(* IEC 61131-3 sources: ml2plc/benchmarks/st (part 12) *)

    weights_3_i : ARRAY[0..4095] OF REAL := [-0.755418241, -0.608314455, 0.360285342, -0.978372037, -0.73372668, 0.0433106236, 0.822168231, 0.994398952, 0.25576961, -0.897847056, 0.964666605, -0.67579025, 0.684332669, -0.809585214, 0.803079665, -0.566751003, -0.408394217, -0.656475842, -0.573797286, 0.747748673, 0.673770845, 0.494365126, -0.699537992, 0.490632325, -0.776397467, -0.676654398, -0.511669755, -0.888815522, 0.76610291, -0.882459223, 0.662760258, -0.724328101, 0.691716373, 0.15585357, 0.931201696, -0.696478367, -0.448318452, -0.338864177, -0.335456759, -0.962986171, -0.592431247, -0.779655039, 0.954741716, -0.817907333, -0.192427114, -0.807255626, 0.855172753, 0.651954412, -0.136959985, -0.420822144, 0.212966338, 0.0445446782, -0.199813604, 0.248965874, 0.838989556, -0.666503072, 0.0486680828, -0.293471068, -0.931513965, -0.615072489, 0.794350803, -0.767282784, 0.800647199, -0.493104696, -1.04894054, -0.839424491, 0.412440658, -1.0782311, -0.610590279, -0.224400103, 0.914384246, 1.09467459, 0.400612175, -0.913536131, 0.880798876, -0.830022335, 0.92901969, -0.925858378, 0.89776057, -0.89756012, -0.580115438, -0.734643281, -0.744657338, 0.821060002, 0.721544206, 0.541094124, -1.03695524, 0.84263134, -1.04971743, -0.930462301, -0.712232709, -0.888018429, 0.880688429, -0.845546246, 1.02739179, -0.692478418, 0.718065321, 0.435147166, 0.961075187, -1.06043577, -0.756034374, -0.573500693, -0.538568377, -0.953424215, -0.810650885, -0.987207532, 1.03647971, -1.00058937, -0.177239105, -1.03699946, 0.988714695, 0.85310322, 0.00717389304, -0.556754231, 0.507442653, -0.0378301032, -0.5122298, 0.447235465, 0.929611444, -0.663908243, -0.0585526079, -0.597246766, -1.02065659, -0.686075151, 0.851084769, -0.72992599, 1.05275869, -0.917103529, -0.811452985, -0.826563954, 0.179984301, -0.835142732, -0.659547448, 0.0863112807, 0.886351824, 0.986944258, 0.135068983, -0.902180672, 0.906524837, -0.855773032, 0.879188478, -0.831542015, 1.05893993, -0.684074581, -0.332585782, -0.95702374, -0.37826848, 0.763411939, 0.510935485, 0.350773633, -0.693967283, 0.556139767, -0.845410943, -0.825000584, -0.515352011, -0.92987591, 1.00201797, -0.865815759, 0.830607235, -0.826742411, 0.697724342, 0.417915851, 1.0467155, -0.983205199, -0.84478277, -0.321441144, -0.468818843, -1.02750862, -0.712836921, -0.86461699, 0.983835578, -0.8388744, 0.0762428418, -1.09817517, 0.828923643, 0.793307722, -0.144390121, -0.211029708, 0.395367414, 0.285318285, -0.472778082, 0.456979275, 0.940658331, -0.763034642, -0.381549388, -0.177495673, -0.90530616, -0.753831744, 0.832921624, -0.774398565, 0.829895437, -0.799162805, -1.21820855, -1.06696033, 0.835389137, -1.26682889, -0.971710622, -0.315437734, 1.23276997, 1.17181158, 0.632770717, -1.20906186, 1.19340575, -1.00084484, 1.0859555, -1.01537168, 1.13232636, -1.02199805, -0.834645152, -1.13640141, -0.815388441, 1.07765841, 0.891493738, 0.978649795, -0.936340988, 0.979935467, -1.06374216, -1.15059888, -0.748942852, -1.1597482, 0.973263681, -1.20231974, 0.933190823, -1.07081246, 0.847544432, 0.364830196, 1.18962157, -0.963554561, -0.808535457, -0.784963489, -0.234990507, -1.13459432, -0.984087408, -0.955592215, 1.10403454, -0.945870757, -0.478384674, -1.300861, 1.14212894, 0.987192571, 0.187816009, -0.865885556, 0.823636711, -0.232717544, -0.0860770419, 0.194109485, 0.987924933, -0.769749939, 0.309627205, -0.921204448, -1.20993173, -0.932157576, 1.02401316, -1.02380764, 1.10313702, -0.987564266, -0.935450852, -0.861052155, 0.385243714, -1.02241755, -0.624481618, -0.0734320283, 1.08894765, 1.13742781, 0.431176722, -1.01322722, 0.922006667, -1.00998127, 0.889069557, -1.04747951, 1.01184118, -0.793883562, -0.560060322, -0.940799952, -0.584474564, 0.723362207, 0.875515103, 0.720968366, -0.911121428, 0.727347374, -1.01887119, -0.835917115, -0.646595657, -1.01109087, 0.976727664, -1.11480069, 0.928580701, -0.732790411, 0.783455253, 0.3726089, 1.02210438, -1.08693635, -0.840154052, -0.561535776, -0.370871723, -1.16396987, -0.911427081, -0.889419734, 0.99090308, -0.945265174, -0.207709432, -1.06947768, 1.11887705, 0.939141095, 0.0903663933, -0.52419728, 0.454987019, -0.0681321621, -0.422043651, 0.423526645, 0.912625194, -0.80558151, -0.0357627831, -0.431746542, -0.890021265, -0.730353892, 0.89218235, -0.759410143, 1.06895053, -0.926181376, -0.741033196, -0.726513982, 0.322699696, -0.972041905, -0.655323505, -0.0292269848, 0.952426255, 0.866428375, 0.11949563, -0.757095098, 0.942866147, -0.796896994, 0.654191136, -0.645846605, 0.824801743, -0.611181915, -0.335965067, -0.810628414, -0.466565788, 0.80544591, 0.691729486, 0.480921775, -0.511504292, 0.702025712, -0.86025691, -0.776957631, -0.29298532, -0.687556684, 0.643776953, -0.739982367, 0.726881027, -0.640373349, 0.57354337, 0.242517203, 0.994883716, -0.606989563, -0.609171987, -0.233668387, -0.257614791, -0.828473866, -0.774299979, -0.623594999, 0.742574334, -0.704159379, 0.0296151433, -0.955602169, 0.968825579, 0.601331949, -0.0735772476, -0.287132144, 0.151510775, -0.0786359683, -0.34978804, 0.133115217, 0.822498322, -0.692448258, -0.215515405, -0.396737725, -0.794197142, -0.61843133, 0.780855775, -0.798789084, 0.636612952, -0.596487164, -1.02452493, -0.733386755, 0.353141606, -0.952989697, -0.727705657, -0.0627208352, 1.21137989, 1.08253932, 0.228804052, -0.90075475, 0.982092619, -0.998478949, 0.896557331, -0.98023051, 1.0387373, -0.700028658, -0.67096138, -0.968751729, -0.84728229, 0.789013982, 0.836730242, 0.688243866, -0.731738687, 0.969447136, -1.06666744, -0.995709002, -0.664720893, -1.05856693, 1.07691407, -1.02315605, 0.728992403, -0.76652348, 0.844830453, 0.179572225, 1.22721124, -0.94140029, -0.715959311, -0.724516153, -0.228294402, -1.1530093, -0.956407428, -0.899410546, 1.09126186, -0.873448253, -0.168818444, -1.22987664, 0.95296061, 1.00769937, -0.0702653304, -0.381446481, 0.512703001, -0.0435364284, -0.11453981, 0.199777916, 1.06700945, -0.684714496, -0.112935178, -0.602526605, -1.02280688, -0.943379998, 0.718487859, -0.927234292, 0.962290883, -0.675989389, -1.04286563, -0.876557887, 0.462482393, -1.0861553, -0.654765189, -0.159290239, 1.07852364, 0.884891152, 0.140386865, -0.963511288, 0.946421504, -1.04198098, 0.839310706, -0.855860889, 0.870488524, -0.702690423, -0.439044088, -0.933871686, -0.589861751, 0.68892163, 0.597560287, 0.425204217, -0.761139214, 0.624503672, -1.02760601, -0.710986853, -0.510669291, -0.832123697, 0.788684607, -1.05656803, 0.902100027, -0.718313038, 0.701382101, 0.336199254, 0.926524699, -0.974620879, -0.690556526, -0.451145768, -0.556159139, -0.986128032, -0.619695544, -0.912777424, 0.842693388, -0.935300767, -0.196174338, -1.05631256, 0.853555441, 0.757244647, -0.184759662, -0.334762543, 0.513675153, -0.0197210051, -0.422626376, 0.306616992, 0.808679283, -0.666823506, -0.0260220375, -0.534840167, -1.05868638, -0.803471029, 1.01640034, -0.656452358, 0.937075615, -0.736741483, -0.969046772, -1.02430713, 0.475471109, -1.01880741, -0.75838691, -0.216517732, 1.14114225, 1.03535259, 0.448151171, -1.05993211, 0.987955809, -0.877148211, 0.88578999, -1.0774231, 1.1040051, -0.910460174, -0.731224537, -0.890228271, -0.725291908, 0.832292557, 0.822500288, 0.545910835, -1.05995345, 0.645671725, -1.10371053, -0.76795429, -0.622391164, -1.10858274, 0.959112167, -1.00889635, 0.884062827, -0.833665311, 0.735249817, 0.367521971, 1.13251293, -0.887471735, -0.932527363, -0.492527246, -0.614649892, -1.0094378, -0.774402618, -1.00567007, 1.00681162, -1.0051012, -0.196057275, -0.977808416, 0.948892236, 0.812963963, -0.00821041875, -0.638639331, 0.399548352, -0.122351654, -0.428168148, 0.473601997, 1.1022259, -0.944955647, 0.0435571112, -0.59750545, -1.01166987, -0.901804149, 0.864712179, -0.801286817, 1.12397861, -0.907543123, -0.968958914, -0.976406515, 0.252034068, -0.996525466, -0.691133738, 0.385438502, 1.00782788, 1.03370297, -0.205928698, -0.884970367, 0.929853916, -0.834381342, 0.924174666, -1.03883147, 1.00104129, -0.721402526, -0.389019519, -0.985671699, -0.479267389, 0.820142806, 0.544877887, 0.263722688, -0.816414952, 0.742167115, -0.977280498, -0.892438114, -0.266501427, -1.07392192, 0.829976678, -0.806288183, 0.836611867, -0.78686285, 0.632151425, 0.518191278, 1.08450913, -0.888277173, -0.780584574, -0.232404694, -0.511793911, -0.958422065, -0.690973699, -0.888970733, 0.83754319, -0.908099651, 0.106050521, -0.930795074, 1.08223093, 0.926879644, -0.449428767, -0.245660082, 0.120277353, 0.183214977, -0.581604123, 0.423586756, 1.03415048, -0.713971019, -0.32305634, -0.0967770889, -0.897503495, -0.723082781, 0.830310166, -0.742337167, 1.02575874, -0.733720362, -0.907611549, -0.854992867, 0.505329072, -0.944037795, -0.70937115, 0.0261288676, 1.01350021, 1.02204335, 0.252643436, -0.978096724, 0.862670481, -0.808062732, 0.896382809, -0.813757539, 0.814833641, -0.642812908, -0.639273047, -0.728571594, -0.703681052, 0.663110316, 0.717055142, 0.489002317, -0.705394208, 0.834371388, -0.781721294, -0.752015114, -0.457937121, -0.792781293, 0.914688826, -0.795861661, 0.595086515, -0.710880637, 0.675870419, 0.406664968, 0.96637696, -0.754895449, -0.686368406, -0.552339971, -0.444466829, -0.997712076, -0.626592398, -0.661046863, 0.88097173, -0.889222741, -0.146164373, -1.08511758, 0.943219721, 0.812917054, 0.0503441095, -0.434279114, 0.274424821, -0.0832945555, -0.193505302, 0.222719252, 0.873863757, -0.539601743, -0.0734653994, -0.442973316, -0.834634125, -0.730556786, 0.631379664, -0.775440812, 0.95656389, -0.50474453, -0.931799293, -0.82169944, 0.194752201, -0.989303291, -0.519775212, 0.112227432, 0.991141856, 1.01745415, -0.0274739582, -0.793622792, 1.06043375, -0.888234019, 0.880099654, -0.893237174, 0.881158412, -0.823377252, -0.437752366, -0.797185361, -0.37659806, 0.858986139, 0.569999754, 0.340523064, -0.836035669, 0.670638025, -0.794342041, -0.702752113, -0.431304663, -0.928568959, 0.926226974, -0.848105371, 0.720710158, -0.622902155, 0.705539167, 0.549153447, 0.870801866, -0.725703001, -0.770241082, -0.183786377, -0.615487993, -0.998608351, -0.745964348, -0.855395079, 0.966465652, -0.77130127, 0.0715011135, -0.96620065, 1.05865717, 0.790433645, -0.268629074, -0.174874589, 0.14475368, 0.0939831361, -0.337278485, 0.395812422, 0.894006252, -0.766367733, -0.176003799, -0.224346429, -0.793370366, -0.638615549, 0.867665052, -0.81962198, 0.82810998, -0.582147717, -0.842648268, -0.783048689, -0.235769719, -0.998877823, -0.327204019, 0.566020548, 0.916653872, 0.854219079, -0.460341662, -0.77112639, 0.933426797, -0.836915135, 0.874533951, -0.83277452, 0.746362567, -0.628461123, -0.084711656, -0.582916021, -0.243317723, 0.525368094, 0.259333014, 0.0327389203, -0.729031205, 0.317607105, -0.839289486, -0.4789671, -0.0461727753, -0.787092328, 0.83384794, -0.75443393, 0.908382654, -0.363875389, 0.546058953, 0.507456422, 0.980222464, -0.675206363, -0.637511611, -0.0142121417, -0.64180088, -0.892539263, -0.407804877, -0.669094205, 0.856718063, -0.493220001, 0.303538859, -0.858540893, 0.940325439, 0.49160096, -0.469009638, 0.17257607, -0.0190391336, 0.469112605, -0.543920636, 0.637618363, 0.764873981, -0.86711055, -0.494828016, 0.157218501, -0.862574041, -0.368994653, 0.676885366, -0.610570908, 0.725115955, -0.861623049, -1.07505918, -0.965862215, 0.60238415, -1.16023743, -0.840752125, -0.105824895, 0.948305309, 0.953172028, 0.288685203, -1.11643279, 1.03585219, -0.971423209, 0.863259971, -1.14757454, 0.967280209, -0.897893667, -0.533795834, -0.847732723, -0.714499772, 0.851787329, 0.7199862, 0.513467252, -0.877711296, 0.906861722, -1.14302409, -0.950012863, -0.768051147, -1.0575242, 0.983039558, -0.990966916, 0.832446694, -0.754112124, 0.893297434, 0.629224181, 0.992561221, -1.00884116, -0.913590014, -0.671533048, -0.474662781, -1.20630717, -0.696899891, -1.07192814, 1.13243151, -0.784192502, -0.15621908, -1.12142682, 1.06379509, 0.912983716, 0.025483191, -0.665657282, 0.413258642, -0.0918736681, -0.556712985, 0.362460822, 1.10431266, -0.784294367, -0.0139337517, -0.611807585, -1.0611099, -0.826119184, 0.902756155, -0.86417675, 1.1229434, -0.856812537, -1.27942991, -0.90530479, 0.625030518, -1.15539479, -0.873494685, -0.260905921, 1.24086809, 1.25946474, 0.39319101, -1.0907501, 1.2032733, -1.08172178, 1.06699085, -1.20631349, 1.22948694, -0.834533453, -0.750264943, -0.992371202, -0.807569206, 0.856315017, 1.08617556, 0.892702281, -1.01682568, 0.886915743, -1.23190653, -1.06336915, -0.932261586, -1.07520664, 1.07185602, -1.12734389, 0.907818377, -0.820663929, 1.01829791, 0.166351378, 1.20455956, -1.17253053, -0.824744999, -0.65868187, -0.317878783, -1.15693378, -0.843500435, -0.920814574, 1.09634209, -0.871699572, -0.450535893, -1.1738621, 1.13490057, 0.895801008, 0.131369889, -0.693567574, 0.74108988, -0.10059008, -0.126341328, 0.0593591593, 1.12989569, -0.740600109, 0.221153483, -0.637960136, -1.14117575, -1.0811311, 1.03810823, -0.89616704, 1.20454895, -0.886058986, -0.818703711, -0.964950979, 0.3011401, -1.05881941, -0.722192585, 0.00358383521, 0.935663342, 0.809548557, 0.160762921, -0.876804471, 0.833429694, -0.830048382, 0.89588958, -0.958845794, 0.874411643, -0.660538614, -0.362247705, -0.670403838, -0.563105106, 0.636587739, 0.495884269, 0.332683057, -0.74164784, 0.724646091, -0.972233713, -0.764483392, -0.447217792, -0.837968588, 0.850412071, -0.983349562, 0.785379887, -0.654432178, 0.724678636, 0.41592297, 0.989545166, -0.950459421, -0.639414907, -0.337752908, -0.484309226, -0.905988812, -0.595648468, -0.844717622, 0.827573478, -0.838856101, 0.0187437031, -0.849463165, 0.889378548, 0.561864376, -0.29927808, -0.392451555, 0.388448268, 0.198650107, -0.559829533, 0.414166063, 0.893056631, -0.908913195, -0.0640959814, -0.374392003, -0.958116055, -0.677774489, 0.828592062, -0.582134187, 0.876991391, -0.876230657, -0.908975899, -0.721173704, 0.494917125, -0.823946416, -0.64437598, -0.217759445, 0.913173795, 0.996590257, 0.367991656, -0.879616201, 0.771492779, -0.98472321, 0.963087082, -0.95259285, 0.839489877, -0.713660777, -0.755366445, -0.73727572, -0.641714454, 0.926426113, 0.728988111, 0.707814932, -0.803486705, 0.719608545, -0.83762908, -0.814273715, -0.611875772, -0.942105889, 0.880182147, -0.971608341, 0.790809631, -0.911215127, 0.898607135, 0.352806628, 0.81870687, -0.761086822, -0.796402991, -0.50277096, -0.537348866, -1.07715547, -0.857042789, -0.950789869, 0.867072821, -0.848236322, -0.411746114, -0.88702327, 1.00351846, 0.825973809, 0.0270913597, -0.71621424, 0.615491807, -0.173585027, -0.227682218, 0.179880247, 0.919904411, -0.736029685, 0.193204731, -0.500456929, -0.822526693, -0.700240195, 0.966011167, -0.801102698, 1.00703526, -0.885540664, -0.713978291, -0.611588717, 0.260023504, -0.922345757, -0.705840707, -0.0141039658, 0.976248503, 0.964204967, 0.26765269, -0.956324041, 0.796898186, -0.789989054, 0.782559752, -0.77758646, 0.867500961, -0.549102545, -0.493753225, -0.801779151, -0.454341143, 0.621101618, 0.647966027, 0.436664164, -0.748553097, 0.54489243, -0.788911521, -0.871274948, -0.460166365, -0.842250288, 0.652063608, -0.863243103, 0.620145023, -0.706633389, 0.78117007, 0.261015654, 0.84503752, -0.820280135, -0.517355144, -0.459893852, -0.314167231, -1.01927006, -0.700387955, -0.742943883, 0.900053501, -0.856171072, -0.0286465324, -0.895612955, 0.856761158, 0.584023952, -0.0770339519, -0.429291189, 0.261452138, 0.0627180338, -0.181542769, 0.112061031, 0.788401484, -0.513115346, 0.077620104, -0.450713575, -0.737526596, -0.571692765, 0.607120872, -0.79032129, 0.799625099, -0.475847691, -1.09786475, -0.772961438, 0.495320827, -1.1611439, -0.766513824, -0.143397436, 0.962765157, 1.06331944, 0.313598633, -1.01686382, 1.1133368, -1.08287513, 0.804114819, -0.856840074, 0.993985593, -0.812854052, -0.610591054, -0.851494789, -0.838413715, 0.978924334, 0.82232976, 0.771277666, -0.730287552, 0.951943219, -0.973897278, -0.990049124, -0.570291817, -0.936770022, 0.858006418, -0.819337249, 0.831573308, -0.891148806, 0.78176415, 0.188151807, 1.05254877, -1.00523531, -0.750526607, -0.642461479, -0.223760605, -1.2113694, -0.936775982, -0.840746224, 1.07401752, -0.79121995, -0.265156776, -1.12808418, 1.07336295, 0.848082721, -0.0801268965, -0.639466107, 0.423318893, -0.197285667, -0.299851, 0.153514013, 0.886098623, -0.601903439, 0.022839861, -0.633413076, -0.839836955, -0.761352301, 0.943436801, -0.842834294, 0.856992543, -0.752803981, -0.976946771, -0.860103667, 0.148241594, -1.17027724, -0.680404603, 0.260861218, 1.1012404, 1.09432316, -0.084494032, -0.919311583, 1.13092101, -1.07132185, 0.954994619, -1.13993835, 1.00824094, -0.845583439, -0.461782247, -0.95956552, -0.488822222, 1.02185178, 0.83047843, 0.552198887, -1.01375663, 0.755363405, -1.0269655, -0.961519718, -0.430978894, -0.921435118, 1.03942025, -1.01963305, 0.888223827, -0.95802629, 0.907438338, 0.721813977, 1.08516002, -1.1015048, -0.968381882, -0.325145304, -0.652126908, -1.28460324, -0.947565973, -0.874286115, 1.05251586, -0.949869156, 0.153231531, -1.18712854, 1.00515926, 0.865185499, -0.298296869, -0.212462679, 0.421099901, 0.405747652, -0.775304854, 0.56657511, 1.02249587, -0.934783936, -0.514021575, -0.20079039, -1.01075089, -0.857002079, 0.987509191, -0.929678917, 0.932180822, -0.886357069, -0.933931828, -0.700244904, 0.369614154, -1.10790706, -0.675352216, -0.188850135, 1.08109188, 1.04684579, 0.308671802, -0.883098602, 1.05010533, -0.929381788, 0.879740238, -1.01128566, 1.10395002, -0.720393658, -0.740107059, -0.99103719, -0.831740022, 0.862007916, 0.894016087, 0.620524406, -0.769335091, 0.897905231, -0.941016138, -0.876742899, -0.708276153, -1.0367837, 0.912421107, -0.825091898, 0.808150589, -0.878788531, 0.916051567, 0.24332048, 1.05220306, -0.952991545, -0.748910844, -0.72116518, -0.374993294, -1.04492664, -0.917863369, -0.86367166, 1.08562934, -1.03882897, -0.218215466, -1.18063104, 1.1076721, 0.878296316, -0.0187482014, -0.528429568, 0.50169456, -0.147743478, -0.122764975, 0.250912666, 0.826420069, -0.730094612, 0.0589699149, -0.46761167, -1.05767417, -0.924309313, 0.804091275, -0.917768538, 0.983291626, -0.721830428, -1.09399235, -1.00202692, 0.562182307, -0.938353002, -0.593690991, -0.0125021413, 1.08856273, 0.906774461, 0.200605094, -1.08938837, 1.09823823, -0.911578178, 0.884976149, -0.867731512, 1.04740059, -0.83649385, -0.525554299, -0.861518741, -0.646086395, 0.715107501, 0.839924991, 0.465662718, -0.874607563, 0.756407976, -1.03819859, -0.815448523, -0.716991901, -0.929483712, 0.948846698, -0.929803491, 0.808668494, -0.6867944, 0.853445053, 0.421883553, 1.09852147, -0.981153369, -0.830782592, -0.503521681, -0.4611803, -1.19973147, -0.676306427, -1.06116807, 0.871525645, -0.893308938, -0.28923732, -1.20726645, 1.16319931, 0.773241103, -0.167875394, -0.538970232, 0.392856359, -0.0467808507, -0.323710591, 0.427655101, 0.908169866, -0.824398875, 0.0668496713, -0.599668503, -1.0336014, -0.750727057, 0.798111081, -0.88163656, 0.99468106, -0.953759074, -1.11895311, -0.975337088, 0.661303043, -1.18804455, -0.69579941, -0.169847563, 1.12572634, 1.17538476, 0.360282838, -0.972973466, 0.919509828, -1.08963072, 0.907667398, -1.18446136, 1.11237955, -0.756965399, -0.708337784, -0.773685694, -0.799184978, 0.745656848, 0.951413512, 0.638455451, -0.967878819, 0.724358022, -1.13330948, -0.790725529, -0.80226022, -1.08631873, 0.949474812, -1.05668902, 0.976779699, -0.861955762, 0.974520147, 0.512347758, 0.955908954, -0.892980337, -0.737581193, -0.617187142, -0.513221383, -1.12916565, -0.880242407, -1.06890917, 1.05162001, -0.815472901, -0.297819644, -1.18346536, 0.946695328, 0.716957748, 0.175897732, -0.667602539, 0.701610804, -0.0740017295, -0.369591564, 0.346157163, 1.05868769, -0.926508367, 0.179177567, -0.475888908, -1.04457426, -0.827824414, 0.98029995, -0.907244384, 0.943478882, -0.924352646, -0.773993492, -0.735044301, 0.0416651331, -0.907257199, -0.422367811, 0.440636724, 0.991895258, 0.759705484, -0.291431665, -0.956883132, 1.00003695, -0.956255972, 0.739793539, -0.74141562, 0.889753878, -0.670551538, -0.231987089, -0.823478103, -0.315503538, 0.595067739, 0.451488137, 0.0750449374, -0.821136713, 0.358170748, -0.763157308, -0.797085702, -0.222883433, -0.833063483, 0.897186339, -0.709599793, 0.797601998, -0.649135232, 0.575399876, 0.694169581, 0.94716084, -0.885367393, -0.612949193, -0.0731305555, -0.618689179, -0.870648324, -0.606274009, -0.917017341, 0.979093015, -0.664984584, 0.407488555, -0.880128086, 0.899560869, 0.68467778, -0.564382672, 0.114791416, -0.0359922089, 0.454897344, -0.658713877, 0.597083151, 0.692245722, -0.672556996, -0.559869766, 0.0941093266, -0.949851394, -0.656304598, 0.892188549, -0.610869884, 0.741495728, -0.754965186, -0.844388545, -0.663963437, 0.100156032, -0.714349389, -0.500820935, 0.0301809032, 0.93849498, 0.795188844, -0.0408474654, -0.778205931, 0.915193319, -0.715432703, 0.726488769, -0.624961197, 0.72919029, -0.444653422, -0.356808156, -0.66607815, -0.495592654, 0.736166477, 0.510713041, 0.304338694, -0.714937925, 0.685840368, -0.841898143, -0.785771668, -0.362618685, -0.843503535, 0.838873625, -0.642146051, 0.515100181, -0.688019276, 0.652499199, 0.163452625, 0.979091167, -0.728121579, -0.39419806, -0.316004902, -0.214974254, -1.02700996, -0.750581741, -0.716689885, 0.746017575, -0.68982774, -0.0666270852, -0.975651443, 0.74363929, 0.783233523, -0.12883997, -0.236293882, 0.151585028, 0.187489644, -0.403225034, 0.297997594, 0.644824266, -0.517803729, -0.261999905, -0.0935142711, -0.751379013, -0.799664259, 0.643151999, -0.769358695, 0.847976506, -0.443437487, -0.865745246, -0.858112276, -0.0854891911, -1.02697647, -0.563964605, 0.411286235, 0.842776775, 1.00849998, -0.220893413, -0.981626332, 0.841228247, -0.869051933, 0.73721987, -0.918379188, 1.00327122, -0.807156563, -0.193718016, -0.772623658, -0.298070163, 0.800232887, 0.408133507, 0.10237436, -0.81515944, 0.44498387, -0.992741346, -0.829405427, -0.15128015, -0.957665145, 0.855219305, -0.923042595, 0.91937834, -0.727190614, 0.777058065, 0.503481328, 0.972717345, -0.792999089, -0.822783053, -0.0296000838, -0.585992575, -1.12478924, -0.65349859, -0.874615133, 0.915536702, -0.865022838, 0.221339598, -0.970219016, 1.03011489, 0.84404099, -0.551715434, -0.000462494208, -0.0881480724, 0.490943015, -0.596435547, 0.544950843, 0.780327618, -0.848713815, -0.504931509, -0.0493441261, -0.965847492, -0.611734152, 0.833947718, -0.779928863, 0.84698987, -0.719679296, -0.888860345, -0.78719759, 0.376279891, -0.800401151, -0.6475631, 0.0540541522, 0.832768381, 0.9913221, 0.254653513, -0.795210302, 0.997577786, -0.926730752, 0.821435809, -0.942105949, 0.994723082, -0.72533679, -0.56359762, -0.830534875, -0.425396651, 0.696741581, 0.705276668, 0.492563456, -0.682713509, 0.685139418, -0.979230583, -0.730480373, -0.522351742, -0.871768355, 0.934757829, -0.723052382, 0.686145604, -0.776319683, 0.605920911, 0.436274976, 0.982208431, -0.929778159, -0.781040549, -0.443694592, -0.353642136, -1.03009582, -0.60700202, -0.745918989, 0.890347838, -0.80710572, -0.0572710522, -0.957512915, 1.00621009, 0.74390775, -0.0205915701, -0.513214886, 0.290729761, 0.10205552, -0.485159516, 0.324673235, 0.780689418, -0.763284326, -0.0712349787, -0.312666744, -0.757450044, -0.674579918, 0.928880155, -0.809836447, 0.961747348, -0.572299957, -0.987814963, -0.665709257, 0.023009887, -1.01407897, -0.491111904, 0.149622276, 1.08481824, 0.813495457, 0.00918790232, -0.988933444, 1.01304257, -0.736413836, 0.713366389, -0.77714926, 0.821009994, -0.718455791, -0.168555468, -0.701443851, -0.444518983, 0.824483514, 0.520365894, 0.331536323, -0.614189804, 0.710616112, -0.939932823, -0.83276999, -0.291009218, -0.740746975, 0.901486218, -0.695580423, 0.65776825, -0.584751487, 0.806130409, 0.480656713, 0.858114123, -0.722780287, -0.544448256, -0.233940363, -0.551465988, -1.09826517, -0.818630636, -0.807670295, 0.881042957, -0.746888697, 0.240349904, -1.04861701, 0.950304866, 0.81671983, -0.239935473, -0.28998813, 0.0921261236, 0.112538286, -0.583798945, 0.515947223, 0.817176998, -0.814985335, -0.317915797, -0.12826775, -0.930432558, -0.836291254, 0.694228888, -0.778837502, 0.935540259, -0.656916857, -0.988335431, -0.956956387, 0.0137774618, -1.12964177, -0.770840764, 0.454703301, 1.08889341, 1.10114956, -0.233997151, -0.9160344, 1.13169825, -0.838038266, 0.851185322, -0.777538717, 0.859436929, -0.862704158, -0.293443888, -0.956585228, -0.420471996, 0.920131326, 0.579383135, 0.173871115, -0.793714345, 0.735676169, -0.859370768, -1.05058193, -0.135776535, -1.05294931, 0.923585951, -0.962093055, 0.725955009, -0.728679836, 0.920734346, 0.429953694, 1.19835913, -0.917490304, -0.828156948, -0.125764608, -0.670550227, -1.15649199, -0.902004242, -0.842370331, 1.06699336, -0.965167105, 0.349797368, -0.910021544, 0.997987449, 0.791344106, -0.4023, -0.198947266, 0.0677236542, 0.388899982, -0.614362538, 0.507743657, 1.02602351, -0.830910623, -0.515007615, -0.0185752213, -0.92261529, -0.795056403, 0.738663793, -0.766319156, 0.822949409, -0.655317307, -0.93890965, -0.991864741, 0.326603681, -0.930119216, -0.815422237, -0.109608583, 0.934924841, 0.920461893, 0.35182032, -1.03809893, 1.10397971, -0.883284926, 0.994623005, -1.07502925, 1.05005991, -0.829090774, -0.672549129, -0.804675579, -0.568975568, 0.760407686, 0.737354517, 0.703553975, -0.8440485, 0.720817268, -0.91479063, -0.810900331, -0.507740676, -1.06939578, 0.840505183, -1.08498955, 0.917757034, -0.803289056, 0.911749065, 0.413806319, 0.992159247, -0.918016732, -0.710864782, -0.431193411, -0.444666862, -1.07377923, -0.78019011, -0.840355754, 0.860853255, -0.819990814, -0.260453254, -1.1637423, 0.952289402, 0.863986433, -0.0693490952, -0.43248719, 0.455752134, -0.168676227, -0.297006905, 0.378284246, 1.08168149, -0.759329259, -0.00800242741, -0.520838499, -1.0476948, -0.675572634, 0.885056794, -0.778042734, 0.970966935, -0.739053071, -1.18367076, -1.00170863, 0.515894175, -1.04622996, -0.734378457, -0.0634912625, 1.05683684, 1.13232851, 0.479658991, -1.14697683, 1.14479041, -1.14973688, 0.966424525, -1.11149096, 1.02778423, -0.863198936, -0.751709819, -0.888835311, -0.804755151, 0.858745933, 0.760714173, 0.756437302, -1.01159966, 0.79420507, -0.995307148, -0.96403861, -0.779833555, -1.0982914, 0.976376057, -0.940571666, 1.07449925, -0.787972987, 0.893660724, 0.253314584, 1.15125144, -0.931932032, -0.726671219, -0.747295558, -0.29423061, -1.28276575, -0.797924876, -0.918390751, 1.14562893, -0.875937521, -0.149294049, -1.15881169, 0.992793918, 0.796081841, 0.0344517604, -0.689107001, 0.556009471, -0.0333260484, -0.188356966, 0.273446709, 1.0719341, -0.849202156, -0.0576614663, -0.497593015, -0.946819425, -0.795422435, 1.04014468, -0.872544289, 1.03207433, -0.746326625, -1.02014303, -0.913138747, 0.174102426, -0.961304426, -0.703736424, 0.142996088, 0.887258172, 1.06656015, 0.0410478935, -0.815817237, 1.11459541, -0.986689091, 0.869543433, -0.807072699, 1.02771664, -0.741206229, -0.168933392, -0.840292573, -0.516178131, 0.788471043, 0.654079497, 0.241704389, -0.678604484, 0.690058768, -0.985296369, -0.889898062, -0.42652756, -0.942365468, 0.840480506, -0.84049958, 0.685397267, -0.654555202, 0.743690073, 0.498869985, 0.984338284, -0.931772113, -0.667692959, -0.149191111, -0.586353421, -1.2004689, -0.613616288, -0.750702798, 1.02661479, -0.968156934, 0.27459839, -1.09536994, 0.869792044, 0.795942605, -0.170552939, -0.119759001, 0.0561317392, 0.298612505, -0.487057149, 0.431264818, 0.776092827, -0.863675654, -0.31945172, -0.222689167, -0.939694643, -0.881493151, 0.77813375, -0.859104395, 0.980753601, -0.835472226, -0.780811608, -0.908254683, -0.0700671524, -0.95471555, -0.243140265, 0.656840563, 0.788265705, 0.808628798, -0.287140399, -0.73185581, 0.784762442, -0.899206996, 0.664094448, -0.895017982, 0.714929521, -0.709218681, -0.0350017548, -0.476985365, -0.132147655, 0.395060271, 0.278724641, 0.0243162718, -0.786040306, 0.254208386, -0.678958178, -0.484509289, -0.143013015, -0.938613236, 0.934693396, -0.907608032, 0.640249074, -0.42963931, 0.273129761, 0.511628985, 0.767143548, -0.835145712, -0.839953721, 0.0871558934, -0.592077434, -0.865831912, -0.400098443, -0.678308547, 0.920655668, -0.61952275, 0.457279861, -0.751586497, 0.815800011, 0.471407712, -0.510838628, -0.0146660823, 0.0550350286, 0.52525425, -0.518903434, 0.713679194, 0.761300564, -0.625218272, -0.626365364, -0.0270288847, -0.688027024, -0.415846318, 0.709429741, -0.505770206, 0.885988295, -0.633718252, -0.976370275, -0.805604398, 0.369813204, -1.09729612, -0.631916106, 0.0831616595, 0.925421715, 0.985631824, 0.132714882, -1.04596221, 0.945217013, -1.06315434, 0.974209487, -1.01574898, 1.08618009, -0.712410092, -0.450384706, -0.97908324, -0.498778701, 0.673285246, 0.646217763, 0.311322898, -0.774297357, 0.543726921, -0.994351029, -0.768154562, -0.448112994, -1.03144801, 1.08958042, -0.900835633, 0.93874824, -0.792783737, 0.862766981, 0.478894234, 0.927475333, -0.916345716, -0.760724545, -0.405634254, -0.749832273, -1.10986936, -0.626981199, -0.970400333, 0.897742629, -0.854419649, 0.0998076871, -0.885941565, 1.02640998, 0.810763836, -0.172908932, -0.219355851, 0.166053206, 0.361918479, -0.608354628, 0.483504057, 1.00468135, -0.954490066, -0.276456952, -0.409829766, -0.833084106, -0.650721133, 0.763146698, -0.666514695, 1.06439698, -0.975921452, -0.976468682, -0.791674674, -0.177903861, -0.843917489, -0.267525673, 0.634957194, 0.920786977, 0.971808851, -0.392000765, -0.850517333, 0.800255775, -0.802226901, 0.909082353, -0.877137661, 0.730122745, -0.851397216, -0.0722328052, -0.537836909, -0.187319443, 0.36514619, 0.253046304, 0.10816586, -0.727519393, 0.41508621, -0.938324273, -0.499514312, -0.12158455, -0.918444216, 0.761836886, -0.689384639, 0.710212231, -0.410224855, 0.548989832, 0.634191751, 0.939039767, -0.704807699, -0.801940441, 0.0953865424, -0.540097415, -1.03223205, -0.523439586, -0.819470525, 0.860700846, -0.656160235, 0.297524452, -0.947977126, 0.90694356, 0.621159196, -0.502045631, -0.0506013669, -0.123203866, 0.503702044, -0.652031302, 0.529158711, 0.842695534, -0.672055542, -0.543978214, 0.20170027, -0.951138258, -0.517390072, 0.885154307, -0.364636242, 0.83135426, -0.658487439, -0.968474865, -0.622928381, 0.308044612, -0.946219087, -0.729095697, -0.020170588, 0.929763079, 0.992177188, 0.0572009496, -0.789075613, 0.864978194, -0.953618169, 0.711665154, -0.742936492, 0.943210602, -0.633800924, -0.483225018, -0.829375863, -0.47125262, 0.61733675, 0.571785808, 0.56263268, -0.589145005, 0.645672798, -0.800022244, -0.656003237, -0.306997836, -0.753312528, 0.707771122, -0.822233975, 0.788333774, -0.610611498, 0.576294065, 0.368350208, 0.956656158, -0.788423836, -0.574761868, -0.428307831, -0.336391181, -0.882566571, -0.633512914, -0.797103524, 0.918003321, -0.843789279, -0.0639619157, -0.80085057, 0.995271385, 0.673964679, -0.0921275243, -0.465578198, 0.266843677, 0.156025752, -0.212184533, 0.420018256, 0.712551475, -0.611166835, 0.0293651894, -0.373225451, -0.869483173, -0.824524105, 0.650054216, -0.835338175, 0.69953686, -0.733144045, -0.94825989, -0.829286873, 0.498820007, -1.10125899, -0.934159279, -0.237553403, 1.17959416, 1.00506413, 0.241874829, -1.10324156, 1.08897948, -1.04178441, 0.961241484, -1.05229485, 1.16768396, -0.701199234, -0.684071183, -0.882459939, -0.842701197, 1.0047071, 0.993355274, 0.698987246, -0.736815214, 0.930523276, -1.00445724, -0.908867478, -0.62573576, -0.918404937, 0.990144253, -1.01239693, 0.988601685, -0.930237651, 0.933457732, 0.253664821, 1.04263794, -0.863427281, -0.590768814, -0.540168464, -0.446616054, -1.17079878, -0.859642208, -0.895760119, 0.942056179, -1.00492251, -0.170379594, -1.21758735, 1.19851482, 0.993596911, 0.113135502, -0.49006626, 0.397776872, -0.213488877, -0.203544989, 0.229960397, 1.05145907, -0.759326816, -0.055846002, -0.525532544, -0.943355918, -0.8732934, 1.04964459, -1.01602924, 0.884545803, -0.781898618, -0.723886073, -0.62977469, -0.204483747, -0.829271317, -0.245969415, 0.436119974, 0.811825335, 0.602030814, -0.28100431, -0.742344499, 0.827918768, -0.690657675, 0.799997211, -0.829492569, 0.817033291, -0.544541478, 0.0358796567, -0.484106064, -0.0552955978, 0.382008195, 0.129058108, 0.0748274773, -0.628724813, 0.250387967, -0.706169128, -0.34636569, -0.116365537, -0.719126046, 0.759861112, -0.715697706, 0.609559476, -0.281813145, 0.249621287, 0.675493002, 0.778470099, -0.730745196, -0.775118828, -0.0318290442, -0.635053277, -0.64971602, -0.264338791, -0.766497374, 0.836210966, -0.335421443, 0.336263001, -0.797662616, 0.600033104, 0.447682649, -0.477033317, -0.00602800678, -0.00347518804, 0.343229294, -0.595320761, 0.690001249, 0.743430614, -0.678604662, -0.573144078, -0.00853874814, -0.787870467, -0.398957372, 0.805735111, -0.208311886, 0.579948843, -0.63110131, -0.929738283, -0.772374809, 0.271806598, -1.01329947, -0.858100355, 0.452278465, 0.916744471, 1.14639127, -0.0263592731, -1.10906065, 1.10039926, -0.990095317, 0.872081578, -1.00980031, 1.0308758, -0.929622769, -0.465474278, -1.04688621, -0.639739394, 0.931501687, 0.756015897, 0.321964175, -0.837107778, 0.727318883, -0.864199638, -0.92858845, -0.460382283, -1.00176477, 1.08890307, -0.86653173, 0.931799054, -0.745827913, 0.919408202, 0.704915285, 0.975672781, -0.900074422, -0.817533493, -0.44180873, -0.754927456, -1.14283717, -0.874060333, -0.996847332, 0.962824225, -1.00731623, 0.143175423, -1.13962972, 0.926433623, 0.944086671, -0.256617039, -0.177992538, 0.234126672, 0.226686522, -0.728595674, 0.598063231, 1.08225262, -0.801509559, -0.299066722, -0.216455579, -1.04918098, -0.889964759, 0.808224797, -0.858967721, 1.00894785, -0.893621087, -1.11113048, -0.911374986, 0.0543966405, -1.00301683, -0.733756423, 0.162385717, 1.0429635, 0.924938262, 0.0733157992, -0.956732213, 1.098562, -0.887375534, 0.966252506, -0.887113035, 1.02406406, -0.76543504, -0.400138885, -0.833865285, -0.589645863, 0.911189914, 0.675319374, 0.241477102, -0.848621309, 0.712136924, -0.961093903, -0.76611954, -0.396515459, -0.87194252, 1.02525055, -0.935948014, 0.96596688, -0.670312822, 0.669189751, 0.521194339, 0.981858134, -0.923735201, -0.834396899, -0.380213201, -0.490119696, -1.01803303, -0.837935627, -1.01692939, 0.893213272, -0.890941322, 0.0512234196, -0.938236773, 1.12978613, 0.822078764, -0.381286681, -0.354263991, 0.140916765, 0.279109687, -0.467644393, 0.549917936, 0.861881733, -0.847081482, -0.202907324, -0.183476627, -0.885915756, -0.69544071, 0.890836477, -0.817651927, 0.933344722, -0.846282125, -1.03862607, -0.947054029, 0.0615682788, -1.11174715, -0.548233747, 0.256683737, 1.14824474, 1.03675997, -0.306727588, -0.964119434, 0.973472714, -0.999305964, 0.839141071, -0.847896695, 0.932551801, -0.85014081, -0.284629256, -0.997696638, -0.367976367, 0.86989969, 0.621583104, 0.341185182, -0.79054755, 0.637244344, -0.795998812, -1.03838813, -0.121878378, -1.02120984, 1.03450096, -0.847081721, 0.791102886, -0.929135621, 0.91503346, 0.493659556, 1.08521104, -0.794698179, -0.783615708, -0.149818674, -0.577271104, -1.22717381, -0.729105532, -0.907890081, 0.904237509, -0.840050995, 0.355233908, -1.16810739, 1.03836215, 0.833904982, -0.270463109, -0.190144002, 0.053217493, 0.424836487, -0.619497418, 0.575297952, 0.876965404, -0.721707761, -0.473643988, -0.0170233063, -0.972761631, -0.806016803, 0.886822879, -0.859126747, 0.807136118, -0.873356402, -0.532830179, -0.612299204, -0.122964926, -0.61621964, -0.069940798, 0.433616072, 0.501196623, 0.503526568, -0.233648106, -0.60350734, 0.448003024, -0.501408577, 0.619695842, -0.559005618, 0.637978077, -0.461325794, 0.105104662, -0.2573511, -0.186585173, 0.354441494, 0.0737063959, -0.0460065231, -0.527710378, 0.219412535, -0.493068904, -0.205879152, 0.105828926, -0.675325096, 0.475340486, -0.548010886, 0.423154175, -0.336760581, 0.255975366, 0.460904866, 0.59745276, -0.58728838, -0.609239519, -0.103507549, -0.399057329, -0.407381773, -0.241226628, -0.419427693, 0.671428859, -0.44988206, 0.220640793, -0.421603203, 0.538674831, 0.297478944, -0.44234702, 0.0603176206, 0.0442613475, 0.371121526, -0.471603364, 0.439350307, 0.667813361, -0.391252607, -0.265212685, 0.00789033435, -0.435489267, -0.239340037, 0.593510747, -0.247391731, 0.534566224, -0.603185236, -0.792371094, -0.739380062, 0.713901758, -0.817053378, -0.852856994, -0.179341659, 0.959845006, 0.770885408, 0.324391484, -0.854621291, 0.786259651, -0.661624253, 0.757754922, -0.741588593, 0.824353218, -0.569926322, -0.575232327, -0.886677504, -0.837767422, 0.783255398, 0.733940661, 0.607587218, -0.757613301, 0.867251217, -0.983041406, -0.95171237, -0.758144796, -0.83637464, 0.595348895, -0.936923146, 0.668096066, -0.798557997, 0.725486815, 0.424645394, 0.707889974, -0.665016055, -0.47084704, -0.67993921, -0.375449032, -0.918146729, -0.776643753, -0.827958047, 0.819822788, -0.888391256, -0.210734129, -0.90350759, 0.928226888, 0.923699737, 0.104914516, -0.624729991, 0.554213703, -0.303485304, -0.377347738, 0.128166661, 0.864066422, -0.585147917, 0.200534806, -0.728587449, -0.80727452, -0.68116796, 0.707198918, -0.795398533, 0.679158926, -0.710352719, -0.962701142, -0.812521577, 0.127895594, -0.848725259, -0.558891773, 0.243628547, 0.956765711, 0.816756129, 0.108055905, -0.944031239, 1.00386214, -0.892733634, 0.766236484, -0.806172073, 0.940659046, -0.641631424, -0.318218708, -0.931178689, -0.340961009, 0.828006566, 0.722664773, 0.248382315, -0.824228764, 0.508430898, -0.891737044, -0.878963828, -0.301210672, -0.746851981, 0.863421857, -0.857524335, 0.777775943, -0.735813081, 0.728388309, 0.34783417, 0.965335965, -0.786547422, -0.812392235, -0.321248323, -0.538291335, -1.09552181, -0.805899978, -0.891295195, 0.924740314, -0.796732783, 0.0918886662, -1.09573889, 0.823742509, 0.724403679, -0.32133618, -0.198802829, 0.122519381, 0.0665191114, -0.591669798, 0.354328364, 0.860146463, -0.769168377, -0.328037053, -0.152577445, -0.765176296, -0.798249722, 0.721755147, -0.802870333, 0.974007308, -0.765210569, -1.02971113, -0.863262057, 0.294929892, -0.873904765, -0.668876112, 0.224371701, 0.850640297, 1.01778233, -0.0772373825, -0.797427595, 1.05826008, -0.930305243, 0.792840004, -0.764625669, 0.843560815, -0.631143749, -0.3468557, -0.82498461, -0.365978032, 0.778761089, 0.538974524, 0.40057835, -0.742695212, 0.532127142, -0.897926211, -0.93071723, -0.499519289, -0.883000612, 0.792768776, -0.867752314, 0.751485407, -0.818368495, 0.623130143, 0.346275657, 1.03179812, -0.977597117, -0.863486946, -0.480615079, -0.519268036, -1.00494742, -0.667935312, -0.914928854, 0.873737097, -0.858839393, -0.0702849999, -1.06019449, 1.0806725, 0.772564471, -0.251107931, -0.252646863, 0.3580468, 0.136758775, -0.557268441, 0.447885424, 0.954984426, -0.92693764, -0.222680256, -0.201380536, -0.79762882, -0.641146898, 0.73164171, -0.804575026, 1.01352036, -0.876159906, -0.993184566, -0.791009843, 0.504641533, -0.921791077, -0.816360116, -0.196006298, 1.17310393, 1.05226195, 0.382271826, -0.894057274, 0.984008789, -1.09940231, 1.00387776, -1.00434065, 0.94280237, -0.691696286, -0.81867069, -0.82539314, -0.828855813, 0.80027622, 0.888840199, 0.800766945, -0.748210132, 0.834859431, -0.880362272, -1.03611803, -0.686120629, -1.06963181, 1.07744288, -1.03263533, 0.885977745, -0.782256365, 0.808066666, 0.316192836, 1.15501893, -0.884240448, -0.611134648, -0.812284827, -0.347036064, -1.00437868, -0.841145515, -0.869562924, 0.925918996, -1.00450277, -0.273400426, -1.16757858, 0.982424915, 0.847116649, -0.0370410681, -0.546299517, 0.568685651, -0.237957954, -0.110121593, 0.262624055, 1.06115329, -0.711271048, 0.201648265, -0.638166785, -0.890225887, -0.771624029, 0.82232964, -1.02269852, 0.905648887, -0.859919012, -1.01018035, -0.852937341, 0.199344724, -1.02075493, -0.557302475, 0.122542568, 1.04583883, 1.05831313, -0.131008953, -1.04885328, 1.13267505, -0.973243535, 0.892987728, -0.859983087, 1.00251496, -0.922155261, -0.49669224, -0.813681483, -0.459259152, 0.90394032, 0.520107567, 0.40480119, -0.884002805, 0.734116495, -0.846735358, -0.961679697, -0.353904635, -0.985855341, 0.886004329, -0.976658583, 0.887159467, -0.660021305, 0.760787725, 0.630375803, 1.00861239, -0.990624189, -0.776782095, -0.300165325, -0.613854587, -1.16555989, -0.739156306, -0.887333751, 1.07783723, -0.886344194, 0.183636725, -1.04426599, 0.903318882, 0.800231457, -0.209712222, -0.32627964, 0.352689356, 0.333587348, -0.646154046, 0.6284917, 1.00177336, -0.7466923, -0.262597769, -0.228939399, -0.921233594, -0.690168798, 0.961507738, -0.825392723, 0.950034082, -0.894637525, -1.07029724, -0.74155581, -0.110260643, -1.01186144, -0.467203647, 0.419715881, 1.02206957, 1.06065667, -0.193051681, -1.01871479, 1.04745793, -0.969526291, 0.882115364, -0.793250442, 1.00953889, -0.881716251, -0.285185963, -0.733971596, -0.430095583, 0.666744351, 0.537245572, 0.197210357, -0.820546985, 0.478942424, -0.867832482, -0.904418588, -0.306358516, -0.987072885, 0.923965573, -0.827970445, 0.942754388, -0.813830674, 0.810630918, 0.598882854, 0.965327322, -0.958405077, -0.789805353, -0.0247831345, -0.64611125, -1.0609479, -0.646289349, -0.943482101, 0.90460068, -0.898542881, 0.241582885, -1.05070531, 0.839297295, 0.659592569, -0.306077451, 0.0500512682, -0.0570018664, 0.510157228, -0.61130023, 0.708471656, 0.852460563, -0.701989949, -0.37463814, 0.00335903093, -1.03780794, -0.670634925, 0.787285209, -0.635788918, 0.847452581, -0.702324629, -1.005234, -0.968812108, 0.447139084, -1.17164814, -0.869274616, -0.0655961037, 0.966442049, 0.993079126, 0.415281653, -1.0261327, 1.03079224, -0.937661529, 0.961169541, -1.15573311, 1.12316489, -0.947063088, -0.609770119, -0.827906549, -0.691708922, 0.942700982, 0.827459455, 0.576645792, -0.842250884, 0.842586279, -1.15715313, -0.955552638, -0.59762311, -1.01382136, 1.08575153, -0.963505149, 1.00307536, -0.936788976, 0.826114357, 0.386973441, 0.980013311, -0.95651722, -0.925170422, -0.611601055, -0.611125529, -1.0324471, -0.726434052, -0.87263602, 1.10575986, -0.897451043, -0.208583012, -1.07795715, 1.14604986, 0.928188145, -0.0521513931, -0.618541777, 0.59916842, -0.193706781, -0.415743053, 0.440905035, 1.14346862, -0.926543593, -0.0363977067, -0.477990896, -0.982643366, -0.867311776, 0.935358524, -0.973981082, 0.931315124, -0.845630407, -0.861772954, -0.721524179, 0.0986454412, -1.03133488, -0.570533097, 0.261758417, 0.965813875, 0.982137144, -0.0293426253, -1.03436482, 1.06985724, -0.950913906, 0.922353983, -0.806497097, 0.783380806, -0.658890784, -0.449607164, -0.89537859, -0.385259211, 0.713460863, 0.729782641, 0.473796427, -0.924663186, 0.578554451, -0.803543389, -0.671633184, -0.382577837, -0.8009305, 1.00022399, -0.933638573, 0.836028934, -0.563164771, 0.629320562, 0.546176434, 0.915136099, -0.869614005, -0.753042638, -0.4967058, -0.524411798, -0.951225638, -0.611946225, -0.92792213, 1.05263615, -0.89749366, 0.0132358298, -1.11050832, 0.983382344, 0.854296625, -0.182954162, -0.181268334, 0.198000371, 0.302228659, -0.43596226, 0.403358847, 0.850450814, -0.853324413, -0.220359758, -0.166480929, -0.943998992, -0.767611206, 0.848755598, -0.657482505, 0.841426432, -0.721938431, -0.808539927, -0.923175871, 0.05690597, -0.875962317, -0.495678008, 0.557142079, 0.931773603, 0.924619436, -0.44155696, -0.836186647, 1.08503079, -0.938528895, 0.992791533, -0.907654107, 1.02695823, -0.728081107, -0.0550730638, -0.679002643, -0.221366316, 0.680275738, 0.391920954, 0.214570433, -0.699837446, 0.654629827, -0.907504678, -0.761733353, -0.138699621, -0.858287454, 0.829922318, -1.01176488, 0.793316185, -0.719401836, 0.715198278, 0.698503673, 1.03310657, -0.94738251, -0.69627142, 0.00782040507, -0.652584016, -1.15452898, -0.698288977, -0.787849724, 1.0273881, -0.834000468, 0.372734994, -1.11593997, 0.926637769, 0.772196352, -0.35649237, 0.12004476, 0.0972433984, 0.553599775, -0.4949072, 0.76016742, 0.810973287, -0.905270457, -0.523971677, 0.0969828069, -0.832741797, -0.768331468, 0.775760949, -0.682405889, 0.883137941, -0.85619998, -0.989380658, -1.03457499, -0.0517622754, -0.932550669, -0.694942057, 0.528805315, 0.975854874, 0.958423674, -0.140165061, -1.08478153, 1.1421417, -0.970185518, 0.968834043, -0.844599009, 1.11847758, -0.774316072, -0.211446851, -0.861546516, -0.456038833, 0.966504276, 0.710692942, 0.214514136, -0.992433667, 0.674419701, -0.838600397, -0.797830403, -0.452291369, -0.87957257, 0.952979147, -1.04137182, 0.756499469, -0.881576478, 0.697081447, 0.495766819, 1.02677464, -0.817020655, -0.823269069, -0.18381232, -0.535384774, -1.06303358, -0.883768439, -0.897187591, 1.11861014, -0.870897472, 0.187550664, -1.03782761, 1.17324579, 0.888868153, -0.341810137, -0.0556954741, -0.0158871058, 0.322948873, -0.588214874, 0.501251698, 1.04257047, -0.742597222, -0.393232524, -0.0918072313, -0.945177972, -0.824784875, 0.926980078, -0.747276783, 0.995664954, -0.691841543, -1.00853765, -0.713255107, 0.647285819, -0.852226436, -0.846004665, -0.168666676, 0.902311683, 0.944902182, 0.267628074, -0.958007157, 0.840322256, -0.887698829, 0.961279511, -0.776420653, 0.94608885, -0.862158537, -0.605205178, -0.915220797, -0.628228426, 0.848300576, 0.839160681, 0.57141012, -0.905398667, 0.858483016, -0.889531493, -0.82938236, -0.598610878, -0.968016028, 0.819422901, -0.985393584, 0.842359126, -0.748422325, 0.876093566, 0.386232138, 0.704279602, -0.881875217, -0.762673676, -0.629377842, -0.501640975, -0.807521403, -0.884190679, -0.717874348, 0.913320184, -0.892254114, -0.298563749, -0.930075765, 0.775691807, 0.863675773, 0.125792608, -0.618853033, 0.577705622, -0.0251189768, -0.432866186, 0.377281308, 0.980280399, -0.649286807, -0.0607887618, -0.45323652, -0.968550265, -0.698687017, 0.831464946, -0.749712884, 0.786249042, -0.669413984, -0.700759172, -0.690960705, 0.219630286, -0.874300182, -0.59967339, 0.000577162486, 0.755742371, 0.729254723, 0.199102446, -0.876938522, 0.794218957, -0.663940489, 0.733607531, -0.698495746, 0.885335922, -0.571763039, -0.293765396, -0.804308891, -0.550076067, 0.569750428, 0.615945041, 0.313869447, -0.587247789, 0.688019931, -0.895350873, -0.723046601, -0.452467203, -0.820372641, 0.6793347, -0.766393602, 0.565901518, -0.507283568, 0.568262339, 0.415052295, 0.915370524, -0.716443479, -0.424843311, -0.460298181, -0.361261994, -0.903628588, -0.648115396, -0.738555253, 0.800467253, -0.795145512, -0.0115165636, -0.944992721, 0.889130592, 0.767579377, -0.139246643, -0.375697315, 0.36367327, 0.143317923, -0.265599102, 0.306399882, 0.68444252, -0.647032976, -0.108279914, -0.276576221, -0.652727604, -0.799071014, 0.564529896, -0.729636312, 0.606915534, -0.580234945, -0.774507999, -0.857604742, 0.429399729, -0.930867374, -0.651145041, -0.0314018019, 0.9284513, 0.950723827, 0.181736708, -0.94284606, 0.777048528, -0.899705112, 0.752479076, -0.709820509, 0.953935325, -0.536857426, -0.453155041, -0.679491878, -0.604841769, 0.783517122, 0.599752367, 0.318136007, -0.594205081, 0.676581621, -0.877049088, -0.731319427, -0.511449099, -0.862341225, 0.892369747, -0.814184546, 0.754008353, -0.715054214, 0.698685884, 0.233145103, 1.01863647, -0.690535367, -0.589026153, -0.334243953, -0.220951915, -0.930629253, -0.559661031, -0.749486089, 0.953985274, -0.831374645, -0.0278570782, -0.82597959, 0.771127641, 0.682325423, 0.0170961022, -0.279765844, 0.382275105, -0.023843443, -0.234016284, 0.137231991, 0.922935069, -0.595442712, 0.0992795452, -0.49003467, -0.927733064, -0.688692808, 0.736590385, -0.632792711, 0.925248921, -0.613666236, -1.16928852, -0.854762793, 0.0468913354, -1.18165219, -0.781460166, 0.331295043, 1.18376422, 1.15690267, -0.241335928, -1.13221955, 1.17465961, -1.12600315, 0.85642612, -1.0159322, 1.13213372, -0.90468365, -0.414374441, -0.809111953, -0.528228104, 0.830214083, 0.714342952, 0.362617999, -0.976914048, 0.72939831, -1.04324293, -0.884737849, -0.339856893, -0.906443477, 0.955860972, -1.04917729, 0.858124316, -0.725417972, 0.743358731, 0.585490286, 1.20731747, -0.850624859, -0.874786615, -0.405697405, -0.565402925, -1.04332829, -0.759941936, -0.922682583, 1.02715707, -1.02701879, 0.190939397, -1.04053569, 1.0984509, 0.769177556, -0.344820887, -0.306929022, 0.040846061, 0.500335574, -0.723776221, 0.589993179, 0.981675565, -0.991475999, -0.425548941, -0.117642395, -0.915643394, -0.815215707, 0.916038752, -0.969600379, 1.12809849, -0.751632512, -0.862899303, -0.829141974, -0.0570159368, -0.737937391, -0.273056149, 0.489814162, 0.882974625, 0.689721644, -0.325598091, -0.854503095, 0.690012515, -0.717048287, 0.858363569, -0.755031466, 0.654838562, -0.727559149, 0.116936356, -0.403147727, -0.0911585465, 0.421337515, 0.204730436, -0.0789451748, -0.842997909, 0.138907969, -0.854771733, -0.345312566, 0.0786507577, -0.880420327, 0.7018255, -0.648191214, 0.608898759, -0.424877197, 0.386772513, 0.689378798, 0.812096119, -0.645421565, -0.738684177, 0.092786476, -0.520626843, -0.807718277, -0.174863353, -0.81000948, 0.828145087, -0.413771659, 0.345121145, -0.790848255, 0.682513893, 0.404779643, -0.457731128, 0.234948263, -0.0156717561, 0.387670338, -0.727176011, 0.640328646, 0.74883163, -0.835190475, -0.563892007, 0.0542730503, -0.864046574, -0.342467546, 0.816046357, -0.424440503, 0.70988059, -0.637702584, -0.937841892, -0.889083564, 0.268207818, -0.805704176, -0.721465349, -0.00490556099, 0.901388884, 0.80767101, 0.213178098, -0.751282811, 0.899395168, -0.725854814, 0.748562276, -0.986488461, 1.00970292, -0.628750443, -0.404512465, -0.834999561, -0.666034818, 0.780131698, 0.580195248, 0.443588674, -0.779767275, 0.75757575, -0.764169872, -0.708934724, -0.357157409, -0.990183473, 0.773827612, -0.729798257, 0.909026921, -0.786345541, 0.774623275, 0.468835086, 0.890515149, -0.753928065, -0.60978061, -0.565818489, -0.363415778, -0.886048853, -0.586931825, -0.881760061, 0.751504302, -0.743851066, -0.00649144407, -0.97195828, 0.961859286, 0.657981575, 0.0401829779, -0.278608352, 0.372902483, -0.131196737, -0.36559844, 0.192959338, 0.882446885, -0.665415108, -0.139419302, -0.510242403, -0.971634388, -0.814798832, 0.688571632, -0.67599684, 0.900357485, -0.822175205, -1.1110909, -0.866408885, 0.537440896, -0.982464671, -0.892360926, -0.0193753131, 1.1145103, 0.985346854, 0.177099958, -0.932675481, 1.0265522, -0.955097854, 0.866545022, -0.951171875, 0.936732709, -0.586589515, -0.753251791, -0.954349875, -0.913152814, 0.846741498, 0.921646535, 0.601255655, -0.841526389, 0.821996033, -1.10704231, -0.938263834, -0.786375642, -0.959054649, 1.06783462, -0.897728741, 0.715040922, -0.954261363, 0.90016979, 0.314348668, 1.08457112, -0.897332907, -0.586558402, -0.513837397, -0.468146712, -1.04694176, -0.997831762, -0.988519728, 1.08274424, -1.03911412, -0.0763379037, -1.19924867, 1.13884616, 0.861875355, -0.035394527, -0.645141602, 0.540617466, -0.00713570463, -0.398186237, 0.188419178, 0.941889644, -0.585887313, 0.0222373828, -0.59352988, -0.954482138, -0.827650249, 0.993924975, -1.01277149, 1.00802708, -0.588631153, -1.02202189, -0.747009635, 0.613322556, -0.897544682, -0.732982278, -0.456595093, 0.962276399, 0.795332074, 0.671077371, -0.967659414, 0.853868723, -0.770793259, 0.833329558, -0.97578615, 0.848643482, -0.857904911, -0.798365831, -0.795888245, -0.857467532, 0.966209948, 0.736484468, 0.695706427, -0.886226654, 0.788673043, -1.01052272, -1.0286032, -0.748519123, -1.0185672, 0.874143004, -1.06077802, 0.694009662, -0.843938947, 0.878933787, 0.349594027, 0.800177395, -0.717908025, -0.594196796, -0.656258881, -0.556953669, -0.846859157, -0.79142803, -0.845962942, 1.04326403, -0.868588626, -0.562533617, -0.85183394, 1.01098347, 0.952204704, 0.282487959, -0.872518361, 0.721074104, -0.31151703, -0.378997952, 0.282929897, 1.03048205, -0.549017072, 0.0635976419, -0.835636377, -0.912023246, -0.88585341, 0.776455045, -0.85138154, 0.971118808, -0.843461335, -0.921734393, -0.891871095, 0.215065777, -0.998061776, -0.627441168, -0.00694472902, 0.936757505, 0.960935533, 0.124367289, -0.888317347, 0.825734615, -0.937575281, 0.886772931, -0.929073453, 0.91916132, -0.616435409, -0.292480201, -0.790857792, -0.357805163, 0.654396594, 0.474305242, 0.45884648, -0.80382973, 0.717312634, -0.807204485, -0.658123434, -0.377325684, -0.822481692, 0.724415779, -0.953108728, 0.76014626, -0.693366945, 0.563358843, 0.411203325, 1.03892446, -0.712390542, -0.538339972, -0.27133134, -0.402222306, -0.99378258, -0.604566932, -0.665674448, 0.884491324, -0.862252116, -0.0283179767, -0.967720449, 1.02005899, 0.699623823, -0.192977205, -0.361554682, 0.226021931, 0.0313617177, -0.443519056, 0.394279808, 0.711178541, -0.585805237, -0.0763858184, -0.431294441, -0.882086337, -0.688799143, 0.765866399, -0.600738764, 0.872073233, -0.585193992, -1.14066052, -1.01628506, 0.468449682, -1.05726838, -0.758302093, -0.319746405, 1.06616163, 1.23968601, 0.471936852, -1.17176759, 1.14338076, -1.0373919, 1.01719534, -1.04405451, 1.15122747, -0.736556053, -0.817210734, -0.87207818, -0.880215645, 0.807342827, 0.825081289, 0.657493591, -0.826831758, 0.96656388, -1.18908823, -0.881948113, -0.884769559, -1.16256285, 1.16519034, -1.12716424, 1.03457212, -0.750531316, 0.834807634, 0.189688057, 1.15967309, -0.925843418, -0.622301936, -0.56216079, -0.412126422, -1.16535819, -0.798312604, -0.987665236, 1.16538191, -1.06542087, -0.114130765, -1.16750205, 1.01994395, 0.928645372, -0.0757360235, -0.509201884, 0.527584434, -0.276150465, -0.224989578, 0.251699209, 1.17536449, -0.669173241, -0.0418375544, -0.71047467, -1.13567662, -0.879538894, 0.937010527, -0.958074749, 1.07342601, -0.771591127, -0.898289621, -0.610124648, 0.23924163, -0.769600093, -0.548261344, 0.402057856, 0.92328161, 0.74641782, -0.33475405, -0.734599233, 0.875175834, -0.87895298, 0.725653946, -0.902100265, 0.764896214, -0.69176358, -0.284559339, -0.494734585, -0.365131497, 0.588428736, 0.344578713, 0.193848446, -0.673172235, 0.547721148, -0.726282358, -0.504092455, -0.417677313, -0.798350036, 0.632530272, -0.857168376, 0.615213275, -0.581914425, 0.578558266, 0.447241008, 0.771184087, -0.820596159, -0.715781569, -0.222367719, -0.712529957, -0.773471415, -0.446331292, -0.862668872, 0.708845675, -0.646493077, 0.343099028, -0.872348428, 0.842768073, 0.437714696, -0.387816608, -0.235918418, 0.238533229, 0.552209973, -0.447900772, 0.586615801, 0.89375782, -0.769779444, -0.455967426, -0.135496899, -0.746009052, -0.653398037, 0.863333583, -0.598646224, 0.710586071, -0.793436229, -0.794035196, -0.644094527, 0.158939242, -0.80322212, -0.477397323, -0.115651518, 0.893703222, 0.991062164, 0.223283187, -0.98810339, 0.848653674, -0.782176256, 0.809766829, -0.796902239, 0.859373271, -0.733840704, -0.315199107, -0.655109882, -0.388337314, 0.85081476, 0.512403607, 0.541898727, -0.789254367, 0.632047057, -0.869125187, -0.689603567, -0.417844146, -0.786599994, 0.844494522, -0.717500627, 0.836738884, -0.683015943, 0.688111186, 0.353871852, 0.881329238, -0.823342502, -0.67863524, -0.404293686, -0.423918992, -0.942907155, -0.587039173, -0.631044865, 0.86594981, -0.908970654, -0.0822079778, -0.929236293, 0.992730558, 0.59928304, -0.179815695, -0.406772912, 0.410552382, 0.0469524488, -0.216171399, 0.170646578, 0.789297104, -0.700347602, -0.127496094, -0.471921772, -0.927259624, -0.822308719, 0.793311954, -0.865695298, 0.687847137, -0.684672594];
    recurrent_3_i : ARRAY[0..4095] OF REAL := [-0.0771211386, -0.041904971, -0.0283814035, -0.0384180062, -0.037035238, 0.0755894855, 0.0912913829, 0.00833980925, -0.040718168, -0.0379342623, 0.0494960211, -0.0679311827, -0.0527894385, 0.0977362394, 0.0656317398, 0.0776981115, 0.06924472, 0.00551402941, -0.00546423346, 0.0256145597, 0.0663869157, 0.0448067561, -0.076562196, -0.0898107216, 0.0113763548, -0.153227463, -0.00167952105, -0.000464737415, 0.00439467467, -0.086409919, -0.0667009279, -0.0556129441, 0.0551343858, -0.120897166, -0.0255078562, -0.0891846493, -0.0639392585, 0.0117626972, -0.0803451017, -0.0123659503, 0.0534541979, 0.0729514435, -0.0211154483, 0.018317543, -4.61786985e-05, -0.0382464863, -0.0782647729, -0.015573822, -0.0043241363, -0.148820177, 0.0135069331, -0.0417309552, 0.0900624469, -0.0594736226, -0.0332042128, -0.0981074423, -0.0342614017, -0.0221951418, 0.0398744494, 0.0292471536, -0.0385849997, 0.00922256242, -0.102232851, 0.00561684091, 0.068692863, 0.0208462477, 0.00374138681, 0.0191529803, 0.000650386326, -0.0334673561, -0.0440338105, 0.0698852465, 0.041924905, -0.0118842367, 0.12935029, 0.125775233, -0.00667375699, -0.0881955922, 0.12345317, 0.0304863304, 0.0154025434, -0.00849951431, -0.0940478072, -0.0569340736, 0.0397216305, -0.0101688467, 0.0636173189, -0.0275668763, -0.0776927918, -0.00831863191, -0.0517599955, -0.00621921942, 0.0752723888, -0.0160099473, -0.0405343659, 0.139895663, -0.0825378597, -0.0492977053, 0.00898302533, -0.00459001446, -0.0101332637, 0.0280130263, -0.000348683447, -0.0557230823, 0.0340168104, 0.0289709847, 0.00258996524, -0.0492569655, 0.0154668484, -0.0495375916, -0.0926592499, -0.00718875788, 0.0474499613, 0.00148090534, 0.014299131, -0.0274025276, -0.0290415343, -0.030516278, -0.0101340506, 0.0522375405, 0.039179109, 0.068894051, 0.0322507881, -0.162401929, -0.0554244108, -0.0205325596, -0.0785830021, 0.0307614394, 0.0223672967, -0.0722827613, 0.0852478743, 0.0494147651, 0.0145334667, -0.0208612103, -0.0429588556, 0.0381661505, -0.0254635643, -0.0736351311, 0.0957547128, -0.0774454325, -0.0347611792, 0.0680866167, 0.016637262, 0.0466553494, 0.033682324, -0.0863118842, -0.0845884606, 0.0137423016, -0.016874576, -0.165303648, 0.0474241152, -0.0929194614, -0.0767099485, 0.0418002605, 0.0954845101, -0.00080230023, -0.0807549134, 0.0121842455, 0.0311720297, -0.0555889904, -0.0261414796, 0.0444951095, 0.0685377568, -0.0603509247, 0.0394478515, -0.0426621363, -0.028166268, -0.111334451, -0.00541599607, 0.0391055457, 0.0406126902, -0.0042554047, -0.0693275034, 0.027714774, 0.0115201902, 0.0424438566, -0.0750981644, -0.0402415507, 0.0593367405, 0.000854386715, -0.114437148, -0.0489385724, -0.0201637335, -0.00409932295, 0.0365078077, -0.0941109583, 0.0433239974, 0.0391140729, -0.0613765344, -0.000776667846, -0.0493680127, -0.0485325456, -0.0351513848, 0.0862187147, -0.00819134247, 0.0379211903, -0.000430813408, -0.0901147798, 0.0257685203, 0.108759008, -0.0223718863, -0.0338063687, 0.0156060597, -0.0172953494, 0.105790891, -0.0348870568, -0.0238552466, -0.00988221075, -0.0594870858, -0.0270350054, -0.0289226882, 0.056025885, -0.0559534319, 0.020340465, 0.0709189698, -0.00690495083, -0.0614235885, 0.0191929154, -0.0386514366, -0.018077353, 0.00255588954, -0.0549483672, -0.00174959237, 0.0446115658, 0.0373613685, -0.0370806232, 0.0284372792, 0.0797402859, -0.00256645121, 0.0148433009, -0.0631293207, 0.0278138295, 0.0731672049, -0.0447285399, 0.0508892573, -0.0192828514, 0.0280563608, -0.111958891, -0.0154376552, -0.0134562105, -0.0191528574, 0.0128744598, -0.0721960068, 0.0127519071, 0.0261764918, 0.00257971184, 0.0371103063, 0.220796183, -0.0201993361, 0.136452839, -0.0829204321, -0.00433726329, -0.0309275035, 0.0139829013, -0.051826857, -0.0566153042, -0.0116139706, 0.142482996, -0.0337721556, -0.0867007822, -0.0408329964, -0.0801567733, -0.0191535316, 0.0158957019, 0.0364312977, 0.0103620645, 0.0660757124, -0.100970119, 0.00712347124, -0.0876183659, -0.0854493976, 0.0477382392, -0.0373322181, -0.10326831, -0.0345545262, -0.0589192808, 0.0612725839, -0.0597315729, 0.0500357635, -0.04096343, -0.0692025051, -0.0106984116, 0.0438899919, 0.0404368266, 0.071749717, -0.0615543127, -0.0598752797, 0.0415351987, 0.02201939, 0.00219875015, -0.0673001781, 0.00924704876, 0.0722749159, -0.00525195571, 0.113458283, 0.0372568965, 0.0262363628, -0.0441234633, -0.157484531, -0.00621980149, 0.00702268817, 0.000515939551, 0.0563302599, 0.0814431012, -0.00974204205, 0.0340133868, 0.10453859, -0.0763610899, 0.181937218, 0.0482747033, -0.0712695792, 0.00854755938, 0.125115588, -0.0461000651, -0.0238136984, 0.053446807, 0.0636589676, -0.0651496276, 0.0328514501, -0.0157776587, -0.0405609868, 0.0313981287, -0.039560575, -0.0540332682, 0.0873858109, 0.0195426941, -0.0589045882, -0.0835158303, 0.00876367651, 0.0174001865, -0.0799380466, 0.0423592404, 0.0804384351, -0.0816923082, -0.0501725748, 0.0174710006, 0.00766914617, 0.0943023041, 0.0225947294, 0.0731049329, 0.0203260779, 0.0116448291, 0.0441071019, -0.0682512969, -0.029621724, -0.0456192233, 0.0643681064, -0.0228619743, -0.0348646864, 0.00293346378, -0.0453966931, -0.0378940366, 0.0893360525, -0.0297199413, 0.0621536076, 0.0571176335, -0.00713542569, 0.00198624004, -0.0263217017, -0.00695461687, -0.062595658, -0.0356898196, 0.0519921929, 0.0773653537, 0.0256005786, 0.0134280697, -0.181774542, 0.0606586337, -0.0386322141, 0.079398334, 0.0183406621, 0.0610715933, -0.0669881776, 0.0885097384, -0.0829677358, 0.0276328847, -0.126968756, 0.0522386208, 0.0957871079, -0.123197556, -0.0739446953, -0.0316405408, -0.0435967892, 0.0860320777, -0.0220160093, 0.0570985079, -0.0832202658, -0.0193082672, -0.0668374896, 0.0475501716, 0.0844978094, 0.000630278606, 0.0638538375, 0.0542233847, -0.0417887084, -0.00277152518, -0.0250559971, 0.0337195545, 0.0427481867, 0.015459504, -0.0582500286, 0.0722409189, -0.0537337177, -0.0623925738, -0.0234598946, -0.00134511478, -0.0242168568, -0.0526385382, 0.00195068866, 0.0186914504, -0.0119787138, 0.0187721029, -0.033073511, 0.0115096737, -0.0633152574, -0.00176272169, 0.030483298, 0.0767166764, -0.138829052, 0.0149489995, 0.0345533825, -0.102163568, -0.104449436, -0.0121117663, -0.0284647569, 0.185877964, 0.00462655164, 0.0652706698, 0.0703491792, -0.0313264355, -0.055347681, 0.0250781216, -0.0712601691, -0.0117419995, 0.0371713117, 0.0855040774, 0.00171021745, -0.079428114, 0.0225222223, 0.0360391289, 0.0283598211, 0.0123287961, 0.0588385053, -0.0281411186, -0.0607317239, 0.0662985221, 0.0331876278, -0.055067122, -0.0299345013, 0.000159702147, 0.0443185419, 0.0587667078, -0.0132936174, -0.00628238171, -0.0756097957, 0.000682532787, -0.050425522, -0.0115786884, -0.00569279492, -0.0613335297, 0.0146273952, -0.0631228238, -0.0581459589, -0.0151755679, 0.0857625604, 0.0821363926, 0.115290247, -0.0549297854, 0.0494527891, -0.0702691972, 0.143419236, -0.000891714124, -0.0305100456, -0.0913166925, 0.0610314682, -0.00264202012, 0.0289883371, 0.135914102, 0.0355210379, -0.00808628649, -0.0574536361, 0.00994824804, -0.0611675978, 0.0921703205, -0.0638784096, 0.020130869, -0.0362409279, -0.00529598212, 0.0173103288, -0.00330379046, 0.0372529067, -0.00947646052, 0.00849558599, -0.0442692153, 0.0606488958, 0.00228718901, 0.0758064687, -0.012268913, -0.094871521, 0.0871430188, 0.0136561962, -0.000904569402, 0.0177231189, -0.0620503128, -0.00116063561, 0.089274697, -0.0410311706, -0.0160198882, -0.0176485721, -0.0251905806, 0.0309642088, -0.0365208983, -0.0692796856, 0.050867036, 0.0156931747, 0.0287272036, 0.0371698886, 0.0470653847, 0.0171248168, -0.038513612, -0.0526604652, 0.0604412891, 0.0703500807, 0.0379981175, 0.129006818, 0.0396738537, -0.0257127378, 0.00598947424, 0.00387466792, -0.0582250282, 0.0306714829, -0.0903960094, -0.0177030656, -0.0494029149, -0.167852327, -0.00442219153, 0.0496009812, 0.013880033, -0.0902066082, -0.00579406694, -0.149498537, 0.0741799176, 0.0138978958, 0.0207201876, -0.029839877, -0.107697017, 0.0754648596, 0.0499061793, -0.0648064092, -0.0602546036, -0.0953533798, 0.00365704438, 0.0356753245, -0.0100625791, -0.0301756747, -0.0183225106, 0.0209142882, 0.000961192884, -0.00425785966, 0.0731755793, 0.0539571531, 0.0307768025, 0.0192657448, 0.121937618, -0.0402431674, 0.0851507634, -0.0264093336, 0.00447697798, 0.00402681436, -0.0473406613, -0.105135515, -0.0504542477, -0.0541321822, 0.00259122159, 0.0348727964, -0.0885458589, 0.0608932152, 0.0967864767, 0.119259723, -0.00126710534, 0.099387981, 0.0255985558, 0.00795432366, 0.0200677458, -0.0657623336, 0.190532804, -0.0352462381, 0.11204578, 0.0583575144, -0.0365644731, -0.0667472258, 0.0420552082, 0.104517318, -0.123279393, -0.025258502, 0.0455506109, 0.0645823553, -0.0150504466, -0.0935732126, -0.0465937927, -0.00506780948, 0.0766709894, 0.016313877, -0.0589278638, -0.0213123448, -0.00999987405, 0.0372834876, 0.0003843382, -0.0424535349, -0.0291266404, -0.0146436654, -0.00614433317, -0.115411565, -0.00276262173, 0.0107895397, -0.032524284, 0.0721799359, -0.115214683, -0.0201889109, 0.0353863686, -0.0889972821, -0.0150663191, 0.0311618596, 0.097947672, 0.0337602422, 0.0297635645, 0.131509572, 0.0590009764, -0.0416336432, 0.0261052232, -0.029010294, -0.0259194914, 0.0256441385, 0.04547894, 0.0276543871, -0.0115486104, -0.00763038546, 0.0314593501, -0.0427584499, 0.0405674614, 0.029487269, -0.0592614375, 0.0180521794, 0.0585754439, -0.0690455586, -0.0602442659, -0.0481735766, -0.0419904962, 0.0475285091, -0.0502720438, -0.0131537914, -0.0166091621, -0.000902149361, 0.0570480227, 0.0707662702, -0.0314460434, -0.0985292792, 0.0363963433, 0.0452788696, 0.0805958211, -0.0927961469, -0.0842332914, 0.0785057843, -0.0252397936, 0.063726902, -0.0157659501, 0.0154123157, -0.0701188073, -0.0163884759, 0.117669068, 0.0686297193, -0.0508072823, -0.00954249315, 0.0685154498, 0.00789694674, 0.0402810648, -0.0445739515, 0.0538645312, -0.0362013169, -0.0298318546, 0.00947535317, -0.022353489, -0.018312728, 0.129584163, 0.0519749038, -0.0102249188, 0.106327176, -0.00141187524, 0.104458824, 0.0900954306, 0.0631913096, 0.0487863906, 0.0143436007, -0.0466737151, -0.0175238848, -0.0134204691, 0.0936064124, 0.0213608462, -0.0548267998, 0.0156905074, -0.0593934953, -0.0977132469, 0.00202449691, 0.00566504337, 0.101919673, -0.0227482766, 0.0688653514, 0.0549680814, -0.0696360543, 0.111353241, -0.0198062696, -0.0470485538, 0.0482638553, 0.0627034158, 0.0686005205, -0.0104259253, 0.0585279539, -0.0265351944, -0.0823240802, 0.0223231334, 0.0155628044, 0.0399463028, -0.0703131333, 0.0192429498, 0.0842892677, -0.0436442904, 0.00773867406, -0.0787202716, 0.0446639024, 0.000940637663, 0.0502416268, -0.0171056073, 0.00118341111, -0.20054698, -0.000826745294, 0.0638445243, 0.115336217, 0.0489696115, 0.0723453835, -0.00212192163, -0.106923357, -0.0138108861, -0.00562525727, 0.10132996, -0.0545146763, -0.0471567214, -0.0582389571, 0.0267263185, -0.0706184208, -0.014614461, -0.0879550129, 0.0106655899, 0.00542923622, -0.0904930532, -0.00561792776, -0.0161186848, 0.106282473, -0.0461229794, 0.095484823, -0.102420568, -0.0115131736, -0.0411330983, -0.0572963804, 0.0411828123, 0.0175885111, -0.00862000976, -0.072997123, 0.0657924712, 0.039794296, -0.00335495267, -0.0449964553, 0.0481781289, 0.0714197829, 0.0511781946, -0.0879000053, 0.0544147305, -0.0406234711, -0.0558374897, 0.0643390119, 0.0160111859, 0.00428581238, -0.0187804457, 0.015720617, -0.0579953454, 0.0280058905, -0.00923684798, -0.0470739752, 0.0321382321, 0.0422517508, 0.0183307044, -0.00781843718, -0.0342937969, 0.0205556918, -0.0981495678, 0.0488321632, -0.011658892, 0.0305980891, 0.118306451, 0.0768781081, 0.024575863, -0.100505978, 0.04237964, -0.189520091, 0.105704762, 0.135003522, 0.010658402, -0.0483942032, -0.0704915226, 0.0844620317, 0.0273216274, -0.0259813722, -0.0111644482, 0.06088854, -0.0766476393, -0.00363370311, -0.0178547688, -0.0920214877, -0.00513554085, 0.0269423816, 0.0703381896, 0.118874483, -0.0575212762, 0.119425707, 0.0529291444, -0.0860894471, -0.0865111127, -0.0148848416, 0.19253251, 0.104712084, -0.0555614047, -0.0672845915, 0.0351972207, 0.00676282309, -0.0296126883, 0.0261259004, -0.00242765062, -0.0275501218, 0.0260865837, 0.10234154, -0.0501713939, 0.0731360838, -0.0291022677, -0.0139559144, 0.0922236666, -0.105612159, 0.0131138563, -0.0829087719, 0.00905138254, 0.0465265922, 0.0365543664, 0.0536549091, -0.0559660532, 0.115871899, -0.0190141965, 0.0573159829, -0.00187401986, -0.0605982132, 0.0414755642, -0.00944722258, 0.0610298775, -0.0544121191, -0.0403051525, -0.0444469973, -0.00737518445, -0.0570647344, 0.0424280278, 0.0314462781, -0.0356462114, -0.00442456827, 0.00501318881, 0.0772018582, 0.0401184224, -0.0479452647, -0.0308884569, -0.0212140195, 0.02648261, -0.0255462639, -0.0302096345, -0.0782852694, 0.0235898439, 0.0513489395, -0.0660517588, -0.00344516197, -0.110358223, -0.0641045943, -0.0483674482, -0.0172280818, 0.0570637062, -0.0584195331, 0.0135480603, -0.0512361005, -0.0377590358, -0.0496845767, 0.00837638974, -0.131501243, -0.0485012457, -0.0867616311, 0.00172824948, -0.0483968779, 0.00378531776, -0.0201999806, 0.0129637346, -0.107964613, -0.0680155903, -0.0121945422, 0.0332003571, -0.142481193, 0.0353830494, -0.0529950261, 0.0895682052, -0.113010526, -0.129145518, 0.0134146102, 0.0746574625, -0.0465294942, -0.0412936099, 0.017362833, 0.0181081146, -0.067679368, 0.0175119545, -0.123860918, -0.0328148454, -0.123511083, -0.0364386067, -0.0311892685, 0.0184607543, -0.0311089717, 0.000620753504, -0.0568052083, 0.011010047, 0.0740614906, 0.0737213343, 0.132467821, 0.0134541467, -0.0517201014, 0.0371107683, -0.0747232139, 0.0175857544, 0.0185665116, -0.085187152, 0.0808551088, -0.0630146116, 0.0255866461, 0.0362472124, 0.0900037512, 0.0042063524, -0.0614381544, 0.0115199219, -0.0224268176, -0.0755639523, -0.010225663, -0.0233745798, 0.08830823, 0.00794417504, 0.100218058, -0.0395819508, 0.00176830171, -0.0245204028, 0.0422842354, -0.0372996591, -0.00241308706, 0.0962401032, -0.113369778, 0.0433700494, -0.114136435, 0.0341613181, -0.130839184, -0.089457199, -0.0233602859, -0.0479965173, 0.0391149297, 0.0692763552, 0.194222391, 0.0147205666, 0.00688768551, -0.0260862112, -0.159773886, -0.00286880438, 0.120641142, 0.0765589625, 0.0160452854, 0.0994570404, 0.00954604149, -0.019290071, -0.0922267511, 0.0113348532, -0.0906397477, 0.046988558, 0.072404258, -0.14337185, -0.0172273871, -0.114456639, 0.0451756306, 0.0412931889, 0.0209460594, 0.0381604433, 0.048741173, 0.0535983518, -0.117481872, -0.0597166754, 0.0416786224, -0.109581009, 0.00134346401, -0.0438084416, 0.00310220965, 0.0906066746, 0.102428459, -0.0467643961, -0.0134145245, 0.00761311688, -0.0128192632, -0.0144976024, 0.0508668683, -0.0244545713, -0.163217515, 0.0707146078, -0.0414909683, -0.020475097, -0.0709300339, 0.110582337, 0.0458872691, 0.0147851352, 0.0236281417, 0.0267456733, 0.0351790637, -0.0111391153, -0.0429372862, -0.0653672218, -0.00234420202, -0.0397546403, 0.000486603472, 0.00611863658, 0.0549708642, 0.00347794965, -0.103336439, -0.0649053305, 0.0232978202, 0.092099525, -0.035087008, 0.0587510988, -0.0260108709, 0.0149294846, 0.149228558, 0.00796078984, -0.0348771624, -0.0376017764, -0.00330119394, 0.0105758226, -0.0476414561, 0.0779505596, 0.0283059888, 0.068600148, 0.00378933013, -0.0553796664, -0.0282109361, -0.00815444812, 0.0270443503, 0.0880057812, 0.0859450847, -0.036509417, 0.0516473651, -0.107805446, -0.00200375728, -0.0827743858, 0.0520797148, -0.0391699858, -0.0311506353, -0.0506948382, -0.031195391, 0.0115020834, -0.0476800315, -0.063335754, 0.132047504, 0.0484156534, -0.0179302748, 0.157283068, 0.0366875157, 0.0251473393, -0.0673718005, -0.0393670425, -0.03770978, -0.0478124507, -0.0309036858, 0.0446205698, 0.0311251916, 0.0245048814, -0.0259537641, 0.0997335464, -0.0605693161, 0.00225354522, 0.0080093611, -0.0326315872, 0.0134006618, -0.0756340176, 0.0391127281, -0.0530095957, -0.0592922792, -0.0589320287, -0.0158974119, 0.0390460417, -0.0620967709, -0.00484201685, -0.0339126587, -0.114744462, 0.0272865258, -0.0148388147, -0.0874240547, -0.130963251, -0.00731145218, 0.0346865393, 0.0248591453, 0.132716715, 0.0567845628, -0.0396426059, 0.0966895819, -0.0279246792, 0.0332853012, -0.0544270054, -0.0434819683, 0.0667337701, 0.0185598992, -0.0217630044, -0.0630863756, 0.0165286437, -0.0175159127, 0.0732632279, -0.0882861689, 0.00874199346, -0.0702120736, -0.00991208293, -0.107882038, -0.057309255, -0.0370102227, 0.0218572132, 0.0131309144, -0.0377560779, 0.00983685162, -0.010612092, 0.00618636748, 0.0234554112, -0.00349855889, 0.032401789, 0.00883803703, 0.0168552957, -0.0251002647, -0.147040695, -0.0349156298, -0.0705754906, -0.0755141303, -0.0358002782, -0.0804489627, -0.0872704983, -0.10116975, -0.0111940997, 0.185184717, -0.0291834772, -0.0106254304, 0.0199537389, -0.0575619712, 0.0327430181, -0.0982737988, 0.00400483515, 0.0415157862, 0.0418619663, -0.0547926277, 0.122650564, 0.0924820527, -0.0236307867, -0.025062155, -0.00689590909, 0.0673624277, -0.059796568, -0.0229343288, 0.1029379, -0.0339142159, -0.0528561883, -0.0526297614, 0.150432065, -0.00509574916, -0.0739349201, -0.084164843, -0.0795581341, -0.00410477351, 0.0224036723, 0.0124150803, 0.0239414368, -0.0398170687, 0.177057952, -0.0192521326, 0.103363805, 0.0614584386, 0.0694947913, -0.0193667188, -0.0576172173, 0.0620115176, -0.0870990381, 0.0496941507, -0.0259861536, 0.0403347239, 0.0496604256, -0.0786272138, -0.0154306944, -0.081339933, -0.0445302837, 0.102406658, -0.061163269, 0.0604605749, 0.057162337, 0.0785773769, 0.049725607, 0.0122487135, 0.0674273595, -0.0874722376, 0.0738762915, 0.0531259775, 0.080693908, 0.106209084, 0.0290892515, 0.0115198158, -0.0458286665, -0.0384727009, 0.0816580355, -0.0311149843, 0.0961059481, -0.035856396, -0.0599000305, -0.0631308854, -0.0129607571, 0.111237794, -0.0191058517, 0.0521618016, -0.00881535746, 0.125796705, -0.0308310576, 0.0099222362, 0.00214290619, 0.00591849908, 0.0316641741, 0.108231694, -0.0540060773, 0.159002408, -0.0459824465, -0.0337038673, 0.113687485, -0.100403123, -0.0782597214, 2.66171992e-06, -0.030309476, 0.0187225994, 0.070588693, -0.021095952, 0.0898897126, 0.0519983917, -0.00222996995, 0.0286504477, -0.0130401272, 0.0265140049, -0.0149852019, 0.034320049, 0.0317233875, 0.0892530233, 0.0787781104, -0.0337975733, -0.0102227032, 0.0430831984, 0.000701051205, 0.0882281661, 0.0165888332, 0.0865149796, -0.0396107659, -0.0339075737, -0.0606385767, -0.0798013657, -0.0987702385, 0.0128210438, 0.0787314102, 0.0952082276, 0.0263865329, -6.64079562e-05, -0.0520985238, 0.048642315, -0.0639183447, 0.120937899, -0.054034628, 0.0577845201, 0.164206862, 0.00996304303, 0.0452152342, 0.012397184, -0.00907938741, 8.59340653e-05, -0.0279395226, -0.064995572, -0.0103277853, 0.0347133391, 0.0380030274, -0.156820685, 0.0496531799, 0.0056411447, -0.0199967287, 0.0349395275, -0.0178748965, -0.0971291438, 0.0238538645, -0.0882459134, -0.0474008173, 0.0881513059, -0.0397922955, 0.0727870688, -0.131201446, -0.0279316753, 0.0408275947, 0.0168356095, 0.0744072869, 0.0187169667, -0.068779774, 0.0426025018, -0.0193063281, -0.0520456582, 0.0416068994, 0.0160504002, -0.0849148706, -0.0781304762, 0.168890104, 0.0400321707, -0.0366453379, 0.0254135281, -0.0447303839, 0.00366006792, 0.00179227069, -0.073159337, -0.0863961428, -0.0180702675, 0.0033401968, 0.0471517816, -0.0329570249, 0.0174799431, -0.0915972367, -0.00979953818, 0.0262655523, -0.00219394523, -0.0771069601, -0.00288106315, -0.0112265646, -0.0510940552, -0.036896605, -0.0146863656, 0.00246440712, -0.1058181, 0.053954836, -0.132233366, -0.0751370564, -0.0461335778, 0.0248641428, 0.0206944253, 0.044601813, 0.0917557999, 0.0854347199, 0.00680780411, 0.0388449728, -0.0178329702, -0.0440684296, -0.0474345945, 0.0536735989, 0.0156669542, -0.0179837942, 0.015049316, -0.0944499746, 0.0255464185, 0.0139696524, -0.0183444917, -0.00965639576, -0.0268477555, 0.135275558, 0.0509962142, -0.0986917242, -0.0227983035, 0.00305658765, -0.0856561884, 0.0290389154, -0.0660269186, -0.0633658916, 0.0124608278, -0.0484014228, 0.010453742, -0.0150720328, 0.0921224728, 0.0343518369, -0.0277125072, -0.0351466686, 0.0913387537, -0.0382746346, 0.0982387662, 0.0597138219, -0.0440888293, -0.0873766094, 0.134155929, -0.000342816114, -0.112505727, 0.0339261889, 0.00784657151, 0.0422569774, 0.0304149017, -0.0174519662, -0.100313917, -0.0682862401, -0.078867808, 0.0252579935, 0.0598724373, 0.0175824519, -0.0580917522, 0.0579990409, -0.00509794895, -0.013098672, 0.0134000657, 0.00295411795, -0.0628975779, -0.0807553232, 0.00282261497, 0.0151576092, 0.0765760168, 0.0573970042, 0.037956208, 0.076710701, -0.029479716, -0.0708900243, -0.0150526743, -0.122771248, -0.0357170552, 0.0486811101, 0.0018941164, 0.0022100471, -0.0338713638, 0.138970211, -0.0620444939, 0.0276888832, -0.0742791072, 0.0107768327, -0.013218767, -0.0233383588, -0.00579264993, -0.122329608, -0.0303021222, -0.105152994, -0.00944907404, -0.0473172814, 0.0247038007, -0.0754274428, -0.00730832759, 0.0661038682, -0.00139894523, 0.0394513085, 0.0232133511, -0.136513174, 0.0769726634, -0.0362442955, -0.0387526341, -0.215772748, 0.0400592461, 0.148775563, -0.0179366972, -0.0344711952, -0.105664037, 0.0565368906, 0.0767515525, -0.0210688021, -0.0248218253, 0.0139113367, -0.0503477789, -0.0919362679, 0.00241893739, -0.150888786, -0.0521079935, -0.0130923521, -0.102624953, 0.0652719885, 0.0720933452, -0.0342555232, 0.143231511, -0.0571466684, 0.0597913601, 0.0616353974, 0.0496004112, -0.00588138867, -0.124242619, 0.0982202068, 0.0385833755, -0.0267478451, 0.0698152184, -0.0226045679, 0.0295436215, 0.0269691981, -0.0145521704, -0.0704007372, 0.0563407354, -0.0541602373, 0.0702264085, -0.0287812315, 0.0237359479, 0.0170573685, -0.0314531364, -0.0559237301, -0.0229936354, -0.0873287767, 0.0505414829, 0.0730561092, -0.12192782, -0.104775615, 0.099988088, 0.0937188119, 0.0256949309, 0.00599367218, -0.0792903006, -0.0849900469, -0.0244031977, 0.0517280139, 0.00284449384, 0.0588323995, 0.0150726568, 0.0705374852, 0.0227077417, 0.0698392466, -0.0465410054, 0.0897336528, -0.140212193, -0.0762655437, -0.0484272018, 0.0781526566, 0.0329838879, -0.0322162881, 0.0493155643, -0.0422493964, -0.0149069745, -0.00729649886, 0.116023973, 0.0208215024, -0.0119661624, -0.0600190572, 0.0152146658, 0.0232678521, 0.031961374, -0.076048471, 0.0752262473, -0.0254874378, 0.0603693463, -0.0214568563, 0.0443627983, 0.0861600712, 0.110576168, -0.0153700281, -0.0522413626, -0.0181858595, -0.102767073, 0.0204370059, 0.00640147924, -0.0462402776, 0.0303416587, -0.014012333, -0.101610146, -0.0537055694, 0.0660692453, 0.0320705734, 0.0438896939, 0.0207390673, -0.0499086902, -0.025366487, 0.0747519806, -0.0316851549, -0.0759165585, 0.0436173193, -0.0106276162, 0.015699055, -0.0377657488, -0.0501587577, 0.106968641, -0.0271445233, 0.114476688, 0.00821631402, 0.0723700747, -0.00975259766, -0.144449532, 0.000877615996, -0.0187783428, 0.0982629582, -0.0616536327, 0.0501482002, -0.00122638233, 0.0282082222, 0.0182234906, -0.0169871524, -0.0162812453, -0.0360330716, -0.0333503634, 0.0434881076, 0.026132334, -0.0594973639, 0.0357384905, 0.10762547, 0.0930696428, -0.032664597, 0.0310225002, 0.0313590989, 0.0207410716, 0.00215228461, 0.0220122356, -0.0219471399, 0.0972534791, 0.0126505364, 0.0284033492, -0.0381177627, 0.0166915413, 0.0413518623, -0.0191520825, -0.000985896448, 0.00584470853, -0.011032097, -0.0880968124, -0.0672093704, -0.00587202143, 0.095265761, 0.126526862, -0.0436578542, -0.0140812155, 0.0604392216, 0.0731392428, -0.0256851912, -0.105274037, 0.106243387, 0.0340439156, 0.131831095, -0.0265626591, 0.0286284406, -0.0759204477, -0.0156980269, 0.00696976855, -0.00866186433, -0.00699613057, 0.0219969749, -0.0664360374, 0.0397608355, -0.113807514, 0.0428919867, 0.132699594, 0.0729412511, 0.0291228183, -0.0552000776, 0.0984611437, 0.0857509077, -0.176901773, 0.0790669769, -0.0925221816, -0.141180128, 0.0706448629, 0.050350558, -0.0397202708, -0.0755624548, 0.0277449936, 0.0465391055, 0.0242460705, -0.0519197322, -0.0352012888, -0.0360889398, -0.0180267282, 0.0771338642, -0.0200135168, -0.0418161638, -0.104534358, -0.0436706729, 0.0487912074, -0.0194058344, -0.110537097, -0.0642443299, 0.0491082668, -0.119076572, 0.108019292, -0.0060014613, 0.0306117442, -0.00466304319, -0.0232913699, -0.0511650331, 0.0275231972, 0.0840327442, -0.134391844, 0.0361698754, 0.0546769425, -0.00451168697, -0.124834865, 0.00793889817, -0.0194791071, -0.047546424, 0.00907409191, 0.0667063519, -0.0414150916, -0.00810996629, 0.0252991784, 0.00813391805, -0.101334795, -0.068073824, -0.00572252087, -0.0330414437, -0.00174164213, -9.43699852e-05, -0.003085576, 0.0486874282, -0.0364591666, -0.0317699015, -0.0173614342, -0.128078446, -0.00707710255, 0.0569778122, -0.00317369495, 0.0616593473, 0.105571508, -0.0600511916, -0.125462323, 0.0620394647, 0.0330251008, -0.0224925671, -0.06249341, 0.0392381921, 0.0241978578, 0.00201773271, 0.0761228129, -0.0289585106, 0.0902938694, 0.0738835782, -0.016410742, -0.117978804, -0.0864401907, 0.039015539, -0.0713666528, 0.0403234623, -0.0509619899, -0.194570005, -0.066731289, 0.0154067371, -0.0439324453, 0.0847003162, 0.107806429, -0.033445593, -0.0332155339, 0.0183431655, 0.0231716502, 0.0285760835, -0.0442197695, -0.089011088, -0.0314625204, 0.0825669691, 0.0989553183, 0.126024291, -0.0403006971, -0.0249300376, -0.00175470766, -0.0387068391, 0.103461869, 0.104851246, -0.078734979, -0.0869031996, -0.00940553006, 0.0473936833, -0.0492781959, 0.011214152, 0.0900023058, -0.139418155, -0.0459762774, -0.0767275542, 0.038480971, 0.0355797447, 0.0246626176, -0.067918703, 0.0173300691, -0.0111240037, 0.00440449361, -0.0675490722, -0.117332205, 0.0323232301, 0.0494250655, -0.039023485, -0.0351693928, -0.0558870584, 0.0212836526, -0.0763815865, 0.0145481098, 0.030264806, -0.0194271654, -0.0656424165, 0.0946357548, 0.0536819957, 0.0625644103, -0.100732088, -0.0241884068, 0.0235884488, -0.00379322818, 0.0470121168, -0.0830290541, -0.00274844444, 0.035193529, -0.00292130839, -0.0975778103, -0.146146074, 0.0253734533, 0.0170242153, -0.0313359797, 0.120178267, 0.0498198569, -0.142378464, 0.00051176548, 0.0584818572, 0.0537292473, -0.108122371, -0.0433480218, 0.0291369781, -0.0533202067, -0.0646765009, 0.00796661153, 0.0651323423, -0.0704324991, -0.0595270172, -0.0637600347, -0.0255695526, -0.0359119177, -0.0329027623, -0.0251953397, -0.00202006707, -0.0203789137, -0.0562391691, -0.080313772, 0.0577877834, 0.0348158069, 0.0304604135, -0.00427031424, 0.137653306, 0.0444946364, -0.135594085, 0.00807581842, 0.0390937254, -0.0484327748, -0.00712263305, -0.00467313454, 0.0213462058, -0.0569633618, 0.014585142, -0.00903347321, -0.0474929325, -0.0491582491, -0.0225354433, -0.060164921, 0.0331706293, 0.033714164, -0.0489883646, -0.000850817189, 0.0880154669, -0.0255647115, 0.0434250459, -0.120299645, 0.00521157775, -0.0519536845, 0.12155582, 0.0670317113, 0.0390714034, -0.0730279163, 0.108900294, 0.0190060548, -0.0151199531, 0.0411870778, 0.0563757047, -0.10859707, -0.0251432694, 0.127860352, 0.0683794245, 0.0160465818, -0.0222009514, 0.0233334191, 0.0192102417, 0.00722608529, 0.0708645135, 0.161178872, 0.0612367056, 0.00366378948, -0.0137775969, -0.0395795293, -0.0202920213, -0.078712672, 0.0827812701, 0.0557660833, 0.00758445263, 0.0559690334, -0.0459271818, 0.0884366781, 0.0462979972, -0.118541867, -0.0199150778, -0.0930863246, 0.0684344172, -0.0483856648, -0.0175752882, 0.00132881314, -0.0874542668, -0.00535436114, 0.0246759802, 0.0050930893, -0.104525492, 0.0308124907, -0.0427543446, 0.0113368044, 0.117691182, -0.00788058154, 0.0374500006, -0.0663976371, -0.0379608162, 0.0824671388, 0.040722385, 0.113066494, -0.0284847841, 0.0628969744, 0.0176786631, 0.106616139, 0.0364625454, -0.0395449772, 0.0711597875, -0.115894616, 0.0616638251, 0.033880759, 0.0842308551, -0.0200199522, 0.0854050592, 0.00240669074, -0.0221695919, -0.0171297081, -0.0368121415, 0.0901898295, 0.0558736101, 0.052049391, -0.044363752, -0.00578884175, -0.139492258, 0.0934761465, 0.0463176742, -0.0893110707, -0.0234638881, -0.0254841838, -0.0230731126, 0.023535518, 0.0606091544, 0.0712842196, 0.0151794199, 0.0228757747, -0.00670690928, 0.0243334826, 0.00760607189, 0.0909763575, -0.0020671133, 0.0380613878, 0.0523210615, -0.00226617698, -0.0527453385, 0.0873451531, 0.00789528619, -0.039309945, 0.0657774359, -0.0373396091, 0.0121234003, -0.0608648509, 0.0955511183, 0.106229104, -0.0227189902, 0.0181806684, 0.0313352682, 0.0983065665, -0.0655134469, -0.0100321807, -0.0214557108, -0.0323480032, 0.0399547108, 0.0510334969, 0.0764594153, 0.120244615, 0.100224771, 0.0613763817, 0.0966042578, 0.119996041, -0.0274828617, 0.0648390055, -0.0121074114, -0.0551745556, 0.0166523531, -0.0572726466, 0.011296981, 0.0738770068, -0.028714275, 0.0734295845, 0.0108936559, 0.0432941616, -0.00889409427, -0.008979748, -0.0243339837, -0.0185373686, 0.00247844215, -0.00585353561, 0.0613322258, -0.0551779605, -0.00296961702, 0.0106428079, -0.0408338606, -0.0757235661, -0.00855779834, -0.0684195235, -0.0265507028, 0.0798603669, -0.0745164007, 0.0298931263, 0.107402548, -0.0163386203, 0.0202664565, 0.0360967554, 0.0445154905, 0.0351002701, 0.0772979185, -0.0847752467, -0.0830296054, -0.0078751957, -0.0517528765, 0.0568756424, -0.0522266701, -0.0157700721, -0.0453625172, 0.121910952, 0.00520794094, 0.0594974682, -0.0149897374, 0.0535635464, 0.0229940414, 0.0360345319, 0.11592412, -0.0503912047, 0.00695486646, 0.0321925282, -0.00204658881, 0.0299749561, 0.0869947672, -0.131942108, 0.0256948676, -0.0761573315, -0.0721464306, 0.0488116369, -0.0233175065, 0.0251011774, -0.0364564434, 0.0703453049, -0.0303190667, 0.020260239, -0.0368825868, 0.0204307344, -0.138143018, 0.0240335371, -0.12227723, -0.000719763339, 0.0397568047, -0.0108157676, 0.0380594246, -0.0454414487, 0.00395573629, -0.079955548, -0.103262126, 0.0717545897, 0.0462553948, -0.0749582872, -0.0598753132, -0.0549320504, 0.167967528, -0.0342475176, -0.0678644106, 0.014138151, 0.0883469209, -0.0422446132, 0.00910017174, -0.0278913192, -0.0617286935, 0.0945532322, -0.0891489685, 0.00157077983, 0.0810243636, 0.036433693, -0.0354036316, 0.0656190589, 0.11084713, -0.0328651145, 0.0968796238, 0.0468874946, 0.0668853596, -0.0326856822, -0.0238782857, 0.0019241781, 0.0953875333, 0.111255117, -0.0768138543, 0.000530576333, 0.000880140811, 0.147702083, 0.0755548328, -0.0203691162, -0.0268486366, -0.044232972, 0.045487687, -0.103220411, 0.0775320604, 0.00794593431, -0.0394486375, -0.0247686394, 0.0284869447, -0.0534544103, 0.00503673032, -0.0112144612, -0.0468843877, 0.0273283813, 0.0793735757, 0.00207741046, 0.0429351106, -0.00290703773, 0.00570422132, -0.0043573156, 0.109113462, -0.0445359349, 0.0418569483, 0.0393498242, -0.0209372249, -0.00551870884, 0.107174665, 7.90264457e-05, -0.042608235, 0.0417940132, 0.0433975756, 0.0341972709, 0.0231017601, -0.0823120326, -0.0285989456, -0.0565683097, 0.00515736546, -0.0216090027, -0.055794172, -0.0425441638, 0.0674974695, -0.0372256935, -0.00943269115, 0.0081518339, 0.169903964, -0.0767062902, 0.0181438327, 0.0594843477, 0.0724104196, 0.0623655654, -0.0627258271, 0.108728275, 0.066685833, -0.00326387049, 0.0191066675, 0.0488062687, -0.0557465106, -0.0717181638, -0.120245077, -0.0263934378, -0.0217542164, -0.0377301425, 0.0505158901, -0.00943231955, -0.0811585411, -0.0633471459, -0.0922307, 0.00297417305, -0.0283020921, -0.00233821943, -0.0317868218, 0.022295991, -0.102933459, 0.0353327431, -0.0564441793, 0.0270108245, 0.111416861, 0.054940667, 0.045586627, -0.0325855613, -0.0276312456, 0.108739905, -0.13752073, -0.0148813566, -0.0878764614, -0.00616987422, -0.0113345832, 0.111377209, 0.0674577281, 0.0334462859, -0.0528105721, -0.0283257961, -0.0640272871, -0.104231998, -0.0182194225, 0.0253928099, -0.010000607, 0.0893871188, -0.0936637968, 0.0359381177, -0.0572381169, 0.0415782668, -0.0515473448, -0.0592029989, -0.0162340757, 0.0372194499, 0.000869643176, 0.0569775514, 0.12664406, -0.00410834746, -0.0598526485, -0.0145936832, 0.00541882915, -0.0387819409, -0.0705848932, 0.131225437, 0.0606011972, 0.0260585826, 0.0326864943, 0.0327170156, -0.0681137666, 0.0398291536, 0.0150668863, -0.0623713508, -0.0654203072, -0.0855273381, 0.0542779416, -0.0772915483, -0.00739911618, 0.111987807, -0.0434356108, -0.109296009, -0.000388567569, -0.0285733771, -0.126296833, 0.0530360192, -0.0114716245, 0.0218612682, 0.0229222216, 0.0851885229, -0.0389903337, 0.0584750213, 0.0194483101, 0.0111343805, 0.0142656472, -0.00225033797, 0.00987144839, 0.00450252695, -0.00685430365, -0.0110871671, -0.064477019, -0.108237572, 0.0994877592, 0.0447605662, 0.0851446614, -0.0512959659, -0.0695576966, -0.056695722, 0.0151356487, 0.0813366249, 0.0509820394, 0.130533665, -0.0970403776, -0.06133876, 0.062047407, 0.000485517085, 0.0295372587, -0.0825812668, 0.103946805, -0.0272734016, -0.0142017547, 0.0348625258, -0.0194650106, 0.054473225, 0.0277187414, 0.00521013513, -0.0750550181, -0.0112232966, 0.061832428, 0.0267357174, 0.0369789787, 0.0242078975, -0.0639228001, -0.076738812, -0.105967775, -0.00552886352, 0.0244175512, 0.0138396807, 0.0793611556, 0.0163184702, 0.017674122, 0.0549585409, -0.0119000934, 0.00208156183, -0.0401373133, -0.062261004, -0.0735801086, -0.0862724259, -0.0881317705, 0.030051088, -0.017848039, 0.0650936216, 0.0235368982, -0.0109532671, 0.0914635584, 0.0342697278, 0.0226438977, 0.1154567, 0.0288205035, -0.0857841223, -0.0564709753, -0.0212000832, 0.0331944302, -0.0697550699, 0.0471978039, -0.0747845024, -0.0133633576, 0.111894704, -0.0159318224, 0.0424069613, -0.0777497888, 0.0269897413, -0.0035970686, -0.0470015891, 0.0703898668, -0.0996557772, -0.0109145269, 0.0119720763, -0.0309154429, 0.0772444978, 0.0240636114, 0.0555266663, -0.0486289486, -0.0358316675, 0.0310520343, 0.0524581783, -0.02964909, -0.0225995835, 0.0202129167, 0.0492513031, 0.0024611596, 0.0920979604, -0.147307992, -0.057231009, 0.0140033029, 0.00698713493, 0.0638547167, -0.12043111, 0.0617109016, 0.0197395254, 0.0250540208, 0.0461532772, 0.0631778687, 0.0675501153, -0.0640308559, -0.0384968631, 0.124442965, -0.0169296619, -0.0591387115, 0.00277835689, 0.03010704, 0.0170286968, 0.0438472293, -0.0421725586, 0.0105780903, 0.0187833142, 0.0932823047, 0.0797822848, -0.0400023311, 0.0413492993, -0.00490421942, 0.0261564571, 0.0153271826, 0.0136942901, -0.0678173229, 0.069321245, -0.0221962631, -0.053999871, -0.0290583689, 0.0566808693, -0.068984136, -0.0322767571, -0.0840166956, 0.0840327293, -0.0266867373, 0.0181480683, 0.141900614, -0.0741518885, -0.0462956466, -0.113084376, -0.0761168301, -0.119766846, -0.0191113465, 0.0263688825, -0.0602698475, 0.0213941634, -0.00738273561, 0.066034399, -0.112135068, -0.0262510292, 0.0678964183, -0.0115228705, -0.0385066345, -0.00596521609, 0.00337880291, 0.0653976202, 0.101864547, -0.0145517476, 0.0115391631, -0.149418652, 0.0152731091, 0.0258516744, -0.141610175, 0.0650391579, -0.0218729898, -0.0738234967, 0.087863043, -0.109388128, -0.0587620288, 0.00153938029, -0.0472481102, 0.0655660331, 0.046287518, 0.00191088393, -0.0099407332, -0.0366902761, -0.0758936703, -0.00195228774, 0.132410303, -0.0897945017, -0.0828643367, -0.0931508541, -0.0858343989, 0.0220552962, -0.0318561718, 0.0606997572, -0.0955435112, 0.0174528975, -0.0370034575, 0.000795804895, 0.0466999449, -0.00521745998, 0.0106653189, -0.0342373848, -0.0102693718, -0.054669518, -0.0429277383, -0.0600964017, 0.0296549965, -0.0716629699, 0.0814423859, -0.0409946404, 0.0218861047, -0.0409745276, 0.0469141454, 3.98382545e-05, 0.0468013287, 0.0229902081, 0.0182137676, -0.0610425286, 0.0229899418, 0.142873287, 0.0214464925, 0.0217601303, 0.0480984598, 0.132810012, -0.0424922258, -0.0198705606, -0.0383956023, -0.0761293694, -0.0926634222, 0.135834634, -0.0136811342, 0.0532483645, -0.01176906, -0.0229151398, 0.0479301736, -0.062715888, -0.130381748, -0.0411189981, -0.0947250798, -0.068229951, -0.0499406345, 0.0430741422, 0.0469632521, 0.032190226, 0.0405618772, -0.0297602359, -0.0669889972, -0.0655034855, 0.078095153, 0.00653720647, 0.0422790386, 0.0746423826, -0.0137710692, 0.00105908152, 0.0166120734, -0.119933531, -0.0162646584, 0.0831588954, -0.0413135663, -0.0308480002, 0.0571599156, -0.0818429664, -0.0296073332, -0.0288697742, -0.0251193624, 0.00306123914, -0.0458743162, -0.121116683, 0.0111547802, -0.112941243, -0.0577419885, 0.0467755049, -0.0507814661, -0.051298175, -0.110015258, 0.00560337678, -0.183197498, -0.0217102468, -0.0208833274, -0.00695190392, -0.123197421, 0.032691773, 0.0942695662, 0.0321684778, -0.0735458806, 0.0188958589, -0.0569661036, -0.0828002393, 0.0375961661, 0.00283417851, -0.0231414177, -0.0458211303, 0.027478531, -0.0677815825, 0.0677349195, 0.0259536654, -0.069852069, 0.0958945453, -0.0408855304, 0.0159991458, -0.0688989162, 0.0626117587, 0.0124521516, -0.0413726643, -0.0320701264, 0.0376031771, -0.126749635, 0.00893450901, -0.0760586113, 0.00351698697, -0.0616703182, -0.0376914926, -0.089731127, -0.0248150546, -0.00226218812, -0.0297166444, 0.0724341646, 0.0295588318, 0.0506805852, 0.0683638975, 0.0346119218, 0.0146825043, -0.0300900675, 0.120438926, -0.00266315043, 0.0247528851, -0.0554317571, 0.0749954581, -0.0660863221, -0.0665542111, -0.0541550033, -0.0416485667, 0.0372959226, -0.127699882, -0.084750995, -0.0336081795, -0.0684883595, -0.0341891944, -0.0812875256, 0.0163575001, -0.0336027704, 0.0934475213, -0.0343994573, 0.0371381752, -0.07674779, -0.0452275723, 0.0257721879, -0.0229448806, 0.114483461, -0.0620328411, -0.0166221671, -9.28267837e-05, 0.00410251226, -0.043749325, 0.0121183004, -0.0199087746, 0.0343265273, -0.0519517921, 0.0498782434, -0.00514894351, 0.105170429, -0.0145044802, 0.0170543566, 0.0612747185, 0.0635284111, 0.0722448826, -0.0402126908, 0.0406716689, 0.180485785, 0.0420826823, 0.011254332, -0.07383883, 0.00756357796, -0.00653190818, -0.118777044, 0.0412342064, -0.00101301633, 0.00468574138, 0.0618331097, 0.129026562, 0.0577140562, -0.119758949, 0.0418074131, -0.10028886, 0.146321386, 0.00203114515, -0.0382076167, -0.0158315971, -0.0185160302, -0.0585700981, -0.0892127752, -0.0502712131, -0.00863518007, 0.00928955711, 0.0245242007, -0.0761695579, -0.016499823, -0.0851950496, 0.0302402433, -0.0451599397, -0.000235274434, 0.134561434, 0.0654707849, -0.039849773, 0.0276978035, 0.0976922065, 0.0597911887, 0.128048003, -0.0642070174, 0.0135878399, -0.014466498, 0.00938953552, -0.00197627768, -0.0473276153, 0.0124964295, -0.0482927561, -0.0500519387, -0.0224759765, -0.117781542, 0.0445974693, -0.00626224931, -0.0716539621, 0.0209659114, 0.0950907618, 0.055297289, 0.0339224786, -0.0361117683, 0.00555084739, -0.115107872, 0.000439941883, -0.0202993192, 0.0453407951, 0.0561007559, -0.11338371, -0.0781322941, -0.0260165855, 0.0112777418, 0.0960166007, 0.0797323436, -0.00932762027, 0.148689911, 0.0673603341, -0.00126363337, -0.0395420641, -0.0616854914, -0.0218652152, -0.0841251686, -0.0654635057, -0.13668707, -0.00122302305, -0.0790907443, 0.0650716498, -0.0057691643, -0.0128726279, -0.0956908092, -0.0315712467, 0.0279215723, -0.101440802, -0.0671161041, -0.0240076855, -0.0446522608, -0.0316099077, -0.00810685288, -0.108626872, -0.022286335, 0.0336487666, 0.0771654397, -0.0866703987, -0.109500088, -0.00691062957, 0.00515462086, -0.120609254, -0.0162109509, 0.0773937255, 0.0669814423, 0.0372542813, 0.0293540005, 0.0399727486, 0.0871676579, -0.0184890218, 0.0546814017, -0.0425825901, 0.067953147, -0.0311761238, 0.0312341489, 0.0876554847, -0.0146615878, 0.0407922156, 0.116035752, -0.0404246673, 0.0638451576, 0.101785071, 0.00436116382, 0.036284972, -0.0171610918, -0.0127823167, 0.123123139, 0.0832545161, -0.0702112019, -0.0220967159, -0.00930657797, 0.0471730381, -0.0502699539, 0.0598344095, 0.00845675543, -0.121706769, 0.147291899, 0.0185488053, 0.0772631615, -0.0692496821, 0.092323333, 0.0531550683, -0.091813907, 0.0341402963, 0.0104403701, 0.008129769, -0.0408172235, 0.0606573857, 0.00977760367, 0.0389199331, 0.0131801832, -0.0922353864, -0.098223269, -0.0419626646, -0.0593111143, 0.10533867, -0.0268028136, -0.00331548043, -0.163931951, -0.033068873, -0.00352114672, -0.0809657648, 0.0686088428, -0.00292867795, -0.0278624669, 0.00411469908, 0.0318309069, -0.0307580922, -0.0397743359, 0.00780036114, -0.0651816577, 0.0145179741, -0.023223361, -0.0542891026, -0.121250667, -0.0295627341, 0.02031634, -0.0493941419, -0.0111236311, -0.0228398573, -0.0352995545, -0.0289986897, 0.0391738042, 0.0846049562, -0.086711213, -0.0735283643, -0.0955764875, 0.00540071353, -0.0682940334, -0.0206642989, -0.0456988215, 0.151994646, 0.0301898979, 0.0369524732, 0.0502344705, 0.0833638757, 0.121431336, -0.0410372801, -0.0254659615, 0.0228950866, 0.0228525996, 0.0083724726, -0.0585110821, 0.0608403683, -0.0204683263, 0.00102710386, -0.0463586897, -0.00256409403, -0.0700236112, 0.0309709981, -0.0577077791, -0.00222884188, 0.0324225649, -0.0529456697, 0.0334489383, -0.0258610249, 0.140200675, 0.027081497, 0.0447089374, -0.0138469264, -0.044828862, -0.0518506318, -0.043909952, 0.0304525048, -0.0991320908, 0.0472474843, 0.0305546597, 0.030144278, 0.0851663947, -0.0152060036, -0.0141895618, 0.0190068781, -0.04600906, 0.137501746, 0.10347534, -0.0207075998, -0.0712871552, -0.0669450387, -0.0113951489, 0.00467752712, -0.040738754, -0.0361441448, -0.00970679428, 0.0331211239, -0.0323049687, 0.00529360026, 0.0707725734, 0.116111211, -0.0430333167, 0.0310098082, 0.00512955338, 0.0163368694, -0.0464587808, 0.0123096537, -0.0234641749, 0.000730314292, -0.112272233, 0.0216336772, 0.0133584049, -0.0161934346, 0.0556386374, 0.0335740149, -0.0173839238, 0.039414037, 0.0958736166, 0.033290185, 0.0287034474, 0.0432678051, 0.017504232, 0.108818457, -0.0528055504, 0.0226539914, -0.0613601804, 0.00927608088, -0.0999047384, -0.0737604499, -0.00714416057, 0.0170378312, 0.0955149829, 0.0398799814, 0.0177485012, 0.080797337, -0.0437004454, 0.00450856751, -0.0644934624, 0.0559109151, 0.0616841912, 0.0297846273, -0.0220688954, 0.0190214403, 0.1088126, -0.00498170266, -0.0906166136, 0.153623462, 0.048660934, 0.0527924597, 0.0132156964, -0.0345814601, -0.047118552, 0.0239117257, -0.0547183156, 0.0468712188, 0.0610508956, -0.00730768964, 0.0571509115, -0.0177728441, 0.108094901, 0.000422280282, 0.0676494464, 0.0548462979, 0.0319501087, 0.0757430568, -0.0270296652, 0.0219633151, -0.0551248714, 0.0401655883, 0.0186556727, 0.0519931801, 0.074958913, 0.0776639879, -0.00639817771, 0.0184700675, -0.0563476905, -0.0846942812, -0.0214337297, -0.0115232533, -0.0333131962, 0.16067192, 0.0255485959, 0.03676489, 0.094095245, -0.0732448176, -0.0146226548, -0.0105268834, -0.0823027566, 0.00527555775, 0.00325848535, 0.103646882, -0.0838223398, -0.0200149957, -0.0291824713, 0.0694787055, 0.0277231112, 0.0374957621, 0.0328506157, 0.0508431233, 0.00787144154, -0.0617377684, 0.00957613159, -0.133195773, 0.0383893773, -0.0733166188, -0.00745590124, -0.0818732083, 0.060960643, 0.0544005632, -0.140092775, -0.0229060613, -0.00408835337, -0.0823066682, 0.0300217345, 0.00907065999, 0.0392521843, -0.0700395405, 0.0079762768, -0.1493496, 0.0583605468, 0.0270410068, -0.0341156311, -0.0386294425, 0.0662309453, 0.0872389451, -0.0472744517, -0.0228074081, 0.0684124902, -0.0888471007, 0.0761127099, -0.0326396823, 0.0732444823, 0.0456608236, -0.0937242955, 0.0504064783, -0.141814753, 0.162431598, -0.102114215, -0.0397514515, 0.0473489277, 0.0336118191, 0.148338452, -0.0122316275, 0.0432145298, -0.109083384, -0.0186488908, 0.0720187798, -0.106312886, -0.0913583338, -0.0169402808, -0.0123407505, 0.00822057761, 0.0596636757, 0.0205631852, -0.0619561039, -0.0609639287, 0.0482201204, 0.0354727581, -0.0402187109, 0.0445601232, 0.0287282206, -0.0440565534, -0.0619057789, -0.0213008486, -0.0699777231, 0.0775571316, 0.0231237784, -0.00883588009, -0.113154605, -0.00541019021, -0.033951968, 0.0411423817, 0.053961359, -0.00288748881, 0.0706721246, -0.0491243415, 0.00054154871, 0.0138199497, 0.127938673, 0.0159905218, 0.0829677731, 0.108012542, -0.0567845702, -0.157686636, -0.0702316687, 0.00892338157, -0.165532067, 0.076706022, -0.057830967, 0.00497925933, -0.0186288226, -0.0808018744, -0.0206770748, -0.0118557923, -0.0637545362, 0.0900221914, -0.0139558092, -0.00739696994, 0.074806042, -0.119168133, 0.0166030899, -0.11083927, -0.0656669214, -0.0363056958, -0.00638495618, -0.0680301413, -0.0248918328, 0.00398088805, -0.0237197392, 0.00691889878, 0.0542797484, 0.0325936712, 0.00915190857, 0.00299844984, -0.0195343439, 0.131595939, 0.118413478, -0.0392579846, -0.0031316895, 0.00834177993, 0.0611352138, 0.00132380705, -0.00584108802, -0.0469935127, -0.0832609683, 0.0250498392, -0.116703823, -0.00103460811, 0.102866396, 0.0110065071, -0.0472957417, -0.0647558421, -0.1213881, 0.183602601, 0.0604174212, 0.0105359852, -0.0726647228, -0.08007323, 0.0142628476, -0.0803629532, -0.077605769, 0.093770422, 0.0476225019, 0.0822985619, -0.0843518898, 0.0317965075, 0.0298086535, -0.0405269526, -0.0544525683, -0.0352851711, -0.0550699346, 0.0060656406, 0.0519128218, -0.0409257188, -0.026854191, -0.0174814686, 0.0396045148, 0.00388014689, 0.0182089992, -0.109553322, -0.0415327437, -0.105616137, -0.00612959452, 0.00763020385, -0.0235190243, 0.0448918492, 0.0302004609, -0.0875566453, 0.00955081545, 0.0885803998, -0.0824447349, -0.0201507267, 0.0728382841, -0.0490038544, 0.0268885419, 0.0938861519, 0.0330029763, 0.00269161188, 0.0447449647, 0.0945401639, 0.119459607, 0.00680486578, -0.0233078562, 0.0511108488, 0.060301017, -0.00174694043, -0.0356153585, -0.0987226442, 0.014362609, 0.0541739948, 0.00264295842, -0.0994685963, 0.0274561457, 0.0371477269, 0.0386635065, -0.0900390595, 0.0335176848, -0.00698496494, -0.0795145631, -0.0263204202, -0.0387219936, 0.0372513533, 0.069616653, -0.016119089, -0.0331068784, 0.0249988548, -0.0215352178, 0.00688688643, 0.0810623392, -0.0860611647, -0.0309012495, 0.0779893696, -0.032125663, -0.0114999395, 0.0288507938, -0.0429686308, 0.0445714816, 0.0473432317, -0.0187126808, -0.129243702, -0.0237859432, -0.0638953745, 0.0924817994, 0.0782472268, -0.0220032651, -0.0668439865, -0.0025732331, 0.0527206101, 0.0441822261, -0.0282638352, -0.0422725491, 0.00705240667, -0.0633908585, 0.0137796365, -0.02615471, -0.00124217058, -0.0351347774, 0.0385856144, 0.030581506, -0.0795791894, -0.0542370453, -0.00510898372, 0.10081286, 0.0338734984, -0.101331621, -0.0985490754, -0.00705705443, 0.0109579377, -0.00333777769, 0.0622152798, 0.00363911875, 0.0481062233, 0.068813026, -0.0234865788, 0.0290710796, -0.082115069, 6.35739416e-05, -0.0284638852, 0.001483083, -0.0426237248, 0.00982693397, -0.082873404, 0.0160913952, 0.0433014482, -0.109392956, 0.00402180618, -0.0129479989, -0.121640407, -0.0853046253, -0.0276072361, 0.0528869592, -0.157933325, -0.041677475, -0.0513420925, -0.0716695487, 0.125380233, -0.0541120097, -0.0270892903, -0.0354004353, -0.00983749889, 0.0150565766, 0.0727557763, 0.0440372378, 0.042118784, -0.0513586737, 0.127804816, -0.08231204, -0.0144347623, 0.144508213, 0.0170834213, 0.018995095, 0.0261083096, -0.0523809604, -0.0183201581, -0.0198718794, -0.0594392829, -0.0548257902, -0.0362088345, 0.17197448, -0.016027078, -0.0518785976, 0.0124345161, -0.0428913534, -0.0327314138, 0.000454797671, -0.0294881854, 0.0233004484, -0.0170797016, 0.0684266165, -0.0772320628, -0.00519311149, 0.0680455938, -0.118872553, -0.0149460202, 0.0620664768, 0.0202575028, -0.0733660832, -0.0887743235, -0.0459058397, -0.0442075208, 0.0459926054, -0.0317461155, 0.0334063917, 0.122998029, -0.0343262479, 0.0153604876, 0.0213850737, 0.0250464212, -0.0142205656, -0.0834608525, -0.126580968, 0.0660800561, 0.0521790944, -0.126256555, 0.0789100155, 0.0505135357, 0.0294168368, 0.0424421951, 0.0443682894, 0.0175621547, 0.0369247049, -0.0763881132, 0.00241885148, 0.123601884, -0.0437575728, -0.0337525159, 0.0584881753, 0.072721459, 0.0268098582, -0.0642768964, 0.0777513832, -0.0668801144, 0.152455807, 0.0384080373, -0.0813715234, 0.123705864, 0.0704651251, -0.0142856771, 0.0225876421, -0.032844767, -0.0282874554, -0.0180452634, -0.0589442588, 0.0211542696, -0.0840755552, -0.0346978456, 0.0624949932, 0.0413371325, 0.0347261764, 0.0189449582, 0.104123369, 0.0629087538, 0.206078738, 0.0759140998, 0.00179275218, 0.0178793985, -0.0904001892, -0.0120746437, 0.125980869, -0.0509332716, -0.0251817312, -0.0342635326, 0.0150608607, -0.0486635156, -0.0707176998, -0.088892363, -0.013950143, -0.144070938, -0.0290455334, 0.103315793, 0.00691494159, 0.0516338274, 0.0357198566, -0.0407630056, -0.0704655498, -0.0061621801, -0.0163742173, -0.00286670402, 0.0717858896, -0.0403173119, -0.0242009424, -0.0255283937, -0.146040618, 0.00370218931, -0.0169456266, 0.0739331171, -0.00640878826, -0.0625880584, -0.0078162197, -0.109838225, 0.00966158137, -0.0124182813, 0.0556307025, -0.040832039, -0.0159406848, -0.0489371084, 0.0553769767, -0.0129255224, 0.00165747106, -0.0153565537, 0.0232416987, 0.0490295142, -0.0645253658, 0.057539735, -0.0697470456, 0.00253124698, -0.0123401824, 0.0267368481, 0.0345181003, 0.0153361401, -0.0566138327, -0.0957990736, -0.0121652279, -0.0328246318, -0.0706163049, 0.0241552666, 0.0602169149, 0.0483116619, -0.00645811856, 0.115425527, -0.0619513579, -0.00985607132, 0.00515981205, 0.121840969, -0.0654161051, 0.0609334558, -0.0703953058, -0.0466380939, 0.00197777338, 0.0263202935, -0.0276529472, -0.0145663982, 0.0825188756, -0.0154785737, -0.00760034472, -0.00398123916, -0.0517241657, -0.0116613209, -0.0224521235, 0.0680376142, -0.00622316822, 0.12626937, -0.042651087, -0.0322515182, 0.0697021931, 0.0727702975, 7.03553669e-05, -0.117054015, -0.0118676685, 0.130442441, -0.0633720309, -0.0175191481, 0.0502342433, -0.0153560489, -0.00189093128, -0.0899978802, -0.0814712644, 0.00397173129, -0.00799734332, 0.112588078, -0.0880026966, -0.0207088478, -0.0840146393, 0.104321539, 0.0305856038, -0.0066149896, 0.00385881821, 0.0438802727, 0.00694280025, 0.031775374, -0.029828202, -0.0140974158, 0.0417685509, 0.0469135605, 0.0260566361, 0.0252963938, 0.000886915484, -0.0506873876, 0.073806785, 0.0405627377, 0.0770382509, -0.0126297167, 0.0539279208, -0.0134933405, -0.0488830209, -0.0149195949, 0.0286664907, 0.0258389022, -0.0504526757, -0.0995170474, -0.0514720455, -0.0692799166, -0.0749276727, 0.163625076, -0.0215796567, 0.101433694, 0.0290257093, -0.0497782454, 0.078620024, -0.0765042529, 0.0157838799, -0.0605206639, -0.109294169, 0.0945193022, 0.070097968, 0.0111340079, 0.00806904491, -0.119950257, -0.117081717, -0.0467412733, 0.00635355525, -0.0328157395, -0.0779284537, -0.0535240695, 0.118558511, -0.0796102732, -0.025870543, -0.0800812095, 0.0445277505, -0.050483115, 0.0729925111, 0.0596612878, 0.0246837493, -0.00155314244, 0.031930197, -0.145665765, -0.0536895916, 0.00893774256, -0.0883497596, -0.0918533802, 0.0466198847, 0.0609964356, -0.0676815137, 0.0174437314, -0.0376639664, -0.0100301281, -0.00489459373, 0.108539455, -0.0867397934, 0.00289764069, -0.0308248531, 0.0253050923, -0.00659247162, -0.0553039759, 0.0530485287, 0.0618184507, 0.0723310336, -0.000700828619, 0.0406789705, -0.0380382352, 0.195782676, 0.0544773676, 0.0280783065, 0.12561442, 0.0357654579, -0.00801739655, 0.00788500346, -0.00631313305, 0.0241355672, 0.0768359303, -0.0964802206, -0.00253858231, -0.100009397, 0.0262479931, -0.0976248756, -0.111943744, 0.0919356421, 0.125938892, -0.0401543379, 0.117040925, 0.0532688424, -0.061242871, 0.0221033189, -0.0276570898, -0.0478152446, -0.0574466176, 0.00819699839, -0.0348973684, 0.0246670842, -0.00592264906, -0.0111077726, 0.0866995007, -0.0227352083, 0.00829381496, -0.103243813, -0.0592893697, 0.0485052206, -0.050603468, -0.0623348616, 0.0450620539, 0.101759166, -0.0575572327, 0.0495275408, 0.0339027867, 0.0608742572, 0.0387787558, 0.0444233604, -0.0218878668, -0.119515583, -0.0267581306, 0.0620956197, 0.0759401843, -0.10464073, 0.039943669, -0.120554805, 0.0142001938, 0.0104443245, -0.0431935564, 0.0729510784, 0.0970963985, -0.0129293296, -0.0586054623, 0.017743174, -0.031778641, -0.0015063294, 0.0412261188, 0.0484331958, -0.0161143709, -0.00549984351, -0.0493346676, -0.0827445388, -0.0279450174, 0.00426994078, -0.0378730223, 0.0813675001, -0.0221152548, 0.162851453, -0.0593155697, -0.113409579, 0.0896707177, -0.0561915897, 0.12033812, 0.0299672019, 0.0382056236, -0.148166642, 0.0616600066, -0.0390294828, 0.076734677, -0.0610635877, -0.0314789601, 0.0106446203, -0.152618423, 0.00824991614, 0.0208676532, -0.0452706739, 0.0296786539, -0.00171152223, 0.0278075878, -0.0647582039, -0.0934415385, -0.00471531227, -0.0295969844, 0.0392355211, -0.0213776827, -0.00345349312, 0.0103437174, 0.0793427601, 0.0244922396, 0.0769085586, -0.0180552974, -0.0139173642, 0.0365448445, 0.110751674, -0.079107523, -0.0148752257, 0.055928126, -0.0583166182, -0.0278848745, -0.0543133169, -0.0146240722, 0.0462388359, -0.0462089404, 0.100065276, -0.0377004668, -0.0627923459, 0.0160569306, 0.122475393, -0.0237609986, 0.0326469876, 0.0121175274, 0.00290823728, -0.0759213045, -0.0410238355, 0.0405264311, 0.0794125274, -0.027770102, -0.0214025844, -0.000634195749, 0.0711863413, -0.0176606383, 0.0656886324, 0.0760930926, -0.0337079838, 0.0103172548, -0.0442149788, 0.0296556819, 0.0896399617, 0.0926107764, -0.0657806844, -0.0730204955, 0.0364074558, 0.0463961698, 0.0280023143, 0.0347175673, -0.0382448807, -0.0151486043, -0.0351293534, -0.0893038735, -0.0119186798, 0.0224835817, 0.0259567983, -0.00618832652, -0.0423954725, 0.0166269671, 0.00578288734, 0.0424060039, 0.00587061886, -0.0524880104, 0.109365225, -0.0914567709, -0.0388044044, 0.0739863664, 0.00929750502, 0.0168155134, 0.0719892383, -0.0457954593, 0.0540598556, 0.0506090075, 0.0544214435, 0.0112028988, 0.000449611805, 0.0767428875, -0.0880494937, -0.00829705596, 0.00506457034, 0.0316372067, 0.037886627, -0.0634205043, -0.0767910033, 0.00139203761, -0.0141287921, 0.065350242, 0.00455083512, -0.0507521704, 0.0327888578, -0.0450044125, 0.0352456719, -0.0213064775, -0.0177522674, -0.00198644958, 0.0105824154, 0.0127733704, 0.0429498255, -0.0461088046, -0.0140869189, -0.032076247, 0.0223935302, -0.0219765306, 0.0266452357, 0.0498517863, -0.0713030845, -0.0465965495, 0.015960671, 0.0765702203, 0.0080312388, 0.0792805627, -0.0662729442, -0.0218281597, -0.0474443845, 0.0242550168, -0.0282644872, 0.033289507, 0.0334301293, 0.0314183831, 0.0155287907, -0.0582918338, 0.0822805017, -0.0742264017, 0.1563963, -0.0114020435, -0.01263176, -0.0115720499, 0.113865636, 0.0781941637, -0.0390629768, 0.0707460418, -0.0352013633, -0.0346395001, -0.0204303395, 0.0684736595, -0.0650949702, -0.10914959, -0.143572226, -0.0396091603, -0.031377703, -0.0407384969, 0.0292514525, -0.0254713856, 0.00264162617, 0.000173193286, -0.085854508, -0.126747891, 0.017126631, 0.134934887, -0.110217519, -0.0356670469, -0.0543404818, 0.0187333152, 0.107053265, -0.0248832926, 0.101865664, -0.0710972846, 0.0722196847, -0.0384056494, -0.0161709804, 0.013287331, 0.00541426614, 0.0130335232, 0.0400547385, 0.0100121098, 0.0154263554, -0.0629646033, 0.0193865523, 0.00167901674, -0.00236805435, 0.0101759396, -0.107627042, 0.00447156373, -0.0081684785, -0.0686657578, -0.105860122, -0.0145202372, 0.105648175, 0.0951744467, 0.0278701279, 0.058870703, 0.0614429303, 0.0409474671, -0.0196230002, -0.059842132, -0.072326608, 0.078839533, 0.0461710729, 0.0051418962, 0.00476863049, 0.0325647667, 0.0355884321, 0.0283987522, 0.0260669962, 0.00147352088, -0.00998620968, 0.014060949, 0.0530263782, 0.0267538447, -0.178208858, 0.0138209928, -0.166257203, 0.00249827933, 0.0588419065, 0.00965133496, 0.0388614498, -0.0354404189, 0.101525106, 0.0155021399, -0.0782295838, 0.00205751229, -0.0115062622, 0.0447000861, -0.0492403507, 0.0462464131, 0.0278545078, 0.0493896231, -0.00348212384, 0.0177688748, 0.0589764938, -0.0141374562, -0.153412342, -0.0877678543, -0.163386658, 0.0293954685, -0.108064502, 0.0414382406, -0.0368895829, -0.00636456022, 0.00416772999, 0.008211473, -0.0767143965, -0.0195856318, 0.0320273377, -0.0896992087, -0.0541382805, -0.114244811, -0.026452342, 0.0807037503, 0.0398947708, 0.00308981165, 0.0229013935, 0.0499595329, 0.126231, 0.105691493, 0.0247283503, -0.0480804071, -0.0219699144, 0.0844142735, 0.0152459517, -0.0940366089, 0.0213311259, 0.0797767118, -0.0654330328, 0.0303749572, 0.0221867338, -0.0245458521, -0.0113317519, 0.00932829455, 0.0289108455, -0.0212216694, 0.00822014734, 0.0457722098, 0.0130141452, -0.16610533, -0.0211480781, -0.0197458994, 0.0688880235, -0.00803674106, -0.0433641002, -0.075563252, 0.0635190159, -0.101971351, -0.164013535, 0.0825247914, 0.0201021656, -0.0529738441, -0.0211677011, -0.0466175154, 0.00472022966, 0.06616579, 0.129757211, -0.0536907986, -0.0515484139, 0.00854382385, 0.0687660128, -0.000543623697, -0.00421395339, -0.0509204641, 0.0787195489, -0.0955284685, 0.0278457161, 0.032738395, -0.0350810252, 0.021184016, -0.00620284677, -0.0157659762, -0.120136291, -0.0488379225, -0.0571413785, -0.00956039596, -0.130700439, -0.0297761634, 0.0620664358, -0.0984532908, 0.036326915, 0.0142956804, -0.0336640477, -0.00327738747, 0.052082818, -0.0302631166, -0.0566398501, 0.00357326865, 0.0498971753, 0.0090519404, 0.0498086736, -0.0356872156, -0.158793435, -0.0531598851, -0.0724413022, 0.0847426951, -0.0579689369, -0.0855806544, 0.0161144361, -0.0345754586, 0.0575088561, -0.0482305698, 0.0408530161, -0.0572958775, -0.0430949926, -0.0452227145, -0.0143297808, 0.136190906, 0.0158195812, -0.047018975, -0.00814411417, 0.029649578, -0.0406708904, 0.0951420739, -0.0738690346, 0.0941496119, 0.0681650266, -0.0519653335, 0.0357567519, 0.0538630001, -0.0222863052, 0.151022032, -0.0852258503, 0.000150131527, 0.0268831402, 0.0451235622, 0.019896077, -0.0390991308, 0.0395388827, 0.0464649163, -0.0528178029, -0.0634406283, 0.032435406, 0.0321994387, 0.0763059929, -0.0442365222, -0.0384837463, -0.0376992933, 0.0821993724, -0.0429838598, 0.0302058551, 0.039350383, -0.0757741854, 0.0359587148, -0.0675518662, -0.100005239, -0.0506118014, 0.0944177061, 0.0117894504, -0.0284820385, -0.0153114414, -0.0337097533, -0.121349752, -0.0296758302, 0.0677160621, -0.0469472483, -0.0317657143, 0.0904516056, 0.00663401838, -0.0561745241, -0.0492588803, 0.0282529946, -0.101061374, 0.0839226246, 0.0480642021, -0.0347557813, 0.0767452791, -0.0702294558, 0.0499737225, -0.0848984867, 0.0706430674, 0.0254755691, 0.0556517467, 0.00553852506, 0.0453726128, 0.0186469965, 0.0565884635, 0.0242560711, 0.0359231979, -0.0724069178, 0.0165634658, -0.135310367, -0.032013312, 0.00181994541, 0.0117271263, 0.121910825, -0.0625010505, 0.0669507533, -0.0225233231, 0.0245092064, -0.126561821, -0.0302848145, 0.035558477, -0.0703105628, 0.0638471842, 0.0306731332, -0.0481522381, -0.0406722277, -0.0409029052, 0.0873740166, 0.0292977374, -0.0487803295, -0.0623919293, -0.0670752674, -0.0582743771, -0.0369736739, 0.00244259834, 0.0422472432, 0.0661929622, 0.0405329838, 0.0844473615, -0.0196251534, 0.0165268667, -0.0535134524, 0.0382272936, -0.0927124992, -0.0902759209, 0.0418790802, 0.00131716207, -0.0810423568, 0.0556469485, 0.145353869, -0.0974263251, -0.0265319683, -0.00157782063, 0.0342672877, -0.0780519694, -0.100708544, 0.00392956845, 0.0333812498, 0.0530423149, 0.0157616548, 0.00743991509, 0.0668429434, 0.0836819857, 0.0426887535];
    bias_3_i : ARRAY[0..63] OF REAL := [0.64754945, 0.691847086, 0.64616853, 0.738801003, 0.681163371, 0.618074238, 0.642219305, 0.681924105, 0.725929916, 0.669821262, 0.642402828, 0.64420867, 0.699106872, 0.731772006, 0.736818969, 0.668383598, 0.68884635, 0.640938818, 0.655000389, 0.732870162, 0.669698298, 0.703552306, 0.687165737, 0.693419755, 0.586305499, 0.688813746, 0.689942062, 0.622232378, 0.665326953, 0.657587767, 0.708570719, 0.641408205, 0.706247687, 0.728076875, 0.694459498, 0.697739005, 0.68515265, 0.63921845, 0.67039603, 0.669698596, 0.672608674, 0.459624499, 0.698169529, 0.630342007, 0.631216407, 0.73681736, 0.703925788, 0.700100422, 0.725266874, 0.671362042, 0.728427231, 0.723560095, 0.694639802, 0.607155502, 0.655874491, 0.73296082, 0.65932858, 0.686508298, 0.673355281, 0.734046161, 0.674785137, 0.674265325, 0.703997612, 0.652445555];
    weights_3_f : ARRAY[0..4095] OF REAL := [-0.0521443337, -0.127342403, 0.0130717456, -0.0596655086, -0.0273111761, 0.0327247679, 0.0394109637, -0.0123401359, 0.0960776955, 0.0669516474, 0.000666379929, 0.111136854, -0.121887974, 0.0318512022, -0.092767477, -0.0571558774, 0.0440648943, 0.0670731962, 0.0755134374, -0.0248164758, -0.0245014653, 0.116271675, -0.0863337666, -0.110264994, 0.0281036198, -0.131201297, 0.121819913, -0.0493896604, -0.108632259, 0.0232308805, 0.11175859, 0.113334209, -0.0309745446, 0.00279828906, -0.0263097361, 0.116411507, 0.134985745, 0.00494657457, 0.00834363699, 0.0148295909, 0.123774081, 0.0418391377, 0.135640502, -0.111531332, 0.109959185, -0.135435939, 0.0361935198, 0.0986461937, 0.0639104098, 0.0740167797, 0.0907477438, -0.0655242056, -0.121550567, 0.0214169323, -0.037972711, -0.0314986184, 0.020315364, -0.0910601765, -0.0322241634, 0.037475571, 0.0928814858, -0.01218725, 0.102777243, -0.0764217377, 0.0783669055, 0.122343868, 0.0670614392, -0.122746259, 0.125813544, -0.136584193, -0.0129609108, 0.0863741189, -0.0260882974, 0.0346245915, 0.0256888568, 0.107945338, -0.101845935, 0.0761630833, -0.0844016373, 0.111051813, -0.009620592, -0.0630434677, 0.0688468665, 0.0351438075, 0.120586038, -0.0786037594, -0.10621427, 0.107332289, -0.1062335, -0.0398073941, 0.0100298226, -0.00765535235, 0.0600221753, -0.0497887656, 0.0726344436, 0.0244747847, -0.133941308, -0.0139969289, -0.0164956525, -0.032233499, -0.0143216625, -0.0229434296, -0.0581621826, 0.0872895122, 0.0427271277, 0.117294371, -0.0419999585, 0.00527742505, -0.0238697454, 0.0134884566, -0.0728438497, -0.0774436891, -0.078616783, -0.0915552676, 0.112122655, -0.104264475, -0.0764580816, 0.0231063664, 0.0415457487, 0.0922157466, 0.112544298, -0.0208588988, -0.00843825936, -0.125481308, -0.0991969109, 0.131200939, 0.0391524434, -0.047940731, 0.00629302859, -0.0649658442, 0.129364312, 0.0668620318, 0.0720915645, 0.117274612, -0.0617987812, 0.10781534, 0.118253678, -0.091769591, 0.0618039668, 0.0271771252, 0.129491687, 0.0751471817, 0.0123195052, 0.12247768, -0.100104749, -0.0376960635, -0.0299254358, 0.0191544443, -0.0680884495, -0.105288088, 0.0125788152, 0.0202235281, 0.0872109234, -0.0292338505, 0.105079204, 0.0722285211, 0.0492487848, -0.0207891911, 0.035598442, 0.0796257257, -0.0816210359, 0.0394578874, 0.10630095, -0.0223288164, -0.0539216921, -0.0801568329, -0.0579407737, -0.0488362312, 0.0901255012, -0.0542660505, 0.123969197, 0.0129767805, 0.0857983679, -0.0723153949, -0.116513394, -0.0345694795, -0.0708460286, -0.0530526638, 0.112991229, 0.110247165, 0.055062592, -0.0358034968, -0.0648803413, -0.00882329047, -0.0386624709, -0.0317198709, -0.0141925812, 0.133358002, -0.119553827, -0.0781110525, -0.0169827417, 0.0419830829, 0.0809727758, -0.0601022243, 0.0752082318, 0.0453452766, 0.0357860625, 0.0793421566, -0.125073418, 0.0902063996, 0.0117165446, -0.0659095347, 0.00580528378, 0.00889448822, -0.12447641, 0.0204410553, -0.0412814021, 0.0495228618, 0.0835448503, 0.116250575, -0.0654591396, 0.136590302, -0.0437139794, -0.130533695, -0.0867854059, 0.072424531, -0.0716329142, 0.099989742, -0.029022947, -0.118508801, -0.00216673315, -0.00964409113, 0.0275921971, -0.0702549517, 0.0168310702, 0.0938851982, 0.0028321445, -0.114841782, 0.0769343674, 0.00749561191, 0.00931432843, 0.129629493, -0.00428524613, -0.0622541383, 0.0181307346, 0.128360391, 0.00720927119, -0.00107601285, 0.135486186, 0.0301079601, -0.122348845, -0.106044114, 0.017554909, -0.0103668272, -0.0536207855, 0.0721321106, -0.11596261, 0.0342057943, 0.0130974054, -0.0751927495, -0.0975918621, 0.0968466997, 0.111900821, 0.0677128434, -0.0339190885, -0.0657791123, -0.0346289575, 0.132123798, -0.107705772, -0.00667120516, -0.0373312384, 0.0983017981, 0.0146001726, 0.0881693661, 0.0728048384, -0.0892456695, -0.0545547754, -0.0606427193, 0.127758384, -0.11426615, -0.0448431, 0.0735787302, 0.0686352849, 0.105652809, -0.0194403604, 0.0510896444, -0.0973827839, 0.0499836057, -0.0842511952, 0.0107224584, 0.0790108889, -0.0802243128, 0.00903344154, 0.133382469, -0.0144729838, 0.00228916109, 0.00299805403, 0.136510193, -0.0606871843, -0.0106766224, -0.0197322518, 0.101590022, 0.034936294, 0.127533883, 0.00446902215, 0.00279822946, 0.115145057, -0.065636538, -0.0213813409, 0.0332797915, 0.0421897322, -0.04739739, -0.03065712, 0.122296244, 0.0230481327, 0.0973794311, 0.0809123367, 0.109200478, -0.0475174636, -0.0738452896, -0.0478056669, -0.0509483814, -0.0712444782, 0.101722687, 0.120032609, 0.0380587727, 0.115555257, 0.0806039274, -0.0530673563, -0.130207911, 0.077729404, 0.0261965245, -0.0817069337, -0.0618148744, -0.00412149727, -0.014915511, -0.103205219, -0.134377867, -0.0374422371, 0.13429296, -0.0570919588, -0.0797002017, 0.0528538823, 0.0800858587, 0.0458294004, 0.0261586457, -0.0560341701, -0.133453399, -0.0814694911, 0.0389332771, -0.0216553807, -0.0522843227, 0.0104800165, 0.054231286, -0.0362112522, -0.121657453, -0.0945644826, -0.0313536674, 0.110182002, -0.0274486542, -0.0645038635, -0.0392875969, -0.054631725, 0.0906170607, 0.0446703285, 0.0665438026, 0.0628865361, 0.0406519026, 0.0847905278, 0.013615489, -0.0455756336, -0.0462128669, 0.0173976421, -0.121880502, 0.117248267, -0.106539533, -0.0776506662, 0.0470769554, 0.0631131977, 0.0956659615, 0.106449336, 0.0514396876, 0.0951529741, 0.0847110301, 0.0335356891, -0.128389612, -0.0655849278, 0.0276690274, -0.0208295137, 0.0726699382, 0.0539053679, 0.0205788165, -0.0640053451, 0.0256249309, 0.132323802, 0.0422382504, -0.00320878625, 0.0842960477, -0.121599346, -0.0290251002, 0.0178422928, 0.0335367322, -0.0237912312, -0.0647743717, -0.104194477, -0.047350511, 0.0779209435, 0.080603987, -0.0237182304, 0.0247604847, 0.0798442066, -0.113430329, 0.101311639, -0.0551978573, -0.0396380946, 0.133087188, -0.0148522779, -0.00979818404, -0.00603397191, -0.10580916, -0.133506253, -0.00967347622, -0.0730265379, -0.0310022905, -0.029996708, 0.129264534, 0.123995304, 0.136550188, -0.0245039761, 0.109209001, -0.0926341116, -0.0518179983, -0.033019796, -0.0177469328, 0.0844373554, -0.0381035581, 0.0177293122, 0.0150468796, 0.103413239, 0.0835546106, -0.0884617865, -0.00752341747, -0.0771219507, -0.110308968, -0.0577309504, 0.0467014909, 0.124507934, 0.100173935, -0.0943341628, 0.0161749572, -0.108874336, -0.0713768005, 0.135854423, 0.0966987014, -0.0205949098, -0.101613097, 0.104421154, -0.0497194603, 0.0223887563, 0.0740994364, 0.0744936168, 0.115517199, 0.0120522231, -0.0541860983, 0.020311147, -0.0562019721, 0.124659091, 0.0691441149, -0.053887479, 0.0724818856, -0.0313050598, -0.0811104104, 0.104190558, -0.0330485925, 0.111697629, 0.0963663608, -0.0238290727, 0.0223227441, 0.0528036952, -0.0996605903, -0.021703206, -0.0652093217, -0.0223025084, 0.0271105915, 0.0292074382, 0.00457368791, -0.068554908, -0.0547924116, 0.108942538, 0.0641764849, -0.0987549722, -0.119499959, 0.0951081514, -0.0419656485, 0.118541718, -0.0252901465, 0.121815503, 0.0855444968, 0.0422533005, 0.0254690796, -0.0655569509, 0.00358602405, -0.0913407132, 0.082400322, -0.0784052312, -0.0180871487, 0.124201268, -0.136227459, -0.0170292258, -0.0532112941, 0.131566346, 0.06952402, 0.0666095465, -0.110658646, 0.113614708, 0.0028873235, -0.109899834, -0.014672257, 0.0058144629, 0.132832855, 0.00573641062, -0.0126792714, 0.0756112784, -0.125071108, 0.0649617016, 0.0426058769, 0.131729156, -0.0732614994, 0.0341416746, -0.0541509688, -0.101108447, 0.0102382302, -0.124604024, 0.130719483, -0.0247230083, 0.00963482261, 0.0265038162, 0.0424721539, -0.123501085, 0.00206148624, 0.0938844234, -0.0733475909, 0.0948895514, -0.120868802, 0.120048553, -0.131673038, -0.0366031453, -0.0553891286, -0.0627916306, -0.0435904413, -0.057633467, -0.0436587781, 0.102742121, -0.0266828611, 0.131982088, -0.0139831528, 0.104467243, -0.0220600367, 0.101302817, 0.0486853719, -0.000630795956, 0.0732958168, 0.0789853334, 0.0535539538, -0.046998024, -0.00175790489, 0.043284148, 0.0617725253, 0.130353421, 0.0918721706, -0.00624765456, -0.131705746, -0.0312967971, 0.128403842, 0.0586179644, 0.0303991735, 0.00364759564, -0.0247948915, -0.0597023666, 0.0240047723, 0.085168764, -0.0661254898, 0.0477693081, 0.0469849259, -0.104816139, 0.0806702971, -0.0418047309, 0.115232438, -0.100655794, 0.125909954, 0.0046890974, 0.0220941156, -0.0794617161, -0.0660549402, -0.0322142392, 0.0484143049, -0.0505887121, 0.0484498292, 0.101025939, -0.0860916302, -0.0568180159, -0.0740828887, 0.132015139, 0.0850556791, 0.0805580616, -0.0910110474, -0.0797288641, 0.0998696536, 0.00483940542, -0.0404196531, -0.029866904, -0.0876832604, -0.0712021068, 0.0319518596, 0.056360662, -0.0139351264, 0.000249356031, 0.0315214694, -0.0407522917, -0.135266572, -0.128061816, 0.0832460374, 0.0479347855, -0.103647217, -0.115489721, -0.0657822117, 0.108107135, -0.089061439, -0.0267519727, -0.058967188, -0.0365279913, -0.0619976595, 0.121219993, -0.0310177654, -0.0474473089, -0.000912636518, -0.11945869, -0.00367443264, -0.0183600113, -0.0413725525, -0.107271016, 0.104627863, -0.100125641, -0.123059146, 0.0906228423, 0.0421913713, -0.0222766176, 0.12505427, -0.114441305, 0.0816470981, 0.0929709375, -0.119069442, -0.0779820979, 0.119288027, -0.110795863, -0.0563212335, 0.118073702, 0.0981317759, 0.0664688647, 0.0602101237, 0.0270466805, -0.10832414, 0.00654751062, -0.0517121553, 0.021417737, 0.095620811, 0.11452195, 0.0508430004, -0.0997347683, 0.0343427062, 0.0199356079, -0.0386759862, 0.0982036293, -0.0412252843, 0.112768382, -0.0958701, 0.0842528045, 0.0155244023, -0.098992601, -0.052829951, 0.104019761, 0.00673630834, -0.0389265865, -0.0390314832, 0.0433861464, -0.0208425373, -0.115250684, -0.00176331401, -0.0448659211, -0.0905172676, -0.0429517403, 0.096448794, 0.059812814, 0.0969527662, 0.120459139, 0.027512908, 0.0399251282, -0.00255598128, -0.135592774, 0.0619364232, 0.118778795, -0.128738359, -0.0909728482, 0.123057872, -0.000388264656, -0.134973079, -0.0446337387, -0.0617902279, 0.0797113329, 0.0840478092, -0.109512709, -0.0891110003, -0.123604089, 0.0288672596, 0.0394423455, -0.045054324, 0.0299270004, -0.0326793268, -0.0441791937, 0.0433877707, -0.0327894092, 0.0628817081, -0.120908603, -0.135370582, -0.129082546, -0.00913827121, -0.133775815, 0.0925979167, -0.0279047936, 0.0137742162, -0.0684487373, 0.0832460076, 0.0778043717, 0.0220358074, 0.116572708, 0.120394021, -0.126439199, -0.0440204367, 0.116596639, -0.00574839115, -0.121665649, -0.117598802, -0.133597374, -0.123539574, -0.0827658027, 0.0988901258, 0.0562292635, 0.0241476446, 0.0646850467, 0.0456878394, 0.114608794, 0.0522514731, -0.0722370073, 0.0649634004, -0.0653436705, 0.00828239322, 0.0441260487, -0.0794956684, -0.112388924, 0.047713086, 0.105907008, -0.0337683558, 0.112112969, 0.00168156624, 0.0221335292, 0.0984038562, -0.0405161902, 0.101812184, -0.0306580663, 0.00638313591, -0.00933606923, -0.0495209992, -0.0118647963, 0.133386314, 0.0972756445, 0.127949864, -0.0170405582, 0.030266434, 0.0644918531, -0.0410653427, 0.0243677348, -0.126150668, -0.0376376882, 0.0793990642, 0.115365475, 0.125485301, 0.132854491, -0.0173375756, 0.123990357, 0.126760542, 0.0199246109, 0.0463828295, 0.133341432, 0.0799899697, 0.0754961669, -0.0465824604, -0.0846978053, 0.0873944014, -0.00712434947, 0.0672320575, 0.0847331285, -0.031734623, -0.0822531432, 0.112729147, 0.091640383, -0.0295949876, -0.101722397, -0.0939373076, -0.0188322812, 0.136161178, -0.111046098, -0.0737150609, -0.00393897295, -0.0723129138, -0.00878252089, 0.0726039559, -0.0808813944, -0.104831845, 0.11933437, -0.0736284181, 0.117690653, 0.132863224, -0.106923886, -0.130747631, 0.0599240363, -0.0373848379, 0.0192611963, 0.00730569661, -0.105000041, -0.0734499022, -0.11048428, -0.134641781, 0.0674274415, -0.105549127, 0.0875730067, -0.0965825468, 0.0865682364, 0.0314493179, -0.0624415278, -0.0868700892, 0.132529616, -0.00267550349, 0.123484045, 0.0232645124, -0.0157514364, 0.100139067, -0.0107656717, -0.031046465, -0.125469819, -0.00878351927, -0.0412467942, 0.051600799, -0.0452794284, -0.0817394853, -0.111147568, -0.10428945, 0.0193194747, -0.0737061799, 0.0928273499, 0.0987958759, 0.0650438666, 0.0444750786, 0.0709429234, -0.0109952241, -0.0512328371, 0.0293803364, -0.0724560991, -0.0101262629, -0.0339284912, -0.102498278, -0.0825525522, -0.0278738439, -0.0327277705, -0.0812947005, 0.033122018, 0.00578024983, 0.0188989043, 0.116528481, -0.027826868, 0.000491172075, -0.106478974, -0.011813581, 0.010574013, -0.0519400612, 0.123747796, 0.0615936518, -0.119706713, 0.0965384394, -0.108477712, -0.0182201862, 0.0777682662, -0.0450730026, 0.0741986185, -0.0867925212, -0.0914172977, -0.0107384473, 0.131009102, 0.100436121, -0.00689902902, -0.0676930621, 0.133405417, 0.0340053141, -0.0278127939, 0.0735555142, -0.00789925456, 0.0237952769, 0.125645787, -0.00715275109, 0.0814768672, 0.0229864568, 0.039741382, 0.0535612106, -0.00911837816, -0.073020339, -0.136608064, -0.0868141353, 0.105997264, -0.108271837, -0.0134975314, 0.0235030651, -0.0706957877, 0.0434921086, -0.0152588561, -0.0328821242, 0.0723848939, -0.0791713893, -0.0699490532, -0.0299490392, -0.090794012, -0.0844306946, 0.133389503, 0.117837787, -0.115428381, -0.0866210312, 0.0410853177, -0.0918630287, 0.118478656, 0.0146174431, 0.0953406394, -0.0962813497, 0.0473799258, -0.0181181654, 0.131747723, -0.120570317, 0.136137247, 0.0953928381, 0.0457116365, -0.00359970331, 0.0654873103, 0.0974072814, -0.119495809, 0.0238964856, 0.0779941678, 0.12287885, -0.0259701163, -0.077402845, -0.0903707147, -0.0973898098, 0.0840773582, 0.084917292, -0.0957877338, 0.00296367705, 0.0508234501, -0.025126718, 0.0773919076, -0.0142726302, 0.0410522819, -0.0980267525, -0.0504460782, -0.117062584, -0.118355528, 0.110945344, -0.0739619359, -0.00828537345, 0.0250171572, -0.0373283327, 0.0482215881, 0.0739530623, -0.00570225716, -0.131928071, -0.0220187083, -0.0621101633, 0.073841244, 0.0657580495, -0.0160987303, -0.0192219168, -0.0456597954, 0.115348727, -0.105435088, -0.0813490897, -0.136476174, -0.0613244548, 0.012233153, -0.0721570551, -0.0675859153, -0.104073301, 0.0922733992, 0.0365638137, -0.0522537977, -0.13286984, -0.129645869, -0.0356296524, 0.108128846, 0.118089706, 0.134406865, 0.000925406814, 0.0339840204, 0.0268510282, 0.136217177, -0.0668128356, 0.0955496728, -0.0347480252, -0.0991844982, -0.0170325562, 0.0585017502, 3.32742929e-05, 0.104093537, 0.0859187245, -0.0749645233, -0.136781573, 0.0874286443, -0.0839600861, -0.0636291578, 0.0829299092, 0.00441795588, -0.0970190763, -0.13331753, -0.0837791264, 0.0838996172, -0.109015271, -0.133527741, 0.0867631137, 0.0342673063, -0.0698866695, 0.0552534908, 0.122101486, 0.097059682, -0.0596561059, -0.0732495785, -0.0900109708, 0.0287191421, 0.0704183877, -0.0147428438, -0.0729215443, -0.02997493, 0.0591437072, 0.0911006927, -0.0470742807, -0.0834658444, -0.128154859, -0.128171474, -0.0141603276, -0.0415874943, -0.0741763264, 0.0191976279, 0.00458350778, -0.0131755695, -0.0289093405, 0.108689323, 0.0278994441, 0.0151216388, 0.0795960575, 0.10847947, -0.0252841711, 0.121694714, -0.09039177, 0.121906906, -0.0624969006, -0.122551583, 0.0379208326, 0.0489537269, 0.0682066679, 0.0822287202, -0.0358567089, -0.105450898, -0.0416091457, -0.0385292098, -0.00931750238, 0.118311584, 0.0558300316, -0.104803734, 0.0148100257, 0.0676030517, 0.0233720094, 0.10112904, 0.0701182336, 0.000294700265, 0.0258774012, -0.0826673359, 0.136286765, 0.104154587, 0.120219171, 0.0439334363, -0.057297565, -0.0512804985, -0.128053397, -0.0474716276, 0.0476621836, 0.031222567, -0.0340055376, 0.050065577, 0.11938867, 0.13348335, 0.12134698, 0.107014388, -0.0903482512, -0.106243461, -0.028781265, 0.119756818, 0.0329640061, 0.053051725, 0.0452067256, 0.0849139988, 0.0232935995, -0.00309948623, 0.0251261592, -0.0166506246, 0.0362438411, 0.0985837728, -0.128518403, -0.0527147353, 0.0568866134, -0.0457645282, 0.0102809668, -0.00682477653, -0.111691199, -0.0985759348, -0.119488858, -0.0336322561, -0.00871042907, 0.0908353776, -0.102891028, 0.0237320364, 0.109722108, 0.0339153707, 0.0781892389, -0.0568968281, -0.070392102, 0.00909925997, -0.0573852882, -0.0305456594, 0.109213173, 0.119168997, -0.132001013, 0.0735763758, -0.04390046, 0.0619595945, -0.132424966, -0.117013089, -0.0970229208, -0.119751304, 0.0943338424, -0.00310666859, 0.0708045363, -0.0581020787, -0.128431141, -0.121518217, -0.0430620909, -0.119222105, -0.00157390535, 0.00488206744, 0.0923803449, -0.0263164267, 0.128791809, -0.091206111, -0.128529444, 0.0107199401, 0.0514403731, 0.00419060886, 0.0311676115, -0.0974185318, 0.105336308, -0.0783051699, 0.00641301274, 0.0655302703, 0.0650752187, -0.0335167795, -0.0150460303, -0.121415116, -0.00268605351, 0.0662408918, 0.0607724637, 0.0548945069, -0.0603127927, 0.132084787, -0.00612483919, -0.061769329, -0.0205898881, 0.0278406739, 0.0459839404, 0.109364167, 0.0521156639, -0.136487722, -0.0256103128, 0.132692397, -0.0793503895, -0.0167675614, -0.0664683804, -0.133050963, 0.0292422771, 0.0520415008, -0.036471352, -0.124928989, 0.0878525674, -0.0451673493, -0.0438311845, 0.0276689231, 0.110060781, 0.0252711177, 0.0686930269, -0.117099896, -0.0133249238, -0.0166052803, -0.120200396, 0.0487333685, 0.133657664, 0.100010395, -0.0016284585, -0.120911248, -0.0790074319, 0.0274080038, -0.11876113, 0.0467091352, -0.0860109925, 0.0293624401, -0.124765135, 0.0377427191, -0.00803343952, 0.128490061, -0.0583512112, -0.111046851, 0.0569658428, -0.105105519, 0.0783790797, 0.122847766, 0.0893425643, 0.0331273377, 0.0140959769, 0.120581686, -0.0513454303, -0.0712746456, -0.0107715577, -0.0754768774, 0.00752152503, 0.123520523, 0.0994419903, 0.042070508, 0.116076678, 0.108907014, -0.0100371242, -0.0502856821, -0.127781808, -0.0959718227, -0.00823584199, 0.103984758, 0.00784423947, 0.136094183, 0.13676849, -0.0667719617, -0.0593828186, -0.111090891, 0.110446766, -0.0694717243, 0.126528531, -0.131870806, -0.126988739, 0.0219853669, -0.0724558756, -0.0417747572, 0.0626463294, -0.0257236287, -0.092297107, -0.0480091572, 0.0706134886, 0.0550106615, 0.0181860328, 0.0275326818, -0.0548655391, -0.101263121, 0.0703497231, -0.0191987753, -0.106192559, 0.0636165142, 0.00324371457, -0.0499303266, -0.0433189198, 0.039193213, -0.0623440817, -0.082757771, -0.108307488, 0.077211827, -0.0241999403, 0.0282767415, 0.100406244, 0.069861725, -0.0870052502, -0.115959577, -0.136538222, -0.105175421, -0.136884451, 0.035523057, 0.0981892049, 0.11644423, -0.0965195149, 0.0948940217, 0.0897577703, -0.119575374, -0.068613112, -0.039985843, -0.0190420374, 0.0148238391, -0.095509544, -0.0392760411, -0.0559469983, -0.0620127767, -0.0302660093, 0.106922835, 0.132595956, -0.0433744565, 0.0305157602, 0.056451723, 0.0654757917, 0.103904799, 0.0396663249, 0.0550738573, 0.0720562786, 0.10757558, -0.026466243, -0.0444748476, -0.0581008419, -0.111512296, 0.0722546428, 0.123054862, -0.0892638266, 0.0384279788, 0.0987899601, -0.0856239945, -0.0184375793, 0.133606642, 0.0523470044, 0.126677632, -0.000685289502, 0.0932309926, 0.0348463953, 0.0536953509, 0.105479881, -0.0786405206, -0.00612908602, 0.0537355691, 0.116253257, -0.0880500823, -0.0127767548, -0.0298942924, -0.0561042279, 0.0919492245, 0.0362647623, 0.0261767954, 0.0154044032, -0.118463717, -0.0106966347, 0.0869911462, 0.0964087099, -0.116868556, -0.0612397343, -0.0924005955, -0.0270310044, 0.0967000425, 0.121895581, 0.130125463, -0.0907645673, -0.0897659287, 0.0844743699, -0.0405976772, -0.0880294144, -0.0699958727, -0.0804035068, -0.113904461, 0.00601027906, -0.0234429538, -0.0116924196, 0.126409292, -0.0303086415, 0.113090932, 0.0786094069, 0.114850223, -0.123965874, 0.04720366, -0.0705588013, -0.0382724777, -0.103151806, -0.0243912116, 0.122166961, 0.12630558, 0.111489579, 0.0731034577, -0.0456609353, 0.0503623039, 0.099888131, -0.063670747, 0.126902491, -0.0737484917, 0.0970897228, 0.00655455887, 0.0902363658, 0.0328852683, -0.120686963, 0.0849710852, -0.102837935, -0.0925061107, -0.0784913525, -0.0852063149, 0.00321094692, -0.0445294008, -0.133646205, 0.109196946, 0.116363645, -0.00162254274, 0.0841408223, 0.0649395585, 0.0306562632, 0.124539614, -0.0997705758, -0.0310134217, -0.102773756, 0.0394320637, 0.0774853081, 0.0297313184, -0.0408617556, -0.0799109042, 0.0766610801, -0.078001976, 0.0935018957, -0.0187650248, 0.0326421708, -0.113368921, -0.0512247086, 0.0387326032, -0.048958458, 0.0846625119, -0.0432993993, -0.113230005, 0.0856152177, -0.107339084, 0.0999075621, -0.0594706386, -0.0687982887, -0.0745980591, 0.0952702165, -0.0735825151, 0.103935629, 0.0240671337, -0.0319503248, -0.055029951, 0.126859069, 0.00795416534, 0.0563020408, -0.10236688, 0.13665995, 0.0107578039, -0.122057773, 0.132144094, -0.0724108815, -0.0900636017, 0.0899018645, -0.0209324136, -0.120483376, 0.0978723913, 0.0331790447, -0.0832656175, 0.0845608264, -0.125201523, -0.0578101203, 0.0134700686, 0.0208921582, 0.104788646, -0.127424389, 0.0944375247, 0.043242991, -0.107128546, 0.0195430666, -0.0772839487, 0.0700984448, 0.0560875088, -0.114404187, 0.0533519685, 0.0696230829, 0.0500552952, -0.0486046374, -0.100405201, 0.133118063, 0.0117811859, -0.0582463518, -0.0252300426, 0.0213049799, 0.118892163, 0.0619460791, 0.0371985584, -0.00492532551, 0.0355799645, 0.0832643807, 0.0933858752, -0.00250583887, -0.0811907873, -0.0571916625, 0.0886474848, -0.13435021, -0.0582796782, -0.0443269908, -0.0121342316, -0.0409444571, 0.0860714465, 0.00317509472, 0.0317439884, 0.0716000348, -0.0742574185, -0.0234479532, 0.0419644117, 0.0696455687, 0.117133528, 0.069949612, -0.054899171, 0.0629307032, -0.00542390347, -0.0756822601, 0.0755674988, -0.088504687, 0.0961316973, -0.120285079, 0.128451705, 0.0585775822, -0.124496162, -0.113663524, 0.0804674625, 0.0603919327, -0.015699625, -0.0458351076, -0.0837002173, -0.036410138, -0.0842880234, -0.0957390517, -0.126437411, 0.055495888, -0.0290719867, -0.115706533, 0.00690737367, -0.106253356, -0.00222922862, 0.00638636947, 0.136639714, -0.130089208, -0.0571671128, 0.0308016837, -0.127073139, -0.0840152949, 0.0520015359, -0.0486909226, -0.0650354177, -0.125432044, -0.0534592792, 0.0923637003, 0.0989185274, -0.120891556, -0.000621885061, 0.13054949, -0.0274071917, -0.113035627, 0.0832538009, 0.113880157, -0.113907561, -0.00255301595, -0.000591561198, 0.130752295, -0.045228824, -0.0526037365, 0.123807877, 0.0970283747, -0.102338865, 0.069728002, -0.104946956, 0.102437556, 0.0581571907, -0.0741001293, 0.0444572121, -0.0030233264, -0.0282619521, -0.0256473646, 0.0676550567, -0.13509123, 0.0396783501, -0.0301795602, -0.0897156149, -0.0638799146, 0.0823161602, -0.0953015238, -0.0743213445, 0.0201806277, -0.0811779946, 0.107954443, -0.00337570906, -0.00971934199, 0.0885137022, 0.0604767799, -0.119999848, 0.0861417353, -0.119649321, -0.0760148987, 0.089216575, 0.0480475128, -0.00522832572, 0.106205195, 0.126377225, 0.13524431, -0.0834581703, -0.000878751278, 0.0671182126, -0.0438458398, -0.0107437074, -0.0491714478, 0.0218756795, 0.0627507269, -0.037882641, -0.0736816302, -0.0426758751, 0.0872242749, 0.128437817, -0.100631341, -0.0738518834, -0.107284829, 0.0454461575, -0.0564804524, 0.0316800028, -0.0166500658, 0.0586845726, 0.0480518341, -0.0206569433, 0.0516817868, -0.00426511467, -0.0620380118, 0.0527656078, -0.0513607785, 0.0292428583, -0.0290877521, -0.0475891903, 0.0364919454, 0.0036188066, 0.0160036981, 0.0517819226, 0.131391287, -0.121882394, -0.0802767724, -0.0106136799, 0.13031289, -0.0857627764, -0.135954931, 0.0724732429, 0.0937915444, -0.00633455813, 0.0220428705, 0.131122321, 0.0100516528, -0.0629529431, 0.0558041036, -0.0757858455, -0.0485834777, 0.0231841058, -0.0111280531, 0.127422839, 0.0986086726, 0.0358464271, -0.0342786312, -0.0679353029, 0.123054206, 0.0904192179, -0.109934345, 0.0577495992, 0.114916652, -0.135566831, -0.0446366146, -0.0408690721, -0.0263216868, 0.12370643, -0.0191679224, 0.124116838, -0.0694237649, 0.130773544, 0.0519571751, -0.0522508249, -0.106997699, 0.0546361357, 0.0576944202, -0.0237817988, 0.059796229, -0.129319265, 0.0842217803, 0.131958067, 0.128440678, -0.00129529834, 0.0223187655, 0.133176416, 0.055896014, 0.0757275373, 0.0713572055, -0.0836920589, -0.103879668, 0.132169753, -0.102196105, 0.0688092262, -0.109179191, 0.13486439, -0.0893321186, -0.0739976838, -0.0681645125, -0.0610896572, 0.0293230712, 0.00956080854, -0.00190111995, 0.0921217203, -0.127043292, -0.0280772373, 0.0288666636, 0.0143638104, 0.0984716862, -0.0585380793, -0.0271505862, 0.03382653, -0.0623259246, -0.00730890036, 2.32756138e-05, -0.0943615884, -0.0858648643, -0.0644539446, -0.0675351471, -0.111309886, 0.019990921, 0.0293648541, -0.047796987, -0.0938501433, 0.0293900222, -0.046621345, 0.113267362, -0.109652013, -0.0356403291, 0.122125745, 0.108362004, -0.0301989838, 0.0521476269, -0.0828424543, -0.103570864, 0.0743227452, -0.0115605295, 0.0945950449, 0.136096179, 0.00197905302, -0.116294429, -0.00212404132, 0.0813746601, -0.0810060352, -0.0970925912, -0.0726671964, 0.12972039, 0.0690163672, 0.124263674, 0.0461698622, 0.1159949, 0.0975343734, -0.0393245518, -0.127924308, 0.0933650732, -0.0110772252, 0.0892811865, -0.0825201645, 0.103403583, 0.0490089357, -0.0741517469, 0.106485367, 0.118132323, 0.0707530826, 0.0261539072, -0.0248588473, 0.0466733426, 0.0414143354, 0.0181136876, 0.115674973, 0.011881277, -0.0440483466, 0.0855888724, 0.00350424647, 0.120592654, 0.0910972953, 0.0350409895, -0.0663104057, 0.084793359, 0.0223444551, -0.0145348832, 0.0328541547, -0.05145026, -0.0464102477, -0.0853003338, -0.114435062, 0.104983583, -0.0497277826, -0.0830415636, -0.0658770204, 0.102298945, 0.00115860999, 0.076831758, -0.0143973753, 0.0154636204, 0.12856555, -0.118063398, 0.0759682059, -0.0122529045, -0.0851866603, 0.118180871, 0.0136093795, -0.136744693, -0.072859779, 0.0305171311, 0.0487162173, -0.0113377422, 0.126042128, 0.091231674, 0.0114648342, -0.0360141322, -0.037275672, 0.0722761154, 0.113058642, -0.00639308989, -0.132716686, -0.0679949448, 0.100947499, 0.104375213, -0.0530837476, -0.0409268215, 0.0480398834, -0.0657091513, -0.00375974178, -0.0540021956, -0.0989605784, 0.0222224593, -0.10744907, -0.0570113212, 0.108316958, 0.0982603282, -0.036241062, 0.0474478602, -0.0650933981, -0.0180442855, 0.028708294, -0.127319127, -0.100772992, 0.126135617, 0.113112897, 0.0675831437, 0.0374301821, 0.0869508535, -0.0204449371, -0.134612367, 0.0226760209, -0.0383700877, -0.0839552879, -0.023379229, 0.0797197223, -0.116203152, -0.0964124948, 0.0375358015, 0.128981233, -0.0111501515, 0.109349832, 0.0896549672, 0.0227474123, 0.0783401728, -0.095428586, -0.114835836, -0.0875191092, -0.0574464351, -0.0511667877, 0.0159212649, -0.0904242545, 0.128912687, -0.100479662, 0.0770364553, -0.0549969152, -0.0592422411, -0.0238574073, 0.13500914, 0.0938336849, 0.0219465941, -0.0315933973, -0.0424854159, -0.0863585472, -0.0336530134, 0.0599575639, -0.0114217103, 0.0038972497, 0.103980511, 0.0115303993, -0.133669689, 0.0990677625, 0.0294876099, -0.091690585, 0.113523692, -0.0224685147, -0.0752440095, -0.129941583, -0.0415092409, 0.0575455874, 0.0270656347, -0.0653796792, -0.117771082, -0.0929383188, -0.111615658, 0.0808861554, -0.0996594802, 0.124172539, 0.0921595991, -0.135693133, -0.0708992705, 0.0151500106, -0.101841167, -0.0409430191, -0.108884647, 0.0614504069, 0.1250543, 0.0496179909, -0.0460122526, 0.0921798944, -0.0285486206, -0.0166778192, 0.00766223669, -0.132137239, -0.0908356681, -0.109672323, -0.0587465316, -0.0917949229, -0.0321453214, 0.0525925756, 0.132113189, -0.0612824336, -0.124468543, 0.00918523967, 0.0290578753, -0.0458133966, 0.0937909931, 0.115016282, 0.0108943731, 0.0714527071, -0.109289736, 0.0439956188, 0.0853204131, -0.0383676067, -0.0620002076, 0.115915984, 0.0567686558, 0.0642954111, -0.0811725408, -0.0673033893, 0.122292489, 0.0605366826, 0.0960350931, 0.0956777781, 0.00737962127, -0.0711956695, 0.0689126849, -0.0438272357, 0.0890601724, 0.00938785076, 0.126547694, -0.0471894965, -0.128692806, 0.00478981435, 0.00796082616, 0.130308151, 0.0800433755, -0.0513560101, -0.110880062, -0.0965960622, -0.131567493, 0.0993641615, -0.0600399971, 0.124575794, -0.0420187265, -0.07880757, -0.00749345124, -0.0227379128, -0.125631228, 0.0740180612, -0.075208813, 0.0675159842, 0.0104151517, -0.026500918, -0.0756703466, 0.0744711608, 0.13343218, 0.12198481, 0.0918223858, 0.0317174792, 0.0774797201, 0.00680048764, 0.0539913327, 0.116550624, 0.0325739086, -0.00708575547, -0.0607766733, 0.051164642, -0.0221630409, 0.018378526, -0.0512623787, 0.0383725315, -0.0461483896, -0.0641455278, -0.0965751708, 0.0970107168, 0.105739132, -0.122537419, 0.0178013295, 0.107133016, 0.0125948191, -0.0135797337, 0.0797807425, 0.0611358136, 0.0529499948, -0.135286316, -0.0640067458, -0.120747462, 0.0661098212, -0.105924435, 0.0982864797, 0.0967068374, -0.0613402873, 0.0689376295, -0.0656040907, 0.0363693982, 0.111808658, -0.0275689587, 0.00758306682, 0.0290805399, -0.131993115, 0.0235240757, 0.0112666488, 0.0848694593, -0.0882292092, -0.120486349, 0.0718367547, 0.0624758005, -0.0758686066, -0.0128832832, -0.136147812, -0.0521976128, 0.113158196, 0.103650421, 0.121767521, 0.0231329054, 0.0155290365, -0.0927346349, -0.0189576074, 0.0683096647, -0.130036056, 0.124609053, -0.0170007572, -0.0893515423, 0.060974285, -0.0451976135, 0.0573027879, 0.0536007732, -0.104038201, -0.123042397, -0.015266858, -0.00371608138, -0.0795646831, -0.0452143624, 0.136367708, 0.118662477, 0.0296504796, 0.135353684, 0.0211382806, 0.0997147113, -0.0202512741, 0.122795224, 0.133774847, 0.0252506733, -0.0868833512, -0.0196186081, 0.11263822, 0.110760838, 0.00225409865, 0.129932493, -0.0822386518, -0.0750381649, 0.112813398, -0.0326290801, 0.0869027376, 0.122541666, -0.117104858, -0.0811770707, -0.00336121023, 0.0891758353, 0.120802879, 0.0851752311, -0.127724662, 0.075992927, 0.00552037358, 0.00993840396, 0.0839840174, 0.000344485044, 0.0288314372, 0.130288333, -0.131219804, 0.0781232864, -0.114732742, 0.00839407742, 0.0153136402, 0.0134378225, 0.0699736327, -0.0791138634, 0.0551245958, -0.0434599221, 0.0988393575, -0.0179145783, -0.106059656, -0.115503855, 0.0305479467, -0.0638865456, 0.101052254, -0.0421021432, -0.0806993544, -0.0345053896, -0.100246072, -0.0207606927, 0.0162339211, -0.0814323127, 0.110953644, 0.00843192637, -0.107001454, -0.0608810782, -0.133155733, -0.0369181558, -0.0392057523, -0.0369349718, 0.0566265434, -0.0147343874, 0.0925732255, -0.00758492947, 0.135466546, -0.0622921661, 0.0643838197, 0.110984847, 0.0497137159, -0.129211992, -0.0791157559, -0.129735216, -0.0425587744, 0.0275189131, -0.00198623538, 0.010402903, -0.0209983289, 0.0361455083, -0.0859315246, 0.0176406354, -0.0969529599, -0.0926274881, -0.0650475249, 0.0944561064, 0.0582294315, 0.0810323507, -0.0295920148, -0.00400814414, 0.0725500286, -0.0864371955, 0.0339131206, 0.0362699181, 0.0280079544, -0.130080238, -0.0683498159, -0.123454332, 0.104002938, -0.0686788633, 0.0247931331, -0.124924809, -0.0422899947, -0.00432136655, 0.0393503457, -0.104298234, -0.0987556875, 0.10403429, -0.0171738565, -0.0580046326, -0.000511705875, 0.0794814676, 0.106441498, 0.125230491, 0.031059593, -0.0224574804, 0.0882577747, 0.112146825, 0.125952125, 0.124437779, 0.0567529202, -0.0847644657, -0.0479874462, 0.00017952919, 0.0494967401, -0.0327971131, -0.101243794, 0.0755880326, -0.0679002032, 0.13497588, 0.135284036, -0.00892116129, 0.0503858775, -0.0320283473, 0.101213798, 0.0958126336, -0.0420148149, -0.0682129934, 0.0186359435, 0.0203741491, -0.110912152, 0.0118872523, 0.0944701731, -0.0212488323, -0.055293642, 0.0734030604, -0.122572541, 0.0197974145, -0.131350681, 0.0986521244, -0.0759862661, -0.111149952, 0.054469347, -0.100436568, 0.00284297764, -0.131670073, -0.0733880699, 0.0850994289, 0.0944229364, -0.105013229, -0.0282981545, 0.062829569, 0.064699024, 0.0377689004, 0.0846547186, 0.0485548526, 0.100507736, 0.0347696096, -0.0923394114, -0.0967936441, 0.122052908, 0.0155787617, 0.0224155635, -0.118212305, -0.0138303936, -0.0780868605, -0.0663772672, 0.0427794307, -0.0591381639, -0.130883992, -0.10663937, -0.0155063197, 0.0224140882, 0.0528750718, 0.0536451787, -0.024905175, -0.0426487774, -0.0544733256, 0.0558504015, -0.127411067, -0.0975524187, -0.0726310536, 0.0948315412, 0.0223526508, -0.0277670547, 0.0418350846, 0.00274203718, 0.0744189918, -0.0387199, 0.0737740546, 0.069701761, 0.0245006531, 0.00366891921, -0.105077311, 0.115573168, 0.102167934, -0.109060846, 0.128638864, 0.0194603354, -0.00553539395, -0.0252884775, -0.0868210196, 0.0409129858, -0.0842051655, -0.123129465, 0.0951313376, 0.108136848, 0.0644914806, 0.0772708505, 0.0613072217, -0.0908147693, 0.0161613822, -0.0360886678, 0.0388506204, -0.00129209459, -0.083115086, -0.0226994231, -0.0842282176, -0.0287849233, 0.0185759068, 0.124659359, 0.0709281713, -0.11003232, -0.0615004823, -0.0553943217, -0.0240448639, 0.101626545, -0.0481623709, -0.126848653, 0.00159649551, 0.0603701472, -0.11553739, -0.125237405, -0.00959676504, -0.105384648, -0.0873550326, 0.00820475817, -0.0992375165, 0.116867542, 0.136130393, 0.0672802478, 0.00716499984, 0.0375452638, 0.0759035349, 0.0346540362, -0.115761377, 0.0666639358, 0.0504043251, 0.00155849755, 0.116153061, -0.0634514242, 0.016740635, -0.068967104, 0.0892555267, 0.102096692, 0.0718745589, -0.0453448221, -0.00494922698, 0.117953748, -0.104866192, -0.121879354, -0.106153905, 0.000722467899, 0.118624598, 0.122366935, -0.105685398, 0.052938208, 0.00407399237, 0.127534032, 0.0891807973, 0.0737172812, -0.0629373342, 0.0883646309, 0.116588742, 0.0395490378, 0.00398141146, -0.119333461, 0.0488301963, -0.087909922, -0.050027743, -0.0825482756, 0.0982488096, 0.0561511815, 0.112053618, 0.056774199, 0.10417603, 0.0557125658, -0.0401355997, -0.0168073252, 0.0910581946, 0.0167201608, -0.102387741, -0.125422224, 0.0131521523, -0.108884811, 0.112588659, -0.0435525402, 0.045208022, 0.133276165, -0.132883936, -0.0581636578, -0.126409858, 0.0481514633, 0.106447443, -0.0236389339, 0.00838337839, 0.0392358899, 0.0361100137, 0.0924970359, 0.0805996209, 0.0609958619, -0.068897076, -0.0304632634, 0.0985625535, -0.00787518919, 0.0128683895, 0.0596730858, 0.0179165006, -0.108517796, 0.0474794954, 0.100393713, -0.126368359, -0.0410906821, -0.0823168084, -0.124741435, 0.0682646036, -0.0176939517, 0.113333404, -0.0434227064, -0.082161054, 0.111413479, -0.102407888, -0.103837714, 0.108590603, -0.107646033, -0.10935656, -0.053814806, 0.116967797, -0.00894407928, -0.128417403, 0.110866383, 0.0655931532, -0.09308213, -0.126885161, 0.125396341, -0.0309519172, 0.0884053707, -0.0797633678, 0.0171965808, -0.0557991788, 0.0771594942, -0.0366589054, -0.106419884, 0.048750177, -0.0136521086, 0.0410774201, -0.0748713464, 0.0949198157, -0.101798534, 0.0459492058, 0.124476016, 0.023176074, 0.131986707, -0.0802201033, 0.0757454634, 0.0892337263, 0.0892047286, -0.0901892632, -0.00974206626, 0.0644918829, 0.0621574372, 0.0015963912, 0.0548603833, 0.0397425294, -0.12043637, -0.131608784, 0.0172828585, -0.0536915958, -0.0561034754, -0.0385942757, -0.0270212442, 0.0921092778, -0.118261471, 0.00721004605, -0.0853868127, 0.109283164, -0.113672599, 0.0950393379, -0.025295727, 0.119675934, 0.066724658, 0.0253613144, 0.127001643, 0.00893771648, -0.101018503, -0.126088798, -0.0837126225, 0.0679278523, 0.0015168637, -0.0761470199, 0.0932754874, 0.0473926812, -0.0625604913, -0.0711588115, -0.0539988652, 0.0252117962, 0.134128273, -0.106004618, 0.0999458581, 0.0067820847, 0.0169609338, 0.0396694392, 0.0647911131, 0.0272307694, -0.100203797, 0.124540418, -0.0220394358, 0.0973239988, 0.0378319025, 0.104935467, -0.135075882, 0.0910106152, -0.0811444297, 0.00515779853, -0.0244440362, -0.00429615378, 0.00323657691, 0.0955038071, -0.108087584, -0.0580240563, 0.113435805, -0.0712489858, 0.0924686342, -0.0845316947, 0.126962543, 0.119404405, -0.127294615, -0.054852128, 0.0818173438, 0.13374573, 0.122065574, -0.050890334, 0.115936667, 0.0850919783, 0.0217027217, 0.10054861, 0.0544310808, -0.132629558, 0.0745338053, -0.0514838248, -0.0640729517, -0.0117925853, 0.104231507, 0.0992470533, 0.0600041896, 0.0808274001, -0.0868516788, 0.0695322901, -0.120368823, 0.0824336559, -0.0589151829, 0.130303711, 0.0340646654, 0.0716471523, -0.110057257, -0.022828348, -0.0792923421, -0.0843452513, -0.110510007, 0.0572808236, -0.0812956542, -0.0672106743, -0.134977549, -0.0448198244, -0.00136695802, -0.104383864, 0.130255163, 0.108304158, -0.0242779329, 0.117537558, 0.0133853555, 0.124705464, -0.0713904798, 0.0847505927, -0.0102681369, 0.0751455426, -0.0946647152, 0.00561927259, -0.0605079532, 0.0664407313, 0.0507230908, -0.0728674829, 0.00553934276, 0.0733247995, 0.0632089525, 0.0795918703, -0.0532236993, -0.027946189, 0.0729770511, -0.0290855989, -0.0484358519, -0.0779489279, -0.126688167, -0.119646542, 0.0279364586, 0.081094414, -0.0893805325, -0.0263148621, 0.0524814725, -0.10716299, -0.126297161, -0.0484121814, 0.0249602199, 0.0150750279, -4.70429659e-05, 0.0681203753, -0.0022893846, -0.0475169718, -0.0594990402, 0.13106221, -0.122276828, 0.0441582054, 0.00520710647, -0.0851201266, 0.0561644882, -0.0806354284, 0.00498379767, -0.0799960122, 0.0132209063, -0.0547764525, -0.114347443, 0.039588213, -0.0227579251, -0.0779782087, -0.0104546249, -0.0720982254, -0.0632655323, -0.117410824, -0.00677169859, 0.00307056308, 0.0790260434, -0.038753137, -0.123694129, 0.0554045737, -0.0127840042, -0.0422151014, 0.105680883, 0.0922319442, -0.0701297224, 0.0485112071, -0.0880366564, 0.0206162632, 0.0991554111, -0.0195788145, -0.0428518429, -0.0933517888, -0.0381260887, -0.0674763545, -0.0809458047, -0.0666443184, -0.120846182, -0.109756187, -0.0856183171, -0.0439622626, -0.00236693025, -0.0287453234, -0.114870936, 0.116978675, -0.00496250391, 0.110881075, -0.136482075, -0.0647615418, 0.0432302803, -0.0730567351, 0.000531226397, 0.0888753831, 0.100618705, -0.060204275, -0.0663503632, -0.0241169855, 0.0145903528, 0.0966626704, -0.0115521103, 0.108025685, -0.0701036379, 0.0920478404, -0.108868659, -0.0930422992, 0.117650002, 0.0365153849, 0.013202861, -0.0132957399, 0.0917621851, 0.0996774286, -0.0853567123, -0.0535529777, 0.0945906639, -0.093339026, -0.00639612973, 0.0694723129, 0.12057814, 0.00187751651, 0.0399993658, 0.0804118365, 0.0169023573, 0.11724025, 0.0893333852, -0.0836961716, -0.0735546649, 0.125247657, 0.0552326888, -0.0383784473, -0.0800489336, 0.0606704652, 0.0844358206, -0.023337245, -0.00983253121, -0.028690666, -0.110367142, 0.0735692233, -0.081581533, -0.0247477815, 0.00873093307, -0.0604812503, 0.00285643339, 0.0435820818, -0.0183207691, 0.125970751, -0.0449164584, 0.0760211647, -0.0174164176, 0.0521882474, 0.0154310316, 0.131391943, -0.105654642, 0.0871497095, -0.12930429, 0.0791472942, 0.119967818, 0.0724800378, 0.103556663, 0.0982557386, -0.075052239, 0.00284892321, -0.00303286314, 0.0167715549, -0.0916907191, 0.0380103886, 0.1012059, 0.11382699, 0.0715570152, -0.0526468679, 0.0258979648, -0.124975972, 0.04145962, -0.121823497, -0.0428962409, -0.0725257024, 0.112746418, -0.112606391, -0.0857898742, 0.0273825079, -0.0616823956, 0.0570104122, -0.0266931728, 0.010204345, 0.134085983, -0.0234495476, 0.05235973, -0.0619190484, 0.11585626, 0.092316553, -0.0101277977, 0.0223333836, 0.0138385892, 0.0317714512, -0.133827046, -0.0973558873, -0.0679819882, 0.040704757, 0.0313572586, -0.0646699965, 0.100117609, -0.1095227, -0.0269814432, 0.0185008496, 0.0289959162, -0.0942840204, -0.101014517, -0.132222846, 0.0744165033, 0.0853347182, -0.0589974895, 0.025514394, 0.0336866081, 0.11872226, 0.116404057, -0.0585095137, -0.120991819, -0.131958634, 0.0961178243, 0.119421154, 0.0768882036, -0.0810848176, 0.0475426018, -0.0964338779, 0.0482020378, -0.00131233037, -0.0689793453, 0.0858920962, -0.051717408, 0.0998160243, 0.00143322349, -0.0966993272, -0.0380304009, -0.116321534, 0.0529877692, -0.0946307629, 0.0773836076, 0.0480381846, 0.0745847672, -0.0095435828, -0.0229893625, 7.28368759e-05, -0.0119988471, 0.106342092, -0.0832643211, 0.0739099979, -0.0376740247, -0.0371220633, 0.0359511524, -0.0101117343, 0.134594142, 0.0809273273, 0.0290460289, 0.133199334, -0.0121408552, -0.0805131719, -0.0777545124, -0.129825979, -0.0182744116, -0.0934727788, -0.136621833, 0.0727443099, -0.0617009699, 0.0640885234, -0.117219776, 0.0810971856, 0.0715808421, -0.0446313247, 0.0381075442, -0.112855285, 0.128142387, -0.0608610287, 0.0955524743, -0.120473906, 0.0758623779, 0.0534533709, 0.131898493, -0.119573385, 0.00469529629, -0.105027527, 0.136736274, -0.0911420882, 0.115644008, -0.120779023, 0.0712350458, 0.132166058, 0.0217978507, -0.0576129332, -0.0669588968, 0.0939740092, -0.0288665071, -0.0685031936, 0.00372621417, 0.124188691, 0.0638543516, -0.090250209, 0.128464311, 0.100386754, 0.0393110961, 0.0161572993, -0.0903270617, -0.116809204, -0.0387688354, -0.0502193123, -0.107288614, 0.0504106283, -0.0631548613, -0.135471359, 0.0155035853, -0.0857766867, -0.0682556629, 0.0239417404, 0.1133551, 0.108482838, 0.0049598366, 0.0244025141, 0.0936750323, -0.129612535, -0.0770145059, 0.124895364, -0.089932166, 0.0558585972, 0.070413515, -0.0977591127, 0.0396927446, 0.00957944989, 0.0690825433, 0.0213024616, 0.0531828254, -0.116070896, 0.13466996, -0.065331623, 0.0635906011, 0.0733023435, -0.126838341, 0.0987905562, 0.0300785899, 0.0175869614, -0.0393739119, -0.0710717812, -0.0538154244, 0.0574035048, 0.0581829846, 0.125308156, 0.050741896, -0.0571570843, 0.107688218, -0.111826457, 0.00187076628, -0.0521990508, 0.132537454, -0.112733975, 0.0644428432, 0.0909367353, 0.0420732498, -0.0581795499, 0.00582098961, -0.100567415, 0.0500706136, -0.0951858237, -0.131025493, -0.130506933, -0.00721807778, 0.0844634324, 0.0347004235, 0.105358303, -0.0805533603, 0.016413644, 0.0652503967, -0.124113314, 0.0472906381, 0.012561217, -0.0957234204, 0.0358997732, 0.126927048, 0.00383707881, 0.047625199, -0.128910661, -0.12394508, -0.0372348949, 0.00634036958, -0.056973353, 0.101630822, -0.102108546, -0.0852196664, -0.131926015, -0.104347952, 0.131746173, -0.0421884283, 0.0719232708, -0.0424370691, -0.128319323, -0.0986432806, -0.0506603047, -0.0872852281, 0.0701775104, -0.0804776549, 0.050581038, -0.0904583037, 0.00325417519, -0.00437450409, -0.133308545, -0.021184288, 0.104108393, 0.10643813, -0.105286255, -0.000865474343, -0.0784510672, 0.0130015612, 0.069292888, 0.0294358581, 0.111727402, 0.114960849, -0.126027331, -0.109669223, -0.0891985595, 0.0976584256, -0.092740871, -0.131682664, -0.00859721005, -0.0230295509, -0.117653981, -0.0115853995, 0.0982471108, -0.0502333492, -0.0591124371, -0.0810497254, 0.0443587601, -0.0881960392, -0.136805639, 0.119254321, 0.00219129026, -0.0968263596, 0.0782870203, 0.0316111296, 0.065927431, 0.0801804364, -0.0725534186, 0.109324574, -0.130468756, -0.0438179895, -0.00459964573, -0.0422631577, 0.135696441, 0.073313728, 0.0217691809, 0.0328913629, -0.0584107265, -0.0056078136, -0.0516480654, -0.0679348111, 0.118013054, 0.103554606, -0.0368776694, 0.0302800536, -0.0708669499, -0.0909005031, -0.0295100734, 0.0803425312, 0.105221972, -0.0530715063, 0.108004138, -0.0654371008, 0.0855426043, 0.117454916, -0.0894752443, -0.0891896486, 0.101815894, 0.0234781206, 0.107075915, -0.0280958787, -0.132728875, 0.034560889, 0.113126278, 0.0127422065, 0.0638370812, 0.0745148063, -0.129952163, -0.0142011642, -0.121911906, -0.0415422842, 0.00148448348, -0.125934094, -0.0422629565, 0.117701173, 0.0734438896, -0.108167827, 0.123293161, -0.0330989659, 0.0116648972, -0.0860403031, 0.0197178572, 0.0785241574, -0.0553176329, -0.0878652036, 0.0872872472, 0.136424303, -0.123370923, 0.0942315608, -0.130185783, -0.113298304, 0.01725097, 0.0379061848, -0.0502171889, -0.0490549356, 0.00814524293, -0.00149901211, -0.0834271908, -0.0654800013, -0.12495736, 0.0160182267, 0.10887444, -0.13011542, -0.019236058, 0.0694419891, 0.0801118463, -0.0405424759, 0.0233606547, -0.0242961794, 0.0188242793, -0.108741462, 0.013283208, 0.115673304, 0.106512398, -0.0631923378, -0.000435307622, -0.0123381466, -0.109843977, 0.110814497, 0.0951025784, -0.0321945176, -0.101717278, 0.0732999295, 0.00233784318, 0.120378256, 0.0691161007, 0.0643844754, 0.045262903, -0.125269949, -0.12051256, 0.0607623011, 0.136048019, -0.127658367, -0.112174928, -0.02291587, -0.0670445636, -0.0282026008, -0.0170222744, -0.048267588, 0.0458327234, 0.0556264371, -0.062001355, -0.052715458, 0.128618449, -0.0033609271, 0.108790204, -0.110544741, -0.112250246, 0.0403413028, -0.0342319757, 0.0865636319, 0.0789161474, -0.0401424542, 0.109872907, 0.00649465621, 0.0405632406, 0.0677405894, -0.0507344157, 0.0765382648, 0.0124416947, 0.0668387562, 0.0241016448, -0.0706546828, -0.0957477689, 0.0703876317, 0.00473046303, 0.112907037, -0.0676834285, 0.0179590434, -0.0391954631, -0.0258670822, 0.0164625496, -0.0768107921, -0.101416856, 0.120916903, -0.051098235, -0.0456515029, 0.0249854922, -0.109967969, 0.00669102371, 0.0631081164, 0.0223971158, 0.0798863471, 0.0106289238, 0.0940352827, 0.0682321191, 0.0200158209, 0.0257198811, -0.0266938582, 0.0936458409, -0.104743533, -0.0450688526, -0.0440693423, 0.115807921, 0.0989186317, -0.0791916251, -0.0976634175, 0.0804375261, 0.100325376, 0.0861642361, 0.00116758049, 0.0185006261, 0.0540115684, -0.0894639492, 0.00134037435, -0.0766617954, -0.0469802245, 0.021985054, 0.0392880142, 0.0889122784, 0.0221657753, -0.0816372335, 0.0418925434, 0.038874805, 0.13672328, -0.118700042, 0.133970857, 0.0724960566, -0.105456181, 0.0891320854, 0.0400934815, -0.132249326, 0.0370177925, -0.0350467414, -0.136630386, -0.0599948764, -0.114977658, 0.0300672501, -0.024529703, 0.102679476, 0.0965716839, -0.115897872, -0.0848692656, -0.0557651892, 0.0978577733, 0.0422261655, -0.0412849933, -0.0855225325, 0.0219302624, 0.00107006729, -0.0936949104, 0.121761292, 0.0296949148, 0.0597975254, -0.0686576441, -0.0261763111, 0.0402729809, 0.0141732544, 0.00385294855, -0.075358212, -0.0799973458, 0.134335518, -0.00835683942, 0.134540707, 0.0402865857, -0.112439305, 0.096138522, 0.134351283, 0.0215957612, 0.0911492705, 0.124521911, 0.0763081014, 0.0521245152, -0.0614289194, -0.124345496, -0.069110848, -0.0927817449, 0.0917175561, 0.0921318382, -0.0975183398, -0.111883029, -0.124598116, 0.1366916, 0.0831387639, 0.118250936, -0.0849632919, 0.0649344027, 0.0577178299, -0.0692275912, 0.0346371233, 0.0829238743, -0.0445555523, 0.0398997813, -0.0678235218, -0.0863944292, -0.0707440376, -0.122544467, -0.104427449, -0.0590443686, -0.0561795458, 0.104862273, 0.073129639, -0.130538493, 0.017612204, -0.0526878014, -0.0478048846, -0.0807929859, 0.113913804, -0.123120949, 0.00855140388, -0.109289438, -0.135410145, 0.0816427767, -0.10365212, -0.0666465983, -0.125489965, -0.072345823, -0.0299374536, 0.0190713853, 0.127223939, -0.0398757309, 0.0719335824, -0.109606437, -0.0117159337, -0.0925998688, -0.0802781433, -0.111190528, 0.048691541, -0.0160998404, 0.0578321964, 0.0629730523, 0.0359464288, -0.0609413087, -0.11633563, 0.00702735782, -0.0541952029, -0.0705175623, 0.123724669, -0.0251282826, -0.113981828, 0.0752968639, 0.0969801843, -0.136530653, -0.1357155, -0.0431622788, -0.0679783002, -0.0875890702, 0.014395386, -0.0735477805, -0.038223736, -0.0617697909, 0.125509232, -0.060923256, 0.0298420936, 0.11359033, 0.102109984, 0.0441154987, 0.00316850841, -0.0258605182, 0.0268177539, -0.0930154324, -0.074634105, 0.0624319613, 0.0813095868, 0.0417106152, -0.00621542335, -0.0825776607, 0.042720899, 0.0354643613, 0.0540966094, -0.0443150401, -0.070054926, 0.124698907, -0.0438814238, 0.126394302, -0.0260835588, -0.00136087835, 0.0776307136, -0.0331936106, 0.0558076352, 0.000338673592, 0.0708984286, -0.0924539417, 0.122926652, -0.0603136718, 0.0778414905, -0.0440241247, 0.118446231, -0.028422378, -0.00781479478, 0.121765494, -0.122393802, -0.0983005911, 0.0714678764, 0.0375824869, 0.114013493, 0.111333489, 0.109208599, -0.105351225, 0.101094529, 0.00853697956, -0.0993187726, 0.00964847207, 0.0076264888, -0.0117033273, 0.0442798436, 0.100322857, 0.0416977108, 0.0282501727, 0.0786968321, -0.118002743, -0.0803775564, 0.0487019867, 0.0637591183, 0.0202346593, 0.029405728, 0.0205045491, -0.0653771609, -0.0149702281, -0.0875260681, 0.00233751535, 0.0659660846, 0.0113362521, -0.0808709785, 0.0892809629, -0.0673984587, -0.0374127179, -0.0614604279, -0.0534706414, 0.0465401113, -0.0111816972, -0.135526076, 0.115498632, -0.127388895, 0.021988377, 0.0960872024, 0.103912473, -0.0414090827, -0.0190828145, -0.128401533, -0.0912638009, 0.112491339, -0.0898963511, 0.0476643145, 0.0100690275, -0.0362614319, 0.0954067409, -0.00241465867, 0.0692979395, 0.0434637368, 0.113373965, 0.00332441926, 0.00841288269, -0.108588122, -0.0047019273, -0.0585729182, -0.0987589508, -0.113126293, 0.118381321, 0.0686590523, -0.0460049734, -0.0282678902, -0.034603402, -0.1207771, -0.0288477316, -0.104355067, 0.031194061, 0.0726336688, 0.0554594845, 0.113435149, 0.115987957, -0.0382946134, -0.0655966476, -0.0986436754, 0.124309421, 0.112208977, 0.128700584, 0.00400534272, -0.0797734559, -0.054966554, -0.0138869733, 0.0288286954, 0.106002912, -0.0873406976, 0.014251411, -0.13395299, 0.122482657, 0.0906396955, -0.00107522309, -0.0834816471, 0.0196638256, 0.0782198012, -0.104809284, -0.00988872349, 0.0432757586, 0.11515224, 0.0648912191, 0.0729929507, -0.0826354772, -0.0464676768, 0.00735852122, 0.0900885165, 0.0800053775, 0.0840630531, -0.0371949002, 0.0792003721, 0.107095212, -0.0442746878, 0.069464311, -0.0907473862, -0.0477131829, -0.00563298166, -0.0923676491, -0.0885544419, 0.0667262524, -0.0393705815, -0.0543792322, 0.104572892, -0.0230908245, -0.0328157917, 0.0994201154, 0.0192306042, -0.0111610293, 0.0373073071, 0.00712539256, 0.0426192731, -0.114879981, -0.112385862, 0.0534262806, 0.0240614861, 0.115970969, -0.0784108192, -0.102334261, 0.113824308, -0.0790179446, -0.0453964695, 0.0692582428, 0.124202102, 0.127219141, -0.0867178589, 0.0876395702, 0.0415853411, 0.00786592066, 0.130917072, -0.0830751956, -0.132702231, -0.0441425368, -0.0370271653, -0.0299352333, 0.0266798288, -0.0492154881, 0.0337437391, 0.136627138, -0.0509986877, -0.131172687, 0.0620774776, -0.102750972, 0.0978041887, 0.0754043013, 0.00464750826, 0.0656031817, 0.114009231, -0.128868997, -0.0304804668, 0.0648151189, 0.0808440447, 0.133106619, 0.00206658244, 0.0769577026, -0.0632543713, -0.076252073, 0.129483283, 0.0541664064, 0.0131216049, -0.132955894, 0.0486795902, 0.0981484801, -0.0124098361, 0.0717148483, 0.07089369, -0.0325427353, 0.078711167, -0.0619804263, -0.12627165, -0.0146004334, 0.107437029, 0.0177870542, -0.0526204556, 0.0679083019, 0.0172071159, -0.0950306207, -0.0398605168, -0.124607876, -0.101674832, -0.0121223778, -0.0710727572, 0.131095648, -0.108607285, -0.0873361528, 0.028038457, 0.00953264534, 0.0808874369, -0.0700527728, -0.00431032479, -0.0563273057, 0.0298001021, -0.128384367, 0.111862361, 0.0518351048, -0.0971349329, 0.116144061, 0.0295843035, 0.0673106015, 0.0173918307, 0.0616193861, -0.0885904804, 0.108766302, 0.0151495636, 0.0822869688, 0.00196191669, 0.0346852839, -0.0770007968, 0.0661608875, -0.0279053152, 0.110463262, -0.0682858005, 0.129971981, 0.110505402, 0.0354239494, 0.0298446715, 0.0156028569, -0.056358546, -0.045260489, -0.0434574708, -0.0388076901, 0.0882522017, -0.044422321, 0.0712821484, -0.0766772628, -0.0953552276, 0.133333117, 0.0522306114, 0.0609820187, -0.0865394771, 0.128399312, 0.089206785, 0.0222623497, -0.00112530589, -0.00341048837, -0.0903844237, -0.111233816, 0.114814937, 0.0682183802, -0.0335946456, 0.0375279635, 0.123001486, 0.0825007111, 0.132988572, 0.111294255, 0.0742075443, 0.122671276, 0.118292987, 0.0564267188, 0.0773493052, -0.105295166, -0.0104848444, -0.0342570469, -0.028912209, 0.0180912614, -0.0432273448, -0.111850291, -0.0919075906, 0.125226796, 0.0321166217, -0.00761538744, 0.0261684358, 0.0809461325, -0.0409804285, -0.0424509048, 0.109816417, -0.0595642328, 0.098117575, 0.0504079461, -0.102097973, -0.0722079203, -0.10379041, 0.126059085, -0.0617830083, 0.0258047879, -0.0672331974, 0.0673811883, 0.0382514447, -0.0780567601, 0.067713201, 0.0869937539, 0.114066571, 0.0104175061, 0.0886221826, 0.0991815627, 0.0399525464, -0.0672446936, -0.0319698751, 0.0211679935, -0.0642305389, 0.107411131, -0.0883418098, 0.0511147231, -0.0988682806, 0.0240443051, 0.0284313262, -0.0969554782, 0.126312643, 0.00484533608, 0.113133132, 0.0272889137, 0.115209341, 0.0560011566, 0.109789029, -0.0259423628, -0.101224698, 0.121979475, 0.0835744888, 0.0586123914, -0.0879128948, -0.13154076, -0.046367608, 0.0159905404, 0.0630668402, 0.0729676485, 0.135843873, -0.0604884624, 0.117527843, 0.0818277597, 0.0671858341, 0.106247276, 0.112086907, 0.125209123, 0.106851637, 0.0560624003, -0.0511105061, -0.0576765016, 0.114818513, 0.0393131524, -0.0629665256, 0.0314871669, -0.0211334229, 0.0119503587, 0.0534743369, -0.0844929144, -0.0758507475, -0.0236985162, -0.000881433487, -0.13324143, 0.124201447, -0.101280786, 0.0426201224, -0.00236819685, 0.030341059, -0.118585721, 0.0681946129, 0.103528187, 0.0872093588, -0.063437812, 0.0486724824, -0.000832781196, 0.0239926279, 0.120768666, -0.00783938169, 0.0206792802, 0.0216434598, 0.0448061079, -0.0583124608, 0.0145533234, 0.120076507, -0.113788821, -0.10148029, -0.0832330137, 0.085065797, 0.0515691638, -0.0328730866, 0.0525225103, -0.0878447592, 0.114821494, 0.0583996624, -0.0957011506, -0.0510933995, -0.121803612, -0.00536073744, -0.0901011452, 0.022209987, -0.130103216, -0.122222833, 0.0185550451, 0.01551193, 0.023330912, -0.11505679, 0.129102111, -0.0902691782, 0.0445156842, -0.00225540996, -0.0986540541, 0.0911066085, -0.0765604898, 0.0420176834, -0.0467577726, -0.0922480673, 0.134012759, 0.0924467593, 0.12404871, -0.0387786627, -0.0172997415, 0.0648670197, 0.119855493, -0.0973559543, -0.0732564032, -0.039557457, 0.0992048085, 0.0768739283, -0.094169721, 0.103476942, -0.00601905584, 0.0255998969, -0.00702269375, 0.00488294661, -0.0297635719, 0.0762206316, -0.0854631811, -0.126439884, 0.116564244, 0.0623750538, 0.0348347723, -0.00128376484, -0.116802223, -0.136688039, -0.118722998, 0.111147925, 0.0696121454, 0.080598712, 0.0576797277, -0.0619806573, -0.133959234, -0.102336191, 0.00499884784, 0.0743276477, 0.0386605114, -0.0876077786, 0.0766717792, 0.05341129, -0.0265279189, -0.0746541172, -0.00088326633, -0.12702325, -0.0920161158, 0.0213638097, -0.0575771183, -0.112095043, 0.0400214344, 0.0427900404, 0.0583102405, -0.0226855502, -0.0267410651, -0.0270384774, 0.127693921, -0.0362102762, -0.115017779, -0.115709893, -0.000587373972, -0.0612432957, -0.0879602656, 0.0445439965, -0.00131204724, 0.00436380506, -0.115925983, -0.109412976, -0.116617411, 0.134762436, 0.0565050691, -0.0234285891, -0.0854096413, -0.0746720731, 0.118881553, -0.132845253, -0.0331647173, -0.112874746, -0.0308153257, 0.00644166768, 0.120229602, -0.0568609461, -0.0585357919, 0.0226747692, 0.0812734514, -0.097241953, -0.123348199, 0.0455345362, 0.133995831, -0.0374899954, 0.0410035104, -0.041514568, -0.0362903923, 0.0674186349, 0.0364922434, 0.121052802, -0.115704045, 0.0657061189, -0.0414375216, 0.0951079577, 0.107390836, 0.0431292802, 0.119400978, -0.03732647, -0.0744007081, 0.0104419142, 0.100902796, -0.0368449613, -0.0367137566, 0.0127672851, -0.130265728, 0.0777427256, -0.116713129, -0.0560514703, -0.0741394386, -0.0983221978, 0.0172569454, 0.0327500999, 0.0802074075, -0.124531128, -0.126084685, -0.0748952776, -0.0538553521, 0.096374616, -0.0237428844, 0.110881954, -0.054667376, 0.120567828, 0.0264597833, 0.0165620148, 0.0454263389, 0.0727924556, -0.0465561152, -0.0515597612, 0.0523216426, -0.0949289948, 0.0587471128, -0.0858276784, -0.0266103819, -0.101605877, -0.0245901346, 0.13028571, -0.0659441426, -0.0201865658, -0.0965605155, 0.0415666997, 0.0587853789, -0.134659737, 0.123420209, -0.00746312737, -0.10369812, -0.0261199623, 0.00347349048, -0.0198397264, -0.070349142, -0.132043451, 0.00241164863, -0.0190812796, -0.0841912627, -0.0336518064, -0.110430181, -0.099938184, 0.0232136101, 0.0790180415, -0.0307973996, -0.0589869767, -0.0460327193, -0.0608371049, -0.0923140123, -0.107069291, 0.00173220038, -0.00213748217, -0.0249190181, 0.0841237754, -0.0491564348, -0.0819401592, -0.0904916078, -0.0765380934, -0.128318384, -0.130968586, -0.00672596693, 0.00731654465, -0.119272932, 0.00399780273, -0.0262283832, -0.0179135948, -0.0912256986, 0.11373052, 0.0277364999, -0.116054609, 0.0413184166, -0.0589451194, 0.0576853156, -0.0696883351, 0.0667781979, 0.130437821, 0.0496585667, 0.112217918, -0.0956312269, 0.130965531, -0.115536831, -0.0920139551, -0.0468032137, 0.0432354063, 0.0889815241, -0.0401219204, 0.0645901859, 0.109863102, -0.0726730749, 0.0509820431, 0.0958648175, -0.129835278, -0.121966325, 0.0389822423, -0.000660374761, -0.0272100717, 0.0320221186, 0.136755437, -0.125418395, -0.0369677097, -0.0671290904, 0.126165777, 0.079549998, -0.0717725456, 0.131064653, 0.131568611, 0.128364712, -0.135854438, 0.0640028566, -0.0336126685, 0.0991562307, 0.105787292, 0.0635974854, -0.0725242347, -0.00602437556, -0.0714441463, -0.0976951569, 0.105480015, -0.0268593132, 0.125822902, 0.132054836, -0.110450946, -0.128546819, -0.0559696555, 0.0677369684, -0.00483433902, -0.119616315, -0.127996877, -0.121783763, -0.0164836347, 0.0532813817, -0.0865568444, -0.12955305, -0.0366837159, 0.0609708577, 0.115923464, -0.0674119741, -0.102059312, 0.0587392896, 0.00531186163, 0.00613969564, -0.115202919, 0.111942619, -0.0805427432, -0.0794878006, 0.0636342764, -0.00813992321, -0.0557605252, 0.122505218, -0.0108366907, -0.121706069, 0.10817948, 0.000266730785, -0.00415407121, 0.0157738626, -0.123610906, -0.0433453619, -0.0628264695, 0.00195345283, 0.10101077, -0.00419478118, -0.0152422711, 0.118645906, 0.0926781595, -0.00647050142, 0.0885630846, -0.013510555, 0.0165005177, -0.00789341331, 0.00234299898, -0.069075264, 0.0701233894, -0.10107547, 0.0182135254, -0.0986558199, 0.00244125724, -0.0555718914, 0.0657515526, 0.01661174, 0.0281449705, 0.114979923, -0.0572134703, -0.133554637, 0.0206375569, -0.132798538, 0.109364226, -0.0577709749, -0.0947145671, -0.0207366347, -0.124801829, 0.0983299762, 0.0373530686, 0.0522623211, -0.00818543136, -0.0105451196, -0.0844118521, -0.132443503, 0.129143685, 0.126591444, 0.0144366771, -0.0874437988, -0.126433775, -0.0210666955, -0.0647376478, 0.0324497223, -0.0995931774, 0.0574104935, -0.0502837598, -0.0986577123, -0.0762417614, 0.0146685988];
    recurrent_3_f : ARRAY[0..4095] OF REAL := [0.0276267845, 0.0778834075, -0.0103492681, -0.0744607523, -0.0235891733, 0.0874153674, -0.0411629118, -0.0455408245, 0.121018052, 0.0665290356, -0.0657219216, 0.0329201072, -0.00274422904, -0.00143206306, 0.0355367921, -0.128572166, -0.0254000276, 0.00422622729, -0.0497977957, -0.107884482, -0.0839469731, -0.0995972157, 0.0171393026, 0.095180437, -0.042353984, -0.00141653558, 0.0157543961, 0.029983785, 0.000925835222, 0.16947484, 0.0323171839, 0.0326515064, 0.0897902623, 0.018178165, 0.0363775566, -0.0409856066, 0.0570905283, 0.0742790326, -0.0228889734, -0.0200854875, 0.14655146, -0.00869555399, -0.127635568, 0.0105345044, -0.175763741, 0.00832119491, -0.0796563253, 0.0856589898, -0.0763150454, -0.0101055317, 0.0509098768, -0.070958212, -0.107807122, -0.147130474, -0.030100286, 0.0723497048, 0.00845288951, 0.0636945739, -0.064222075, 0.0175831374, 0.0119359689, -0.115816012, 0.0522544794, -0.0982318148, -0.0472634248, 0.0361897647, 0.0101031261, -0.0489332788, -0.0116338767, 5.04208729e-05, -0.00485811196, 0.0140675995, -0.0241822638, -0.0200194586, 0.0138263563, -0.0323163718, 0.0775291175, 0.137315288, 0.0592403524, 0.044101432, -0.0215705782, 0.0510005988, 0.0458572581, 0.0762273818, -0.0735793114, -0.0131371357, -0.10611774, 0.0773431063, -0.0776968151, 0.103860594, -0.172173351, -0.0415139236, 0.0194315352, -0.0212643966, -0.151790828, -0.0179847367, 0.0484757423, 0.0307152029, 0.0421229042, 0.0702095032, -0.0646686181, 0.0781433582, 0.0650567412, -0.0842932612, 0.054781612, -0.0744340867, -0.0162227675, 0.0112652071, 0.11347425, 0.0359552875, -0.0447856411, 0.0804083273, 0.0511757433, 0.0256622955, 0.142961532, 0.0726723894, 0.022950599, -0.0208708569, -0.0481408685, 0.00293323398, 0.0609455109, 0.0895497799, -0.0592034236, 0.0735294372, 0.0619786754, -0.00692794286, -0.0364842191, -0.0353424735, -0.0379250944, 0.0665906742, -0.0557924509, 0.0317343399, 0.0445529222, 0.025091812, -0.0108365398, -0.0722248256, -0.0516175255, 0.0125512714, -0.00739217084, -0.140388846, 0.165483698, -0.0160229895, -0.0233327709, 0.117798842, 0.0199612379, -0.00104783289, -0.0995874852, -0.113499865, 0.0333949402, 0.0256775357, 0.0206598788, -0.0237453412, 0.0170767289, 0.115832195, -0.106836759, 0.0458271354, 0.0256607533, 0.0414232425, 0.0621618144, 0.052170679, 0.109323516, 0.0860360786, -0.0905868113, -0.0100239106, 0.1080672, -0.0656371489, 0.00931994431, -0.0038321279, 0.0401097611, 0.00792204682, 0.0529838987, 0.0661005676, -0.104935095, 0.0282656569, 0.177242756, 0.030860221, 0.0232190192, 0.00489316136, -0.0280467011, -0.0872856453, 0.112857506, -0.060964413, 0.0821129084, -0.0359297954, -0.0646201745, -0.0685314462, -0.047921367, 0.000689394772, -0.0156825706, 0.0395166278, -0.0205429271, 0.0632746369, 0.0511896871, -0.0456937328, -0.0065044607, -0.00493180193, -0.0219476502, 0.113088779, 0.0534259155, 0.124904476, 0.0165670104, 0.0124835651, -0.00975962728, 0.0421168581, 0.0743560269, 0.0656922087, 0.0356202573, -0.137974605, -0.0721958131, -0.0520997494, 0.00206599198, 0.00811368134, -0.00539792283, 0.0219378807, 0.0561054908, -0.064646095, 0.131130621, 0.00360493362, -0.0183087997, 0.0767865553, -0.00241419114, -0.126514271, 0.0338337868, 0.131273717, 0.0998243913, -0.00292811543, -0.0368826836, 0.026254341, -0.11510919, -0.0414858982, -0.0864703506, -0.0110396165, 0.0484672636, 0.0299077779, -0.00726315472, -0.0402911007, -0.13991636, -0.0930280238, 0.0743694007, -0.0416963287, -0.0448754951, 0.0493883081, -0.0209460966, 0.124651983, -0.00897292979, -0.0554884896, -0.0280842222, 0.00291465595, 0.017124854, 0.018812485, -0.0390971974, 0.111629933, 0.0406235009, -0.0499143042, -0.124398246, 0.0383958817, -0.0640870929, -0.0559696518, -0.0776950717, -0.0143224336, -0.0880903974, -0.0378183872, 0.00415299973, 0.0561259538, 0.00693550333, -0.0477888435, -0.0382287391, 0.106731229, 0.00695215724, -0.102382094, -0.00333046354, -0.0834395736, -0.0753800869, -0.0247985087, -0.0248108655, -0.00424603559, 0.0763958469, 0.000766523182, -0.0562923141, 0.0260026045, 0.0233972184, 0.0869431421, -0.0252733957, -0.0487635657, -0.00802836008, -0.0178021323, 0.0300631672, 0.0275071897, -0.0259648655, -0.0149930902, 0.0773592889, -0.0286083166, 0.176284045, 0.0504190959, -0.0271145403, 0.0428201929, 0.0388792977, 0.0409477279, 0.0788895041, 0.00187323615, 0.0357947797, -0.103402451, -0.0169337615, 0.0222416036, 0.0400698185, 0.0634492561, -0.0610400513, 0.0388830453, 0.0535402447, -0.0396373235, 0.0768852681, 0.0208990499, -0.0966856033, -0.0236835927, -0.021708075, 0.0998882055, 0.00736593828, -0.0319053605, -0.0933315605, -0.0752548501, 0.0828225464, -0.151994556, -0.0419516638, -0.0925463066, -0.0540611185, 0.0451452918, 0.0149277728, -0.0840564668, -0.0223734863, -0.0251482297, 0.0451211482, 0.0190184806, 0.0019075356, 0.0333289243, -0.0352753252, -0.0215215012, 0.108203687, 0.00498744845, -0.0732392371, -0.0205856413, 0.0958089978, 0.0266844258, -0.0181558337, -0.0573500916, 0.000876855105, 0.0212557092, 0.073691681, 0.0874110535, 0.0341733508, 0.0070808325, -0.029903058, 0.0169168487, -0.0500960425, 0.0316428915, -0.0106053678, -0.0327092893, -0.0220670514, -0.0430492982, 0.0249179378, 0.122212604, -0.0631195009, 0.147385895, 0.058004722, -0.0378661528, 0.056999892, -0.0387807339, -0.0253789835, 0.0125110587, -0.0135396095, 0.055055134, -0.0385147259, -0.000293814694, 0.0048414655, 0.043078322, -0.0352888107, -0.106486864, 0.0206717663, -0.0054615289, -0.0897730738, 0.0712116137, -0.0993916541, 0.0491969883, -0.00737866014, -0.0107107237, 0.00675116433, -0.0168835912, 0.0506908558, 0.0372393169, -0.00395770976, 0.0833560228, 0.0354306586, 0.0103737712, 0.186585799, -0.0313842967, 0.0664263815, -0.0204714742, -0.0189028531, 0.0234329421, 0.0326043889, -0.013008602, 0.00553647615, 0.0626571625, 0.0265436284, 0.0676244646, -0.0283828378, -0.0112249292, -0.0267706476, 0.0869987756, -0.00317775458, 0.0222008992, -0.0644882992, 0.172908515, -0.0423217565, 0.0521393716, -0.0217889454, 0.09204714, 0.140652388, 0.0138055375, 0.0237383004, 0.0546265692, -0.0521529913, -0.0195349455, -0.0260922201, 0.0804242194, 0.0932194293, 0.0239222832, 0.0541057773, 0.0057645794, 0.055589553, 0.0829703361, -0.0766370669, -0.099370189, -0.0325682238, 0.00413249712, 0.0893853605, 0.131128833, -0.0251873657, -0.0982452556, -0.00451026205, 0.0472679585, -0.0029271394, 0.0373515338, -0.0238827392, -0.00691052154, -0.0706449896, -0.0259895846, -0.104922801, 0.0589773953, 0.00281834044, 0.130397022, 0.0197244398, 0.0262956601, -0.06928581, 0.0612638481, 0.135235518, -0.0230377316, 0.0334037393, 0.0434927382, -0.0267194975, 0.0117335487, 0.00885398872, 0.01622249, -0.0356796235, 0.0442460962, 0.0246567838, -0.00231462903, -0.0558599457, -0.0167908035, -0.0654707626, 0.0589314178, -0.0005340036, -0.00911000557, 0.0545933172, 0.111552633, 0.118486814, -0.0135540823, -0.0498979874, -0.0308784936, -0.0928313807, 0.0581183732, -0.0557660237, 0.0123628909, 0.0320827328, 0.0237374455, 0.0448954403, 0.0244392715, -0.002323105, -0.0162450802, 0.113559991, -0.0630255938, 0.0285602678, -0.0891122222, 0.0421227068, 0.0516199805, 0.132833034, -0.0428373627, 0.0876899511, -0.000412254827, 0.0492112786, -0.12743333, -0.0282597281, -0.0837111026, 0.0153183267, 0.0240087807, 0.0325392373, -0.0527864397, -0.0255600698, 0.0983394086, -0.116439737, 0.0368556231, 0.00516265072, 0.0797701851, -0.0156673174, -0.0878382549, -0.11339692, 0.0907338709, 0.0471590348, -0.0426403694, 0.0200875401, -0.0677194223, -0.0317382477, 0.170553893, 0.0325528756, -0.0387691446, -0.0575980768, -0.0394682959, -0.0399673507, 0.108603969, 0.00595466234, 0.0047010975, -0.0561040342, 0.106402919, -0.00859841984, 0.0572765507, 0.0154354759, -0.0306560453, -0.0971538574, 0.00949621946, -0.0469833501, -0.0551642478, -0.0193370599, -0.0372382104, -0.146381453, -0.0591826551, -0.0790911317, -0.0179479383, 0.0747570768, 0.019080719, 0.029013196, -0.0217684507, 0.0474928208, 0.0348910801, 0.0321962088, 0.120455749, 0.0586258397, 0.0509419441, -0.0583040155, 0.0331591256, 0.0149813853, 0.0332693458, 0.0155607369, -0.0437836722, -0.0417690426, -0.0013211146, 0.0433956534, -0.0804323405, -0.0839931369, 0.177810907, -0.0123451389, 0.0074120881, -0.00407789089, 0.0635630265, 0.0805817693, -0.106101677, -0.0521158576, 0.0295793116, -0.00020130453, -0.12579751, 0.0765392557, -0.0772586167, 0.0788546726, -0.0367428586, 0.0553745404, 0.0550354384, 0.0683907568, -0.00927887205, -0.00990959164, -0.00779848965, 0.0501311272, -0.0189925693, -0.0580634326, -0.0781877339, 0.0524611175, -0.0897354931, 0.0409517065, -0.0357711911, 0.0281049646, 0.026691597, -0.121823505, 0.066384092, 0.170445055, 0.0123317391, -0.0792309269, 0.0396172814, 0.0646545589, 0.036375571, 0.0160046462, -0.0333954133, 0.216201812, 0.0607321858, -0.0363657959, 0.0379377306, 0.039432168, 0.0278355181, 0.0076213479, 0.0817003697, -0.00598295033, -0.0264766868, 0.0441265218, -0.0433689617, -0.0388295129, 0.0686738566, -0.0352787822, -0.0304050781, 0.0748571306, -0.0786491632, -0.00977970287, 0.0496253185, -0.0828825012, 0.0273060314, 0.0342963114, -0.00108088367, -0.00712981634, -0.037951842, 0.0866919458, -0.0274873488, 0.069787696, -0.0762793124, -0.0975182503, -0.0076374542, -0.0104313446, -0.0366204269, 0.00793519337, 0.0160504226, -0.0248389766, -0.0900964886, 0.0673006624, -0.0399499536, -0.0302191917, 0.0292349495, -0.0117437597, -0.016261097, -0.0275819451, 0.0394761264, -0.153206393, 0.0105548687, 0.0237286091, 0.0510497056, -0.00309844781, 0.051635351, 0.0491371974, 0.0652216002, -0.0916533545, 0.098590143, 0.0117061827, -0.0180703457, -0.0236576032, 0.0953428224, -0.0725917369, 0.153911442, -0.0811349154, 0.0544362739, -0.0608034357, 0.0148433773, 0.0577383637, 0.0579786748, 0.0452385582, 0.00966212898, -0.0155348061, -0.00141282612, -0.0312072951, -0.0449209511, -0.0147062279, 0.0734401718, 0.0128087737, 0.00818270445, -0.0274562202, 0.0853120014, 0.0253571477, 0.0421272106, 0.0105010262, -0.0227784328, -0.139948875, -0.0518930703, -0.00139628723, -0.0693598017, 0.0521380641, -0.0769442394, -0.058106754, -0.00313672423, -0.0107978769, 0.0196863841, -0.105449758, 0.0598196499, -0.0582633764, -0.0491204783, 0.0519072115, 0.019961508, -0.0575122423, -0.0578518659, -0.100139901, -0.029793065, -0.0197158866, -0.0664063692, -0.00158447213, -0.0644674152, -0.0932202041, -0.0436364934, 0.121767096, -0.0827639848, 0.0558819436, -0.00489118509, -0.0340615064, 0.0719996169, -0.0211785063, -0.0701259151, -0.0215637889, -0.00434000045, 0.026677506, 0.0279644411, 0.00832990743, 0.00468205148, 0.0324429497, -0.0713917539, 0.0478803813, -0.0197821781, -0.0237986706, -0.0697306767, 0.0103871413, 0.0119485846, -0.124443188, -0.0176573843, -0.093250066, 0.0987015739, -0.0283948407, -0.0673283413, 0.0300612226, 0.0507432446, -0.00921790395, -0.0216732174, -0.0697327927, 0.0925988778, -0.141845405, 0.0380981714, 0.0242363531, -0.0278652348, -0.117147855, 0.0346155204, -0.0860534012, -0.0410589948, -0.0318844244, -0.0441891551, -0.0359862894, 0.0390880853, 0.00613613147, 0.0451142266, 0.0674476102, -0.100861497, 0.0259292554, -0.00844479166, 0.130780205, -0.0079379864, -0.0226700492, 0.0798050538, -0.0247144084, 0.0253063831, -0.105039403, -0.046898365, 0.0842678398, -0.0366897359, 0.0214723554, 0.0473555513, -0.055253543, -0.171288013, -0.0079167923, -0.0332513377, 0.0334649608, 0.0702540725, 0.0518734567, 0.0235949606, -0.0121659916, 0.0378262065, -0.00815439969, 0.0631355196, 0.0175808761, -0.0535941049, -0.113027379, 0.114974804, -0.0294245481, -0.0168667119, 0.0769506991, 0.041246891, -0.0417153202, 0.00328607857, -0.00829841476, -0.0476484969, 0.104405276, -0.00478654075, 0.0633919761, 0.00487193838, -0.0223508384, 0.0229758546, 0.0359540433, 0.00338172447, -0.0314126164, 0.00425323425, 0.0432219766, -0.0181352403, -0.00976060703, -0.0727678165, -0.0377514586, -0.0454478636, -0.0393960699, 0.0532217659, 0.0514795147, 0.0326012745, -0.0553580411, 0.0290599465, -0.0104210451, 0.021786755, 0.117320709, -0.00249710213, 0.035161864, 0.0611025169, -0.0521535352, 0.0874923468, -0.0371837243, -0.0916585624, -0.0399489738, 0.0173878893, 0.0524088778, 0.0618739054, 0.067790851, -0.0511785187, -0.0165023468, -0.0443992354, 0.0267018378, -0.0709752068, 0.0309787393, -0.0123873185, 0.0524093285, 0.166492477, 0.044890292, -0.0179800801, -0.0090075545, 0.0526536815, 0.00220896071, 0.0744047463, -0.095130384, 0.0403482504, 0.0580226704, 0.00316831097, -0.059943229, 0.138218015, 0.0430112556, -0.160671562, -0.0695708394, -0.101794459, -0.020484345, -0.0693882331, -0.091619961, 0.0373188332, 0.00426862761, -0.0174853448, -0.0501007251, -0.00902946573, 0.0161609203, -0.0942868665, 0.0426980928, 0.0376003534, 0.10906364, 0.107950538, 0.0122947861, 0.0501212329, -0.0193471238, -0.0711034611, 0.0710516572, -0.0236673653, 0.0808256716, 0.0446840636, -0.0132715125, -0.168829888, 0.000191729516, -0.047774449, 0.0726029202, -0.0575729273, -0.0533700101, -0.0500758216, -0.0353930257, 0.0487678945, -0.0898481682, -0.00667860033, 0.0345959663, 0.0293661207, -0.00399904791, 0.0761804655, -0.0924610198, -0.131129608, -0.00818804093, -0.138613045, -0.0288205147, 0.0945906639, 0.0336667001, -0.0694148168, -0.0976273865, -0.0579356849, -0.0228484198, -0.0254474506, -0.0488359705, 0.0430157743, 0.107594274, -0.121932, 0.0539984927, -0.0371713117, -0.0981085002, -0.0697977394, -0.0532799251, 0.0253474433, -0.110270783, 0.118532553, 0.00828219205, -0.0147727989, 0.0224355478, 0.114749759, 0.0134166041, 0.0100993365, 0.0302147605, -0.0616264269, 0.0164625756, -0.0269575045, 0.0407821685, -0.0655083209, -0.0261696782, -0.0356126353, 0.0241052546, 0.0595569313, -0.0462748855, -0.0350691006, 0.0236181822, 0.00645787409, -0.0356341712, 0.0371175483, 0.0225381665, 0.0264469627, -0.126046687, -0.0399434045, -0.0103638256, 0.0444374606, -0.013379287, 0.0129591804, -0.00825375132, 0.0110765491, -0.0152498707, -0.0628566295, -0.0528210178, 0.0729828998, -0.023598589, -0.0516347326, -0.0467721224, -0.0395186767, 0.0377548784, -0.0133530702, -0.0323004611, -0.0710792691, -0.00553263398, -0.00794718042, -0.0408787504, 0.0044202311, 0.0457714945, 0.0707524568, -0.0285768993, 0.0161392055, 0.0443773121, -0.0142677454, 0.0305150691, 0.0242762659, 0.0190181993, 0.154013336, 0.0422201566, 0.114203885, 0.0222654641, -0.0880129859, 0.0278606303, -0.0973212942, 0.0853921399, 0.0183042437, 0.100987755, -0.0663685948, 0.0815383792, -0.00941291172, -0.0481990837, -0.124416962, -0.0406667218, -0.0162412208, -0.00595320947, 0.0032361825, 0.031011045, 0.019682467, -0.075315617, -0.0190552492, 0.0739473924, -0.00606909767, 0.0223029517, -0.0621659011, 0.000501278788, -0.00518693402, 0.0780989081, -0.00401983224, 0.13280955, -0.0990944058, 0.0387860686, -0.0940815657, 0.0773592889, 0.0100899041, -0.0467104279, 0.0561033636, 0.0445901528, -0.0375650786, -0.0528708734, 0.064040564, -0.031365864, -0.0371827185, -0.0677808598, 0.0163462386, -0.0760296881, 0.035737019, -0.00653896201, -0.097026892, 0.00360603072, 0.0301804561, -0.0484979041, 0.00511585688, -0.0159156322, 0.172754407, -0.0712055191, -0.0490743592, -0.0394720808, -0.019216828, -0.0547491536, -0.0643174574, 0.0990366936, 0.059529271, -0.0276015252, 0.0649328455, -0.0908271447, 0.156656563, 0.08819516, -0.12236318, -0.0196664967, -0.0659141839, 0.00179660565, 0.0613880791, 0.0624515079, -0.0116601586, 0.102876745, -0.0246958975, 0.0568032786, -0.0222071633, -0.0348611213, -0.017749425, 0.0832483172, -0.044667352, -0.025525976, -0.0598883145, 0.02995928, -0.00320852548, 0.0039303638, 0.0583930053, -0.0114898607, -0.0415797196, -0.0381443761, 0.0636005774, -0.0242465008, -0.0142912148, 0.0233572088, 0.0652015209, 0.0644668862, 0.0677169189, 0.0548725389, -0.00183511619, 0.00228425069, -0.0254884101, 0.18426235, 0.00145971868, 0.128193334, -0.0476288535, -0.00143218529, 0.0351231061, -0.0400157794, -0.00919232331, 0.0617430992, -0.103689373, 0.119491838, -0.0132442545, 0.0613399334, 0.0426465534, -0.135750562, 0.0360346399, -0.0545150228, -0.0467315316, 0.0236612074, -0.0221177563, -0.0244334154, 0.105033837, 0.0226969942, -0.000489488244, 0.0761136785, 0.0482234135, -0.0794991404, -0.00481206179, -0.106624469, 0.0562642217, 0.0771199092, 0.0600172579, 0.0300480239, -0.0363876298, -0.0542106107, 0.122086033, -0.085374251, -0.101806223, 0.136858463, 0.0153162982, 0.0231618434, -0.0113082211, 0.0245782323, -0.0018151179, 0.0313763693, -0.02448171, 0.163983524, 0.0320217498, -0.000721093267, -0.0591716915, -0.0385272689, 0.0153833553, 0.081110999, 0.0562967584, 0.0514531918, 0.064648971, 0.0388543382, 0.030849725, -0.0770836994, 0.0371506959, 0.101925671, -0.113064058, -0.0569647178, -0.0932790712, 0.000484623015, 0.0390667394, -0.0557390302, -0.0129645923, -0.0249501951, 0.0831834525, -0.117803365, -0.144049972, -0.0508971103, 0.01006178, 0.0446771234, 0.0711698681, 0.000169315375, -0.0746516511, -0.0442662612, -0.0367913283, -0.0166040938, -0.147426054, 0.126584828, 0.0815402269, -0.0158583, 0.0719577968, 0.0399554595, 0.0766077787, 0.00782243256, -0.0126045439, 0.0056044329, 0.0393951088, 0.0509159118, -0.148480535, -0.0138257202, 0.0323465168, 0.090733692, 0.0376416855, -0.074334994, -0.0210058801, 0.0901881307, 0.0860579312, -0.0322047956, 0.0130539443, 0.0561757609, 0.0482928939, 0.0290104989, 0.0708320066, -0.041296564, -0.0387580171, 0.0143743753, -0.0736321062, -0.0251991376, 0.0245742612, 0.0282834992, 0.0773978084, -0.0316123739, 0.10029839, 0.162557796, 0.0692890882, 0.00957362354, 0.0313948244, 0.0636036992, -0.0513825044, 0.0582485422, 0.0868949145, 0.00296425726, -0.0895669982, -0.0512948744, -0.0260608159, 0.0525535569, 0.147869065, 0.0200805236, 0.0429268964, -0.0297400095, -0.060366936, -0.017079629, 0.0192887615, -0.105146252, -0.0285737682, 0.0110281073, 0.0373185389, -0.00278113782, -0.0409983918, -0.085228838, -0.000425591832, -0.0653898567, -0.12126714, -0.0164024942, -0.0511298999, 0.12210837, 0.0756268576, 0.0311745051, -0.0232168846, -0.0180412885, 0.0667902678, 0.0554291233, -0.00916605815, 0.0211446267, 0.101497486, 0.0405851305, 0.0179103985, -0.00936181657, 0.0239127278, -0.0658170283, -0.0443514846, -0.0332392491, 0.0663462654, -0.0275074113, 0.0445375778, 0.020484101, -0.0414097533, 0.0619492047, -0.04526712, -0.0873442888, 0.0256291665, -0.115405358, -0.0211622771, -0.102648005, 0.0556548461, 0.101996705, 0.00444091763, -0.0222102664, -0.0527037159, 0.032726068, 0.0366003104, -0.0532781631, 0.0317719951, -0.0118753295, -0.045661971, 0.0378678776, -0.0272480994, -0.0553724319, -0.0747216269, 0.0585324913, -0.0480772667, 0.00916196778, -0.0701200292, -0.0478666835, -0.0104456758, -0.0861236975, -0.04853791, 0.0166006926, -0.0393693, -0.107133716, -0.131640494, -0.107033223, 0.0102711059, 0.0198268387, -0.0458422229, -0.0364775583, -0.0427006744, 0.00621484872, -0.0616488345, -0.0565045439, 0.0139565356, -0.0816714913, -0.00613524672, 0.0908650011, -0.0401851982, -0.00791749731, -0.0041699037, -0.00302503258, -0.0469855145, -0.102442905, -0.0332288221, 0.0179278255, -0.0549743287, -0.0382256806, -0.0101215448, 0.0481217578, -0.100039989, -0.0130919358, -0.00839087367, -0.0108038299, -0.076164037, -0.0340772122, 0.0493117459, 0.0133731924, -0.0575711578, -0.111356691, -0.034679234, -0.000580328517, 0.173043355, -0.0522343367, 0.0313820131, -0.0866574571, 0.024845235, -0.0022381451, -0.0337380469, 0.122597046, 0.0795823783, -0.0384944305, -0.0845909417, 0.0860818028, -0.0858907476, 0.000777278212, 0.065255478, 0.0355430692, -0.0449581183, 0.0708855093, 0.0126589285, -0.0444815792, -0.0881559849, 0.12831077, 0.0268991403, -0.00962767098, -0.0226503573, -0.0780454203, -0.124609888, -0.0527346916, 0.0810714513, -0.00405854732, 0.127448723, -0.00771148317, -0.0591236167, -0.0253387615, -0.0923302695, 0.11081659, -0.0645495728, 0.0129736671, 0.0140675232, -0.119131312, 0.0518907756, 0.119847506, -0.0971204117, 0.0401668958, 0.0531841479, -0.0145524619, -0.0561505929, -0.139895648, -0.0370193534, -0.142768562, 0.0015139468, -0.091987595, -0.0287524927, 0.00338715687, 0.0516831018, 0.00500003202, -0.0005025235, 0.0297835451, 0.0939352289, 0.0155069632, 0.0469068363, -0.0370668322, -0.0145718567, 0.0454644971, 0.00610159338, -0.0833748728, 0.106487498, 0.00536149973, 0.0242451616, -0.0672092587, 0.0336811915, 0.0740466863, 0.0258674808, 0.079587698, -0.0125749856, -0.0816959366, -0.00260167196, -0.00541039044, -0.0254305098, 0.0468157306, 0.0102681387, -0.0616014004, -0.0157675687, -0.100866489, -0.0549495332, -0.0671589673, 0.0212359782, 0.0392321609, -0.0469639637, 0.0934868678, -0.0741141364, 0.00606553629, -0.0229185987, -0.0681928098, -0.0247458573, -0.0125977397, 0.00922178384, -0.0419256017, -0.0353480242, -0.0467184409, -0.0549502596, -0.0359600261, 0.0482556969, -0.0443457142, -0.0357290357, 0.0218887758, 0.0613992922, 0.0656010434, 0.0125575829, -0.0768133551, -0.0795111358, -0.00719533674, -0.0286065452, -0.155287325, -0.00168394856, -0.00289841462, -0.0484960936, -0.0138900131, -0.0818947628, -0.067168504, -0.0455951989, 0.0105412081, 0.0283603873, 0.00543168606, -0.00640318915, 0.0996480584, -0.0224644281, -0.0738120526, -0.0427065007, 0.0028442461, 0.0979737192, 0.055029206, 0.0410822444, 0.0316695832, 0.0427988954, 0.138028324, 0.117585309, -0.0575526506, -0.149498731, -0.102408424, -0.0200677589, 0.0279945601, -0.0359599963, 0.158086777, -0.0726164505, 0.00356145902, -0.0204066485, -0.0545061603, -0.0134659177, 0.0549237728, 0.016884014, 0.0248378795, 0.0142182671, -0.0746796131, -0.0852554142, 0.0378703848, 0.0909717977, 0.00462599006, 0.0558372587, -0.0587875508, 0.0725072175, 0.0821963996, -0.0238831583, 0.0262895785, -0.0335867107, 0.0308206435, -0.00831976905, -0.0695241988, 0.0276419744, 0.0422261134, -0.067484647, -0.0773139745, 0.0560456179, -0.0571268164, 0.0890280083, -0.0362367108, 0.0376504436, -0.0364428908, -0.0611719862, -0.00495194923, -0.0430841781, -0.0224512853, 0.0151121337, -0.0984745398, -0.0142731834, -0.0204926021, -0.151235819, -0.0347992592, 0.0262647327, 0.0782487839, 0.104661651, 0.144609123, -0.0254833978, 0.0122834109, -0.0233472697, -0.109932914, -0.0398592539, -0.0454275981, -0.00417191349, 0.0297568776, 0.065614298, -0.0299435779, -0.00776641723, 0.000355281984, -0.119662762, 0.0176112708, -0.00972170662, 0.0255980138, -0.092962034, 0.0671037063, -0.07684692, 0.0895235687, -0.0319885872, -0.109269544, 0.0530828461, 0.0178599507, -0.0214530416, 0.00541489571, 0.0182606727, 0.0712672099, -0.0782635659, 0.0873126388, 0.0580067113, -0.00491835829, -0.0694229677, -0.016263729, 0.0561622418, -0.133922532, -0.0287080575, -0.0110522937, -0.0606177598, -0.0806637332, -0.0448358394, 0.0825461298, 0.108007774, 0.0265101567, -0.0628000498, -0.105438285, 0.0257399306, -0.00810558721, -0.0601903126, -0.102254443, 0.0286549516, 0.0144121833, 0.0046322234, 0.0356625021, -0.0105615696, -0.0869713277, 0.116149001, -0.053020414, -0.0101888254, -0.0623870678, -0.0515521467, 0.101372384, 0.00673363917, -0.0548822433, -0.0259544831, 0.0649443269, 0.0917908549, -0.0618304014, 0.00186282955, 0.0358409509, 0.0975381136, -0.00424220972, 0.025559213, 0.0071483599, -0.0458838083, -0.0397334918, 0.032838773, -0.0252329372, 0.0205975659, 0.0433797576, 0.0200363118, 0.101649307, 0.033176519, -0.132551327, 0.0928541496, -0.013792973, 0.0235332306, -0.0196877997, 0.0430779457, -0.0357286334, -0.0742985308, -0.0354737267, -0.11291834, 0.0495139807, 0.0966337472, 0.0471990705, -0.0870929137, 0.0204199422, 0.0545303449, 0.0114289969, -0.0813261569, 0.0657888278, -0.011528587, 0.0364979282, -0.0526293404, 0.012105016, -0.13439101, 0.0949862748, 0.00961158611, -0.00760424137, -0.0449970439, 0.110175908, -0.0454588011, -0.00223047845, 0.0432530977, 0.026621975, 0.0294894129, -0.0362779498, 0.0301470868, -0.0114687597, 0.00213264814, -0.145600528, 0.00341855362, 0.0859211832, -0.0550648123, 0.0024333708, 0.0471789986, 0.00949459523, 0.0241043456, -0.0305060595, -0.0457053967, -0.0523490421, 0.0121598095, -0.127904385, -0.0779877007, 0.02386529, 0.028169807, -0.0430005789, 0.0548254699, 0.0127683422, -0.0149258683, -0.0513531305, -0.0124367736, -0.0102245156, -0.00304678548, -0.0926316455, -0.0198847689, 0.0068387948, -0.0938480571, -0.0422939137, 0.0657038912, 0.0833018422, -0.0571104512, -0.136549219, 0.0981272012, 0.0487134904, -0.0736659467, -0.104583159, 0.0547016859, 0.0765616745, 0.0216471236, -0.122321486, -0.0057147718, -0.0287457928, -0.00439980533, 0.110909104, 0.0370060131, 0.00946681388, 0.00182579574, -0.0203108117, 0.0757886767, 0.0462026335, -0.0191739816, -0.0240432322, 0.00599499326, -0.0247333795, 0.112040974, 0.0710326433, -0.0132521493, 0.025671225, 0.04283081, 0.0482489988, -0.0999715105, -0.0471145473, -0.0238512456, -0.013720654, -0.0681484565, -0.00458434317, 0.045012258, -0.0280752182, -0.01533313, -0.06075418, -0.12869665, -0.102331474, -0.116610646, 0.0796660483, 0.115857214, -0.0874134898, 0.0216424353, -0.00621220935, 0.0542049631, -0.0239136666, -0.142160639, -0.0528354086, 0.0882580802, -0.0275049396, 0.026900474, -0.00388861075, 0.00402097497, -0.0723807514, -0.0109073566, -0.0328807645, -0.0870240703, 0.122565828, 0.0404417776, -0.0816257447, -0.176563606, 0.0406126902, -0.0415037572, 0.00465927832, -0.0401557833, 0.0494681075, -0.0657459274, -0.0857940167, 0.0614018068, -0.0744198263, 0.0515401252, -0.0367939919, 0.0130056217, -0.0903343707, -0.0616297945, -0.019426737, 0.0113249645, 0.0109562408, 0.00422757212, 0.0807014704, -0.0600789301, 0.0444570519, -0.0201776028, 0.0302677713, -0.0613848716, 0.00584103912, 0.0198996514, -0.00236675143, 0.0820359215, 0.0177068859, -0.0731515661, 0.027250275, -0.023199711, 0.0768154785, 0.0262477733, 0.0422141477, -0.0783138573, 0.0929277763, 0.0532470271, -0.0353746265, 0.0595109165, -0.0133373532, 0.0345207229, 0.0911046714, 0.0357785709, -0.0595634803, 0.0214134399, 0.0675902814, 0.0977605134, 0.0393491499, -0.0259091072, -0.0661039576, -0.00498206913, -0.0656896159, 0.0255991668, 0.0297918543, -0.08824718, -0.0350323133, -0.213301316, 0.0560267381, -0.0834940895, 0.0436079539, -0.000368729234, 0.0140293194, 0.0741158798, 0.0676812977, 0.0274782702, -0.0496785045, 0.0717103332, 0.0582054518, -0.0205099247, -0.0580840036, -0.0282324441, 0.0537903458, 0.0179879162, -0.0351910293, 0.0292758942, 0.0939930156, 0.0150582055, -0.00845210068, -0.026137121, -0.022329269, 0.052387204, -0.0195460096, 0.0665599331, 0.0173845123, -0.116979122, -0.0689442381, -0.00149144232, -0.048639141, 0.03158525, -0.0637245625, -0.0338874273, -0.0258239191, -0.00121663976, 0.0147538427, -0.0816596448, -0.0349283814, -0.0888563544, 0.0574568436, 0.000261821784, -0.0608855113, 0.00376400584, 0.0206797868, 0.0518240258, 0.0137401456, 0.0475946628, -0.0534197539, 0.0460028611, 0.0148029719, -0.116431646, -0.0347482376, -0.00917745382, -0.0195992384, -0.104110003, 0.081328854, 0.0134043181, 0.0689869523, 0.0413136855, -0.0543257929, -0.0528486297, -0.0353603922, -0.108183078, -0.140077874, -0.00420097914, -0.0198462624, -0.14790307, 0.0543909706, 0.00603879616, 0.0376893654, 0.0150249451, 0.128007486, 0.0490811355, 0.0449011326, -0.0148460632, 0.0884043872, -0.0275698435, 0.119991362, -0.0424752608, -0.015652664, -0.0483740643, -0.0403228626, 0.0285162032, -0.105744757, 0.0441899151, 0.122427568, 0.070006758, 0.0966597944, -0.0198720768, 0.141583428, 0.00877555646, 0.0519657731, 0.0328696594, 0.131512254, 0.0348169841, -0.0649639219, 0.041316092, -0.0124402158, -0.112384975, -0.0351362303, 0.0106712766, 0.0267674774, 0.0377509184, -0.018236842, -0.114149056, -0.0475013852, 0.0148228519, -0.00647458062, 0.108922824, -0.0142396037, 0.0181112271, 0.0726897418, -0.00843647495, -0.0776845887, 0.0938300714, 0.0300238859, -0.0908047855, 0.0263987463, 0.0571178272, 0.0359571092, -0.103003591, -0.0203244258, -0.114223197, -0.0480621271, -0.0987882316, 0.00282947742, -0.00835656654, -0.0698296875, 0.148698375, -0.0148173235, 0.0150935678, -0.00255804509, -0.0946870223, 0.0613125488, -0.014418656, 0.00857045408, 0.0614193417, 0.0596820265, 0.0177507345, 0.0559728891, -0.181324556, -0.0278531574, 0.00976899639, -0.177840382, 0.00378304534, -0.0313072093, 0.0460807569, 0.0113175539, -0.00496873446, 0.0356606878, -0.0155126862, -0.0799271017, -0.0440439433, -0.0554237552, -0.0692486614, -0.0143908225, -0.0288912561, 0.0335224345, 0.0177780092, 0.00611956045, -0.00160448253, -0.0462504402, -0.0263912417, -0.0789472014, -0.0172664374, -0.0172368772, -0.0941013247, 0.00152368471, -0.045190081, -0.0421784148, 0.000120194629, -0.0244634412, -0.156365126, 0.0244521853, -0.101134881, 0.0198621918, 0.00260684546, -0.0166848544, -0.0375618339, 0.0289886352, 0.0483401716, -0.00755636953, 0.157385617, -0.0644231588, 0.0916382298, 0.0133219799, -0.0789644644, 0.076259844, -0.0675739199, -0.0290857702, -0.0437033921, 0.0740086809, -0.0278980359, 0.0540284403, 0.0300789047, 0.0524086542, -0.0501037315, 0.0305736139, -0.0348226354, 0.105279304, 0.00997264311, 0.0628920197, -0.110923313, -0.105412729, 0.0428671241, 0.0800431371, 0.0553773791, -0.0808367133, -0.0825851113, -0.00815194007, -0.059644822, 0.0635647699, 0.0746527314, -0.0334484242, -0.063693516, -0.0314016193, -0.0109553076, 0.0379749984, -0.0273102317, 0.0369705893, 0.00235534785, -0.0869214162, 0.0199391786, -0.0363283679, -0.067059271, -0.0682186186, 0.0180275477, 0.0244324394, 0.111806169, -0.0235493518, 0.0127768219, -0.0372357108, -0.0964351371, 0.00127715617, -0.0259582046, -0.00576917687, -0.0475290641, -0.108457178, -0.0406387448, -0.0632742718, -0.0431753695, -0.0774208754, -0.0623700544, -0.0668238103, 0.0587851219, -0.0292074103, -0.0700882673, -0.161216155, -0.0884933323, -0.0363693163, 0.0310810842, 0.0184593685, 0.069669202, 0.0235222019, -0.041215051, 0.00900858827, -0.0271204226, 0.0905612484, 0.00707535399, -0.168668151, 0.0368606597, -0.114431351, -0.100348927, -0.031082103, -0.0125700599, -0.00921351463, 0.0297830272, 0.086480923, 0.0227117687, 0.0762094632, -0.0291293003, -0.0170153324, 0.106906302, -0.00213321717, -0.00311509892, 0.014121687, 0.112796411, -0.0815579295, 0.0354602076, 0.0105573311, 0.0593064688, -0.0428368337, 0.0183864608, 0.0406582132, -0.0865894258, -0.0569191165, 0.033496581, 0.104773507, 0.112658523, -0.032157205, -0.118458435, -0.0632474422, 0.0574487112, -0.0101115815, -0.0151285306, 0.0592922382, -0.0550483167, -0.0395899154, 0.0197976474, 0.0303206705, 0.0156443734, 0.0673312768, 0.0523109548, -0.0257555544, -0.106031105, 0.0693425164, 0.0439740121, -0.100053124, -0.0262068175, -0.0102712754, 0.142336726, -0.0173963662, -0.0112469895, 0.101109751, 0.0116365636, -0.0438814349, 0.0218322873, 0.0940738395, -0.0646073222, -0.0944069475, 0.00866631046, -0.0885271132, -0.0316675082, -0.0251205899, -0.0366964377, -0.0254941378, 0.00700463168, -0.0347229317, 0.0174051449, 0.0491306856, -0.0764860287, -0.0659225658, -0.206083834, 0.0320833102, -0.0137055544, -0.0827429742, -0.021857921, -0.0659870133, -0.00459354604, -0.0265307315, -0.00924318377, 0.0696139634, -0.00635738485, 0.0815096647, 0.0839185491, 0.0924746692, 0.0606887378, 0.0974813402, 0.0961243957, 0.107581683, -0.0234480202, 0.0372893214, -0.067663081, -0.0340908505, 0.0727412626, 0.0147353336, -0.0413069949, 0.0437746905, -0.117486268, 0.0271948557, -0.0324148946, 0.0239764899, 0.0774679035, -0.0878255665, 0.0378226191, -0.0659895316, 0.0870889574, -0.0238326192, -0.00075709261, 0.107023209, 0.0366341583, -0.0666124746, -0.0199184678, 0.0404325463, 0.105382271, 0.120067455, 0.0167561304, -0.0586326271, -0.0481569655, -0.0384623595, 0.086619705, 0.0554256216, -0.0225764923, -0.0264306087, 0.0563653857, -0.1117649, -0.0339303054, -0.00584283471, 0.0811603367, -0.0149027826, -0.0315104946, -0.0712907761, -0.0741213635, -0.0229922999, 0.0645033941, -0.0640056506, -0.0107341763, -0.0726029351, -0.0223778933, -0.0526950732, -0.0569055565, -0.100772694, 0.0223133732, -0.0365555957, 0.101154171, 0.0467195064, 0.0580710545, 0.0954319835, 0.0468503982, 0.00901551172, -0.0271212906, -0.0913109928, 0.00329800509, -0.0067952862, -0.111107588, 0.0107333539, 0.033717297, 0.00348317064, -0.0342534035, 0.0338598713, 0.118039094, -0.0977534354, 0.0388599709, -0.00923171267, 0.0222635008, 0.136701614, 0.0278155729, 0.0662524104, -0.0156912915, 0.0780156851, -0.000531308353, 0.00660186261, -0.0535319597, -0.0187308602, -0.0565812439, -0.103111409, -0.042703934, -0.0658376589, 0.108823501, 0.0278005134, 0.0279895477, 0.00938743912, -0.0197750926, -0.02436544, 0.00132394675, 0.0272722207, 0.0455947891, -0.15036571, 0.0206530131, -0.0287563056, 0.00874983333, -0.0613366663, 0.0202093963, 0.0496432669, -0.06733495, -0.00105546601, -0.0139328474, 0.0412373804, 0.0259128474, -0.0394407809, 0.018373033, -0.00244013872, -0.0199421439, 0.0208409335, -0.00395375676, 0.0909849182, -0.00336564519, -0.0965609625, -0.0541225933, 0.0113390535, 0.024501875, -0.00267631747, 0.136285141, -0.0676976964, -0.068165347, -0.0194261651, -0.0252997018, 0.0371229202, 0.0703057423, 0.0285101589, -0.0912475809, 0.0438459329, -0.0412334874, -0.0737582222, -0.0340520851, -0.0666497797, -0.0603474118, -0.00526899379, -0.0953447819, 0.0252543818, 0.00852817483, 0.0832459107, 0.0131681375, 0.0871343166, 0.0238419212, -0.0988228768, -0.0965645537, 0.0275926143, -0.0120506231, 0.100779429, 0.0438304208, -0.0185401104, 0.00821355358, -0.0275065843, -0.057371676, -0.0191882253, -0.0274337493, -0.0610427521, 0.0686004981, -0.0557524338, -0.0839272216, 0.025922738, 0.0267450139, 0.0762207881, -0.0596573874, 0.00319804996, -0.0246729814, 0.018641917, -0.00725796074, -0.0845991075, -0.150740564, 0.102307722, 0.0878596678, 0.000597964972, 0.00947313569, -0.0185569394, -0.0225639734, 0.0630040914, -0.0470955856, -0.0631883442, 0.0581199862, -0.0454104319, 0.0119898366, 0.0950364247, -0.0187070537, 0.0278689079, 0.00482106209, -0.0445957035, 0.0879273564, 0.01416553, 0.0752837956, -0.0841275901, 0.031832695, 0.054853946, -0.0380109847, -0.0242544021, 0.0356314108, -0.0395874493, 0.054618489, 0.0724350736, -0.0234302543, 0.0550535545, 0.0742077231, 0.0241387226, 0.0248916317, -0.042491015, -0.0110113677, 0.0841251835, -0.0860129967, 0.0462181307, 0.0543998331, -0.00481114164, 0.0382955484, -0.000164110214, -0.0340259001, 0.0159670766, 0.0907138139, -0.0506838821, 0.0622301549, -0.0442873873, -0.00586003391, -0.0237447936, 0.00180438999, -0.0756357759, -0.0226934068, 0.0195800383, -0.0694289878, -0.0963376462, 0.0281871129, -0.0826276839, -0.114991233, 0.0856650472, -0.0477097109, -0.0318853408, 0.050218638, -0.0497703403, 0.0553212762, -0.0291117318, -0.0408396646, 0.0703237951, -0.023559384, -0.0167339034, -0.0508203991, -0.0846404433, 0.0361634865, -0.00759056024, 0.0354068503, 0.102165632, -0.0129358051, 0.0454409756, -0.00629037246, -0.0998744443, 0.0445272624, 0.0427902527, 0.044069469, -0.010450772, -0.000717507675, -0.0275748651, 0.0337798074, 0.0920240134, 0.025363069, -0.00666651595, 0.0218137503, 0.100137047, 0.0854654908, -0.104413718, -0.0179716647, -0.0531542152, 0.0223929007, -0.112598956, -0.00974037498, -0.00443734089, 0.0305987876, 0.00918162987, 0.0571104735, -0.0417709127, 0.0434319898, 0.011724811, -0.00738081336, -0.0333152264, -0.0211941041, -0.0455726944, -0.141913846, -0.000475797802, 0.0318516009, 0.0661471263, 0.0242665522, 0.0249190237, 0.0412931219, 0.0168129504, 0.221240774, -0.0586944185, 0.0440724008, -0.00523108803, -0.0882016644, 0.0350061469, -0.0609114654, 0.003586662, -0.0185525306, 0.072258383, -0.013778029, 0.0180858765, -0.00233441405, -0.0618245453, -0.103737198, 0.066192627, 0.0605058558, -0.0465829372, -0.061645925, 0.0113967434, 0.0287732519, 0.0335765779, 0.0362343378, 0.0210650656, 0.0708194673, 0.0817322731, -0.0845245197, 0.0709974468, -0.137797415, 0.026311649, -0.0351894908, 0.0220105629, -0.00946608, 0.0502205342, 0.0544866174, -0.00846912339, 0.0641718507, 0.0436456501, -0.0471215397, -0.0139182424, 0.00323314592, 0.0236360133, -0.0778807625, -0.0487293005, -0.0522835851, -0.0136034656, 0.0589259714, -0.0218560249, -0.0836950615, -0.0683193952, 0.0377402231, 0.0201920476, -0.0186200626, 0.0232431144, 0.0983216166, -0.0624195375, -0.151127651, 0.0304338858, 0.0565972254, -0.132229865, -0.0492863134, 0.045629058, -0.0667893663, 0.0702022016, -0.159955785, 0.0310174562, 0.0325252861, -0.0762316436, 0.0126808137, 0.00231238455, 0.0764733106, 0.00279476959, -0.000984776765, 0.0503465161, -0.0993743017, 0.000858929241, 0.0643585548, 0.020712072, -0.0572571903, 0.0564348474, -0.0501290299, 0.0797260702, 0.011028273, 0.00314432522, -0.00841390342, -0.0630448088, -0.0368616059, 0.0859456137, 0.0981466323, -0.00424607098, -0.0324059241, 0.0982252359, 0.004036217, -0.00422089547, 0.0194093175, 0.041565977, -0.0748232752, -0.00728494674, -0.0819440335, -0.0687295794, -0.0478123128, 0.0844143555, -0.0165800788, 0.0541284867, -0.0162004642, -0.0223157257, -0.0333321244, 0.0223181639, -0.00780511275, 0.0357124209, -0.0282233432, -0.0102435034, -0.0231489986, -0.0614142567, 0.0691181496, -0.0113397669, -0.0159037784, -0.0188351218, -0.0869471133, -0.0463133715, -0.053492479, 0.0269318037, 0.0211484898, -0.050763797, 0.0454574153, -0.0404711105, 0.00201751082, 0.12735267, 0.0472284853, 0.00344345719, -0.0787052959, 0.00798316672, 0.151326329, 0.0530946478, -0.0468464717, -0.0323870927, -0.135204494, 0.0992696583, 0.0560667962, 0.0126236863, -0.0541401654, -0.0208979044, 0.0346535519, 0.0827640444, 0.051830288, -0.00992063992, 0.0176306982, 0.0418458581, 0.0450494215, -0.0335798599, 0.0568372309, 0.0343140587, 0.0298828147, -0.0613671616, 0.0575395748, 0.0685044155, -0.0196285844, 0.0500025973, 0.0528129265, 0.0129889362, 0.0174888466, 0.0621642135, 0.0598305464, 0.0568624213, 0.0200459845, 0.04858822, 0.151778519, -0.0163452439, 0.0332901105, -0.0430720821, 0.00395502895, -0.0365964733, -0.0114995511, 0.0251075998, -0.0728207752, -0.0403402448, 0.0479753762, -0.000144526362, 0.123901382, 0.0949953347, -0.118506193, 0.0900831744, -0.0533235967, 0.110629909, 0.0602999255, 0.039721705, -0.0442778356, 0.0143862246, -0.0793745816, -0.0323134363, -0.0552904345, -0.101991773, -0.0738248229, 0.0752219856, -0.0972978845, -0.0433921032, 0.0376465321, 0.0327817202, 0.0923409462, 0.0164377745, -0.106922053, -0.00282330438, 0.0510833673, -0.0601668768, 0.0797404572, 0.0947562754, 0.0831111297, -0.131288752, -0.00261359662, 0.0361528173, -0.0347429737, 0.0411818773, -0.00933422148, -0.0599134676, -0.0811960474, 0.104828157, -0.0385075621, 0.0942785591, -0.0858461112, 0.0235991441, -0.0250264313, 0.143718734, 0.0424035974, -0.0484768748, 0.0371883027, -0.0363548994, -0.0578930825, 0.0119521134, -0.0783274397, -0.0144689437, -0.0306567214, 0.0364124067, -0.0054134354, 0.0280878469, -0.0150399217, -0.0605220869, 0.0365434662, -0.0429414809, -0.0874371752, -0.084737733, -0.0284669474, -0.00027795136, -0.00535637699, 0.0300112106, 0.0710914582, 0.00663156528, 0.0634959564, -0.0252170917, -0.0672535747, -0.0992471203, -0.121038042, -0.122596808, -0.103546612, 0.136604309, 0.0546582341, 0.0450151451, -0.0328086577, 0.0302524846, 0.0516724288, 0.00445816852, 0.017112175, 0.0279781688, -0.0144226169, -0.0471476614, 0.00232590269, 0.020784894, 0.062216524, 0.14323622, 0.0947486684, -0.0975060761, -0.0630379766, 0.0551736429, 0.0272936188, -0.0327061228, 0.0241358243, 0.0834462345, 0.00165981613, 0.0352062508, 0.0788913891, 0.061352279, -0.0136815449, -0.137421459, -0.0873375684, 0.04423289, 0.0928741395, 0.0175065659, -0.152105838, 0.034042988, 0.00609864853, 0.067395553, -0.0200141016, -0.062433295, 0.0683686212, -0.0784452036, 0.0666098893, 0.0167714655, -0.00195736811, 0.0827242583, -0.015840482, 0.0293768179, 0.0287430938, -0.0528315827, -0.0487425625, -0.0476527661, 0.0227714311, -0.0603982843, -0.00276599452, -0.00982682407, -0.0613137856, 0.0194683149, 0.111207522, -0.0329744816, 0.0180632714, -0.0277960561, 0.113179952, 0.0714195967, -0.0922473595, 0.0346989632, -0.0360110439, -0.0509209372, 0.0390068069, 0.09611696, -0.0317361504, 0.142144367, -0.00931211375, 0.0285686031, 0.0755387545, -0.0336252339, -0.0820314959, -0.00351422234, -0.090317674, 0.00216507539, -0.0193462279, 0.00121027697, 0.0549942292, -0.0397241116, -0.0373528898, -0.0850885585, 0.0145735182, 0.0101744374, 0.0459378734, -0.0485076159, -0.0156543739, -0.029549662, -0.0150020318, -0.0405511446, 0.00372639764, 0.0566977262, 0.0587288998, -0.0292388871, 0.0628593042, 0.0538965799, 0.00830060244, -0.0495379567, -0.010630006, -0.0420277491, 0.0350283161, 0.081842877, 0.0462984554, -0.108877569, 0.00830176845, -0.0626424253, 0.0868911371, 0.0879024044, 0.0167592186, -0.0509877428, 0.0340212025, -0.0563313365, 0.0674078465, 0.0184202008, -0.0409834757, -0.0448917001, 0.207921356, 0.00522281602, 0.0267671365, -0.0865953341, -0.12583293, 0.00882677361, 0.128603145, -0.0716311038, -0.0249648057, -0.0101192147, -0.0190372095, -0.0285220258, 0.0444820672, 0.108935997, -0.0453445204, -0.0262198839, -0.076182209, -0.0283298343, -0.0793861747, 0.0793103576, -0.000419715419, 0.0347146653, 0.126520619, 0.0171729233, 0.0263565816, -0.0195104741, 0.0119538968, -0.0243394822, -0.0298109278, 4.73773107e-05, 0.0918163136, -0.0306263641, 0.125044405, -0.0710958689, -0.0133536747, 0.1263109, -0.0519147553, -0.026283456, -0.0121188015, 0.00148760295, 0.0056181727, -0.0720495805, -0.00194830447, 0.0599225014, -0.0211344212, -0.000633669086, 0.0346792042, 0.0389237329, -0.124458246, -0.0140282195, -0.0335521623, 0.0724248886, -0.0798201859, -0.16313453, -0.0821877867, -0.0174706504, -0.041992031, -0.116840281, -0.00623239391, 0.0369415469, -0.0207696892, -0.0645512268, -0.0768746063, 0.0926358774, -0.203775376, 0.00378085556, -0.0720583946, 0.0155537501, 0.0122184753, 0.0743987337, -0.0757792592, 0.0133273741, 0.0360077918, -0.0826895311, -0.00601030141, -0.0717547387, -0.063256979, 0.0398155637, -0.0075883083, 0.0629392788, 0.064047806, -0.0193110071, 0.0717843771, 0.000419157557, -0.0109396819, 0.022268666, -0.0361923277, -0.048635412, 0.0706237033, -0.0865295678, -0.0195865296, -0.0974688381, 0.0637935326, -0.137107149, 0.0296059176, -0.120595969, -0.124285549, 0.0771401301, 0.0220322218, -0.0595416278, -0.0374364853, -0.125871897, 0.0143538974, 0.0768904462, -0.0548554398, 0.0585917532, -0.112802684, 0.0463209003, 0.0520551726, -0.0705382675, -0.112795375, 0.00205419119, -0.0202029012, 0.128671736, -0.0811489373, 0.0316166803, -0.0747596547, -0.155343816, 0.0308889616, 0.0291859191, 0.00397870317, 0.018676823, 0.0143547319, -0.0706743672, -0.0561404526, 0.139850274, 0.056702394, 0.0258671101, -0.0714369342, 0.0307094008, 0.112720586, 0.0194525626, -0.0431945622, -0.0717279315, -0.0168336295, 0.0378105044, 0.0148544069, -0.125727549, 0.0822669119, -0.0551071912, 0.0213356502, 0.0236175414, 0.144435346, 0.0782963783, 0.173167676, -0.0118138026, 0.0891125202, -0.0136344414, 0.136959225, 0.0388533063, -0.00414486602, -0.106506161, 0.114196539, 0.0323584564, -0.0598234199, 0.0395343862, -0.0201786719, -0.0310909338, 0.141745508, -0.0909626633, 0.0144927464, 0.00156159699, 0.17056635, 0.0707120299, 0.00328813866, 0.126776889, -0.0716742426, 0.0656434298, 0.0656622946, -0.0778835192, -0.0630527735, -0.0554898903, 0.0316421613, 0.0807764307, -0.0445900299, 0.0321348272, -0.0259241238, -0.00800019037, -0.0399757326, 0.012875665, -0.0284602307, 0.0919920504, -0.0733514503, -0.00825741235, -0.00269941613, -0.0959233493, 0.0263982601, -0.00916188397, 0.0067764204, -0.050063841, 0.034068536, 0.0281936489, -0.0741143078, 0.0872939155, 0.108753093, -0.050483413, -0.0458577871, -0.0479609407, 0.0412913114, 0.0500612557, -0.00867055543, 0.0104127787, 0.0509211048, 0.0971171111, 0.143516332, 0.0317348391, 0.037279129, -0.0715883523, -0.0260122232, 0.0446442813, -0.0640992895, 0.115151927, -0.036190562, -0.00168597046, 0.0308016185, -0.0117924362, -0.0442319661, 0.00668676384, -0.0129320882, -0.0455180332, 0.0223680343, -0.000283910893, 0.127435595, 0.116857767, 0.0482462049, -0.0936985612, 0.03473996, 0.0152194463, 0.0819397792, -0.00564387999, 0.0438897386, 0.0461231992, 0.0095021911, 0.0327440538, 0.0327969454, 0.0374337584, -0.0834925696, 0.0993662775, -0.0446608663, 0.00705635129, -0.0580409989, 0.022538932, 0.0252450965, -0.00245221518, 0.053560812, -0.0212774128, 0.0702632964, 0.0702260286, 0.0111957714, 0.020327501, -0.0251179747, 0.0171322934, 0.0563229062, 0.0547430143, 0.00369137153, 0.0546198077, -0.0383057669, 0.00339738489, 0.00934015121, 0.0598048307, 0.0594764203, -0.0582049526, -0.083817035, 0.0735156313, 0.0635233819, 0.00630174205, 0.0795494914, -0.0911415666, 0.0466910675, 0.0606360137, 0.0401503444, 0.104378313, 0.105895989, -0.000811231788, -0.00740461051, -0.0155261792, -0.0452880338, -0.0281637385, 0.136133492, -0.0461421348, 0.0414155424, -0.0511175282, 0.0308285542, -0.0485993885, 0.0388431549, 0.00904206932, 0.0438649692, 0.0180817153, -0.0261081811, 0.00678093592, 0.00653930008, 0.0518569201, -0.105377048, 0.0530258678, -0.0549291931, -0.00393442996, -0.10040538, -0.0164066926, 0.0446909443, -0.00204299577, -0.030420579, 0.0292901881, 0.00487748347, -0.097163558, 0.134119615, 0.0427111983, 0.0701625273, -0.138018221, 0.0978135094, 0.0160789564, 0.0650686845, -0.0316936113, 0.0265970547, 0.0948237479, -0.0604418069, 0.02479068, -0.00676343124, -0.0436989181, 0.0941133797, 0.0125063611, 0.0326087102, -0.0110648759, -0.0485574827, -0.0663554221, 0.104777887, -0.0760637224, -0.0330644213, -0.0229540989, -0.0970492288, -0.0717062205, 0.00749311689, -0.0269734412, 0.139105693, -0.0410516784, -0.134367764, 0.0682754368, 0.0560388267, -0.0519007705, 0.0243832786, 0.0182770249, -0.00779117644, -0.0135297179, -0.00136886211, 0.0331867635, -0.0290039703, 0.0371391252, -0.0251131728, -0.0355404615, -0.0989934579, 0.0485571586, -0.0372378156, 0.0246049389, -0.0341279879, 0.0109996349, -0.00988118537, -0.0680833906, -0.0436525084, 0.0165211149, 0.0181577485, 0.0323311836, -0.111874267, -0.161264598, 0.0270574838, 0.00629270636, -0.0532361306, 0.075439319, -0.0711706281, -0.0803600773, -0.0332396403, 0.114705563, 0.0862880722, 0.0744256005, -0.00143556297, -0.0620327406, 0.0148407146, 0.0388584845, -0.00118256919, 0.0284797251, 0.0640596971, -0.0465310998, 0.00145616196, -0.042187281, 0.04777788, -0.074447453, 0.0418466218, -0.0709764361, -0.0779289827, -0.0337267406, 0.0491694771, -0.0726052672, -0.122968994, 0.0689677894, -0.0198880583, -0.0677938014, -0.026422061, 0.0110124759, 0.104051597, -0.0462275334, 0.0898115784, 0.0329568759, -0.0294124577, 0.0774988756, -0.0281288326, 0.00680770911, -0.00884689298, -0.0350825191, -0.0337942913, 0.0772518516, -0.0566374809, -0.0389257595, -0.0306435749, 0.0877659619, -0.0310595259, 0.124964863, -0.0957588702, -0.115030549, 0.0550060421, -0.168131307, 0.101320773, 0.0891779736, 0.0849423707, -0.0732070655, 0.0714477524, -0.0499479771, -0.129221916, 0.0923667774, -0.0191568155, -0.0199776571, 0.0437719747, -0.1454366, -0.153990969, 0.07490962, 0.0153739918, 0.00195262721, -0.047920987, 0.127082318, -0.00285737775, -0.020199148, -0.0281331018, -0.00304718688, -0.100617148, -0.0431944318, 0.0251088198, 0.0088349469, 0.0880591199, 0.126945108, -0.0247219168, -0.0834257454, -0.0288124979, 0.165753037, -0.0436757207, -0.0211461913, -0.0292444266, 0.000162766315, -0.136034176, -0.0554456934, 0.161701843, 0.018463254, -0.0145777967, -0.0396678783, 0.0550153181, -0.00914106239, -0.120041952, -0.062959373, -0.0311751068, 0.00457889214, 0.028921159, -0.04066699, -0.0387526862, -0.0486108586, -0.0575057119, 0.0117322393, 0.0264256336, 0.0285620634, 0.118608408, -0.04984276, 0.0472168364, -0.0576146431, 0.0461757481, -0.0471321195, -0.0531005524, 0.00734813325, -0.00708643347, -0.0386020727, 0.0182450432, 0.00401454419, -0.106816277, 0.026848428, -0.020396037, -0.0116738006, -0.0581501648, -0.133722037, 0.0108819343, 0.0582929961, 0.082653366, -0.0165933352, -0.0128453784, 0.018747801, -0.050871402, -0.0701920167, -0.123694293, -0.0183124952, -0.0472935364, 0.0113076176, -0.128444076, -0.067465052, 0.106249548, -0.0496149883, 0.0989708602, 0.045899801, -0.0105147501, -0.024327632, -0.037630409, -0.0423040725, 0.102868497, -0.0730754361, -0.0269970186, -0.0874037966, -0.0669640675, 0.0568245426, 0.0240096431, -0.154584557, -0.02182246, -0.000544991344, -0.0731352568, 0.0325741172, 0.0722889826, 0.0577225424, -0.0352375172, -0.0123152044, -0.0482738577, 0.052247908, 0.0364501178, 0.0320600197, -0.000175455119, -0.00185240433, -0.0490202308, 0.0151405148, 0.0390618369, 0.0541663617, -0.0169732273, -0.0401358791, -0.0519654788, 0.02727082, -0.000694720075, 0.117084451, 0.124064468, -0.0290039089, 0.0606490932, 0.00299782678, -0.0359059349, 0.159433454, -0.0585865378, -0.0258554295, 0.0684467703, -0.0201539062, -0.010478653, 0.119220629, 0.0118390899, -0.0207507387, -0.0349295698, 0.0235170927, 0.0574315935, -0.00832277071, -0.120146774, -0.0366767943, 0.00209335983, 0.0373839624, 0.0184952058, 0.0847397819, -0.014911063, 0.0476309359, -0.0663685426, 0.0595663264, -0.0110730212, -0.0163978934, 0.0383992419, 0.0552380085, 0.0535435937, -0.151276633, 0.0284492746, 0.134271145, 0.0758550689, -0.149602249, 0.052758228, -0.054195568, -0.175280422, -0.0555837564, 0.0581984259, 0.0288196802, -0.0114671625, 0.0299345441, -0.0529778227, -0.120665342, -0.0380313396, -0.0197654366, 0.0526419692, -0.0717780143, 0.00545177236, 0.0699172541, 0.132046402, -0.0448216349, 0.0279292557, 0.0307166651, 0.0311485939, -0.0444991067, -0.148809329, 0.0300705507, 0.056306839, -0.00903391, 0.0541236885, 0.127085209, -0.023981763, -0.0465383194, 0.00582119543, -0.0387304723, 0.00631576171, 0.0433832034, -0.0196737684, 0.0221379288, 0.0802582428, 0.0106961038, 0.0898146331, 0.103875116, 0.163770944, 0.0458479598, -0.0153884897, -0.0774732232, -0.0277616382, -0.0273456778, -0.00433784723, -0.017673092, -0.113373205, 0.0323634371, -0.0682597682, -0.0126066599, -0.0416358039, 0.02411565, -0.00372025091, -0.0063503515, 0.0217203088, -0.0791368932, 0.016960999, -0.0145828836, -0.0119992048, -0.0300915577, 0.000444486272, 0.0592254288, -0.0565110482, 0.00295438711, -0.0351124629, 0.00868484937, 0.00933773629, 0.0537636578, -0.0649817139, -0.0775154755, 0.0783688277, 0.0604816526, 0.00487851165, 0.0054111965, -0.0332669951, -0.07896474, -0.0327083468, -0.0994815603, -0.025841251, -0.123208925, 0.119442396, 0.0655044466, 0.0155529398, -0.110433713, 0.0112173911, -0.0965983644, -0.0716264173, -0.0125765596, -0.153670549, 0.0229726229, 0.0666033551, -0.0385708921, 0.0793999657, 0.0241617579, -0.00533927558, -0.0243451893, 0.0961167812, 0.038312234, 0.0576939657, 0.042851232, -0.0358315036, 0.0358997472, 0.0227629617, -0.0913492963, 0.118889272, -0.170795202, 0.0561172776, 0.0246566199, -0.0585237965, 0.0758079141, 0.0172428824, -0.0729951486, 0.0906477943, -0.0378021449, 0.115066767, 0.00613665208, -0.0619825646, -0.0250669532, -0.0636628121, 0.0441154093, -0.019137457, -0.0105001479, -0.0122354859, 0.0685944334, -0.0693055913, 0.00828789547, 0.0978689343, -0.00773450546, -0.0937277973, -0.0795447379, -0.111284032, 0.0214230344, 0.104236171, -0.0593462884, -0.00263052806, 0.0837748647, 0.0186597165, -0.0234428924, 0.0279572494, 0.0456273481, -0.0144679435, -0.0184127931, 0.00534057338, 0.00311607309, 0.0779221281, -0.0149843711, -0.0653924793, 0.0711301118, -0.0248427521, 0.0697843358, 0.0482382253, -0.0853462443, -0.0220317487, -0.0295238029, 0.0387399159, -0.0366771407, 0.0418762974, -0.0797430575, -0.0295413602, -0.027681293, 0.0048418371, -0.0680969357, 0.0610560663, 0.0213241484, 0.0801980197, 0.000836689956, 0.0595580488, -0.002605699, -0.0123861041, 0.0163292475, -0.0453969762, -0.0630998984, 0.0538237207, 0.0827814341, 0.0514547154, -0.0844336525, -0.0359347127, 0.0588213541, -0.112257935, -0.134003744, -0.0699817091, 0.0242702048, -0.0130902752, 0.00326215429, 0.00262629264, 0.0739195794, 0.0576854125, 0.0291830432, 0.0199246891, 0.0276506953, 0.0269868672, 0.0166296102, -0.0333934054, -0.0564064533, -0.00877703261, -0.00936939009, -0.012725818, 0.111339904, -0.0216438472, 0.0299144294, -0.0356176086, 0.0400863141, 0.0132308975, 0.0651910454, 0.0412254408, -0.0251634661, 0.0584020615, 0.0126364361, -0.100437343, -0.00917152222, -0.00577493664, -0.0548890941, -0.157526746, -0.0826172382, -0.0152674215, -0.0538601354, 0.03166743, -0.0649304539, 0.0297401026, -0.0556121282, -0.0529944152, 0.0018012803, -0.0200358368, 0.00875069387, -0.0129886027, 0.0642298087, -0.0318649113, -0.0249860566, 0.0507242568, 0.0252665393, -0.0570531376, -0.0496048965, -0.0387844183, 0.0397206992, -0.0445796251, 0.0273695514, -0.0526615046, 0.0205880478, 0.00826173089, 0.0736790225, -0.060041599, 0.0982105285, 0.0730360523, -0.0569852106, 0.0983446613, 0.0245305374, 0.0598854646, -0.0352758244, 0.0892537236, 0.0121544097, 0.0320136063, 0.156756759, -0.0688542649, 0.0425491184, 0.0524674244, -0.0254217647, -0.0428709164, 0.0224039089, 0.115825444, 0.0710413605, -0.0101484805, -0.147773981, 0.131913662, 0.0641956031, -0.0947205573, -0.0457786918, 0.0453664921, 0.0708878562, -0.0115118288, 0.042543374, 0.0586548671, -0.0088423267, 0.0621570162, 0.00521691889, 0.104976267, 0.00832910836, -0.0261728764, -0.0277918801, -0.0952738971, 0.00914620981, -0.0518588796, 0.0325142294, -0.0550612956, -0.0453606695, 0.0100926971, 0.0297810044, -0.00653575361, 0.0744574219, -0.0348829105, 0.0315345079, 0.0596710779, -0.0488631055, 0.0117433313, -0.0260070302, -0.167032167, 0.000464372337, -0.0159767233, -0.157046124, 0.00397387706, 0.0281003937, -0.0524692088, 0.0904591978, -0.0523954257, 0.000903403386, -0.0144094601, 0.0875321627, -0.0349024348, -0.0938078091, -0.0228116382, 0.0777692348, 0.0438611731, -0.0585822165, -0.0166053288, 0.0438468941, -0.0614718236, 0.0500500128, -0.00265980139, -0.021987861, 0.126459837, 0.0849078521, -0.0262422077, 0.0693567172, 0.0389528126, 0.0512110926, -0.0754294991, 0.102317944, -0.0537033789, 0.0107139423, -0.04735367, 0.192314222, -0.00361257233, 0.0323533192, 0.0773674548, -0.0103753805, 0.0534867197, -0.0322413296, 0.175135925, -0.0222816858, -0.104840487, 0.0621830262, 0.0228022113, -0.0180504862, 0.0273270085, -0.0918684676, 0.0479792058, -0.0748050585, -0.0950439796, 0.0519897789, -0.0730442777, 0.0447922684, 0.00429253373, 0.0324358344, -0.020763699, 0.164352432, -0.000862773508, -0.00612956006, 0.124670595, -0.0340847783, 0.000145215541, -0.0460306033, 0.0876810551, -0.0355497375, 0.0055465959, 0.0166269355, 0.0153367063, 0.013447959, 0.0440620184, 0.00886172894, -0.0985550582, -0.032873679, -0.0370585248, 0.107536547, 0.0554145761, 0.00197463296, 0.0831993148, 0.0925370827, -0.0853444487, -0.0166519657, 0.00820638519, -0.025233116, -0.0604022034, 0.0390485562, 0.0451029316, 0.121790454, -0.116757512, -0.0264542401, -0.000161452219, -0.0983723849, -0.130126551, 0.0948483124, -0.0265996456, -0.00503839366, -0.0308538359, 0.0407007113, 0.103136219, 0.0671191439, 0.0408682302, -0.0336545333, 0.0618165657, -0.133005187, 0.0909017399, 0.091140531, 0.00702103414, -0.120794117, 0.0383883938, 0.0595010221, -0.0496434644, 0.00300184451, 0.0901205391, -0.0843699649, 0.0660540685, 0.0656372756, 0.014720019, -0.0656864047, -0.095156543, -0.0208353922, 0.0162730925, 0.136528566, -0.0762757137, 0.0709100738, 0.000927855261, 0.0602045208, -0.0161736943, 0.0852523372, 0.00159708038, 0.114528716, -0.116141349, 0.0145223513, 0.0342769064, -0.0981167257, -0.0759822354, -0.071397692, 0.0175059326, -0.0462377518, -0.0960905775, 0.00514982268, -0.0450254455, -0.134848282, 0.0206391588, -0.0299922824, 0.0754823312, -0.0334678032, -0.0131102493, 0.0750454068, 0.0507376194, 0.0940473676, -0.0720524043, -0.042138543, -0.0398096591, -0.0515284427, 0.0031810496, -0.0395970047, -0.0165582485, -0.100258149, 0.0412577689, -0.0349645726, 0.0866794884, -0.0420196466, 0.0171162989, 0.0119688986, -0.138056234, -0.0304361545, 0.0326685905, -0.0688718855, -0.000287668779, -0.0186870769, -0.0103182103, -0.0332754441, -0.0209563076, -0.0379594117, 0.0822373107, 0.0228411146, 0.0978683159, -0.0880096182, 0.0827165097, -0.0966300666, 0.0599336326, -0.0818612427, -0.0082848547, 0.033376269, -0.0442513339, 0.03609588, 0.0417950228, 0.0540762842, -0.0918703824, 0.0685817301, 0.0535970032, -0.0517048649, 0.0436669178, 0.0668945089, 0.031383872, -0.0770094395, 0.122002475, -0.0635105744, 0.0505352803, -0.0293868016, 0.00382741168, 0.145384833, -0.0608801991, 0.0577654243, -0.00978171732, 0.0539359711, 0.0359628424, -0.0735183507, -0.0201065, 0.0343457274, 0.0284094196, 0.0148093421, -0.0801174641, -0.0722824037, 0.0226920303, 0.0432471819, -0.0294586197, -0.0607275479, -0.0118639246, -0.00447471254, -0.0370622277, -0.000830128789, 0.0693000555, -0.0361630209, 0.0744672269, 0.0957773328, -0.135049164, 0.0345977768, 0.0578934625, -0.013735557, -0.0654508024, -0.104584284, -0.063762024, 0.0443658456, 0.00429359451, -0.0338540003, 0.0351315103, -0.0106531754, 0.0452211611, 0.0214158781, -0.0723168477, -0.0667011738, 0.0394572914, 0.0334803313, 0.011356825, -0.00861832965, -0.0663884133, -0.0160783753, -0.0339693688, -0.0907160491, 0.141522542, 0.0181954131, 0.170019135, 0.00692077167, -0.0264775753, 0.0479528494, -0.0225476027, 0.0269292295, 0.0809427947, -0.0253310855, 0.0377794057, -0.00843248144, 0.0642494485, 0.0684372634, 0.0347917527, -0.000772092491, 0.0418730788, -0.02787471, -0.0284226909, -0.0300512835, 0.0551576689, -0.0606302544, -0.0264060684, 0.0356873237, -0.00265506236, 0.000962077756, -0.0381548181, -0.0767370239, -0.027814012, -0.0226326361, 0.0131381098, -0.0450338796, -0.0522808395, -0.0437729172, 0.0382389128, -0.0230580717, 0.0433934256, 0.0261253901, -0.0148409186, -0.0296442285, -0.103537112, -0.0723207593, 0.0763290673, -0.00249677664, 0.0718548149, 0.0908411518, -0.0655037537, 0.0488255247, 0.0769326165, 0.0368216634, -0.0558381081, -0.0323771052, 0.0441647843, 0.00403788686, -0.0530877262, -0.027564805, 0.00694148894, -0.00826103054, -0.0533859655, 0.0937855169, 0.0245898645, 0.0251932982, -0.0142583689, 0.037413571, -0.101187021, -0.0932473168, 0.0609707758, 0.00984138064, 0.0113916602, -0.163416862, -0.00436028652, -0.0916275308, 0.0961952284, -0.0618586764, 0.0216272175, -0.0299923122, -0.0320265442, -0.0407082513, 0.117185362, -0.019825317, 0.0277280193, -0.0392001495, -0.0866438672, -0.138311774, 0.0382229872, 0.0126878386, 0.00636984501, 0.00362016377, -0.0347380824, -0.0153270848, -0.0163740031, 0.0650544912, -0.0733646229, -0.0946579129, -0.046073962, 0.00693581533, 0.032058537, 0.0921451673, 0.0729097575, 0.00332806678, -0.0258130282, -0.0480049998, 0.0519877337, 0.0930817649, -0.105404966, -0.121177405, -0.0140856961, -0.0863415077, -0.0653534308, -0.0452476293, 0.107658163, 0.0322528258, -0.0567492209, 0.0348825678, -0.0698981881, -0.0723470896, 0.133577704, 0.0569301993, -0.0838846639, 0.045235876, -0.111871928, -0.0214537028, -0.0961486697, -0.109154761, 0.0162440911, -0.0132249352, 0.0133098364, 0.0824577957, -0.0105112828, 0.00409429567, -0.0610876679, -0.0857018009, -0.0681799352, 0.0514959395, 0.040572457, 0.0791241825, -0.0431395508, -0.0560610518, 0.0119373035, 0.0100756027, 0.0577928461, -0.0119281216, 0.0206011236, -0.0271528438, -0.0906230956, 0.0610706285, 0.0664898679, -0.0648542941, -0.0489872321];
    bias_3_f : ARRAY[0..63] OF REAL := [1, 1, 1, 1, 1, 1, 1, 1, 1, 1, 1, 1, 1, 1, 1, 1, 1, 1, 1, 1, 1, 1, 1, 1, 1, 1, 1, 1, 1, 1, 1, 1, 1, 1, 1, 1, 1, 1, 1, 1, 1, 1, 1, 1, 1, 1, 1, 1, 1, 1, 1, 1, 1, 1, 1, 1, 1, 1, 1, 1, 1, 1, 1, 1];
    weights_3_g : ARRAY[0..4095] OF REAL := [0.334696651, 0.459893674, 0.588931501, 0.225918621, -0.529859424, -0.711596608, -0.268382728, -0.238952905, 0.723561168, 0.347821832, -0.492707103, 0.39439711, -0.440663218, 0.408884048, -0.351317674, 0.456424505, -0.539472282, -0.545774877, -0.470176607, 0.532276869, 0.597730339, 0.566391468, 0.388534904, 0.435214907, 0.468310148, -0.526900053, -0.448725283, 0.255596548, -0.517045259, 0.446985215, -0.481767774, -0.553763509, 0.555955768, -0.521494985, -0.472606957, 0.391773045, 0.460757047, -0.396523476, 0.646327257, 0.214222342, -0.504349291, 0.443324357, -0.410986096, -0.392339438, -0.590739787, 0.221475571, -0.17983003, 0.462024987, 0.664287388, -0.468381584, 0.467875272, -0.819812417, 0.581035912, -0.578730881, -0.447773635, 0.617174208, 0.785593748, -0.443258554, 0.43781063, -0.341597468, -0.45279187, -0.403854162, -0.444021106, 0.499367118, 0.378389984, 0.492821187, 0.646293938, 0.336553544, -0.353956044, -0.889889121, -0.39690426, -0.450034857, 0.929169297, 0.32170251, -0.586820602, 0.588153839, -0.465774029, 0.510198236, -0.485173404, 0.50339222, -0.716529965, -0.240741417, -0.687259197, 0.463590443, 0.584574938, 0.612124085, 0.436245888, 0.510803878, 0.354973525, -0.441401333, -0.673492253, 0.440029919, -0.537557483, 0.517918825, -0.596777618, -0.442761987, 0.349172026, -1.03222752, -0.379008055, 0.424729556, 0.751009285, -0.69054985, 1.09924674, 0.312436014, -0.400820464, 0.488747716, -0.328508258, -0.220668525, -0.912406683, 0.319938749, -0.469002426, 0.406208754, 0.823793292, -0.534058332, 0.619498849, -0.956825078, 1.38313961, -1.41096985, -0.334248006, 0.753053725, 1.0035913, -0.532719493, 0.520589411, -0.318735421, -0.4105739, -0.296536863, -0.565646112, 0.587440848, -0.258787662, -0.39195779, -0.650093973, -0.242794752, 0.475784689, 0.630811572, 0.314297467, 0.30150044, -0.813092411, -0.126978844, 0.247311935, -0.4207353, 0.380223364, -0.382250518, 0.322775573, -0.337508619, 0.69236964, 0.44791162, 0.590113819, -0.648905575, -0.669354558, -0.622273088, -0.298255354, -0.645075738, -0.151741654, 0.521941304, 0.69219476, -0.261719167, 0.384286761, -0.233402565, 0.279928684, 0.517069697, -0.600000441, 0.647710621, 0.198059693, -0.444062859, -0.379430979, 0.580145299, -0.660138488, -0.367549092, 0.527287781, -0.454349965, 0.190091997, 0.382158488, 0.703072608, -0.169629559, 0.109911256, -0.448498189, -0.70116961, 0.577127695, -0.549189329, 0.660310805, -0.501063824, 0.680603743, 0.376381904, -0.390215158, -0.634619534, 0.747808337, -0.348204255, 0.591025889, 0.422861278, 0.5795874, 0.341520756, -0.348781049, 0.36977157, 0.491182476, 0.725632966, 0.452657253, -0.60983628, -0.961705744, -0.553472817, -0.496075541, 0.699398637, 0.346367508, -0.437914968, 0.466125488, -0.539875805, 0.4927122, -0.501847804, 0.764431417, -0.502617002, -0.284993052, -0.64147675, 0.442549109, 0.635759532, 0.481588095, 0.596530914, 0.59095484, 0.565535247, -0.362338454, -0.569893837, 0.484379172, -0.483971238, 0.513303697, -0.451245606, -0.560657918, 0.37872982, -1.08903956, -0.578953922, 0.534648061, 0.691077471, -0.653672218, 0.911954463, 0.3548567, -0.467105925, 0.54097718, -0.42201364, -0.497504473, -0.686189473, 0.587780774, -0.408520192, 0.371105641, 0.958120167, -0.531876326, 0.475154728, -0.882420003, 1.38590026, -1.68719566, -0.448663771, 0.703568816, 1.0761044, -0.596032262, 0.355891466, -0.311855733, -0.462226927, -0.540922701, -0.54588747, 0.649262846, -0.393689126, -0.506876469, -0.465987682, -0.400442183, 0.421407014, 0.879044533, 0.357684165, 0.324539781, -0.829124808, -0.322396666, 0.417395115, -0.3696132, 0.579591274, -0.310370296, 0.41139549, -0.496556252, 0.452449828, 0.287400097, 0.607891381, -0.473392457, -0.397284269, -0.495738983, -0.58298701, -0.590240419, -0.299706757, 0.455185026, 0.486282051, -0.473806709, 0.433027029, -0.321802765, 0.520485818, 0.423597455, -0.337682098, 1.12769508, 0.524797797, -0.553971231, -0.722507238, 0.62597698, -0.886188865, -0.538565278, 0.332679719, -0.592859387, 0.448146135, 0.385972828, 0.765457809, -0.470907003, 0.279049307, -0.491523653, -0.879431605, 0.498989612, -0.668206632, 0.869883657, -1.27968061, 1.24609447, 0.52986902, -0.762102604, -1.01468563, 0.551170945, -0.455807596, 0.339573801, 0.426975101, 0.272426426, 0.479562461, -0.574861467, 0.370637774, 0.409491122, 0.591502607, 0.304184049, -0.452153653, -0.730533779, -0.240931228, -0.38228786, 0.665357172, 0.335496962, -0.35340178, 0.347838283, -0.45989576, 0.444312304, -0.200159147, 0.484028488, -0.389273971, -0.508607149, -0.441756874, 0.43076247, 0.473969847, 0.562401533, 0.402652562, 0.56135577, 0.178501114, -0.466243595, -0.610224783, 0.331260443, -0.342666566, 0.413177401, -0.33043465, -0.526860893, 0.587673604, -0.552634001, -0.448599517, 0.450187564, 0.440405279, -0.646909952, 0.441380024, 0.390686184, -0.585748971, 0.409217119, -0.276743174, -0.542910695, -0.73798573, 0.379657477, -0.308137774, 0.351353407, 0.549951792, -0.407486767, 0.589478374, -0.787027538, 0.700253665, -0.520758331, -0.428434104, 0.480139792, 0.669792235, -0.590756178, 0.312144458, -0.479037255, -0.326317668, -0.471595615, -0.259286463, 0.386178464, 0.3984465, 0.328214943, 0.465490848, 0.492737502, -0.434407651, -0.878537118, -0.512350559, -0.444377542, 0.770180702, 0.412139475, -0.427146405, 0.479131669, -0.355318755, 0.404837072, -0.286447823, 0.457547575, -0.365542769, -0.420703381, -0.595457256, 0.355077416, 0.598927498, 0.450168937, 0.502180457, 0.548574269, 0.381900549, -0.450617582, -0.516253531, 0.52879107, -0.326660872, 0.450721622, -0.585836351, -0.455070317, 0.542164266, -0.969287753, -0.565889716, 0.486150384, 0.636408508, -0.532597244, 0.823236585, 0.396210968, -0.511359334, 0.520103633, -0.340114862, -0.403221905, -0.676262379, 0.446127415, -0.455957532, 0.394790441, 0.891266406, -0.440120697, 0.624995589, -0.886184514, 1.11586559, -1.09366536, -0.427211881, 0.721240342, 0.887889087, -0.558480859, 0.460597366, -0.367894202, -0.499132186, -0.444942594, -0.552337587, 0.543708801, -0.552899837, -0.590657473, -0.625323653, -0.394068003, 0.567751646, 0.908171058, 0.448856622, 0.544118643, -0.665149629, -0.385490745, 0.575014949, -0.553586543, 0.360419333, -0.457954288, 0.357944012, -0.615689158, 0.647890031, 0.404805332, 0.638076305, -0.507503927, -0.497962564, -0.514615595, -0.55763799, -0.503329933, -0.454292297, 0.370624751, 0.496337712, -0.542248368, 0.396027684, -0.476377934, 0.482300222, 0.296015918, -0.473766983, 1.01016963, 0.345653385, -0.392501682, -0.516385019, 0.496517181, -0.928887665, -0.329730719, 0.467229247, -0.397571534, 0.528575122, 0.320062995, 0.819152772, -0.467998594, 0.469339401, -0.402863324, -0.894191086, 0.570362389, -0.618255913, 0.79585731, -1.06189966, 1.43001997, 0.312423766, -0.584950745, -0.937776625, 0.45877704, -0.513584912, 0.284058779, 0.524194717, 0.364320427, 0.353972256, -0.550919294, 0.578206897, 0.48984924, 0.69370687, 0.388696134, -0.561883867, -0.992671549, -0.318962038, -0.459210902, 0.788012385, 0.438168347, -0.569898069, 0.413392037, -0.606889427, 0.540551424, -0.380481958, 0.72546345, -0.466777831, -0.348223746, -0.583220243, 0.366624147, 0.414185166, 0.740230799, 0.465056241, 0.584235311, 0.472829133, -0.318938136, -0.702742338, 0.341313392, -0.61872977, 0.467518032, -0.504496038, -0.456522644, 0.407123357, -1.05130374, -0.530595839, 0.633368313, 0.758280516, -0.653592288, 1.1052438, 0.548134983, -0.459854603, 0.457486421, -0.531135678, -0.424228668, -0.697049618, 0.398558646, -0.403776497, 0.409781426, 0.89905709, -0.715407073, 0.650818467, -0.859829724, 1.45971441, -1.61062896, -0.408946753, 0.762522101, 1.11483479, -0.515048027, 0.502049148, -0.416843981, -0.524300814, -0.410066843, -0.416641206, 0.507241547, -0.149781063, -0.324028343, -0.752295971, -0.270423025, 0.634717822, 0.662036777, 0.300237924, 0.306726158, -0.985477507, -0.30977422, 0.335294098, -0.278767616, 0.383350074, -0.169481948, 0.224124998, -0.503835678, 0.554356933, 0.648512602, 0.760522485, -0.521800339, -0.681355357, -0.654676735, -0.245198816, -0.683879256, -0.2702896, 0.412531048, 0.660841942, -0.27498427, 0.447191566, -0.372911632, 0.353137344, 0.548924148, -0.49649927, 0.449731916, 0.213543788, -0.414980084, -0.384420782, 0.705915034, -0.545251369, -0.136144951, 0.445821047, -0.313231587, 0.348674387, 0.442032456, 0.883140683, -0.161886886, 0.256801873, -0.550170898, -0.658088923, 0.631792367, -0.68034339, 0.628093898, -0.673520327, 0.64886272, 0.119231351, -0.50938499, -0.804269433, 0.753493547, -0.185574532, 0.596072435, 0.262295187, 0.389022321, 0.287074447, -0.486778438, 0.250325918, 0.538377404, 0.510265708, 0.402326643, -0.485398233, -0.616941094, -0.315257162, -0.406355083, 0.596790731, 0.18312791, -0.404126465, 0.422671884, -0.393740088, 0.318197966, -0.25652051, 0.571402431, -0.417811453, -0.516532421, -0.387963712, 0.446619213, 0.357654065, 0.453591824, 0.444609344, 0.386659116, 0.38722384, -0.435420364, -0.661135852, 0.44653216, -0.484769344, 0.259573221, -0.412828475, -0.403533816, 0.384532601, -0.575521946, -0.387747854, 0.454900146, 0.480018318, -0.606047392, 0.763270438, 0.431678325, -0.428464323, 0.473017037, -0.264299035, -0.353988141, -0.570904732, 0.277915627, -0.35870567, 0.451273471, 0.608966708, -0.444660515, 0.513376057, -0.643585145, 0.602900028, -0.745459914, -0.424295068, 0.563931882, 0.712498069, -0.500777125, 0.454909146, -0.547409654, -0.485119253, -0.312746674, -0.495797604, 0.32361263, -0.369999141, -0.274437666, -0.830233514, -0.275556445, 0.395280749, 0.688363492, 0.215288535, 0.252460241, -0.908234477, -0.223420769, 0.441514313, -0.221607223, 0.418126971, -0.172671214, 0.395999551, -0.511529863, 0.499575227, 0.61242044, 0.731697261, -0.439214081, -0.635171473, -0.688619077, -0.261818945, -0.665220976, -0.343080789, 0.566583395, 0.692079067, -0.362523615, 0.277867764, -0.240296155, 0.311870784, 0.588594913, -0.621245146, 0.607721269, 0.320387125, -0.442105383, -0.525579929, 0.703559637, -0.434066415, -0.175712481, 0.41918993, -0.470500737, 0.24285765, 0.440820158, 0.792357266, -0.243547395, 0.212502658, -0.435832828, -0.552155077, 0.636577249, -0.763701439, 0.726608872, -0.604545772, 0.475039542, 0.189554021, -0.509402573, -0.720934331, 0.827649891, -0.156637803, 0.395130992, 0.264884233, 0.476940721, 0.424625099, -0.392070442, -0.201435775, -0.145421937, -0.889556706, -0.0334893428, 0.515543103, 0.759575665, 0.0796553791, 0.131943747, -1.01996541, -0.124912679, 0.133945867, -0.306471616, 0.380480796, -0.0820675567, 0.0171267111, -0.363614708, 0.625686467, 0.399404764, 0.685859203, -0.421578974, -0.636531234, -0.696741164, -0.373195618, -0.402644753, -0.144492716, 0.4790003, 0.705023348, -0.315900654, 0.397456825, -0.232213512, 0.206000745, 0.629172921, -0.488669991, 0.575407445, 0.318706483, -0.211487189, -0.288516939, 0.64677757, -0.616002798, -0.0493387058, 0.575370491, -0.339981735, 0.0908434242, 0.411362767, 0.698846638, -0.267184108, 0.120071314, -0.387268871, -0.743495464, 0.744130731, -0.753035486, 0.681229651, -0.452962041, 0.493415207, 0.106875949, -0.345991582, -0.665692985, 0.895840168, -0.231874719, 0.528325856, 0.34730798, 0.579094172, 0.326672941, -0.44514811, -0.379020154, -0.552117646, -0.583376825, -0.403383613, 0.560118139, 0.838045418, 0.426518053, 0.449755877, -0.950022161, -0.366163343, 0.566114843, -0.517285287, 0.385128051, -0.421297103, 0.406334072, -0.590950608, 0.569421947, 0.335460126, 0.477841407, -0.461394578, -0.657734036, -0.602584183, -0.407084286, -0.534729183, -0.509853005, 0.310842156, 0.575707912, -0.600672722, 0.428758174, -0.328980982, 0.590953529, 0.537787855, -0.353013575, 1.32499146, 0.537784994, -0.5213238, -0.794690311, 0.596389472, -1.06295025, -0.413854271, 0.370082051, -0.523847461, 0.452758998, 0.306363106, 0.841760755, -0.503774643, 0.522657037, -0.289535373, -0.964939833, 0.540059924, -0.712263703, 1.04526448, -1.39220119, 1.67677188, 0.545932949, -0.637877941, -1.09805894, 0.569246829, -0.490861267, 0.393194348, 0.553323865, 0.466682971, 0.543824136, -0.613097787, -0.45459044, -0.526309431, -0.656021953, -0.360541224, 0.493327439, 0.94922632, 0.432517469, 0.447921336, -0.784917772, -0.483460277, 0.394886047, -0.380217671, 0.537025988, -0.406661958, 0.567315757, -0.581099629, 0.445839286, 0.506797969, 0.60057503, -0.50637722, -0.457914561, -0.541372657, -0.638620198, -0.469011158, -0.346902698, 0.32197392, 0.520140231, -0.462037832, 0.406483203, -0.568840146, 0.495454609, 0.477592647, -0.549679041, 1.22428346, 0.51539135, -0.620455503, -0.7584759, 0.657343328, -0.960747957, -0.320510834, 0.474521577, -0.445617288, 0.576519907, 0.404500723, 0.763330579, -0.384348094, 0.479164243, -0.28476873, -1.08730137, 0.524687052, -0.528642774, 0.796124756, -1.45506251, 1.68722606, 0.416689515, -0.708642185, -0.872421026, 0.67956537, -0.338394463, 0.509331703, 0.415006071, 0.284865111, 0.395193964, -0.646475673, -0.519450188, -0.408038735, -0.669812858, -0.460419625, 0.544404685, 0.965421259, 0.334380925, 0.427261978, -0.688262522, -0.482213318, 0.436046243, -0.557914376, 0.550275803, -0.394222558, 0.266022086, -0.556367815, 0.582908273, 0.232151061, 0.593837261, -0.441053957, -0.623476326, -0.68651104, -0.490153819, -0.470621079, -0.420426637, 0.308802545, 0.554715633, -0.536234438, 0.488165826, -0.295128345, 0.374501228, 0.332178563, -0.306417704, 0.859841526, 0.490419835, -0.549588799, -0.556348741, 0.60651201, -0.965358794, -0.481981128, 0.353077471, -0.527126312, 0.521532238, 0.212866038, 0.678860307, -0.316059381, 0.499297678, -0.424193054, -0.920252204, 0.533778548, -0.637087762, 0.947617471, -1.18541038, 1.30223703, 0.486311972, -0.584093332, -0.925763726, 0.600028932, -0.414735883, 0.299502432, 0.382199168, 0.377447367, 0.507400393, -0.49268657, -0.348576099, -0.638164461, -0.654438496, -0.511897862, 0.38483867, 1.05617762, 0.40306291, 0.385520309, -0.931462169, -0.484654516, 0.540201187, -0.36378026, 0.609431267, -0.351228058, 0.451720685, -0.524651229, 0.59331584, 0.183681786, 0.486204088, -0.361741871, -0.570030332, -0.540829837, -0.499595255, -0.588362515, -0.371888518, 0.487349182, 0.680457592, -0.499818385, 0.484998554, -0.458688289, 0.63367027, 0.428558171, -0.34848398, 1.15294933, 0.43114838, -0.375435561, -0.609408438, 0.630841613, -0.980268121, -0.525109529, 0.528841376, -0.644025147, 0.304991603, 0.340026647, 0.744779706, -0.420617998, 0.32421428, -0.320957214, -0.907028258, 0.626452088, -0.604258895, 0.928714931, -1.23938906, 1.5700357, 0.304795176, -0.7467978, -1.03154445, 0.686517894, -0.536533952, 0.438258648, 0.594017684, 0.252035111, 0.453340054, -0.552311063, -0.417818069, -0.26190424, -0.571614742, -0.384781599, 0.407266974, 0.815615833, 0.381351292, 0.354994088, -0.646592796, -0.372202933, 0.304195464, -0.434438199, 0.362853259, -0.31584686, 0.244136646, -0.318957031, 0.557140708, 0.34489131, 0.647323191, -0.528444409, -0.426986545, -0.464227885, -0.3825261, -0.498808682, -0.27001974, 0.350429475, 0.60395205, -0.384024262, 0.44076103, -0.427232414, 0.292858958, 0.433880299, -0.551758647, 0.696217895, 0.371488482, -0.293180257, -0.368783623, 0.60285145, -0.723924816, -0.434112787, 0.478570819, -0.43966046, 0.256822228, 0.365054816, 0.759034336, -0.374474615, 0.177014709, -0.535215199, -0.719300807, 0.411476582, -0.615099013, 0.783845127, -0.775601685, 0.571797609, 0.438532174, -0.581321478, -0.681845486, 0.673450589, -0.338453203, 0.363810748, 0.478750885, 0.470316291, 0.296830237, -0.566006243, 0.333698362, 0.363307953, 0.55199939, 0.442035705, -0.383573115, -0.641640782, -0.238909602, -0.437409729, 0.557771504, 0.452482134, -0.366771102, 0.408661455, -0.449404359, 0.44643265, -0.496670514, 0.614964604, -0.55154413, -0.420596242, -0.391293526, 0.515248299, 0.515675664, 0.480643153, 0.466191739, 0.350003153, 0.246595368, -0.505883515, -0.550677359, 0.459182978, -0.349407881, 0.240475357, -0.495883316, -0.493301719, 0.547659457, -0.796995044, -0.404546887, 0.462239355, 0.690047085, -0.649240434, 0.635555208, 0.307751626, -0.33474806, 0.439349443, -0.41000542, -0.266249061, -0.498849511, 0.403698564, -0.321013868, 0.337660193, 0.690214396, -0.572486222, 0.36732161, -0.684773982, 0.846628606, -0.905601263, -0.439664632, 0.602699637, 0.952240467, -0.650907397, 0.423727244, -0.329724222, -0.420888394, -0.383269608, -0.580309629, 0.547902167, -0.170367301, -0.264708668, -1.23543537, -0.281020641, 0.595188439, 0.972505629, 0.114389509, 0.203577861, -1.20719492, -0.226515099, 0.372065395, -0.251373738, 0.487018257, -0.425378203, 0.124593131, -0.328524411, 0.750639796, 0.577434361, 0.787221491, -0.617882967, -0.712628722, -0.877430677, -0.366920322, -0.492048949, -0.413935483, 0.620500267, 0.753165126, -0.204818472, 0.480239779, -0.391652584, 0.369886041, 0.567533493, -0.595628917, 0.676325142, 0.205830216, -0.425586939, -0.392195761, 0.801529765, -0.57094568, -0.198260024, 0.519222796, -0.265541017, 0.329809964, 0.588505149, 1.02412498, -0.170681179, 0.229564667, -0.617393553, -0.749539435, 0.825480998, -0.949508309, 0.797777176, -0.552113235, 0.761866033, 0.152554587, -0.649764657, -0.794153631, 1.05037129, -0.278679997, 0.626122355, 0.265911728, 0.445403248, 0.374678463, -0.342580229, 0.520656407, 0.573103964, 0.570444465, 0.469456106, -0.323329389, -0.804567158, -0.414154291, -0.45882231, 0.69754827, 0.423725516, -0.403667986, 0.528419435, -0.480837435, 0.351441741, -0.402553022, 0.510046721, -0.433772177, -0.380496413, -0.394198567, 0.438342214, 0.452685267, 0.528034925, 0.508481562, 0.526894748, 0.405712545, -0.541407049, -0.453555733, 0.353487968, -0.461078554, 0.25179401, -0.418590248, -0.387028962, 0.396600813, -0.931244195, -0.451324731, 0.361082554, 0.667675436, -0.600020528, 0.732300341, 0.469670475, -0.290680736, 0.456329077, -0.346446723, -0.342414051, -0.650512278, 0.255548, -0.352853209, 0.513713658, 0.790771365, -0.432831019, 0.639716625, -0.766357005, 0.857613623, -0.896571994, -0.269599527, 0.680787742, 0.710606635, -0.652714789, 0.399893761, -0.433409244, -0.524610639, -0.312088192, -0.488375127, 0.50994873, -0.425768435, -0.554442286, -0.642301738, -0.514117539, 0.529879212, 0.885797977, 0.496357262, 0.295032829, -0.736831605, -0.471642882, 0.551495135, -0.37344867, 0.467153907, -0.50650388, 0.523668885, -0.700668454, 0.602751136, 0.272464365, 0.532313824, -0.550322473, -0.548169196, -0.682784617, -0.469020545, -0.365018487, -0.521782041, 0.366236746, 0.615229726, -0.569497585, 0.61587429, -0.476180643, 0.395663947, 0.301352024, -0.546463788, 1.10225439, 0.404533267, -0.343092173, -0.656097829, 0.585557759, -1.00944042, -0.432898998, 0.380420029, -0.366831154, 0.279304773, 0.32894209, 0.681732297, -0.449885547, 0.333303005, -0.32521987, -0.949812949, 0.548179746, -0.481482506, 0.915706933, -1.3460927, 1.35060477, 0.532778621, -0.723563313, -0.819175363, 0.622870684, -0.380322933, 0.5157758, 0.464462489, 0.337888867, 0.526917517, -0.445044607, 0.541099072, 0.50325352, 0.677245975, 0.323587775, -0.332000583, -0.780857503, -0.447883099, -0.575264573, 0.773923576, 0.378291875, -0.479982048, 0.38349238, -0.465763003, 0.429923743, -0.379493684, 0.653094172, -0.675943851, -0.274701029, -0.524045706, 0.344420135, 0.461033851, 0.612487614, 0.530505002, 0.339211583, 0.565088928, -0.49296841, -0.638410091, 0.389825881, -0.448829889, 0.33532396, -0.434196651, -0.519870758, 0.556106865, -1.06203532, -0.368413895, 0.551040351, 0.732794225, -0.64174813, 0.996447682, 0.481682241, -0.316285402, 0.401805967, -0.550898135, -0.403002381, -0.770289898, 0.298914105, -0.33248207, 0.366171002, 0.814904511, -0.528657913, 0.587772429, -0.838930607, 1.35731173, -1.42681801, -0.546971798, 0.529041708, 1.04821432, -0.572809875, 0.30376783, -0.396251172, -0.536933064, -0.454127043, -0.454506367, 0.501756847, 0.167578146, 0.279935271, 0.858329535, 0.0272319373, -0.428495228, -0.759695828, -0.0834374204, -0.229138091, 0.89569056, 0.156982735, -0.188633591, 0.104403786, -0.328891963, 0.305502087, -0.248880729, 0.220129564, -0.800334871, -0.432452083, -0.545947075, 0.521066368, 0.592346787, 0.802690208, 0.217045441, 0.455956817, 0.194578528, -0.55685991, -0.588694334, 0.113738872, -0.385351121, 0.274045944, -0.186730936, -0.495718777, 0.424346268, -0.534337282, -0.192227274, 0.131534874, 0.49832347, -0.818950772, 0.47277391, 0.188198686, -0.467730343, 0.416054726, -0.2915079, -0.565653443, -0.851156473, 0.110739999, -0.209598735, 0.480854392, 0.553064585, -0.814000607, 0.801790953, -0.669766188, 0.616795599, -0.643502414, -0.256751955, 0.294647217, 0.662411213, -0.880029142, 0.209213212, -0.595876157, -0.270994693, -0.529327273, -0.287460744, 0.243372083, -0.325894624, -0.432371646, -0.550504088, -0.407037705, 0.514226615, 0.731068254, 0.374798119, 0.201470315, -0.727335334, -0.325077504, 0.346012741, -0.439286411, 0.333308727, -0.311294168, 0.342066079, -0.433207601, 0.47755152, 0.541718185, 0.395483285, -0.564353168, -0.379612327, -0.489284933, -0.371704191, -0.483742148, -0.390651584, 0.342548281, 0.565155149, -0.32511133, 0.485053867, -0.406071633, 0.326123238, 0.326088279, -0.462968737, 0.64342612, 0.239119932, -0.466389418, -0.558311999, 0.495003492, -0.52469945, -0.295910805, 0.554481924, -0.413308203, 0.155392587, 0.401756227, 0.617788911, -0.389093965, 0.257562876, -0.330855161, -0.685748398, 0.532081962, -0.518495023, 0.632078648, -0.645799041, 0.523082376, 0.398365796, -0.467045575, -0.663691282, 0.499885321, -0.175572664, 0.367428869, 0.305096716, 0.563034654, 0.438041508, -0.249610364, -0.283272624, -0.358795941, -0.982903302, -0.136733636, 0.603000462, 0.80477351, 0.249172851, 0.0673773363, -0.964687824, -0.0387507528, 0.282203943, -0.165284917, 0.239011973, -0.347310096, 0.171225876, -0.340983927, 0.693488359, 0.576028287, 0.566512704, -0.444235176, -0.567874968, -0.66565913, -0.267314732, -0.643461585, -0.303208411, 0.470927477, 0.714222848, -0.172081769, 0.192168161, -0.299989909, 0.449971706, 0.610318601, -0.434900492, 0.557600677, 0.196471184, -0.4122141, -0.530112386, 0.717300832, -0.408176243, -0.235542536, 0.576590061, -0.402583748, 0.134950235, 0.474380821, 0.833194613, -0.103588447, 0.0891227648, -0.468323857, -0.62792027, 0.803580105, -0.785261929, 0.806756794, -0.529432118, 0.61572814, 0.0892420486, -0.379495978, -0.550534964, 0.783187747, -0.207133546, 0.526591837, 0.294110864, 0.426459879, 0.285217106, -0.409641266, 0.238512605, 0.350833744, 0.681291521, 0.373441249, -0.589262605, -0.710154951, -0.22372216, -0.236419693, 0.734089375, 0.262492955, -0.512194276, 0.495519727, -0.348198861, 0.37896961, -0.24169825, 0.604631305, -0.567785203, -0.632024229, -0.659040213, 0.452594221, 0.588926911, 0.551869154, 0.403056443, 0.536315143, 0.439422786, -0.535578847, -0.734873116, 0.280560791, -0.537309289, 0.382309318, -0.398091793, -0.600111365, 0.458581388, -0.61039114, -0.375132948, 0.313789517, 0.609071791, -0.762822688, 0.569715619, 0.210205153, -0.666683614, 0.546203732, -0.245516315, -0.399653822, -0.887548089, 0.239415944, -0.355282068, 0.459468871, 0.782193363, -0.621101201, 0.778309584, -0.882275045, 0.711607456, -0.741972089, -0.470179409, 0.547727883, 0.693549812, -0.625376284, 0.45952943, -0.596325576, -0.31700471, -0.441045702, -0.507005632, 0.40017575, 0.299462408, 0.368873566, 0.757138789, 0.177711442, -0.468171895, -0.63479054, -0.15623793, -0.349899977, 0.877961874, 0.217684776, -0.402990162, 0.29281044, -0.21595934, 0.159143612, -0.244624108, 0.492553622, -0.667261958, -0.594178855, -0.5580585, 0.446866333, 0.493617356, 0.711934805, 0.370906264, 0.424997389, 0.216546372, -0.397282213, -0.51699847, 0.301145464, -0.253507674, 0.191388696, -0.437795579, -0.446385235, 0.55781734, -0.590693653, -0.226021156, 0.433810204, 0.508008897, -0.73411423, 0.604632795, 0.201233909, -0.498512536, 0.430822849, -0.268948436, -0.565350115, -0.585544229, 0.131844267, -0.0985700637, 0.60331738, 0.477022439, -0.737276614, 0.739348412, -0.780957878, 0.636857212, -0.673156261, -0.186896667, 0.412021995, 0.679868221, -0.754024267, 0.234325513, -0.448603541, -0.395069182, -0.378739357, -0.315825313, 0.479964375, -0.321257651, -0.295059592, -0.77799046, -0.221850574, 0.551184118, 0.706216156, 0.139173999, 0.142288312, -0.878085554, -0.0342805311, 0.234268114, -0.20716235, 0.388903022, -0.338036746, 0.243292049, -0.325317711, 0.592056155, 0.409110278, 0.756002605, -0.567251861, -0.53929919, -0.694564223, -0.425141931, -0.428060889, -0.277496874, 0.521914542, 0.84954536, -0.163342029, 0.208043978, -0.207859054, 0.189960539, 0.428250879, -0.38938725, 0.596192539, 0.240633845, -0.327855945, -0.427874893, 0.684532583, -0.519488037, -0.0568759963, 0.502675712, -0.278195858, 0.100424267, 0.410603642, 0.890421689, -0.341502815, 0.205754891, -0.48490423, -0.678747535, 0.619363606, -0.755045891, 0.557381153, -0.416407853, 0.631267071, 0.17229794, -0.423768014, -0.644227743, 0.889907777, -0.332315803, 0.558386028, 0.248280406, 0.617097437, 0.392860234, -0.351015836, -0.443047941, -0.353078872, -0.501930773, -0.518282115, 0.431032598, 0.859903872, 0.323263586, 0.390713632, -0.651903689, -0.396405339, 0.491211265, -0.305729717, 0.493661255, -0.283780128, 0.260419399, -0.455788523, 0.616844773, 0.450010449, 0.505137086, -0.315073639, -0.623857677, -0.617228568, -0.342319965, -0.363650113, -0.533531845, 0.248784035, 0.645062923, -0.400124162, 0.498861045, -0.457104534, 0.474639595, 0.399738759, -0.292998791, 1.02576375, 0.51698333, -0.367574304, -0.567398429, 0.546049654, -0.727638423, -0.442172617, 0.480285525, -0.56605351, 0.499985546, 0.243005559, 0.572674751, -0.281488627, 0.414541632, -0.299860507, -0.909291744, 0.403057963, -0.603531122, 0.701785803, -1.06234276, 1.17074287, 0.347060531, -0.725450873, -0.910402179, 0.653182209, -0.395115227, 0.50289017, 0.545734346, 0.348768085, 0.512140214, -0.596556962, 0.347126722, 0.468261927, 0.477998018, 0.335079044, -0.590415716, -0.854746044, -0.447128892, -0.55043757, 0.614228666, 0.422970176, -0.569780469, 0.327640414, -0.436567426, 0.342652917, -0.305259734, 0.684629917, -0.448736697, -0.307220906, -0.663768709, 0.459859699, 0.390889198, 0.423822314, 0.54664737, 0.432333559, 0.327140361, -0.371867955, -0.474025309, 0.323286563, -0.483154684, 0.491285264, -0.581923842, -0.536662221, 0.493367463, -1.03564882, -0.524836361, 0.517686188, 0.757357776, -0.492390007, 0.791603804, 0.399490923, -0.430052042, 0.508883536, -0.438035756, -0.330016404, -0.793897152, 0.357776165, -0.374079734, 0.275550365, 0.810435951, -0.662917733, 0.463717222, -0.844937503, 1.17519164, -1.39522147, -0.4581227, 0.750042021, 1.01812994, -0.525968909, 0.530613244, -0.388203204, -0.325991809, -0.355104208, -0.375738889, 0.654266715, -0.246238187, -0.328388274, -0.900334358, -0.102514587, 0.444142222, 0.828398049, 0.165270939, 0.338851839, -0.883268535, -0.197197318, 0.213587329, -0.413152337, 0.274834216, -0.199403107, 0.364259809, -0.410779357, 0.786017835, 0.441939741, 0.665733218, -0.523882747, -0.604177415, -0.620881855, -0.333371997, -0.590572059, -0.245860413, 0.500872076, 0.806275427, -0.37275514, 0.291275263, -0.145374492, 0.297142118, 0.446176827, -0.455065727, 0.630103111, 0.384944916, -0.316880941, -0.53316617, 0.624569774, -0.632713258, -0.20398733, 0.435037136, -0.41079697, 0.35267365, 0.477758348, 0.753579497, -0.236058086, 0.0966574922, -0.60752362, -0.696536541, 0.776510596, -0.815420151, 0.803661168, -0.62879616, 0.45567295, 0.123660304, -0.384508193, -0.609552443, 0.632402658, -0.243827447, 0.630169272, 0.324621022, 0.417416543, 0.453456402, -0.293153346, 0.0629724562, 0.282054573, 0.948353469, -0.01112503, -0.446363509, -0.906694233, -0.150774568, -0.198606119, 0.92327565, 0.215320408, -0.165527165, 0.200482354, -0.0939625949, 0.156043261, -0.145319119, 0.457442015, -0.845342398, -0.455728769, -0.698774934, 0.537646592, 0.652544141, 0.686487436, 0.31823799, 0.447897047, 0.140797585, -0.536412895, -0.618760943, 0.295252204, -0.196979925, 0.123686709, -0.237342492, -0.453248322, 0.622943342, -0.64648217, -0.135725662, 0.318282932, 0.330090076, -0.852190971, 0.630669713, 0.107867919, -0.49712202, 0.346709013, -0.246710822, -0.349392205, -0.772212863, 0.0380674526, -0.178112671, 0.396954775, 0.611174643, -0.890879571, 0.771946013, -0.717363358, 0.662966669, -0.449829489, -0.250934422, 0.308512032, 0.613217592, -0.794438183, 0.244610265, -0.550646484, -0.172934994, -0.598853469, -0.233596042, 0.388285547, 0.244651794, 0.445050716, 0.875652254, 0.26988253, -0.561746597, -0.779444218, -0.252824008, -0.321111292, 1.06848943, 0.295377821, -0.437555999, 0.28307265, -0.298364878, 0.313521653, -0.384158015, 0.469548076, -0.732281268, -0.471832573, -0.816568553, 0.70611918, 0.528583646, 0.701247394, 0.343509763, 0.659085929, 0.207387581, -0.523094058, -0.754302621, 0.365032524, -0.324296981, 0.212653041, -0.365114331, -0.520832002, 0.636939704, -0.526777864, -0.464013755, 0.348045558, 0.390014023, -0.904298842, 0.610676527, 0.301345497, -0.565652311, 0.51331532, -0.341150373, -0.661861956, -1.00385046, 0.235195249, -0.210188031, 0.689216793, 0.803023756, -0.903787851, 0.910963118, -0.853248477, 0.592033148, -0.748203695, -0.244562104, 0.615952373, 0.863976896, -0.866574466, 0.332677424, -0.471797168, -0.259435207, -0.515951276, -0.506270468, 0.45248574, 0.250391096, 0.311859429, 0.938711584, 0.199012324, -0.552551389, -0.907712877, -0.0292224251, -0.142828003, 1.08049381, 0.163844496, -0.165308148, 0.117217541, -0.282036901, 0.333034098, -0.261533737, 0.327806175, -0.846170902, -0.55871141, -0.650601804, 0.527476907, 0.672261059, 0.672039866, 0.250090748, 0.662484229, 0.301278502, -0.519129634, -0.772370279, 0.326487094, -0.215952232, 0.293516815, -0.254435033, -0.407296091, 0.609227419, -0.400611013, -0.128699973, 0.156874925, 0.300926089, -0.827643514, 0.606920302, -0.0399293937, -0.560712278, 0.333961189, -0.25337407, -0.460930228, -0.756155908, 0.111029588, -0.174785942, 0.58958739, 0.740321219, -0.831516504, 0.781675041, -0.69119364, 0.521212041, -0.625474393, -0.274716079, 0.486845255, 0.629193842, -0.930688083, 0.189789623, -0.364750236, -0.354482323, -0.394587129, -0.149066895, 0.230414256, 0.215836838, 0.491596997, 0.700585723, 0.456593513, -0.471093863, -0.765746415, -0.411722928, -0.339567959, 0.773355126, 0.4266541, -0.456761658, 0.435377479, -0.48741737, 0.263097525, -0.322128475, 0.584900379, -0.605951905, -0.51968956, -0.671521008, 0.419011503, 0.549039543, 0.685625732, 0.509464741, 0.435605973, 0.270741463, -0.371719927, -0.519246757, 0.485465646, -0.563619912, 0.445907414, -0.393643916, -0.561774611, 0.599427164, -0.604217708, -0.329256952, 0.36250639, 0.431041032, -0.664941609, 0.698059738, 0.237263456, -0.597527325, 0.4369798, -0.416730851, -0.551124096, -0.818866313, 0.292731255, -0.283123583, 0.386692315, 0.747513235, -0.759241045, 0.477275133, -0.876334906, 0.692796648, -0.780430257, -0.417433083, 0.614516079, 0.733170033, -0.64263171, 0.47454381, -0.590557456, -0.432523668, -0.537426829, -0.28477335, 0.598722696, 0.494717032, 0.416905552, 0.48906666, 0.305307806, -0.310949534, -0.781238675, -0.529275, -0.464254379, 0.612940907, 0.385181993, -0.40740639, 0.438032657, -0.529878378, 0.49949199, -0.339031696, 0.560534358, -0.602270961, -0.491503745, -0.411578536, 0.524442792, 0.391362816, 0.542233586, 0.445596069, 0.364454538, 0.385163277, -0.462802112, -0.640788853, 0.336987823, -0.525584102, 0.53296423, -0.419788688, -0.45423907, 0.284706265, -0.82703644, -0.582333028, 0.544609964, 0.646183848, -0.647284746, 0.84342742, 0.384108216, -0.344146848, 0.48592487, -0.277876347, -0.463913679, -0.755639732, 0.404296011, -0.448455602, 0.504308105, 0.942184687, -0.548759162, 0.59737891, -0.753717542, 1.01575744, -1.19051194, -0.384594321, 0.508125007, 0.987443507, -0.604132056, 0.276406139, -0.28799814, -0.513938189, -0.353042334, -0.361533374, 0.453560591, 0.257468492, 0.174677595, 1.06680763, 0.197333381, -0.432188094, -0.901422441, 0.00785290264, -0.0305271856, 0.978117228, 0.0125726229, -0.18139945, 0.208148539, -0.250057399, 0.0882064477, -0.124524973, 0.309836417, -0.575959444, -0.568242967, -0.492013246, 0.337933064, 0.653048873, 0.771532297, 0.305375427, 0.601883709, 0.074381493, -0.336813509, -0.7794981, 0.291799366, -0.318551421, 0.118420988, -0.144757107, -0.437134564, 0.42022863, -0.652765036, -0.0306711029, 0.147376224, 0.412145913, -0.779087722, 0.394711316, -0.0504994206, -0.483489096, 0.129640549, 0.0219485927, -0.481859624, -0.845748067, 0.207463354, -0.0415801294, 0.536965311, 0.6556077, -0.844672024, 0.902707696, -0.853960752, 0.686929762, -0.60263145, -0.190143779, 0.40874663, 0.555190384, -0.821312368, 0.104288623, -0.405631512, -0.180742934, -0.41993174, -0.141889408, 0.345394313, -0.173090056, -0.37151432, -0.89373517, -0.144356117, 0.580647528, 0.757459641, 0.271152824, 0.288030565, -1.21821094, -0.190606788, 0.418052495, -0.414365053, 0.200714469, -0.354893804, 0.360974938, -0.277544767, 0.693278193, 0.487686127, 0.745655298, -0.472692281, -0.509124577, -0.721267521, -0.359080553, -0.532743514, -0.186544225, 0.491743058, 0.648181081, -0.28698644, 0.296985894, -0.196287811, 0.414783567, 0.585468769, -0.665569186, 0.524442494, 0.230066538, -0.285188287, -0.540552557, 0.847329855, -0.620200098, -0.0617543682, 0.611717999, -0.372248262, 0.114533916, 0.447834253, 0.834647715, -0.231694281, 0.194736198, -0.584714651, -0.648753703, 0.69645226, -0.840352893, 0.883932114, -0.568629682, 0.651081681, 0.117869407, -0.346449167, -0.771529496, 0.939396024, -0.114048921, 0.459198624, 0.236674815, 0.386042893, 0.297888905, -0.507050455, 0.370574802, 0.346722215, 0.970172942, 0.361205697, -0.661324263, -0.681496918, -0.155864239, -0.385353893, 1.09318161, 0.142546028, -0.344489872, 0.229719281, -0.237668097, 0.205861554, -0.272000253, 0.294067025, -0.583343863, -0.656137347, -0.721691668, 0.440148592, 0.574711859, 0.715354085, 0.252608985, 0.600980401, 0.246709153, -0.573691905, -0.669599295, 0.344540894, -0.366140991, 0.328274399, -0.496813327, -0.424318522, 0.465786636, -0.583664656, -0.240473375, 0.294938207, 0.348787427, -0.83149159, 0.668540895, 0.298399955, -0.628243804, 0.320712656, -0.233344361, -0.487331241, -0.743381739, 0.327826619, -0.13167651, 0.467116892, 0.560980082, -0.784882069, 0.861600399, -0.695126057, 0.516500831, -0.639968395, -0.362884641, 0.474332809, 0.84183985, -0.746321261, 0.240386918, -0.427387923, -0.317123204, -0.501971781, -0.254804373, 0.445564926, -0.274497837, -0.371203661, -0.81181246, -0.104722269, 0.587726295, 0.83375293, 0.0862023681, 0.120025091, -1.13786316, -0.134314433, 0.272340983, -0.218453079, 0.417520106, -0.247756392, 0.222074315, -0.484334558, 0.779378235, 0.500625908, 0.520362437, -0.451774746, -0.707401037, -0.70885694, -0.252805799, -0.430832148, -0.32242313, 0.395950526, 0.825463712, -0.349297196, 0.189277649, -0.245836556, 0.287911505, 0.626974523, -0.621457577, 0.441190481, 0.383288652, -0.355456591, -0.482093692, 0.757665277, -0.625357687, -0.27123785, 0.468763202, -0.38299346, 0.135283798, 0.383362055, 0.845267773, -0.150662273, 0.0670877844, -0.533522427, -0.485103965, 0.896404982, -0.853809059, 0.660401702, -0.464548022, 0.505587339, 0.240668386, -0.496136367, -0.676835537, 0.919556737, -0.300272137, 0.510092676, 0.377860934, 0.589589417, 0.223942578, -0.407478958, 0.238767207, 0.152297005, -0.497014403, 0.20083943, 0.523349702, 0.488241553, -0.297424942, -0.11050307, -0.424515069, 0.258165359, -0.0239214823, 0.00964505691, -0.211816877, 0.113309771, -0.200172976, -0.0213771127, 0.597614646, 0.490241587, 0.603444338, -0.318409353, -0.524104834, -0.547398746, -0.00229556975, -0.460378677, 0.0956893861, 0.523315251, 0.619601786, 0.000513757928, 0.0314135253, 0.247382417, -0.174128637, 0.409572214, -0.511606574, 0.176335603, -0.115851603, 0.174122453, 0.102504335, 0.34038797, -0.245521232, 0.304468989, 0.569809794, -0.0304452796, -0.210962147, 0.323326409, 0.412501127, 0.0954742059, -0.0871605054, -0.303121656, -0.19844754, 0.556379914, -0.555037439, 0.310386121, -0.202452675, 0.0985213071, -0.0476110503, 0.0682585835, -0.200383335, 0.361906916, 0.0280265305, 0.397911787, -0.0576226115, 0.349537134, -0.0180170164, -0.0896787047, 0.4951092, 0.466181159, 0.756273031, 0.386582553, -0.487607718, -1.01005042, -0.263797164, -0.519615412, 0.69736433, 0.284120619, -0.590482831, 0.567264199, -0.549500048, 0.353119105, -0.430186599, 0.611936212, -0.673284411, -0.179817289, -0.644586861, 0.479300439, 0.476005584, 0.509333968, 0.434473187, 0.645393312, 0.340523094, -0.348291606, -0.519281805, 0.519528091, -0.511090934, 0.521959364, -0.490335047, -0.33156094, 0.380160511, -1.24818444, -0.424234033, 0.602386892, 0.717675209, -0.704489589, 0.933558166, 0.304948956, -0.291118622, 0.630240679, -0.437776536, -0.207699716, -0.933814406, 0.297022551, -0.416699886, 0.231116354, 0.945163608, -0.673645198, 0.639742434, -1.02563167, 1.33432353, -1.31458652, -0.377561837, 0.793118119, 0.879839957, -0.751712799, 0.526335776, -0.36455819, -0.578779817, -0.424948007, -0.456062466, 0.645958662, -0.2009359, -0.263773561, -0.826967478, -0.370625407, 0.542275846, 0.664447069, 0.163287491, 0.308100998, -0.861048281, -0.194696158, 0.220512033, -0.226582944, 0.255048186, -0.391231298, 0.259909332, -0.366343468, 0.597054541, 0.455798388, 0.659468412, -0.614014566, -0.647925377, -0.698584259, -0.326418251, -0.557808101, -0.242764115, 0.526800513, 0.620785058, -0.445572495, 0.289413214, -0.157801181, 0.286088079, 0.357253224, -0.527151227, 0.596771777, 0.321921706, -0.27184999, -0.376095653, 0.710879803, -0.425363064, -0.171487629, 0.5395118, -0.450492084, 0.21501489, 0.539113343, 0.83319509, -0.383878738, 0.368128002, -0.379428864, -0.662463963, 0.711876512, -0.745887399, 0.634167373, -0.650651455, 0.43601051, 0.135384589, -0.317399323, -0.631690204, 0.703509033, -0.401612073, 0.605592549, 0.437430501, 0.561705887, 0.209696889, -0.247922003, -0.189277992, -0.217304081, -0.749578297, -0.323254317, 0.539204717, 0.728956282, 0.277090937, 0.401523799, -0.825991809, -0.273026973, 0.268642157, -0.259769022, 0.263589621, -0.369773448, 0.168386191, -0.398087293, 0.564016044, 0.56983453, 0.568054676, -0.587791443, -0.682538807, -0.597797394, -0.310886979, -0.43280828, -0.351940542, 0.402026504, 0.725551724, -0.344901413, 0.25086841, -0.196568683, 0.458823591, 0.439975411, -0.501341105, 0.593206704, 0.25059554, -0.413169742, -0.54639858, 0.653652191, -0.637274921, -0.249179304, 0.464290261, -0.275205404, 0.341593593, 0.595168829, 0.751112401, -0.206167787, 0.135927692, -0.549307406, -0.547307491, 0.795383632, -0.634439886, 0.570365667, -0.557982981, 0.481782705, 0.307791501, -0.332375437, -0.816478491, 0.704833806, -0.147440225, 0.529172719, 0.320238382, 0.521421075, 0.297512829, -0.503937423, 0.392369986, 0.499026537, 0.557706296, 0.327456534, -0.496750325, -0.806194127, -0.319533408, -0.565670192, 0.720564544, 0.48260507, -0.500139296, 0.591555655, -0.445721447, 0.368455052, -0.401765376, 0.465892136, -0.489378363, -0.32572189, -0.425057948, 0.53074944, 0.550350606, 0.526860058, 0.570775211, 0.531260967, 0.519740224, -0.387945533, -0.507647395, 0.342835128, -0.498815536, 0.530000448, -0.616143346, -0.524641216, 0.59048146, -1.07204616, -0.579604506, 0.595958531, 0.764025152, -0.573009431, 0.904218435, 0.536760688, -0.508265793, 0.575817525, -0.304201633, -0.414322197, -0.709731221, 0.430216879, -0.465025872, 0.497060329, 0.958866954, -0.588998675, 0.457746476, -0.919173658, 1.10236216, -1.0048908, -0.424213499, 0.66981113, 1.00544739, -0.533460557, 0.347768635, -0.371134102, -0.373428643, -0.514042914, -0.594967484, 0.5132671, 0.200290054, 0.433623224, 1.02203405, 0.323877335, -0.533810377, -0.895527661, -0.23163414, -0.221574798, 1.16609228, 0.242880151, -0.403969616, 0.390322924, -0.460030466, 0.314850211, -0.172071725, 0.421792865, -0.638126731, -0.667486489, -0.694238424, 0.527170718, 0.664319515, 0.715590179, 0.302289575, 0.578976989, 0.205042839, -0.539689541, -0.828820109, 0.283062279, -0.366143584, 0.302690804, -0.372769684, -0.439584941, 0.569364607, -0.628790855, -0.25392738, 0.372507393, 0.570168674, -0.735647976, 0.628451467, 0.155496806, -0.427494824, 0.265664279, -0.354848415, -0.61978972, -0.98301357, 0.38858366, -0.273800701, 0.470405549, 0.843349397, -0.718695521, 0.748915255, -0.826158106, 0.740480959, -0.694378436, -0.217282176, 0.380821168, 0.817043483, -0.926361382, 0.180015951, -0.503372788, -0.471371621, -0.694792211, -0.458219498, 0.384510249, 0.351474315, 0.443674266, 1.11125815, 0.0880905017, -0.574157894, -0.7908234, -0.241150007, -0.177079871, 1.15466774, 0.107747041, -0.32727164, 0.150086567, -0.269126058, 0.190451279, -0.263872623, 0.417925298, -0.800326765, -0.461136878, -0.68378824, 0.486337036, 0.450565308, 0.787122309, 0.423443973, 0.653326154, 0.202834353, -0.634362876, -0.797869921, 0.15107286, -0.236876383, 0.225229248, -0.364838928, -0.512411535, 0.453049272, -0.470336407, -0.151961684, 0.423445672, 0.451209217, -0.802669287, 0.619109154, 0.108615965, -0.482686907, 0.248642474, -0.112961367, -0.577998638, -0.908955812, 0.204193041, -0.128125697, 0.484464437, 0.741138995, -0.795964062, 0.815873981, -0.699818075, 0.497804135, -0.464158088, -0.255229384, 0.552704036, 0.656278312, -0.871029079, 0.153432593, -0.462791413, -0.269675344, -0.470113456, -0.290688753, 0.342632353, 0.581155956, 0.547519386, 0.702668667, 0.413780421, -0.462375402, -1.02571797, -0.435773402, -0.566165447, 0.923119962, 0.374345988, -0.550363183, 0.380189627, -0.480621606, 0.441591889, -0.535251796, 0.534693241, -0.61400193, -0.397097945, -0.641558051, 0.549189746, 0.585095048, 0.481853157, 0.572160363, 0.376207411, 0.485279858, -0.488048553, -0.515832007, 0.539535582, -0.437932134, 0.577877045, -0.436782032, -0.466930658, 0.410578787, -1.12756717, -0.619950473, 0.414643645, 0.646280527, -0.622953176, 0.961902022, 0.361166805, -0.417870075, 0.636564612, -0.457520604, -0.23916246, -0.731118917, 0.489576697, -0.454277247, 0.506435752, 0.873826027, -0.631583631, 0.688300431, -0.798250198, 1.41198325, -1.59610319, -0.506833971, 0.706683099, 0.950876176, -0.499421388, 0.554268241, -0.469414741, -0.393041342, -0.50618428, -0.384822369, 0.545894444, 0.187190652, 0.246423274, 0.907203317, 0.328936011, -0.457639575, -0.776459277, -0.273714513, -0.283097863, 0.956705511, 0.172773972, -0.357948363, 0.233617485, -0.280701131, 0.340278476, -0.412458807, 0.340041906, -0.543849349, -0.637045979, -0.690804124, 0.501034617, 0.6456936, 0.742468536, 0.32371518, 0.530948997, 0.282261461, -0.668399513, -0.695456266, 0.387465715, -0.474695861, 0.392627031, -0.257529676, -0.424579382, 0.47605449, -0.546476066, -0.232761502, 0.337502718, 0.459151506, -0.750615001, 0.585467041, 0.272855312, -0.660907686, 0.454055041, -0.371678919, -0.593729734, -0.833883345, 0.209032804, -0.277053595, 0.453939617, 0.632635891, -0.675260067, 0.576594055, -0.825086117, 0.61530441, -0.604878306, -0.275764316, 0.376866043, 0.804845572, -0.856445074, 0.417382002, -0.570453465, -0.334888935, -0.597369671, -0.360090256, 0.48273614, -0.306990504, -0.230070278, -1.09909689, -0.1636675, 0.621702254, 0.674601734, 0.246477932, 0.310195655, -1.19192541, -0.132746786, 0.273221135, -0.155066922, 0.404253751, -0.352336407, 0.0401428342, -0.261068016, 0.688155115, 0.407058001, 0.545624852, -0.415766388, -0.59605509, -0.769288957, -0.417391121, -0.459224135, -0.200203508, 0.509438396, 0.850664914, -0.106015339, 0.262042522, -0.155878112, 0.385848731, 0.426718652, -0.419342548, 0.518178821, 0.140892014, -0.216667786, -0.464685053, 0.663083613, -0.514115274, -0.0205285326, 0.480129719, -0.164312139, 0.127549663, 0.47528711, 0.803208768, -0.299954206, 0.155377299, -0.492197812, -0.7155779, 0.905318856, -0.851143837, 0.793637991, -0.630919576, 0.630528569, 0.136860833, -0.528074563, -0.722409546, 0.753608525, -0.112982698, 0.485640645, 0.263396174, 0.542774737, 0.150543123, -0.289700896, 0.20876804, 0.280848503, 1.12810469, 0.160258099, -0.445825994, -0.8189798, -0.111164495, -0.337912649, 1.11674368, 0.169844672, -0.422637522, 0.306197077, -0.37622112, 0.223766327, -0.141381279, 0.525833845, -0.760584533, -0.603213906, -0.679515362, 0.677870452, 0.667746663, 0.618115246, 0.410314053, 0.644465446, 0.351321876, -0.457629204, -0.907127917, 0.294997036, -0.341109276, 0.135668993, -0.462654084, -0.567560136, 0.566696882, -0.472471774, -0.23072736, 0.352127045, 0.377069652, -0.68234545, 0.621890903, 0.186982349, -0.554198325, 0.465716451, -0.109229639, -0.41909343, -0.997850299, 0.162804559, -0.125065714, 0.618347406, 0.588448882, -0.898933053, 0.854276121, -0.761164665, 0.476102471, -0.740566373, -0.115307286, 0.570333898, 0.680743039, -0.838994622, 0.172854736, -0.538978517, -0.314399689, -0.387903869, -0.303288966, 0.385495961, 0.513157368, 0.637085974, 0.697108865, 0.516586721, -0.521081865, -0.895427465, -0.527276158, -0.517107248, 0.850408673, 0.453525662, -0.436300814, 0.574615359, -0.44233796, 0.528130233, -0.526731849, 0.521550715, -0.560411513, -0.297717661, -0.489339918, 0.448840976, 0.554962039, 0.708843946, 0.525428712, 0.626448989, 0.306288451, -0.343715847, -0.695142388, 0.382899463, -0.650318503, 0.355282784, -0.586688161, -0.300500751, 0.419991016, -1.07795775, -0.477047384, 0.521976352, 0.731458366, -0.684702337, 1.02854943, 0.283347398, -0.322144657, 0.43163833, -0.470982909, -0.368042976, -0.814351916, 0.423651695, -0.488408267, 0.336329997, 0.885656655, -0.756266534, 0.525726438, -0.884774446, 1.26688993, -1.57740438, -0.313142389, 0.579769969, 1.15113521, -0.765965581, 0.286212295, -0.331682473, -0.59841001, -0.454794675, -0.535127342, 0.663455546, -0.449571431, -0.359366149, -0.614765048, -0.237218067, 0.503638923, 0.659786403, 0.20122166, 0.242923573, -0.716324866, -0.227706954, 0.485323578, -0.335747004, 0.400215924, -0.419744015, 0.358518779, -0.472834647, 0.390084386, 0.391275764, 0.551161826, -0.565886676, -0.565476894, -0.642740428, -0.482294619, -0.333216578, -0.31584534, 0.381909132, 0.480554253, -0.468462378, 0.463644147, -0.28018856, 0.381048083, 0.446304619, -0.317517132, 0.542756379, 0.240631983, -0.401492715, -0.488540888, 0.496728241, -0.627157092, -0.316725284, 0.4836936, -0.453904361, 0.206610352, 0.359172821, 0.536408186, -0.258754224, 0.271194994, -0.511703968, -0.604014456, 0.518659055, -0.539535344, 0.745565355, -0.495848358, 0.606330574, 0.353892505, -0.605881035, -0.584356546, 0.647493839, -0.246999145, 0.560672104, 0.343967468, 0.412044287, 0.371602744, -0.42312637, 0.385247678, 0.527204573, 0.494672686, 0.357852072, -0.446920693, -0.656830728, -0.415859967, -0.245454639, 0.688588798, 0.192023784, -0.462693393, 0.466143817, -0.34368515, 0.311748415, -0.349412858, 0.387468249, -0.465777159, -0.50558424, -0.463219017, 0.569537461, 0.631559134, 0.689584315, 0.398396522, 0.53982842, 0.419469833, -0.345557123, -0.472127229, 0.479387909, -0.509029508, 0.338222176, -0.483616114, -0.508775294, 0.54947257, -0.520134211, -0.395031244, 0.29339993, 0.391059607, -0.520817459, 0.629955411, 0.372585475, -0.366463721, 0.379386872, -0.240199834, -0.546734095, -0.638515234, 0.450689405, -0.225037992, 0.47898218, 0.777923703, -0.691686928, 0.638843358, -0.653266966, 0.620898366, -0.599992275, -0.372237623, 0.655808747, 0.788578629, -0.57462132, 0.209120348, -0.409739405, -0.337165087, -0.436498135, -0.483499289, 0.329910994, 0.326199949, 0.481177688, 1.16359544, 0.206624717, -0.695663691, -0.813543081, -0.222134441, -0.301099747, 1.06720877, 0.0982987136, -0.222558349, 0.333435118, -0.282705396, 0.197784811, -0.149085388, 0.533713043, -0.908872724, -0.375418842, -0.770307124, 0.534855247, 0.623711944, 0.782452703, 0.323662639, 0.528443277, 0.245449454, -0.427402496, -0.861736715, 0.305742264, -0.256901175, 0.232547522, -0.466381431, -0.667825401, 0.504195333, -0.644258857, -0.322387427, 0.322032034, 0.407531679, -0.931643844, 0.470853716, 0.272893697, -0.60111773, 0.315316379, -0.156917512, -0.595057487, -0.969385326, 0.285556108, -0.096228078, 0.561174691, 0.708949447, -1.00587761, 0.982372761, -0.87020725, 0.698471189, -0.751767635, -0.152550936, 0.41984272, 0.71415025, -0.829321861, 0.167760983, -0.592690527, -0.355854481, -0.628726721, -0.381899953, 0.365675807, -0.0465951785, -0.358047932, -0.880212724, -0.182319552, 0.405644357, 0.728266537, 0.168842494, 0.102600455, -0.979417503, -0.171121135, 0.249877661, -0.0723972321, 0.247325465, -0.146962449, 0.119723082, -0.278888047, 0.820329845, 0.501146317, 0.533150673, -0.355726987, -0.473440051, -0.777638435, -0.218270808, -0.633167028, -0.279746026, 0.528565109, 0.798648238, -0.241700843, 0.1608098, -0.148207545, 0.334849149, 0.45928672, -0.425278515, 0.567445517, 0.135615841, -0.226115391, -0.478285968, 0.630218744, -0.475862682, -0.173051909, 0.539743662, -0.183654457, 0.219358683, 0.597796619, 0.865054846, -0.0468610898, 0.181407824, -0.600174129, -0.685601771, 0.706922352, -0.684688866, 0.618187666, -0.551391065, 0.675044656, 0.216130883, -0.331861526, -0.643832803, 0.690533459, -0.104342632, 0.547348022, 0.0965096131, 0.487036079, 0.227805495, -0.373000652, 0.272583604, 0.448061585, 0.805707335, 0.258710206, -0.661880612, -0.83204633, -0.239843041, -0.233504981, 0.763569772, 0.420496315, -0.307486683, 0.360896736, -0.52702266, 0.38465327, -0.393024206, 0.586225748, -0.672779083, -0.507444561, -0.685064197, 0.452422559, 0.529536486, 0.705149531, 0.435184658, 0.66582185, 0.290264338, -0.638234258, -0.592290163, 0.46619603, -0.361524403, 0.441005886, -0.447277158, -0.530420244, 0.578502774, -0.690500975, -0.451319009, 0.422686636, 0.495203406, -0.744223893, 0.652014732, 0.422241926, -0.633214891, 0.532111347, -0.382185489, -0.370549172, -0.732441664, 0.351130724, -0.223976329, 0.440156221, 0.73801893, -0.763945758, 0.564236581, -0.898421705, 0.557333767, -0.735742986, -0.297184855, 0.48788625, 0.910363436, -0.63786, 0.367409468, -0.611377954, -0.418537736, -0.521284461, -0.398774475, 0.349797189, 0.322694331, 0.376694143, 0.483070672, 0.388009012, -0.465679318, -0.685029089, -0.372201383, -0.488534719, 0.659292161, 0.440502822, -0.572985113, 0.54666692, -0.301185608, 0.366004974, -0.492218494, 0.48372364, -0.551055729, -0.426280618, -0.55951786, 0.500045598, 0.609633029, 0.432803243, 0.418478787, 0.341789871, 0.266200423, -0.401765853, -0.45946312, 0.516252816, -0.405258238, 0.44367519, -0.526319504, -0.450157285, 0.51572758, -0.946239173, -0.333996683, 0.50093925, 0.525497079, -0.536529601, 0.717539907, 0.516171455, -0.510850608, 0.58161217, -0.454105675, -0.296858281, -0.552912414, 0.44778496, -0.322999477, 0.311096311, 0.931384265, -0.629501402, 0.430051267, -0.768526435, 1.15942299, -1.1840452, -0.426751763, 0.708617389, 0.76344198, -0.656803191, 0.49345389, -0.352077842, -0.452331662, -0.446800828, -0.505934715, 0.548232555, 0.435045362, 0.611051857, 0.586130261, 0.517834306, -0.594725966, -1.10093296, -0.305011481, -0.399400473, 0.873429179, 0.470877677, -0.59704572, 0.602522969, -0.374939591, 0.552463233, -0.445587784, 0.490479171, -0.684512138, -0.352469385, -0.65754658, 0.338127553, 0.507106483, 0.651831031, 0.467000216, 0.489944369, 0.54797256, -0.471258074, -0.557674468, 0.449789762, -0.417932302, 0.368801236, -0.469076157, -0.356696755, 0.411393166, -1.21022117, -0.542315781, 0.455763042, 0.742555141, -0.538927376, 1.01949358, 0.461236, -0.401985794, 0.643230975, -0.460425049, -0.387737989, -0.990588129, 0.376649112, -0.46267876, 0.227371603, 1.13518035, -0.672486246, 0.518971264, -0.949415922, 1.45657301, -1.72685742, -0.501710832, 0.561250091, 0.971298099, -0.720059156, 0.441240877, -0.487569004, -0.51516062, -0.502963305, -0.484737247, 0.71079886, -0.335233152, -0.271280438, -0.750459492, -0.259238869, 0.676791847, 0.763187468, 0.320925623, 0.339963764, -0.868400574, -0.259744734, 0.256180644, -0.464681864, 0.359568775, -0.316238672, 0.285438597, -0.546080232, 0.708462059, 0.444063425, 0.755364239, -0.604672909, -0.572135627, -0.764483094, -0.389026016, -0.605620563, -0.206244096, 0.517358661, 0.765020907, -0.214551583, 0.477057189, -0.258695334, 0.468147933, 0.5390324, -0.54779017, 0.527488887, 0.359281659, -0.264136821, -0.401367247, 0.538585126, -0.651461184, -0.358718276, 0.426010579, -0.448634714, 0.351415902, 0.378670961, 0.68447113, -0.33796376, 0.286270261, -0.463992238, -0.729223788, 0.557461619, -0.614458859, 0.694635451, -0.52258724, 0.682086825, 0.266150683, -0.527700484, -0.648811996, 0.734942138, -0.316290408, 0.497466117, 0.398887843, 0.521968305, 0.336227506, -0.492103726, 0.332263976, 0.615848899, 0.692319274, 0.292124122, -0.340897322, -0.896990776, -0.522168338, -0.454930693, 0.771187186, 0.51408571, -0.381135941, 0.319291353, -0.396299392, 0.513851106, -0.321677834, 0.574206471, -0.627758503, -0.450472832, -0.567882717, 0.533085883, 0.608325303, 0.54108125, 0.502676308, 0.500716805, 0.3959122, -0.455117047, -0.604221284, 0.498871863, -0.535170317, 0.470866203, -0.514008045, -0.409502894, 0.541882992, -0.995882154, -0.554353237, 0.397705227, 0.650923967, -0.479975075, 0.766558826, 0.527585924, -0.485788852, 0.585933208, -0.496550322, -0.435983121, -0.588755131, 0.306980014, -0.35280174, 0.340765566, 0.731039464, -0.456854671, 0.609621465, -0.724508047, 1.21012235, -1.1626178, -0.268344313, 0.552504182, 0.840840757, -0.487748384, 0.356611967, -0.412433714, -0.318199605, -0.280455112, -0.598447025, 0.552642286, -0.0823746175, -0.368743777, -1.28527319, -0.125558391, 0.489598453, 0.92858988, 0.151855797, 0.207859918, -1.19165063, -0.0845686197, 0.159458771, -0.136885136, 0.23361814, -0.346603334, 0.107563451, -0.274093926, 0.782895505, 0.456464618, 0.669142663, -0.499088913, -0.683417022, -0.76996237, -0.231725663, -0.511193573, -0.276256144, 0.579197228, 0.73528856, -0.125234902, 0.245472834, -0.0668956712, 0.302175611, 0.464659721, -0.353863329, 0.513849616, 0.160740286, -0.232221365, -0.499522179, 0.851555467, -0.518513322, -0.0543271862, 0.597059727, -0.264653802, 0.029031517, 0.375719279, 0.989020646, -0.105796792, -0.0100124637, -0.340240657, -0.655018032, 0.930915117, -0.934472203, 0.782848477, -0.73290652, 0.581017554, 0.115213677, -0.563700259, -0.84416908, 1.03586972, -0.28631711, 0.613704264, 0.112773769, 0.601791799, 0.397840977, -0.45470351, -0.399902165, -0.342745692, -0.651657581, -0.426776886, 0.434126675, 0.630537808, 0.242508605, 0.21467042, -0.815545499, -0.372527987, 0.375150442, -0.308599353, 0.363367289, -0.217578188, 0.410380304, -0.37141639, 0.452133477, 0.385216027, 0.604691982, -0.455466539, -0.44274798, -0.602021873, -0.498366833, -0.378014654, -0.424305975, 0.526997805, 0.647332489, -0.364250004, 0.313919902, -0.208091632, 0.424899787, 0.462396145, -0.623451471, 0.455604434, 0.488979101, -0.260600299, -0.444555968, 0.543094218, -0.552497685, -0.423459947, 0.373722285, -0.39831695, 0.415886432, 0.350337267, 0.726949036, -0.263986647, 0.191010877, -0.465301007, -0.712843597, 0.666446149, -0.451596469, 0.763687015, -0.535221338, 0.709298611, 0.234257802, -0.370692283, -0.680726469, 0.717993498, -0.340359509, 0.606472075, 0.399768472, 0.614197791, 0.451405078, -0.487950206];
    recurrent_3_g : ARRAY[0..4095] OF REAL := [0.0437946171, 0.0356089249, 0.0603230521, -0.047727257, 0.0527745113, -0.0189226475, -0.0241641942, 0.0327949636, 0.0177599974, -0.0603852458, 0.0436201915, -0.0783402696, -0.0551882461, 0.0699121878, -0.0924036205, 0.0366497971, -0.0238315072, -0.00604448188, 0.0312895998, 0.0653170645, -0.0206472874, -0.00161674921, 0.136747956, -0.0611768775, 0.0407048985, -0.0706192032, -0.0110838432, 0.00552614965, -0.142643765, -0.0407231301, 0.0423699431, 0.00962346513, 0.0594425835, 0.0545211732, 0.081631884, -0.0662707612, 0.0716799945, 0.102387987, -0.0507300831, -0.0454611555, -0.000158276409, -0.0192562193, 0.0904988125, 0.0182701088, -0.0298902728, 0.0263758805, -0.114956796, 0.0309427306, -0.0314933062, 0.0783589929, -0.00715179555, 0.0234887991, 0.010805523, 0.140529901, 0.16488184, 0.0483169854, -0.118740082, -0.01462573, 0.0226182155, 0.100963861, 0.0138853434, -0.00705660135, -0.00206182431, -0.0792749226, -0.0148940068, 0.00602765102, -0.104199164, 0.0608550683, -0.0199380163, 0.050144691, 0.00877667032, 0.117468834, 0.0279638786, 0.0734397992, 0.0104080345, 0.0327590629, -0.102873877, 0.0137347775, -0.0160454288, -0.0478321053, -0.0793856457, -0.0851908699, -0.0456838571, -0.00442230422, -0.0483222157, -0.0110697336, 0.0691818371, 0.0551628917, 0.0461301282, 0.13791132, 0.0542764217, -0.0094403699, -0.0145909479, 0.0446228385, -0.0798043311, 0.0351968035, -0.00239900127, -0.0216923095, 0.0198777616, 0.0117041674, 0.0234491155, 0.0286384039, -0.0521193594, 0.147994921, -0.00586513057, -0.177775338, -0.0365150087, 0.0110691376, -0.107153893, -0.0682319626, -0.065542005, -0.0448637232, 0.049820751, 0.00115479529, -0.0050499998, 0.0331660323, 0.00934460573, 0.0182071663, 0.0295800325, -0.0609124899, 0.0178401917, -0.00110952184, 0.0541258082, 0.0991318226, -0.123389289, 0.0675796419, 0.0106140636, 0.0117992163, 0.0358371325, 0.026860375, -0.0437087417, 0.0830354989, 0.0910087898, -0.125799388, 0.0410022661, 0.0622523315, 0.0903293714, -0.020052718, 0.0990970209, -0.0561684892, 0.052668646, 0.0394487269, 0.00786635187, -0.0703451931, -0.16498898, 0.0851500556, 0.00694400165, -0.0826949626, 0.0243108328, -0.00454433076, -0.0468683913, 0.119009882, -0.123177044, -0.0138613358, 0.075883992, 0.00786806736, -0.0666241199, -0.0459856205, -0.184698358, -0.00130390562, 0.109424487, -0.0366346501, -0.0273824614, -0.0252181198, 0.0802295133, 0.0631064773, -0.0307271816, -0.0314257964, 0.0113007426, 0.0589789711, 0.0141819082, -0.0472304896, 0.0570724495, 0.0251741074, -0.0257351082, 0.0107673928, 0.0312493294, -0.0469326861, 0.00426948443, 0.0475220047, -0.0241182875, -0.0623387396, -0.0727202073, -0.0186802577, -0.0754899904, -0.015733581, -0.0207592733, -0.073164165, 0.0301877949, 0.0588661656, -0.0571453497, 0.0751569569, 0.0497234352, -0.0723318681, 0.10679587, 0.120137013, -0.00436050165, 0.0479413234, 0.0432624929, -0.017382456, -0.0119392565, 0.0874863118, 0.0779123306, -0.0820801929, 0.0308495313, 0.0483643897, 0.000151194632, 0.0132592842, -0.0532415919, 0.156844929, -0.0889991224, 0.0466540977, -0.00542534236, 0.052643165, 0.0944159999, -0.0841197595, 0.0489070415, 0.13224946, -0.0398661047, -0.00405186508, -0.0369656347, 0.0862073079, -0.0447398797, 0.0679130256, 0.00494718924, 0.00776614249, -0.0107311355, -0.00242555514, 0.0230813213, 0.112902462, 0.00745940581, -0.0547661372, -0.0408829004, -0.0865405202, -0.0188274235, 0.039733775, 0.0572599843, 0.0630219281, -0.0873965323, -0.0515896417, -0.0239288099, 0.0359626487, -0.0478699505, -0.0354774334, 0.0345449969, -0.121963739, -0.0157069825, -0.0204777457, 0.050551746, -0.0958625376, 0.0306946002, -0.00928554311, 0.0333284661, -0.0331369452, 0.00537282368, -0.0615441427, 0.0251101125, 0.000117624528, -0.0441348292, 0.0852627754, -0.142903864, 0.00483416952, -0.03087583, 0.11638502, -0.0100253616, 0.047723867, -0.088887237, 0.0330978818, 0.0326048173, -0.0474701859, 0.0313171484, -0.0164919831, -0.0664947629, -0.0222432278, 0.00963285659, 0.0122138774, 0.0797647089, -0.0517733544, -0.013356572, -0.0725202039, 0.0505522378, 0.0556567684, 0.0587954037, 0.0960235819, -0.018330384, 0.0348234773, -0.0270340387, 0.0644792169, -0.0591062456, 0.0521139726, -0.0150095671, -0.0127190668, -0.0711883381, 0.118938558, -0.0924677551, 0.0654087067, -0.0321329907, 0.000495560467, 0.021288326, 0.0482438281, 0.0321638435, 0.118991397, -0.0275172107, 0.043107938, -0.0112965489, 0.0265220366, 0.0333517343, -0.0251479745, -0.090136759, -0.08812996, -0.0158685707, -0.00131812692, -0.0162508562, 0.130799323, -0.131101459, -0.0359286293, 0.090195559, 0.0210224055, -0.0396175012, -0.0372376852, 0.0551964156, -0.0129464772, -0.0430404879, 0.00627431972, -0.0170405973, -0.051235117, 0.000174651272, 0.154698536, 0.028191451, 0.132395819, -0.0533527248, 0.0131867975, 0.116268821, -0.0110508706, -0.0617204681, -0.0537770241, -0.0189973228, -0.0177845135, -0.079368256, 0.0624092519, -0.156656563, -0.0685066655, -0.0819371194, -0.106309488, -0.0632021725, -0.00902509317, 0.104553789, -0.0124902353, 0.0336680412, 0.0348187499, -0.0835888088, 0.012579713, -0.0593955405, 0.0388434641, -0.0716860294, -0.0238554925, -0.0567766726, -0.0262237191, 0.0294644162, -0.0667560399, -0.0895431116, 0.0326211862, 0.106111214, 0.00555678084, 0.0310179908, 0.13451387, 0.0534371436, -0.0246243253, -0.114113376, -0.0370281786, -0.031641461, -0.0690283328, 0.0637342483, 0.00548026571, 0.0456839353, 0.012929339, 0.00080434233, -0.0783343017, 0.150892809, 0.0514784381, 0.0400711745, 0.0469036326, 0.0110388082, -0.0856724009, -0.161606595, -0.0264695883, 0.0206598118, 0.0175653882, 0.000188273843, -0.0173688307, 0.0498335361, -0.0430916734, 0.0238943584, 0.0332063362, 0.0169303417, 0.0244698878, -0.0920069665, 0.130756572, 0.0356508382, -0.0250255261, 0.0372642428, 0.0596290752, 0.130397707, 0.0624236278, 0.0770095065, -0.0595984049, 0.0839890838, 0.0480631627, 0.00205892883, 0.0400260799, 0.0854125619, -0.00825265795, 0.0601388887, -0.0207331721, 0.0845742598, 0.0588131547, 0.0327210799, -0.00686559826, -0.0743021667, 0.0396478847, 0.0202707425, -0.0367234275, 0.0350457281, -0.0431323051, 0.13371563, -0.0158024039, -0.119976334, -0.0317550935, -0.0251746066, -0.0534133017, 0.00945022795, -0.0602518767, 0.0540190041, -0.056983605, -0.0853763744, -0.0217396393, -0.00645941868, 0.0480292961, -0.118101686, 0.105877288, 0.016640082, 0.0146705657, 0.109670684, 0.0365797132, -0.05524607, -0.0345163681, -0.0551316664, -0.0256243218, 0.023326274, -0.00774309505, 0.0180745181, 0.0171112828, 0.0374728218, -0.0147281364, -0.0635587201, -0.0141743403, -0.00960662868, 0.0283385515, 0.0632124767, 0.0150674786, 0.0697335452, 0.0306217596, 0.0380299389, 0.0667182654, -0.0629971325, 0.0495261326, -0.00300480612, -0.0805550143, -0.038471438, -0.111067154, -0.0715867728, -0.0457849875, 0.172186196, -0.0997939631, -0.00552320667, 0.0930173025, 0.102501474, -0.0294463784, -0.0210591052, -0.0852635801, -0.0136373937, -0.0037564002, -0.0517212152, 0.0480001494, 0.0566151775, 0.0043565128, -0.0654382631, -0.0351467319, 0.0771682858, -0.0347881168, 0.042618379, 0.0587576069, 0.0292062052, -0.0258947276, -0.159660488, 0.0489060842, -0.018367704, 0.0105593121, -0.0294862911, -0.0171457306, -0.0400918163, -0.0324743837, 0.0031289123, 0.0610611439, 0.0781589001, -0.0922509432, 0.0229052138, 0.00348528847, -0.0473426692, 0.0523510277, -0.159925371, -0.0465800986, -0.0122167766, -0.141957864, -0.129894435, 0.0323161334, -0.0164559279, 0.0278466679, 0.0280659683, 0.103070319, -0.00847487338, 0.0279524438, 0.0639277697, -0.0317392014, 0.0852497295, -0.1059516, -0.0229070429, -0.00117459055, 0.0272169113, -0.0367145352, -0.0505845957, 0.000724893995, 0.047852166, -0.027406659, 0.0764742047, 0.0088911783, 0.0391752049, -0.0724412352, -0.0185030978, -0.0420969129, 0.052846171, 0.0419014767, 0.0729342401, -0.000822759932, 0.170634523, -0.0271994472, 0.196600974, 5.87867107e-05, -0.000332868658, 0.149793342, 0.0597085431, 0.0186867677, -0.0379116163, 0.0748567283, -0.0277350917, 0.0116728554, 0.0739852637, -0.127848178, 0.0326416269, -0.0604896434, -0.0738109052, -0.0144443847, 0.0316269845, -0.0584234297, -0.0265611038, 0.00339804962, -0.0695790052, 0.0347188041, 0.0253881328, 0.0141136907, 0.0628068075, 0.0825641975, 0.0321616828, 0.0247248765, -0.0157543868, 0.14644742, -0.0436226167, -0.0909949839, -0.0472625569, -0.0932573304, -0.0240172558, -0.00556543656, 0.0106262509, 0.0286489781, 0.0179347768, 0.0266251303, 0.096784018, -0.129549295, 0.0610996448, -0.0123506086, -0.0571338609, -0.0249893423, -0.0134870503, -0.0308243297, 0.0957151949, 0.114217326, 0.00636703894, -0.0221208446, -0.0188888833, -0.0924003273, -0.0725656375, 0.071031481, -0.0668210611, -0.0875139013, -0.0980054885, 0.0498619005, -0.0237564482, 0.00874692947, -0.0761414915, 0.0165116824, 0.0761271939, 0.0404123813, -0.0355446041, 0.0969976187, 0.0125186481, -0.030749321, -0.0255624391, -0.0528403372, -0.00695202872, -0.0742891133, -0.0610548705, -0.0334467143, 0.0159592722, 0.0100142546, -0.0294853207, 0.0551163591, 0.142635047, 0.0973949879, 0.0729607493, 0.0390121602, 0.0748167709, 0.0232498776, -0.0357143432, -0.0562612638, 0.0554807857, 0.0389705524, -0.0214845818, -0.00878978148, -0.079347454, -0.0323549211, -0.0884832144, -0.0644469857, -0.0392639711, -0.000336792786, -0.0540650077, 0.0109412167, 0.125446856, -0.0250293761, 0.0186739359, -0.0117511516, -0.0218843631, -0.00308746286, -0.0873689577, -0.00294509716, -0.141816035, 0.0173082575, 0.0648783594, 0.0891337991, 0.0881629139, -0.0388818868, -0.0232140925, 0.106614292, 0.112443253, -0.0189327225, 0.0219631847, -0.0715802386, -0.120316476, -0.0698842779, 0.0486293137, -0.0946422741, -0.0173603185, 0.0489539728, 0.0487572476, -0.135705695, -0.0360559896, -0.0279911906, -0.069363296, 0.0271106046, 0.0947534814, 0.0394816212, 0.072985746, -0.0139287785, -0.0752114803, 0.0410046317, 0.0383616909, -0.00506154727, 0.0967616886, 0.0770343095, 0.0543256104, 0.0633872002, 0.0736746565, -0.0112913623, 0.0688676909, -0.0473245084, -0.00795318186, -0.107369207, -0.0280095339, 0.0371930487, -0.000496821944, -0.034586072, 0.102976426, 0.00583893806, -0.0248779319, -0.0423515812, -0.0370051935, -0.0692012832, 0.0519177765, -0.0506054051, 0.0584365577, -0.00616674684, -0.163525388, -0.0298826657, 0.0515844822, -0.0106118005, 0.0375536233, -0.0850021318, 0.00840512291, 0.00965516455, -0.00963456556, -0.0331755243, -0.0101903621, -0.0672248453, -0.107034124, 0.0180644989, 0.00325294305, -0.0403223932, 0.0494849384, 0.0390063636, 0.100751936, 0.0426795334, -0.00151113793, -0.138964891, 0.0598751158, -0.0356394164, -0.141031131, -0.0873572081, -0.0435702503, 0.0296391472, -0.10683994, -0.0339005888, -3.21324915e-05, -0.0809328109, 0.0142500456, -0.062498305, 0.071800366, 0.0750214681, -0.0512118042, 0.070118323, 0.0925361514, 0.0134849921, 0.0534225926, -0.0853061154, 0.00885172002, 0.107762806, -0.0316386446, 0.0954414606, 0.0463188998, -0.00821089745, 0.0275785625, -0.0388389155, 0.0500948057, 0.0780036077, -0.0547428131, -0.000319614075, 0.0682679787, 0.166067064, -0.125245243, -0.0136718787, -0.0695996955, 0.0516639724, 0.0543026775, -0.0547133908, 0.017105151, -0.0922205895, 0.0209775716, -0.0707204491, 0.0399549976, -0.0995192155, -0.0084136501, -0.0942412093, -0.0410260521, 0.0820243508, 0.00997671857, -0.0268852543, 0.0573237389, -0.0136433821, 0.0293774568, -0.0858073756, -0.0918708295, -0.0321989432, -0.0552604236, -0.0387189165, 0.035827443, -0.0134981479, -0.0365950391, 0.138456702, 0.0899098143, -0.0215687752, -0.030826319, 0.00056686264, -0.0375713259, -0.0888281167, 0.0463074297, 0.0906105936, 0.0328093693, 0.00806281902, -0.0143647939, -0.0290142447, -0.128904045, 0.0432190374, 0.0413971022, 0.0102096684, 0.0145965451, 0.0203530248, 0.0213261396, -0.0929430202, -0.0385406688, 0.111956365, 0.072554715, 0.016495958, -0.0531439185, -0.0913725644, 0.0261270534, 0.0032450743, 0.103315681, 0.00636581564, 0.00297954958, 0.0518578663, -0.0598627739, -0.0019322671, 0.0304874051, 0.0135562597, -0.0974083766, 0.071473442, -0.00723022595, -0.0314555876, -0.00950273965, -0.04266458, 0.0446846038, 0.0513164736, 0.133749142, -0.0480514839, 0.063508369, 0.0181249008, -0.0350980461, 0.0370739549, 0.107270136, 0.0394912735, -0.00284807663, 0.0801917687, -0.104331933, 0.0578683242, 0.0624231696, 0.0903098658, -0.0134294704, -0.148465961, 0.0783245787, 0.0889386088, 0.0439603627, -0.0269809961, -0.0990409702, 0.0207240134, 0.0699846447, -0.0860875696, 0.0596522167, -0.176039472, 0.0454411097, -0.0113939233, 0.121883236, -0.0918860734, -0.0581154823, 0.0493174717, -0.0657394081, -0.0781332701, 0.0253242292, 0.115182795, 0.000212859362, -0.0260990784, -0.0301430412, -0.0608325116, 0.00667643175, 0.172523201, 0.0539123863, -0.133342639, 0.00103351474, 0.0458128788, -0.113308929, -0.104017951, -0.0218024086, 0.0538804606, 0.00108002499, 0.023010917, -0.00699742138, 0.0315718353, -0.126293331, -0.137346834, 0.0416493192, 0.0511883572, -0.00309673278, 0.0223449841, -0.0562600829, 0.0401032791, 0.0197832678, 0.0653053969, -0.0603515506, 0.0662093535, 0.0212488547, -0.0267507266, -0.00525549427, -0.0696200505, -0.0162829664, -0.000987504609, 0.0200190675, 0.0105028823, -0.0418067947, -0.00827357918, -0.0372207314, -0.108828753, 0.0437548086, 0.0150941126, -0.0137074897, 0.0154122002, -0.0506977923, -0.055614017, 0.0546899401, -0.0549833775, -0.0191186909, 0.0672337413, -0.0758709162, -0.0442107879, -0.0708327442, -0.0274153966, 0.0041588773, -0.0316219553, -0.0592753813, 0.0515885055, -0.0405231752, -0.039121788, 0.0517694727, -0.0545876324, -0.0308018252, 0.0907936916, -0.0495968014, -0.0555784591, -0.0687647611, -0.0486076102, -0.00530659221, -0.00447174488, 0.0680043995, -0.0821079835, -0.0332670212, 0.0555731244, -0.0779806301, 0.0515601635, -0.0351043716, -0.0787500739, 0.142117232, 0.0848803967, -0.041535344, -0.00458858721, -0.0887318626, 0.0253921691, -0.132499978, 0.0268349275, 0.121834077, -0.0276161917, 0.0237504281, 0.0597131103, 0.0353505239, -0.0747668967, 0.0314463936, 0.0379308388, 0.0526249707, 0.00122246426, 0.134960487, -0.0244314764, 0.0112246312, 0.0398989096, 0.0200127065, -0.139424801, -0.0749389082, -0.0684033334, -0.0303652063, -0.0969503298, 0.0607842468, -0.163150176, -0.0508852974, -0.0710474029, -0.0449129269, 0.0586251542, -0.096247822, 0.0372614935, -0.0776774362, 0.105325088, -0.0022131186, 0.00872825086, -0.0458002314, -0.0809246674, -0.0169954151, 0.111101709, 0.083675392, 0.02178872, 0.0552256182, -0.0480520763, 0.00167967752, -0.0283478163, 0.0972101912, -0.0557188392, -0.0293560829, -0.0151757039, -0.0568278804, -0.129950389, -0.0472627729, 0.0224157963, -0.103854284, -0.0244820174, -0.0232927725, -0.0488482602, 0.0975339711, 0.00959583372, 0.0167419314, -0.0765229836, 0.0571237989, 0.0981060565, 0.0187965352, 0.0275197197, 0.0153497206, -0.0164502952, 0.0781833529, -0.0640570819, -0.0223630294, -0.0512625873, 0.0948705524, -0.00737074623, -0.0406470597, 0.0855391696, 0.00104976445, -0.0489106365, 0.0386628583, -0.049393747, 0.0482431389, 0.128723338, -0.0799038112, -0.00600087643, 0.069760263, 0.0176393054, 0.0399047956, -0.136307523, 0.00941477809, 0.0291418005, 0.038658265, 0.018319685, 0.0535182096, 0.103093863, -0.105153397, -0.0332286134, 0.0923775136, -0.00476696622, -0.015503712, 0.0167125538, -0.105730057, 0.0423004404, 0.00941983983, -0.0161771607, 0.012389929, 0.0570268594, -0.00442304276, 0.0505149961, -0.0329311863, -0.0419432819, 0.0837120935, 0.0277116988, 0.0908375531, 0.0193081945, -0.00156955514, 0.0512244627, 0.0735181347, -0.153968588, -0.0451854579, 0.159297869, -0.0523338839, -0.0399141759, -0.00561910681, -0.0613095276, -0.0217277408, -0.0732570589, 0.0493326038, -0.0538512804, 0.141228542, -0.0702890605, 0.0273352452, -0.0610188022, -0.0434649028, 0.0250576101, -0.0102382116, -0.10538885, -0.156915814, -0.0500253588, 0.0375902019, 0.0501928851, -0.00860014558, -0.0792337209, -0.0436643362, -0.0800104141, -0.010623673, 0.0315528996, -0.0441206023, -0.0351912789, 0.0456732437, 0.0770347491, 0.068646051, 0.0309985131, -0.0264771022, 0.0136799794, 0.106181353, -0.101247281, 0.00716032647, -0.0408449396, -0.0535017066, -0.0051052738, 0.0946858674, 0.0242261644, -0.0390941948, -0.0625560358, 0.00658260658, -0.076573804, -0.0862258747, -0.0481125228, 0.0418758541, -0.00847311504, -0.00545511208, -0.0101117939, -0.00177318323, 0.0204412527, -0.00323768146, 0.0360398777, 0.00858668145, -0.0231021009, -0.0973089859, -0.00149125606, -0.0038880147, 0.0788744241, 0.0618985519, 0.0666652322, 0.2110921, 0.0674087927, 0.0564186759, -0.0712232739, -0.0317184143, -0.0590486154, -0.0132799931, 0.0294683054, -0.139294863, -0.00962675177, 0.0224994365, -0.00741684157, -0.0319934711, 0.0909804925, -0.0395711623, 0.0193202663, -0.0559785254, -0.0205036402, -0.019171726, -0.056551937, -0.0766943991, 0.0503951311, -0.0932497755, 0.0556321405, -0.0627518296, 0.0377981663, 0.0272609759, -0.104310051, 0.191026971, -0.0306752324, -0.0364861265, 0.00643242709, 0.0465070345, -0.142535791, -0.10215266, -0.194120646, -0.0375697426, 0.0995707512, 0.0109131085, -0.0108391717, 0.0271665007, -0.0635344833, 0.0248441957, -0.00897011533, 0.104523025, 0.040006049, -0.000857563689, -0.0264638551, -0.139202476, -0.0894379616, 0.0602872446, -0.0622471124, -0.00761811202, 0.0242898799, 0.046970021, 0.0349155627, -0.0676321983, -0.00321237277, 0.0724524632, 0.0545906723, 0.0993178934, 0.0166767687, 0.075340949, -0.0495018288, -0.0174664669, 0.0612922013, -0.083954975, 0.0417406894, -0.0289455056, 0.116475232, 0.00986072794, -0.038338203, -0.0991577953, 0.0278481692, 0.00784622598, 0.0222188458, 0.0747227669, -0.0709641278, 0.0544451959, 0.0255802348, 0.0384010524, 0.0719087645, -0.121760406, 0.00481382245, -0.000585127622, -0.135935485, 0.131211936, -0.0212898143, -0.100280263, 0.0234243162, 0.0385998935, -0.0521546677, 0.000743210316, -0.0485991612, 0.0633290112, 0.00902856141, -0.0536569618, -0.0259502549, -0.070486486, 0.0699209571, -0.0808160752, 0.0215099882, 0.0344036594, 0.0252323449, 0.113571994, -0.0237386972, 0.00102477893, -0.0636270344, -0.0479459763, 0.0595086254, 0.0212391801, 0.00761640444, -0.02714606, 0.125518873, -0.0605320223, -0.024817124, 0.0637853816, 0.0428128652, 0.0255031958, -0.0587189943, -0.0793529972, 0.0415715612, 0.0257545151, -0.03283263, 0.124993481, -0.0263969898, -0.0741453245, -0.142258525, 0.085048914, -0.0610307381, 0.0985249057, 0.0733609125, 0.124186732, -0.0451595187, 0.0245973989, 0.000429265201, -0.0152498158, 0.0265254863, -0.0166501552, 0.0820592195, -0.0544047058, -0.0366440862, -0.0184330624, -0.0064102374, -0.0554670207, 0.0298923515, -0.0218889229, 0.0658498853, 0.0132339271, 0.0137840025, -0.140885025, -0.0141397743, 0.101898417, -0.0621680319, 0.0623553656, -0.0405295193, 0.0477350689, 0.0925273001, -0.0547095165, 0.0178646371, -0.0165670179, -0.0690489188, -0.0857473761, -0.00542651583, 0.0364890173, -0.0502478592, 0.049791947, -0.0734185055, -0.0420475565, 0.0241549481, -0.0773289055, 0.0125149591, 0.0397351831, 0.0522903278, -0.149520159, 0.00103199854, -0.0288832635, 0.0365350395, -0.0788434967, 0.167386547, -0.053527493, -0.0972103924, -0.0274927318, -0.090696454, -0.0482012853, 0.0376947597, 0.0427852497, -0.0886414424, -0.022442041, -0.0300389715, -0.0246035717, 0.0559815913, -0.109197244, -0.123624139, 0.0855253935, -0.0205873251, -0.0521289706, 0.0506267324, -0.0276604183, -0.0260408148, -0.0194663163, -0.073949255, 0.0656063855, 0.0984442085, -0.0363203399, 0.00517521612, -0.0710335448, -0.100124128, 0.0446914211, -0.0244415887, -0.018025497, 0.0328585804, 0.00530130602, 0.0336090177, 0.0946201086, -0.0695398226, -0.00348007702, -0.0507431328, -0.0307467021, 0.00232117064, 0.00388779677, -0.0054759616, -0.0568126366, -0.0708990619, -0.0729758516, -0.0739225075, 0.0282083396, 0.0806478411, 0.0702341124, -0.0148573108, -0.00354283582, 0.141048834, 0.0648447871, -0.0209369324, 0.0628284216, 0.130696818, 0.0560673662, 0.0442488045, 0.110877894, 0.00242006779, 0.092648007, 0.0348521024, 0.0457123034, 0.0247226395, 0.150713116, -0.0591204129, 0.0159223545, 0.121485777, -0.0118759088, -0.0285220463, -0.142771378, -0.0510081872, -0.0845190585, 0.0647980347, -0.0218373518, 0.0133634191, 0.00249534845, -0.0972629488, -0.0427954309, 0.0626154095, -0.0368622132, 0.0474482886, -0.068202123, -0.0760832503, -0.0341768563, 0.00673387293, 0.0679354221, 0.055270575, -0.0451835059, 0.0363239571, 0.0502698347, 0.0347895473, -0.0702535734, 0.0685315281, -0.0720399022, 0.0283862576, -0.00326366536, -0.0221029334, 0.0623328909, 0.0263358131, 0.00373769365, -0.0535679832, -0.033660166, 0.0476006716, -0.0416463092, 0.0593384691, 0.0715817586, -0.102924123, -0.0700130984, -0.0813510939, 0.00335601438, 0.0687512308, -0.0356222466, 0.000196982175, 0.0343504511, 0.0293396767, -0.0721163005, -0.046208512, 0.0197926909, 0.0648469925, 0.0130615383, 2.45030969e-05, 0.0312840566, 0.0907965004, -0.103790373, 0.0603147969, -0.021862518, -0.0561037287, 0.0671753958, 0.0168595016, 0.0351376496, -0.0853875354, 0.0600750856, -0.0497095324, 0.0549683496, -0.0383790806, -0.0493463464, 0.0513246953, 0.0231574848, 0.144823939, 0.0106753595, -0.122087643, -0.0430514142, -0.0712743551, 0.0699730068, 0.033647038, 0.0390554629, -0.0669165626, -0.142801285, -0.0887139142, -0.090604879, -0.0405369438, -0.094409138, 0.00243717106, -0.0394747518, 0.0999782383, 0.0605793595, 0.00866577774, 0.151486427, 0.00252250768, -0.0707776099, -0.0278639309, 0.0627456903, -0.0253402889, 0.0949090198, 0.0137950182, 0.0522881374, 0.0801687166, -0.135862023, -0.099721998, 0.0482338406, -0.0161890853, -0.0260213986, 0.133775517, -0.0883678794, 0.0320810154, 0.0457535759, 0.0321318246, -0.0374644287, 0.0290767401, 0.106415644, -0.0282021873, -0.0931792483, -0.0204625074, -0.0141848698, 0.128663749, -0.0187942162, -0.0817958862, -0.00397646427, 0.013728112, -0.0369062759, 0.0798454732, -0.0521001816, 0.000768011436, -0.0146153392, -0.19150342, 0.00350939482, -0.0477405153, 0.0111964084, -0.054836046, -0.020611167, -0.0394426696, -0.00418617483, -0.0509541184, -0.0776007622, 0.0714660585, -0.0822863728, -0.00419231132, -0.11209897, 0.165123612, 0.0628670454, 0.0720339343, -0.055249542, 0.0142350784, -0.000623517553, 0.0416886806, 0.0718994364, -0.0426993072, -0.0128279617, 0.0078166509, -0.0851455182, 0.107675701, 0.0461743027, 0.0567564219, 0.0580719374, 0.046490714, 0.0280795991, -0.0102832951, 0.00057309214, 0.0537007079, 0.0306451935, 0.00600591348, 0.0439060591, -0.0219222531, 0.053899698, 0.139480621, 0.0100344419, 0.0554072373, 0.0904727131, 0.0399847664, 0.00795942172, -0.00132137607, 0.034675885, -0.0730519071, -0.0352918729, 0.00681896321, 0.0363368392, 0.015803175, -0.0659515709, 0.0792124718, 0.0414071083, 0.0187042244, -0.078536883, -0.147206619, 0.0138750505, -0.0551111251, -0.0819048882, 0.094347246, 0.0334293395, -0.072604306, -0.0268384926, -0.0780775324, -0.100536868, -0.0181026869, 0.0574925616, 0.0317317061, -0.0599300638, -0.0922840089, 0.0240945481, -0.0227659624, -0.0538291372, -0.0015925481, -0.0168934315, 0.00094248727, -0.10671404, -0.0244659185, -0.0720363706, 0.0417134613, 0.0163070504, 0.00145395077, -0.0409966148, -0.0131505886, 0.0447876006, -0.0347378813, 0.00917446241, 0.0464757346, 0.090196386, -0.0873175934, -0.0105880387, -0.0714944825, -0.073655732, -0.100576505, -0.0413407125, 0.0515581518, -0.0570369922, 0.0754417479, 0.0129967798, 0.0407805704, -0.0517806783, -0.0111719631, 0.0206973609, 0.102774009, -0.0296073705, 0.0436041653, -0.0436578318, 0.0331462622, 0.0696561262, 0.0633508563, -0.0269959196, 0.0560168959, -0.0204678625, -0.0105428472, 0.000873768702, -0.0737785473, 0.00165817142, 0.103466406, 0.0452754237, 0.135777235, 0.0421848744, 0.0108114081, -0.0517719164, 0.0458985604, -0.107405782, -0.0433868989, 0.0601125881, 0.0141843874, 0.116243437, 0.0124012493, 0.0429210663, 0.143503532, 0.0188111514, 0.0729792938, -0.0132237189, 0.0451103523, 0.0768657923, 0.0932494551, -0.0361936502, 0.0410550237, 0.0626893789, 0.104756847, 0.0675333366, -0.0214108061, 0.0146081541, 0.00682398677, -0.184808701, 0.000971930102, -0.139394328, 0.0386681147, -0.0291126892, -0.0752831846, -0.064819701, -0.00680194981, 0.0139545994, -0.125681713, -0.0722900182, 0.0462356061, -0.00403481536, 0.1265627, -0.0249409229, 0.0217421856, -0.0497171357, 0.0663138777, 0.00784896221, 0.0243969224, -0.0133483764, -0.00118255941, 0.0374216661, 0.00596168265, -0.0497410558, 0.0533350334, 0.00643436285, -0.0244669765, 0.082441777, -0.00629646005, -0.074900955, -0.0630012751, -0.00968787819, -0.0976695642, -0.0704948306, -0.0360274687, 0.000799583271, -0.0431389697, -0.00170373544, 0.0448879451, -0.00148361549, 0.041238077, 0.0212126318, -0.0162574016, -0.0226290226, 0.100230105, -0.0183195584, 0.0644439459, 0.0140053127, -0.0192868691, -0.00844751857, -0.0207381658, 0.00976939872, -0.01147871, 0.0127085727, -0.0451914221, -0.0628271252, 0.0789558515, -0.0472965129, 0.0631449744, 0.00230306224, -0.0105378479, 0.0496447049, -0.0845899135, -0.037281774, 0.0284127202, -0.0275899787, -0.00769925211, -0.0490412638, -0.0175798703, -0.0174107552, 0.000279257074, -0.0547183007, -0.0793882683, 0.073726967, 0.00389581756, 0.0021273694, -0.100327522, 0.0442019515, 0.0743178725, -0.0317084976, 0.0326897204, 0.0196805485, -0.0343016721, 0.0856743306, -0.0585709959, -0.0663912892, -0.0728461668, 0.102971382, 0.067562446, -0.0714981109, -0.0220408849, 0.0162682533, 0.0014283543, -0.0249595884, 0.00233403407, 0.014955312, -0.101020649, 0.0143048419, -0.0836860538, -0.0047298409, 0.0233665742, 0.00511474768, -0.0967540666, -0.00166017143, 0.00208768435, -0.064734444, 0.115568392, 0.0485841781, -0.0555278324, 0.0548014641, 0.0650715753, 0.00909797102, -0.0709947795, 0.0871347338, 0.0659923404, 0.0780614242, -0.039166104, 0.0549587905, 0.0337862782, -0.0225313343, -0.0279758964, -0.0510044694, -0.0279935114, -0.0108422348, -0.0277980529, -0.0805196762, -0.0508307926, 0.0516238324, 0.087843731, -0.0512280837, -0.127194941, 0.0325051807, -0.0624534748, -0.0666571483, -0.00466810027, 0.00552304182, -0.0307798721, 0.0522661172, 0.0429992154, 0.0172167644, -0.0307729468, -0.00634042546, 0.104772612, 0.0692303255, 0.0452383049, -0.0464258827, 0.0437597558, 0.0202586707, 0.0266393237, 0.0373419672, 0.0305527691, -0.0502583869, 0.0169429891, -0.0472056679, 0.125663429, -0.00132889021, -0.0609000959, -0.0721376017, -0.0122957211, -0.0904405266, 0.114251956, 0.0261210557, -0.0109617058, 0.0528109595, 0.0850625336, -0.0787649825, 0.0203561224, -0.0762541518, 0.0469586998, -0.124386266, -0.0650305003, 0.0318567194, 0.0884649009, -0.0395232216, 0.00912176259, -0.00156698935, -0.0237864926, 0.0628394112, -0.0310049783, 0.145956889, -0.180878565, -0.0932578295, 0.0530016609, 0.0197299588, 0.0327863991, -0.0185660832, -0.0288810134, -0.0991030261, 0.0312827453, 0.0646031499, 0.0909827799, 0.021856159, 0.0632118508, 0.0284301713, 0.0398473777, -0.0264934339, -0.0446981937, 0.0158659667, 0.0283399075, -0.037050534, -0.0483466461, -0.0210409537, 0.0471282862, 0.0197772644, 0.0697801635, -0.0211002231, 0.0741760209, -0.0962772518, 0.132653832, 0.0807051063, -0.129630685, 0.0134090241, 0.0773689225, 0.0872647911, 0.0290719457, 0.051416669, -0.0403712988, -0.0461892113, 0.0585625395, 0.104173683, -0.116810843, -0.0399346314, 0.0956466421, -0.0116801169, -0.0489421189, 0.0770190135, 0.0214442611, -0.00871430337, 0.0975948423, 0.0567379706, -0.0255699027, -0.0113099217, -0.0360292867, 0.0156615302, 0.0483391322, -0.0122865429, -0.0974645466, 0.0352514535, 0.0364700928, -0.00654026866, 0.0264619142, 0.0518023297, -0.0511320457, -0.107179612, -0.0546540543, -0.0425088033, -0.0400190055, 0.0379188731, 0.028835481, 0.110043764, -0.118229181, 0.132413253, -0.0260019638, -0.00179817993, -0.0718525127, 0.0525665507, -0.0688994676, -0.109416455, 0.0218855906, 0.0209810734, 0.0362401195, 0.0370858535, -0.0306485593, 0.0218540076, 0.0857129171, 0.00725148804, 0.106594212, 0.0666264892, -0.0932988375, 0.0983042642, 0.0261039287, 0.0814470202, -0.0939739123, 0.00537273055, -0.0733297691, -0.00407380983, -0.0868249834, -0.0615938157, 0.00309805223, -0.0696139708, -0.0386956148, -0.0845719576, -0.0120726656, 0.0433476195, -0.069937177, -0.0525638983, -0.0689182207, -0.0235140957, -0.0142088626, -0.103356443, 0.130989671, 0.0602310523, -0.118296012, 0.112171404, -0.096265316, 0.0574163646, 0.0342530943, -0.0384196267, -0.0522846505, 0.0136580449, -0.0331682488, -0.00488113426, 0.0158302635, 0.065959923, -0.0713930801, -0.00882580504, 0.0457118526, 0.0114411172, 0.051590018, 0.0216312446, 0.00814935565, 0.00165256113, -0.0923497006, 0.0677519664, -0.0764443278, 0.0237499196, 0.0364104323, -0.107571043, 0.0143316826, 0.0849279463, 0.127444774, 0.0533001982, 0.0706099123, 0.00492518814, 0.0281565841, 0.0331864581, 0.0118441675, -0.0509792343, 0.0117349327, 0.0745007619, 0.0129846651, 0.0637511164, -0.0261296742, 0.0869919807, -0.00305290497, -0.00747031532, 0.0584041737, 0.0427736603, 0.0565930679, -0.0409131944, -5.24949282e-05, -0.0613957644, -0.115305781, 0.0029191887, -0.192310482, 0.0606861934, 0.0714496523, 0.0175157879, -0.00142147206, 0.0995120183, -0.0232723281, 0.0598310307, -0.0720922351, 0.0347911343, -0.0151916109, 0.00969898328, 0.0675180778, 0.0386909284, -0.0762500167, -0.0604409277, -0.0242063254, -0.00873011537, -0.0973661318, -0.071706824, 0.0965816528, -0.014882125, -0.0498527735, -0.000836196356, -0.101627484, -0.0195913967, 0.0240739845, -0.0423791073, 0.0609532706, 0.0327545479, -0.0525795519, -0.00975584239, 0.0466445349, -0.0127064232, -0.127163246, -0.0500615165, -0.175369546, 0.0732934475, 0.0926145688, -0.00979442708, -0.0385508053, -0.0402889065, 0.0624731071, 0.109680936, -0.0551848784, -0.0393319018, -0.0126019623, 0.15673244, 0.0938641503, 0.0176030211, -0.00406331755, 0.0399236791, 0.0672533512, -0.097016409, 0.0942300856, -0.00518544484, 0.0406865925, 0.0361760184, -0.00501667056, -0.0490368716, -0.0705912039, -0.0268043913, -0.0248467419, 0.0241681952, 0.0266908891, 0.0714592189, 0.118875682, -0.113458589, -0.010585146, -0.0540569797, 0.111083098, 0.0573106967, 0.041275356, -0.0378045216, -0.0253973324, -0.0294718668, 0.03418421, -0.0233394913, -0.0810486823, -0.00492007378, 0.0166646875, -0.0905492753, 0.0722334906, 0.0518001951, -0.0232825167, -0.0632262677, -0.0325615406, 0.00574617088, -0.106573209, -0.0353691578, -0.056216646, -0.00598251633, 0.058860749, 0.0410870649, 0.00477697235, -0.0403814539, 0.0765264407, 0.0781923607, 0.00636186078, -0.0794806704, 0.0306790229, -0.0729174614, 0.107677236, -0.0641774014, 0.0832683668, 0.0429744795, 0.014143426, 0.00199605944, 0.0352672562, -0.0266628619, -0.0777618662, 0.00522227585, -0.00872307271, 0.0299021732, -0.0692151785, 0.0714731663, 0.00498901587, -0.00988451764, 0.046215333, 0.0865805596, -0.0413954109, 0.0942449123, 0.0229305271, 0.178092733, -0.0119531453, -0.0209411364, -0.0396620631, -0.162027255, 0.0692444965, -0.0287034065, 0.0743346512, -0.0933155268, -0.078818053, 0.015656963, -0.057860747, 0.0272766128, -0.010528543, -0.0427199826, -0.115701452, 0.0226454455, 0.0340868011, -0.00896725617, -0.102600589, -0.0168602169, 0.0379630961, -0.0265942067, -0.00583999231, -0.0536883473, -0.0228712708, -0.0569861345, -0.0202108286, 0.0512893759, 0.0235828571, -0.090308398, -0.00875595212, 0.0364642069, -0.00624114182, 0.100476727, -0.0275988206, 0.0177504029, 0.0677875951, -0.0312764123, 0.0255969185, -0.0475961789, -0.0893026814, 0.102229014, 0.0318019092, -0.0880804881, -0.0341381207, -0.0775652826, 0.109055713, 0.0389091298, -0.00721085491, -0.133825496, 0.0292821452, -0.0490448475, -0.0279632192, -0.0538782924, 0.0549394563, 0.0116169024, 0.0506189093, 0.0241269004, 0.0205132738, -0.0110282889, -0.118196547, -0.0879877955, 0.0980909169, 0.0125246141, 0.0132735148, 0.00421023276, 0.00766414404, 0.0230970271, -0.016962789, -0.0133748781, 0.0148830432, 0.0139891095, -0.0416689701, 0.0671331808, -0.0416659638, 0.00626912434, -0.0716214105, -0.0256802849, 0.154157624, 0.0246896371, 0.170036525, 0.110943325, 0.0153374225, -0.0427210554, 0.00444331393, 0.0567055121, 0.045100946, 0.0431459695, -0.0686186925, 0.0263333209, -0.0364395976, 0.0205337666, -0.0805044472, 0.0895597786, -0.0163414143, 0.0716475397, -0.021895051, 0.0231063385, 0.0609122664, 0.0702821016, 0.0887054205, -0.0207948647, -0.0262887571, -0.0318973549, 0.0220195111, -0.0431260243, 0.0272719078, -0.00729568396, -0.0468490347, 0.0241231918, -0.00332220132, 0.0665162802, -0.00979762338, 0.00268718414, 0.0270736963, -0.0263445787, -0.0462097898, 0.0983998477, 0.142941073, -0.0173285939, -0.0187439974, 0.0384108536, -0.000604720786, -0.00764884241, 0.0493435785, 0.0361661911, -0.102939367, 0.0348074585, 0.0186017789, 0.0890035033, -0.0620062053, -0.123102114, 0.0189398136, 0.0322313532, -0.0880542323, 0.0226614214, -0.0179917049, -0.00357672945, -0.137373656, 0.0560070612, 0.0145020261, 0.014131885, 0.0080353152, 0.115074217, -0.0704478845, -0.0678179115, 0.0297717992, 0.0139532229, -0.0182477962, 0.0286403485, -0.0381069183, 0.0565833561, -0.0521315522, 0.117785603, -0.06498041, -0.0302871168, -0.0244761445, 0.0804481953, -0.0470589288, 0.053675659, -0.000120382989, 0.0443907082, -0.00708061643, -0.00847005472, 0.0579286963, 0.0204689633, 0.0334026441, 0.00568646425, -0.0196375214, -0.0472955704, -0.00667147012, -0.0108636962, -0.0977132767, 0.084812507, 0.0454593971, 0.058382187, 0.00400101626, 0.00271226792, -0.0359828435, 0.0340488367, 0.00440640887, -0.0531270541, -0.124580257, -0.0619477555, -0.0151804052, 0.07764218, -0.0315744057, 0.0791214705, 0.0357466936, -0.0193881635, -0.0780572444, -0.0151949544, 0.0288224891, -0.0171508677, 0.0507715307, -0.0347277448, 0.0392509252, 0.029503759, -0.0230431929, -0.0235765222, -0.0273565724, 0.0994564667, 0.154242977, 0.104842618, 0.01064061, -0.0653373227, 0.0158497728, 0.0982126072, -0.0323495418, 0.0412263945, -0.0274225194, 0.00928175822, -0.0700863823, -0.0126185548, -0.0481140427, -0.110683724, 0.00204109075, -0.0346254632, -0.0557617471, -0.0449180901, -0.0185930319, -0.0487626866, -0.0261884034, 0.000402662903, 0.00724694878, 0.00715393014, 0.0157046467, 0.00747553445, 0.175108254, 0.00763161853, -0.0284311641, -0.00659791939, -0.00911832694, 0.189467505, -0.0138703454, 0.0498847142, 0.0456825048, 0.0100442879, 0.000860460394, 0.0190563016, 0.00465693232, 0.0689635128, 0.121737257, 0.072102204, -0.0167927817, -0.106841668, 0.0721223429, -0.0485170111, 0.0310632214, 0.107406653, -0.0670796335, -0.0776340291, -0.000516461208, 0.0275814347, 0.0219014846, 0.113322169, -0.00862146914, 0.0119417608, 0.0405449569, -0.083949402, 0.0824499503, -0.0888166726, 0.0796885192, 0.00595818087, 0.0163861047, -0.0162338875, -0.0160393417, -0.051034946, -0.0172632523, 0.031616468, -0.0387321189, -0.0550529212, 0.0404613987, -0.0506636351, 0.0261437744, 0.140823364, -0.0181520749, 0.0682502836, -0.0272460841, 0.0573712811, -0.0531866513, -0.0507071242, -0.140722081, -0.0486198626, -0.0313069746, 0.0318313166, 0.0030388087, -0.0904056728, 0.0770314634, -0.0629537031, 0.144287646, -0.0777157992, -0.0206424855, -0.0746879056, -0.00726333167, 0.04891105, 0.00108227378, -0.0597574525, 0.0997128189, -0.105341837, 0.0839004889, 0.0156475604, -0.0974263325, 0.0926717743, -0.0496987775, 0.00667825527, 0.0774569958, 0.0248641334, -0.0287548527, 0.0251867939, 0.0682732463, 0.056832023, -0.14815712, -0.152774483, -0.00806592591, -0.0812081471, 0.0657070056, -0.0158116817, 0.0562619343, 0.0382694714, 0.014002772, -0.0730709657, 0.0390523523, -0.0153085552, 0.0152415093, -0.104275167, 0.0160007104, 0.0384664349, 0.0399441868, 0.029574398, -0.0846777856, 0.00428233342, 0.0539140329, -0.104484819, 4.73223627e-05, 0.0130600445, -0.0288190208, -0.101809412, -0.167075172, 0.0589084849, 0.0624491945, 0.00359798223, -0.0976154506, 0.0226364322, 0.0280424114, 0.0279548801, 0.0672514811, 0.00151229091, 0.112621374, -0.148344576, -0.0609819666, -0.0942541063, -0.0045774444, 0.108871028, -0.0157754738, 0.0239076316, 0.0926381499, 0.0407576486, -0.0546267778, 0.00330870738, 0.0594512895, 0.0391017087, 0.100008741, 0.0229085963, 0.0144934468, 0.129886657, 0.138421834, 0.202237085, -0.0488092899, -0.106104404, -0.127182171, 0.140045702, 0.0195568651, -0.042009484, 0.0023471443, -0.0124771129, -0.0525485054, -0.0321902111, -0.0598530322, -0.0238469355, 0.0105025843, 0.105921045, -0.040500097, -0.104203798, -0.123370424, -0.00493984763, -0.0520417728, 0.135451317, 0.0797963291, 0.0345563665, -0.0304996558, -0.0236270837, 0.00763001479, 0.0268944819, -0.0393782593, 0.0173147637, -0.119337618, 0.0287307538, 0.0204598997, -0.0249669515, -0.0166518576, -0.110001728, 0.1414489, -0.0243376717, 0.037391603, 0.026425831, 0.0210525542, 0.0763184428, 0.00978232361, -0.0696094781, -0.0116163269, -0.0441209674, 0.00933783688, -0.0344432257, -0.0348093845, 0.0585200451, 0.0546467565, -0.0746126324, 0.0792612135, -0.0579427816, -0.0362479016, -0.0722054243, 0.0175139569, -0.0634530708, 0.0731814951, 0.0826667249, 0.0390245728, -0.0406836458, -0.0573929474, -0.0556985624, 0.0221883394, 0.0792178512, -0.0473814979, -0.0501485467, 0.0223699566, -0.0150356572, -0.0356437825, -0.097396858, -0.0324046537, -0.0381281227, -0.0639146939, -0.0311654508, -0.0273824278, -0.00857670978, -0.0172075648, -0.0535460226, 0.0413416438, 0.052817151, 0.00622142479, -0.0135286078, 0.0564800166, 0.155078873, -0.0140154464, 0.0965329483, 0.0188998114, 0.0855375379, -0.0237015449, -0.0114426389, 0.00449711643, -0.101439632, -0.0201820228, 0.101011068, -0.0459432714, -0.0814798102, -0.059483178, -0.0981562585, -0.016080277, 0.0917451754, -0.0211254191, 0.0458478481, 0.0196815468, -0.0430021584, -0.0124979597, 0.0597104803, 0.0379433818, -0.0129831508, -0.0704780668, -0.035309501, -0.106383897, -0.113434687, 0.0720949173, 0.142024264, 0.0482250713, 0.0869400203, 0.024321977, -0.0513647273, -0.061458651, 0.0312121026, -0.0836775452, -0.0357919298, -0.0385029055, 0.00472303713, 0.0281314719, 0.0530263931, -0.0338873267, -0.0686981305, 0.0673258677, 0.0663697794, 0.0220062099, -0.0857022926, -0.0279790089, 0.0347468518, 0.121966712, -0.0903875604, -0.00051197689, 0.083435744, -0.098616302, -0.0455025621, 0.0710037202, 0.049734354, -0.0277393311, -0.074851498, -0.127413362, -0.0393713079, 0.0638672113, 0.0972380638, 0.0782679617, 0.0282186829, 0.0307427626, -0.125974193, -0.0156838764, 0.03603293, 0.0354317278, -0.0520452783, -0.030842822, -0.127955064, -0.0206850488, 0.0801726803, -0.0711221546, 0.0466404818, 0.00843494479, -0.102944702, 0.111014113, -0.0138135571, -0.0288607311, 0.15750353, 0.0950316116, 0.0253728963, -0.0476113297, -0.0766708553, 0.0188851319, 0.0623863451, 0.0779190287, -0.0145162176, 0.077103287, 0.0321669355, 0.0419032648, 0.0290212743, -0.0358486883, 0.0410093255, -0.020871412, -0.0874204263, -0.0103911841, -0.0230735075, -0.0871427506, -0.0251351949, 0.109724522, 0.046122767, 0.15514186, -0.0875300467, 0.0916077495, 0.00663397741, -0.0366500989, 0.0436698422, -0.0243947916, -0.00254984992, 0.0115132378, -0.115491979, 0.00776752084, -0.162884951, -0.0681987256, 0.115944222, -0.0134022869, -0.0295315348, 0.0199481957, -0.0817723796, -0.0848150402, -0.022584198, 0.0720470995, 0.0935427025, 0.0242063813, 0.0491375923, -0.0667804927, 0.0553878173, 0.0513403639, -0.0871435106, -0.0125644505, 0.136929899, -0.0185936913, 0.0357742272, 0.0745036602, -0.0637116134, -0.000253515784, -0.00456688181, -0.0888854563, -0.00787032209, -0.0653275475, -0.0470996276, 0.0401108973, 0.0293646026, 0.0269251727, 0.0218654945, -0.00038456358, -0.0814960003, 0.12124972, -0.139008224, -0.0902290195, -0.0852909461, -0.0579606593, -0.0611784011, -0.0354469717, 0.00831349008, -0.0428700298, -0.0286098439, 0.0049347654, -0.00185555394, 0.0018765874, 0.0950348601, -0.136039987, 0.103304163, -0.051251702, 0.0291565079, 0.0170655232, -0.00371781224, -0.00404358096, -0.0361152366, -0.0748850927, -0.00313647278, -0.0121474154, -0.048149433, 0.00205307128, -0.139730215, -0.025061287, 0.00728390552, 0.0600511432, 0.125428885, -0.0214866064, 0.110261917, 0.0415897071, 0.0657242015, 0.0332009569, 0.086841099, 0.00965492055, -0.0103395563, -0.0934640467, -0.075351581, -0.117179863, -0.0697006583, 0.0560305603, 0.0395296887, -0.0951981768, -0.00094571407, 0.0486060679, -0.0205072798, -0.0520721301, -0.0566285402, -0.0093741538, -0.0825339407, -0.014649719, -0.0127280708, -0.0585734844, 0.0695354715, -0.0239905361, -0.0615869351, 0.0710724816, 0.0403406955, 0.117892355, -0.0467934944, -0.0536303706, -0.0917998999, 0.00857593864, -0.0600094125, -0.00587335974, -0.0639679655, 0.109467648, -0.0736873373, 0.00173493661, 0.0803547874, -0.0180815551, 0.152160585, 0.00586829102, 0.00685735513, 0.0161523987, 0.00273610884, 0.0928805172, 0.0172556099, -0.0594666079, 0.140449777, 0.0452360436, 0.09790048, -0.0426957905, 0.00118520786, -0.0630539656, -0.010144094, -0.0550332516, -0.00452411361, 0.00447760802, 0.0285070017, 0.0143113295, 0.0327335373, 0.0203294139, -0.00945917889, -0.0666053593, -0.0397759154, -0.0957391709, -0.0381244794, 0.0531936213, 0.101422444, -0.0250406899, -0.0865593404, 0.083240658, -0.0642483607, -0.0289912075, -0.0546493232, -0.0989327952, 0.0289384127, 0.0893297195, 0.0185334608, -0.090652369, -0.15490438, 0.0216342956, -0.0248842537, 0.0648047775, 0.00288182031, -0.00312125077, 0.0448402353, 0.0197437573, -0.0275688525, 0.0364223942, -0.0666818842, -0.065710187, 0.107973948, -0.0360418744, -0.136318251, 0.0900088623, -0.0150246825, -0.0776477754, -0.0301514305, 0.0682968497, -0.0421132743, -0.0105228536, 0.11666584, -0.0176557209, 0.0285506602, 0.000275290397, -0.0390105769, -0.0915179849, -0.00695179636, 0.0226125512, 0.0689990893, 0.0236087814, 0.00152092613, 0.0360011458, -0.0115603423, -0.0711627081, -0.0399818122, 0.0289487019, 0.0469247214, -0.0928768516, 0.0597802624, 0.043441426, -0.0224812459, 0.0153060146, 0.141000524, 0.0847784281, -0.0554950535, 0.0218526982, 0.0127653889, 0.00524556637, -0.0266199168, 0.0704327375, 0.0428918302, 0.0520454049, -0.00144251995, 0.0293037407, -0.037911512, 0.0666712821, 0.126513213, -0.0661098436, 0.00601828657, 0.0332474075, -0.0853715315, -0.0421932414, 0.0378726721, 0.0251711383, 0.0215205625, 0.12652427, 0.0584723763, 0.168696269, 0.147201896, -0.123411678, 0.0225127097, 0.0350973755, -0.0734753385, -0.0269031078, -0.05928424, 0.109620102, 0.0696091205, 0.0246586911, 0.0349624977, -0.00974949077, -0.0736110285, -0.0833904222, 0.0745322704, -0.0584283061, -0.00409571873, -0.0644469261, -0.0186214987, 0.0604012795, -0.0130289616, -0.0658816844, -0.167622387, 0.0468659028, -0.00255789887, 0.0180664584, -0.00309908763, 0.0660267174, 0.0262318868, 0.0333178416, -0.0863818675, 0.00206708349, -0.0449012071, 0.00837402791, 0.0975734591, -0.0319099054, -0.092674911, -0.0375814177, 0.0536681339, -0.0336510614, -0.0316907503, 0.00489718001, 0.172486976, 0.0984627604, 0.0162389502, -0.0759479403, 0.137941867, 0.0564778, -0.186370775, -0.145751894, 0.0268903412, -0.00823681988, -0.0767542943, -0.0105237737, -0.0458372831, 0.0584962256, -0.0454248786, -0.0303541441, 0.107962802, 0.0026203189, 0.116626881, -0.0379451402, -0.0913221836, -0.000347240828, 0.0683971345, -0.0513534993, 0.0227791574, 0.0186891872, -0.113208465, -0.0286537167, -0.0135107599, 0.0741883293, -0.0418629572, 0.0141527243, -0.111806907, -0.0225812737, -0.00333454553, 0.0087531656, 0.02541456, -0.0806892142, -0.0795634165, 0.0417286679, 0.0073676724, 0.0754420459, -8.69674841e-06, 0.0618547387, 0.116478667, 0.124463335, -0.0539749488, -0.0723885, -0.0410638526, 0.0832498595, 0.0991948768, -0.0411506481, -0.053838972, -0.126852006, -0.0704327971, -0.00975695997, -0.134048343, -0.0205160789, -0.00728553068, 0.0248512998, -0.0572459772, 0.0241649915, 0.0394840166, -0.0294689443, -0.0130902128, -0.0307996403, -0.0439605713, -0.0165045951, -0.0589099377, -0.0384153016, 0.049819842, -0.0804864466, 0.0400228947, -0.0583529174, 0.0382517129, -0.018521592, 0.0323187038, 0.0170512833, -0.069307521, 0.0128049441, 0.0420619473, 0.13756758, 0.148205727, -0.0125464173, -0.00821778178, -0.013742133, -0.0136860721, 0.00903412234, 0.000459158095, -0.00412421022, -0.0837509707, -0.0286138654, -0.0843880624, -0.018315535, 0.0310477465, -0.0153143387, 0.0975566059, 0.0831105858, 0.00831545424, 0.101737715, -0.0765080005, 0.0601868257, 0.0491592735, 0.0567918234, 0.03369404, 0.00878577773, -0.0287505332, 0.0522962511, -0.0721106157, 0.0456669852, -0.0848702416, -0.0543546528, -0.118371673, 0.0458883382, 0.0382733978, -0.0653831437, 0.0139406342, -0.135031193, -0.018430613, -0.00310835498, -0.0302646365, 0.0553676635, 0.0249326266, -0.0488271713, -0.0833251625, 0.16396299, -0.0709491596, -0.0897723213, -0.0411927961, -0.00261087855, 0.139643729, 0.0499558002, 0.00537344441, -0.0298536941, 0.0134182097, -0.0773302764, -0.00185759016, 0.0069890134, -0.0675218105, 0.01860434, 0.00779228937, -0.0381149501, 0.0593951941, -0.0191692039, 0.00991781522, -0.0443587713, -0.042884402, -0.0669235662, -0.0343478806, 0.0107349874, -0.00460115913, 0.0558882095, -0.051443398, -0.0375989228, 0.0252242703, -0.0192703307, 0.00528108981, -0.119038127, -0.0258288756, -0.0187699273, -0.107284747, 0.0263836943, 0.0469239056, -0.0584763102, 0.0482227355, 0.115086578, 0.0244016424, 0.126681373, 0.0803363249, 0.0779946595, 0.0199340861, 0.056405127, 0.0255166739, -0.11494597, 0.0363894776, -0.00947960466, -0.0123206228, -0.0499268174, -0.030287439, 0.0794981346, 0.0401173271, -0.0196512267, 0.0891385972, -0.00637649931, -0.0235760808, 0.0618417189, -0.089240104, -0.0106881671, 0.097762309, -0.0233596209, -0.0252768584, -0.0341228433, 0.0590369478, 0.0705460683, 0.0662270188, -0.0589481853, 0.102004878, 0.0481266901, -0.0075664483, 0.105016321, 0.0387468785, 0.0399596393, 0.0248953514, -0.114118606, -0.0362095013, -0.0961689204, 0.0675708279, -0.00994038954, -0.0795983076, -0.0637072176, 0.0743477792, 0.0424333625, -0.0580955856, 0.0883712918, -0.0932756513, -0.0508273803, -0.0552809015, -0.00379231572, 0.00728871487, 0.00522963703, 0.0359473377, 0.0478033125, 0.0493336581, 0.036497537, -0.0257146955, 0.0334913656, -0.0160065442, 0.0965906903, -0.114628188, 0.0917936414, 0.0817024186, -0.0815619528, -0.053349942, 0.0164614078, -0.051201731, -0.0701888427, 0.0927311927, 0.0053817872, -0.0659030825, -0.0182525869, -0.0481519885, 0.0572492704, -0.0427130871, -0.117971838, 0.0760072917, -0.0401136726, 0.0293068942, 0.0550760813, -0.0239000563, -0.0589896366, 0.0628921464, -0.0111487992, 0.0621845052, 0.086983569, -0.0491983071, -0.0577365048, -0.0127178021, 0.138659984, 0.0136703849, 0.0203418899, -0.0167258903, 0.0277019888, 0.0735571161, -0.0304019712, -0.0960620493, -0.0633719116, 0.0529922768, 0.0849122927, -0.0568064377, 0.0386673808, -0.0278773811, 0.050119333, -0.0261830483, 0.034985017, -0.152361751, 0.0646530166, -0.0399732925, 0.136056826, -0.0667104572, -0.0361961722, -0.0589022413, 0.0238616355, -0.0694033131, 0.0244187303, 0.0998045802, -0.0942119583, -0.0533202514, 0.0396387354, 0.0239462368, 0.114358447, 0.0064926222, -0.104682855, 0.0867709965, -0.0643172339, -0.0639604703, 0.00978600234, -0.0619044527, 0.0231725276, -0.0677455589, 0.0646953359, -0.0423314348, 0.0663801804, -0.0126665328, 0.00079670985, 0.0959830657, -0.110948384, -0.044717893, 0.0259171184, 0.0029677581, 0.0488119237, 0.0493388921, 0.00315413391, -0.0227418393, -0.0178110264, -0.0601525865, 0.027275715, -0.088893421, 0.0418855622, 0.0274772923, 0.140218884, 0.0181001052, -0.0606117174, 0.06166403, 0.0290223863, 0.0379726216, 0.00176884793, -0.0619544983, -0.113230765, 0.0179323647, 0.0539414436, 0.0379320905, -0.0695518777, -0.01092791, 0.046230603, 0.111597657, -0.0614224002, -0.0463933796, 0.114856675, 0.0644582435, -0.0229518507, 0.0425222665, 0.0858408734, -0.022010956, -0.0496490076, -0.0161762908, -0.069172442, 0.0167976283, 0.0731301457, 0.031990163, -0.0184318796, 0.00955096819, 0.0271152854, 0.00406571478, -0.0171847772, 0.0719815716, -0.0642897189, 0.0493998863, 0.0200924762, -0.048813574, -0.107431218, 0.183275014, 0.0607612506, -0.0243136864, 0.0676074103, 0.0395074077, 0.0465932786, 0.0137261245, -0.00171791879, 0.0695903301, -0.0239852108, 0.0242714286, -0.068965137, 0.00273539126, -0.0015002396, 0.0600375347, 0.0173954852, 0.0670008585, 0.0440744758, -0.0366984978, 0.0297529325, -0.013167493, 0.0899660215, -0.0560335293, 0.107497431, 0.0661580861, 0.00595683604, 0.00238380814, 0.0377494916, -0.0699493736, 0.0643459782, 0.0511911288, -0.0730385259, 0.0119525827, 0.0373752676, 0.0551899299, 0.136423483, -0.0847420022, 0.0085307071, 0.0273791179, -0.155341387, -0.0718755499, 0.00317818695, -0.021483358, 0.059964031, -0.0139861833, -0.0545050725, -0.00458152406, -0.0441917852, -0.0474866927, -0.0565952584, -0.129597649, 0.0728063211, 0.117210492, 0.0266580842, 0.0400655344, -0.000703627244, -0.0180977527, 0.0945833772, 0.0798216909, -0.0532262921, -0.105724111, 0.0408700742, -0.0284206569, -0.0114606041, -0.0305638704, -0.00290533714, -0.0632611215, 0.0861598328, 0.0256097484, 0.0844868124, -0.000183494762, -0.0455897413, -0.0256120246, 0.0113333175, -0.111941621, -0.0550071299, -0.0449723192, -0.064906612, -0.03743729, -0.054785993, 0.0944822505, 0.107955337, -0.015555135, 0.0125486013, -0.0451906845, 0.0486560874, 0.106059976, -0.0436536148, -0.0731038451, -0.0328179821, -0.153650373, 0.175019264, -0.0898246169, -0.0821646303, -0.0357303731, -0.0403635167, -0.0485206768, 0.0380006582, -0.0622984804, -0.0668045878, 0.00871956907, -0.0706435144, 0.00537299924, -0.016637437, 0.000934959156, -0.0461767055, 0.0162912272, -0.106971629, -0.0329704285, 0.0481520593, 0.0348616503, 0.15222162, -0.043573834, 0.0131295677, 0.0767574236, 0.0578459017, 0.0762267262, -0.00305164605, 0.092621848, -0.029637143, -0.00944327191, 0.00712501444, -0.0606836006, 0.0510030985, -0.0753934234, -0.102620661, -0.0575833097, 0.0277523324, -0.0143347122, -0.0758434534, -0.0029467647, 0.0339226723, -0.000715362839, 0.0876091048, 0.0113643324, 0.0300263166, 0.0788765326, -0.166643038, -0.0178198162, 0.0597060695, -0.0446988866, 0.0398542471, 0.082441695, 0.0270468146, -0.0937431976, -0.106794089, -0.0490684099, -0.0100667747, 0.0191480406, 0.0430809408, 0.0157079231, 0.0402602889, 0.0352774523, 0.0488876179, 0.0284086131, 0.103776187, -0.050829839, -0.0636555329, 0.0761722252, -0.017574966, -0.0136346314, -0.00153193809, -0.0907893553, 0.0106897913, -0.00721007586, -0.0455814004, -0.0274666324, 0.132764012, -0.00797156524, -0.0648535267, -0.0230660569, -0.074524045, 0.0204962678, -0.00375608355, 0.0140180029, 0.00653832406, 0.112480484, 0.027561035, -0.0248970166, 0.109508477, -0.00834539626, -0.173050672, 0.115768574, 0.0501624346, -0.0799136609, 0.0317795277, 0.0402359404, -0.0141283646, -0.00416751718, 0.0445878245, -0.00390318967, 0.0575758331, 0.060521476, -0.0186978076, 0.0303580873, 0.125115544, -0.0513926707, 0.00387083925, -0.0724220201, 0.0174948629, 0.0088728508, -0.0107462611, 0.0018973964, -0.0517203733, -0.0887014046, 0.114802465, -0.0590937883, 0.0275189262, 0.00887892395, 0.0216434933, -0.0426986478, -0.0313229226, 0.0518602468, -0.0875830799, -0.00910915248, 0.0359561704, -0.00148514286, 0.0651171207, 0.0269932542, -0.0336639211, 0.00721887406, -0.0195665993, 0.0188093763, 0.0226376913, -0.0242027529, 0.00973877963, -0.0061116931, 0.0547311604, 0.100967787, 0.0165629853, 0.0685569644, 0.0689111799, 0.0394094065, 0.0280195456, 0.00132902246, 0.0477260053, -0.0404579267, -0.0369920358, -0.130704299, -0.0458741412, 0.0621027425, -0.0414835215, 0.0446288101, 0.0479787812, -0.00596900098, 0.0777240247, -0.126405433, -0.0535859205, 0.0484512933, -0.0213578939, -0.117705531, -0.0974955186, -0.00615936238, -0.0250316542, 0.107710242, 0.106493741, 0.0641418472, -0.249681562, -0.085394904, 0.133077845, 0.0378696136, 0.0707044601, 0.0831430182, -0.0327371471, 0.0103407362, -0.0455160141, 0.010422606, -0.0569669046, 0.0566515699, -0.106681749, 0.0259751454, -0.0748780742, 0.0451363102, -0.0373559445, 0.0923741609, -0.0696469918, 0.00254642963, 0.0329135135, -0.187503844, -0.052324798, -0.0181447789, -0.0591514371, 0.0904739276, -0.0337331519, 0.0167032741, -0.00704860501, -0.0159117319, -0.0179821216, 0.0642585605, 0.00898541883, 0.00861603394, 0.0209293086, -0.0784179494, -0.108045213, -0.00232136622, -0.00986678712, 0.0890319794, -0.152924716, 0.0819708481, 0.00200564042, 0.0530426539, 0.01184092, -0.0440359004, 0.104986049, -0.0365393162, 0.0884416103, 0.0599602573, -0.0107538439, 0.0194925535, -0.0341205262, 0.0571896136, -0.0533981174, 0.0233363323, 0.0596668795, 0.0871201307, -0.0247691311, 0.0373147354, -0.114223137, 0.0742914751, -0.0549120381, 0.0501485057, 0.120348699, -0.02612832, -0.0183286592, -0.018494878, 0.0161769576, 0.0828156173, 0.0461297557, 0.0128012542, -0.0769066289, 0.0790741742, -0.00357566122, 0.0436053798, -0.0245894808, -0.0223144125, -0.0220041722, 0.0379337072, -0.0103706392, 0.00153468736, 0.0624835864, 0.0850405395, 0.024067156, -0.00428088615, 0.0557614118, -0.111060604, -0.0223824289, 0.0581790432, -0.0457777381, 0.0456162393, -0.0478162318, -0.0326411352, 0.00537061505, -0.00958615635, -0.0609744713, -0.0442263521, -0.0463129207, -0.107833549, -0.0163411275, -0.00114361942, 0.0292104185, 0.0859159529, 0.0728753656, -0.0311700739, 0.0540612936, 0.0569870621, 0.0930427238, 0.00829934608, -0.000418767333, 0.0162471086, -0.0319710225, 0.020500008, -0.111190327, 0.068059817, 0.118636273, -0.0440578759, -0.0292991549, 0.013629185, 0.0557562411, -0.0407737046, 0.043614842, 0.00416432088, 0.109360605, 0.071429424, -0.0104594212, -0.0330514796, -0.0686237291, 0.0673070848, 0.0333955437, -0.0829327703, -0.0704844445, -0.10953521, 0.00395125942, -0.0176604614, -0.0467942767, 0.106587887, 0.0155349486, -0.098312512, 0.112085514, 0.0174507685, -0.0107421074, -0.0780705959, -0.0142569952, -0.0747745857, 0.0658345744, 0.0170356836, 0.100902855, -0.0549179353, 0.0417767651, -0.00449547637, -0.031248197, -0.143883869, 0.0302504878, 0.0342233106, -0.00832069665, 0.032918077, 0.0602471754, -0.053038042, -0.0583118834, -0.026515875, -0.0283092558, -0.0478704199, 0.00196344964, -0.00386855006, -0.0416286923, 0.0186591726, 0.116214231, -0.0479242057, 0.11823874, 0.0271770097, 0.128326997, 0.0627788603, 0.0833879262, -0.0209303666, -0.048543714, 0.0222873241, -0.0666813925, 0.0515412837, 0.0382827297, -0.0208170004, 0.0806695968, -0.0787518024, -0.0102268904, 0.00101332366, -0.0423842669, 0.0684128255, -0.0985557362, 0.0622128621, 0.112807639, 0.0251122955, -0.090466395, -0.0766488239, -0.130260751, 0.00460057333, 0.0115046855, 0.0837528482, 0.00989025831, 0.0135682449, 0.0959551185, 0.0315829068, -0.0684198886, -0.065401271, -0.049925413, -1.29854307e-05, -0.0541259088, -0.142021701, 0.0256385431, -0.00497178547, 3.00398096e-05, -0.0939675793, 0.0956874639, -0.0105419774, 0.0773193613, 0.0756074339, -0.000617986545, -0.0258587524, -0.051476296, 0.0667045787, 0.0564629249, -0.0826095641, -0.0622458458, 0.0488035679, -0.0948024839, 0.00421141461, 0.0218561217, -0.0710685626, -0.0398794897, 0.0498290919, 0.0121802893, 0.141747281, -0.0258814152, 0.0790584758, 0.0159207918, 0.0768742114, -0.0653464645, 0.0181863923, -0.0297055468, -0.0193152018, -0.0178055726, -0.113849759, -0.0337221883, 0.0694251657, 0.0116117969, -0.0961880386, -0.0454436839, 0.0377202854, -0.155266061, 0.0593413934, -0.10687308, -0.0910210013, -0.0327585004, -0.0620710738, -0.0562722534, 0.0250459593, 0.0365692563, 0.132199362, -0.0338924527, 0.0118484823, 0.0577498563, 0.0110551566, 0.00460951589, -0.104437836, -0.122865118, -0.0673350766, -0.117810078, 0.0118398815, -0.00491665211, 0.0664852709, -0.0978418514, -0.0444246791, -0.0100815902, -0.0132434759, -0.0199350044, -0.043047417, 0.102522574, 0.0316540152, 0.0435058847, -0.00691261422, 0.0313382559, -0.0488980338, -0.0568745509, -0.0511014275, 0.0387725495, -0.0609640367, -0.0392125249, -0.0782465711, -0.0220331904, 0.0118650086, -0.0984330475, 0.0376985185, 0.0505482443, -0.0179485623, 0.0403323062, -0.00975354947, -0.0124219991, 0.0620927662, -0.00846980698, -0.0260278098, -0.0648871064, -0.0383695513, -0.0655695945, 0.0692879111, 0.0739795864, -0.0279878862, -0.0813971236, 0.0392812863, -0.0667336732, 0.00884250551, -0.092331782, 0.00155604817, 0.104298919, 0.0446757749, 0.00293998979, 0.0343209803, -0.117243633, -0.0795073211, 0.0196571629, -0.0242567509, -0.0630038381, -0.0679314584, 0.127634004, -0.0228610989, 0.0336672142, -0.0767852962, -0.0971866176, 0.109788693, 0.0115219671, 0.0200405233, -0.00252956804, -0.101939827, -0.0680609494, -0.0552854091, -0.0130165182, -0.0220800638, 0.0889879093, -0.0253602713, -0.0368813276, 0.0690257475, 0.0186834186, 0.0520263724, 0.0178525299, 0.0536663979, -0.0112049319, 0.0426837578, -0.0543723479, -0.0565344803, -0.111514412, -0.0807457715, 0.0242693294, -0.0477078333, 0.0532605611, 0.0260250792, 0.101735026, 0.0196578596, 0.0530879833, 0.150528371, 0.0270590596, 0.0216656048, 0.0183170252, 0.038476333, 0.0363754183, -0.00643502921, 0.0986894593, 0.0146187143, -0.0338521004, 0.00314715691, 0.145085782, 0.0213162638, 0.0134689678, 0.0412761569, 0.0083153192, 0.0612720177, 0.10603711, 0.0102780461, 0.0228238292, -0.0131024839, -0.0574563406, 0.0242601968, -0.0848699063, -0.0106664002, 0.0425618142, 0.0520266257, 0.0504437052, 0.0842870772, 0.0189924669, -0.0257215034, 0.034089908, 0.0388914682, 0.0680603161, -0.0327357575, 0.0598302893, 0.0607175231, -0.0325971618, 0.0172564089, -0.017632056, -0.0158231035, 0.055588115, 0.0849860013, -0.023146078, -0.0382568575, -0.0274798982, 0.141526893, 0.000534346327, 0.0186242927, 0.0309525579, 0.0410873219, -0.0652645156, 0.0316977054, 0.0600645952, -0.0116240755, -0.0558668301, -0.0120358625, -0.122412905, 0.0980276614, -0.043831192, -0.000924725085, 0.126647115, -0.0425914824, -0.0582012236, -0.157272249, -0.0717187524, 0.117454834, 0.00537696946, 0.087025553, -0.0758102834, 0.0979601443, 0.000509545207, -0.0418811403, -0.0103687942, 0.0545176975, 0.0680027902, 0.00620109495, -0.0500163622, -0.0547868386, -0.144743323, -0.0525846742, 0.0445867665, -0.0276343748, -0.0108135547, -0.0125181824, 0.0491529927, -0.0380190909, -0.0281884409, 0.133458331, -0.00868008938, -0.0351189785, 0.0557060204, 0.0135073587, 0.031397596, -0.0558718219, 0.0215338599, 0.0199673884, 0.0130196167, -0.0113997431, 0.10981223, -0.114531495, -0.0470215119, -0.0262132138, -0.0359893739, 0.036365591, -0.0104049221, -0.0112302322, 0.0648007318, -0.0163590498, -0.0248691905, 0.0054326402, 0.0560142621, 0.0272602811, 0.0773605704, -0.0472747125, -0.0088899415, -0.0411600545, 0.062161155, -0.0507184938, 0.00648374716, 0.108063564, 0.0123401582, 0.010986045, -0.0979975685, -0.0677843094, 0.081748955, -0.133338869, 0.0752991661, -0.0337115377, 0.0233293884, -0.0605040304, -0.0309929531, 0.0952119455, -0.0337813981, 0.0954767764, -0.0226832312, 0.0311467424, -0.0704929382, -0.048751682, -0.0309597924, 0.0493566394, -0.0420945846, -0.0220461339, 0.125588834, 0.0230162293, 0.035337273, 0.00818438455, -0.108411923, 0.0272332616, -0.0150138922, -0.0837059394, 0.0132295843, -0.109569795, -0.0151005071];
    bias_3_g : ARRAY[0..63] OF REAL := [0.163410932, 0.00982454699, -0.253855884, 0.142040685, -0.0493585207, 0.188220978, 0.0856736451, -0.0228934381, 0.0585524477, -0.258745402, 0.138000697, -0.242126435, -0.217821762, -0.0803337693, -0.0995026082, -0.0447086543, -0.0128557226, -0.177110955, 0.100215703, -0.260479718, 0.12717104, -0.0670361519, 0.0299517773, 0.223402619, -0.190082416, -0.229975134, 0.279827267, 0.230623558, -0.243755728, -0.049167417, 0.085180819, -0.251186341, 0.202504918, 0.2934784, 0.209657758, 0.248753935, 0.0865690559, 0.187145323, -0.253240734, 0.266585112, -0.243525207, -0.234963253, 0.00984069612, -0.221670508, -0.23716642, 0.17273961, 0.283333808, 0.228506699, 0.0613409132, 0.259918302, -0.231624246, 0.24294205, 0.0134335794, -0.168851465, 0.193654865, 0.243644968, -0.201259643, 0.281881571, 0.110072479, 0.0182489343, -0.256670356, 0.0609042794, -0.188948065, -0.22111927];
    weights_3_o : ARRAY[0..4095] OF REAL := [-0.810416162, -0.632364571, 0.331948847, -0.821512341, -0.507959008, 0.0525717251, 0.991340756, 0.827381432, 0.322914451, -0.926556051, 0.891123295, -0.926926672, 0.902667105, -0.899319947, 0.890559018, -0.727114797, -0.498999655, -0.813281596, -0.611148655, 0.663062811, 0.697072089, 0.433967948, -0.716905773, 0.534796298, -0.727120101, -0.704625726, -0.407410085, -0.842695415, 0.760583341, -0.916013658, 0.700237095, -0.662591875, 0.622441232, 0.258318961, 0.981015623, -0.91827482, -0.66032654, -0.408986866, -0.448537946, -0.861857176, -0.638492882, -0.745996058, 0.746864259, -0.692002416, 0.0104521355, -0.928194761, 0.993612349, 0.839406133, -0.0757885575, -0.481726378, 0.359193832, -0.123859867, -0.224441871, 0.334864855, 0.880186021, -0.563822925, -0.0141965002, -0.416545779, -0.746655285, -0.82704401, 0.883453608, -0.717097402, 0.864148557, -0.58061862, -1.0829134, -0.823607743, 0.572485864, -1.00121653, -0.647507966, -0.17820327, 1.12907946, 1.01044905, 0.507915974, -0.915899992, 1.05370569, -0.995482206, 0.909505427, -1.04414809, 0.91023916, -0.717669547, -0.544866025, -0.747128725, -0.593837857, 0.839194238, 0.872573912, 0.59611553, -0.974419534, 0.732646525, -0.947464764, -0.994947076, -0.683214068, -0.876485527, 0.938078463, -0.89297086, 0.903191984, -0.679340899, 0.746241748, 0.385734856, 0.998169899, -0.9376055, -0.837572753, -0.752655745, -0.527543306, -0.898670256, -0.850015163, -1.00882041, 0.926407754, -0.793875337, -0.347495645, -0.972094357, 0.977655232, 0.792688608, -0.038234923, -0.679934561, 0.5187729, -0.242143422, -0.288187236, 0.184791446, 1.04193676, -0.675273597, 0.0186059177, -0.598705471, -1.10505998, -0.813861609, 0.930217981, -0.746753037, 1.05715287, -0.809303463, -0.940164447, -0.854803741, 0.24817504, -1.1066283, -0.776414752, 0.0166122951, 0.978725016, 0.837585747, 0.0429907143, -0.807737112, 0.908838451, -0.96965009, 0.770339072, -0.83129108, 1.0117346, -0.668943942, -0.350848824, -0.953844428, -0.498169988, 0.73163563, 0.571662128, 0.429476619, -0.686127603, 0.652506173, -0.979750335, -0.751914382, -0.531791091, -1.00555015, 0.935287297, -0.863976479, 0.884518743, -0.826017678, 0.857592881, 0.54308641, 0.972898602, -0.896204948, -0.735711873, -0.369015187, -0.526894152, -1.10453975, -0.616772652, -0.97835052, 0.893984854, -0.889170647, -0.00660305377, -1.0944196, 0.900211632, 0.845365882, -0.2042716, -0.219385967, 0.382736534, 0.175510496, -0.529986739, 0.541858077, 0.79762882, -0.788721085, -0.118985958, -0.422704041, -0.930683792, -0.835422397, 0.724398673, -0.666998327, 0.800106466, -0.672537446, -1.21783662, -1.17573047, 0.78739357, -1.09857368, -0.828098714, -0.453535378, 1.0436126, 1.17363417, 0.444279522, -1.05227125, 1.17594826, -1.09437108, 1.17424655, -1.15257657, 1.18182039, -0.857873917, -0.797113597, -1.02761841, -0.97269243, 1.1315037, 0.892705262, 0.901616156, -0.899816573, 0.930284619, -1.25181115, -1.05530977, -0.884327471, -0.990078449, 1.0200175, -1.10096228, 1.08617961, -0.873265266, 1.05974436, 0.182358101, 1.2616334, -1.16774404, -0.790593207, -0.827829599, -0.360842198, -1.3289628, -0.916279733, -1.09493852, 1.15986085, -0.978571773, -0.456383198, -1.23530328, 1.19807053, 0.873382449, 0.0915719122, -0.777729273, 0.654820323, -0.371243298, -0.217018098, 0.139695868, 1.18950987, -0.883746326, 0.258074164, -0.815478861, -1.03686059, -0.880235136, 1.11851799, -0.887662232, 1.24477851, -1.04366267, -0.927076042, -0.874570608, 0.533207953, -1.16950655, -0.779000759, -0.083556816, 0.951717854, 0.917973876, 0.338150859, -0.943543792, 1.00813174, -0.978224397, 1.07276583, -0.953902841, 1.1061393, -0.839955568, -0.725721776, -0.780686796, -0.70376271, 0.789752841, 0.698594868, 0.555514634, -1.00540328, 0.807863235, -0.89325738, -1.00011432, -0.616469324, -0.920194507, 1.0268898, -1.05868495, 0.838855624, -0.710130394, 0.753563881, 0.407444149, 0.969546795, -1.02390778, -0.844037473, -0.572696447, -0.526845813, -1.20472968, -0.805530846, -0.890259385, 1.01292598, -0.807973027, -0.193706661, -1.09777975, 1.00725722, 0.929887593, 0.0525590107, -0.484539688, 0.504222751, -0.073785454, -0.382982701, 0.398180306, 0.874454677, -0.773526311, 0.0202719271, -0.548354626, -1.09213746, -0.703610122, 0.85308969, -0.938794494, 1.02478063, -0.852784634, -0.936436951, -0.810628295, 0.288247049, -0.800110638, -0.589985073, -0.0933668166, 0.772421777, 0.757540822, 0.199742839, -0.801299274, 0.860473394, -0.686715603, 0.627428293, -0.692731142, 0.864281654, -0.673476934, -0.344178736, -0.891158879, -0.45599556, 0.79197222, 0.535070777, 0.450350076, -0.736960471, 0.511235356, -0.711736679, -0.79555124, -0.451936543, -0.875041425, 0.742317915, -0.709822178, 0.622409999, -0.778374851, 0.819654644, 0.405972481, 0.919927359, -0.852057397, -0.605770648, -0.493412256, -0.282300323, -0.878022552, -0.785930812, -0.627949417, 0.963491678, -0.66732502, -0.0732551515, -0.824094117, 0.858006001, 0.797196329, -0.209460884, -0.225955248, 0.386500329, 0.0264633521, -0.273642331, 0.268181503, 0.72968328, -0.503906906, -0.0299764499, -0.306860924, -0.956261933, -0.625701129, 0.71547991, -0.708829939, 0.674921751, -0.728674889, -0.915051341, -0.797267556, 0.433978826, -1.0648638, -0.6611467, 0.0321726426, 1.08708584, 1.12441766, 0.234147027, -0.929795682, 0.99306953, -1.08476818, 0.824155271, -1.00790703, 1.09197402, -0.597972572, -0.724727213, -1.03516269, -0.765102029, 1.04485929, 0.915707231, 0.655611098, -0.655327201, 0.71146667, -0.880531907, -0.981864512, -0.740608275, -1.03925431, 0.930697083, -0.873291016, 0.911698699, -0.866153359, 0.988849938, 0.287267536, 1.16864264, -1.01967359, -0.613336205, -0.448691189, -0.459558576, -1.23740065, -0.727345526, -0.729569435, 1.07527161, -1.07307291, -0.0634794161, -1.22114217, 1.12967038, 0.993716061, -0.182771757, -0.5244748, 0.398529768, -0.0358487628, -0.169554666, 0.145709008, 0.93377161, -0.82277149, -0.0796993673, -0.429104477, -0.868583977, -0.865877926, 0.919038713, -0.770574808, 1.0103364, -0.68764925, -0.890600622, -0.950234771, 0.401323825, -0.893950284, -0.695562005, -0.0654199645, 1.09919572, 1.08195078, 0.418035686, -0.925168157, 0.909039557, -0.835556626, 0.831402361, -0.886672556, 0.954080224, -0.688357234, -0.507279396, -0.802634478, -0.71169138, 0.651136994, 0.734781146, 0.547465682, -0.788385808, 0.576072156, -0.897289217, -0.694975615, -0.537301123, -1.0356313, 0.943917215, -1.06196761, 1.00949574, -0.728529334, 0.698269427, 0.31463933, 0.88976413, -0.813047767, -0.795124829, -0.407622576, -0.511002719, -1.14938819, -0.665442586, -0.86580056, 0.883992434, -0.792700231, -0.298728853, -1.12042487, 1.09476519, 0.796541691, 0.0641986281, -0.612924635, 0.550003648, -0.163035363, -0.310238063, 0.350732625, 0.928103864, -0.645643055, 0.112292618, -0.374293506, -0.931672096, -0.76144731, 0.781069636, -0.738246799, 0.84312427, -0.876054585, -0.998094082, -1.08876646, 0.515163481, -1.15523279, -0.830414474, -0.142749056, 0.978087723, 0.955117822, 0.231328219, -0.923584521, 1.04953003, -1.08466709, 0.992961228, -1.1137923, 0.939355493, -0.825798988, -0.61003089, -0.78512007, -0.613310874, 0.969524741, 0.824490964, 0.776512802, -0.932790995, 0.742941618, -0.900355458, -0.9948439, -0.615561187, -0.964486122, 0.94518733, -1.09343207, 0.820304751, -0.764077961, 0.709186614, 0.484983563, 1.11687851, -0.992166936, -0.778622925, -0.721719861, -0.573230445, -1.2238555, -0.784993351, -1.03999794, 0.952664912, -0.967082858, -0.277411133, -0.950065911, 1.12379968, 0.951396823, -0.0440048873, -0.532876551, 0.481933951, -0.214262694, -0.340115547, 0.396563977, 0.99284333, -0.985861361, 0.119726598, -0.610663295, -0.966425061, -0.942896128, 0.92907536, -0.970526457, 0.906409562, -0.798956156, -1.02111459, -0.753185213, 0.117250703, -0.906496763, -0.665380478, 0.204478219, 1.10296369, 0.883347929, -0.107981846, -0.959355295, 1.01197875, -0.965763092, 1.03240323, -0.93674159, 1.05728674, -0.838105738, -0.469058692, -0.942238271, -0.448442072, 0.852513254, 0.64448148, 0.46084258, -0.790699005, 0.735133529, -0.947204649, -0.805781782, -0.240231529, -0.894147396, 0.902454317, -0.935602069, 0.902245462, -0.773278713, 0.743646502, 0.467320234, 0.968215585, -0.861793816, -0.856672049, -0.328923166, -0.482819319, -1.02827752, -0.673876643, -0.871224225, 0.857278049, -0.962392449, 0.0221720692, -0.910921991, 1.12360692, 0.732678175, -0.329954594, -0.349990964, 0.26402244, 0.364810199, -0.507242978, 0.513254046, 0.909919739, -0.758439422, -0.252318591, -0.135316879, -0.926355362, -0.812086701, 0.931882501, -0.729283214, 1.0493387, -0.765120804, -0.804593861, -0.659718633, 0.30722028, -1.00459397, -0.580626965, -0.0642664582, 0.999902546, 0.988400936, 0.228875384, -0.922962606, 0.937314987, -0.900100827, 0.931499064, -0.919784844, 0.934259295, -0.68171823, -0.493394107, -0.836679757, -0.632992744, 0.69272691, 0.597598314, 0.592400312, -0.682136595, 0.697678328, -0.946909785, -0.73916775, -0.591615677, -0.993152678, 0.967339456, -0.887237012, 0.670074522, -0.875521541, 0.764205933, 0.351264328, 0.867913961, -0.706009448, -0.531604886, -0.551608384, -0.471202791, -1.10206652, -0.847554624, -0.71665436, 1.0344516, -0.861289918, -0.15096508, -0.859748065, 0.962192059, 0.884995639, -0.180134848, -0.274881512, 0.299877554, -0.0388779677, -0.341524154, 0.338437259, 0.948013246, -0.570307732, -0.016347697, -0.405836463, -0.971495569, -0.813150704, 0.775648654, -0.701681197, 0.979956031, -0.507858992, -0.99926132, -0.834581017, 0.150933355, -0.937754929, -0.623434842, 0.235489368, 0.946184456, 0.796016395, -0.0865933225, -0.81420064, 1.05355406, -0.81036061, 0.820183754, -0.950138688, 1.03194857, -0.74544251, -0.340459824, -0.700592935, -0.393653452, 0.831653118, 0.672556698, 0.291230351, -0.804058552, 0.684855282, -0.89992702, -0.817008674, -0.323869884, -0.979623735, 0.913924515, -0.761783361, 0.695838988, -0.643045425, 0.682716787, 0.404558837, 1.04299521, -0.850374699, -0.782303751, -0.256804198, -0.500572741, -0.982827604, -0.58911258, -0.880953491, 0.95238328, -0.769976437, 0.103830218, -1.08127451, 1.02889311, 0.827016592, -0.177144453, -0.323171794, 0.193605378, 0.0550227277, -0.563002169, 0.455436468, 0.891213357, -0.713749588, -0.228870392, -0.167340696, -0.775992036, -0.758684337, 0.875997066, -0.644207895, 0.740553379, -0.792784989, -0.763025641, -0.869977295, -0.141083822, -0.858258784, -0.155874968, 0.617544353, 0.761046886, 0.834283769, -0.40854311, -0.952244759, 0.999913692, -0.905873001, 0.862693667, -0.946360767, 0.726966619, -0.811755896, 0.140796348, -0.725439787, -0.00370721216, 0.369660318, 0.391838104, 0.00369962049, -0.77247864, 0.346269578, -0.911159098, -0.540566862, -0.0250921566, -0.816935599, 0.751808822, -0.76211369, 0.836097598, -0.37434271, 0.306137383, 0.684277534, 0.978217006, -0.706481874, -0.784281194, -0.101461731, -0.58521682, -0.824986577, -0.390577048, -0.703053236, 0.963286042, -0.553001523, 0.434846967, -0.761681676, 0.909804046, 0.552850544, -0.538155854, 0.237592116, -0.029913513, 0.598290741, -0.559893727, 0.703335643, 0.810537755, -0.869511962, -0.491411507, 0.0602072217, -0.840365767, -0.541884303, 0.730098963, -0.573116302, 0.895701945, -0.646713376, -1.10362172, -1.0343647, 0.625229597, -0.966908932, -0.786028624, -0.0236303955, 1.01053905, 1.05751252, 0.423132211, -0.991263628, 1.1076951, -1.10686457, 0.897074044, -0.996542513, 0.976140618, -0.888659418, -0.538049161, -0.936811507, -0.829706073, 0.798595905, 0.720476151, 0.565481722, -0.942914486, 0.897380471, -1.01677799, -0.766943991, -0.594139338, -1.01186037, 1.08429587, -0.908107579, 1.02614713, -0.714129567, 0.858112097, 0.498025328, 1.18397164, -0.948625684, -0.949648619, -0.569084764, -0.603996336, -0.984670818, -0.746285081, -1.03612423, 0.919023871, -0.876065433, -0.218191743, -1.21176338, 1.0998441, 0.808486104, -0.0352619179, -0.547369719, 0.501274347, -0.153296247, -0.385932058, 0.55224669, 1.02470732, -0.862100363, -0.0121623455, -0.670730591, -1.0616188, -0.841974497, 0.92963171, -0.843917966, 1.15794456, -0.987858057, -1.1626066, -0.907478213, 0.608027399, -1.04968715, -0.760365307, -0.372121871, 1.29686201, 1.16345382, 0.475312084, -1.18424737, 1.12401259, -1.10074651, 1.09850311, -1.23719478, 1.26403427, -0.927538157, -0.840142608, -1.099141, -0.962609053, 0.95902282, 1.04031742, 0.882834673, -0.86096251, 0.840710521, -1.05500627, -0.936419845, -0.831271827, -1.06475711, 1.08530521, -1.19739676, 1.05378163, -0.805482388, 1.02937388, 0.318793297, 1.21964955, -1.15052366, -0.921993971, -0.815229237, -0.500185549, -1.08583772, -0.884286761, -1.13556266, 1.21759999, -0.973459661, -0.237898231, -1.11604416, 1.09505701, 0.849362075, 0.0284092836, -0.774505138, 0.624827445, -0.103781968, -0.357599229, 0.324987113, 1.07510328, -0.762163043, 0.206534103, -0.649940372, -1.20459843, -0.979830325, 1.03374135, -0.847493351, 1.08690441, -0.961402118, -0.840717673, -0.876441598, 0.251978606, -0.848592162, -0.624835968, 0.0422926657, 1.06422901, 1.01123154, 0.192406863, -0.844975054, 0.830052674, -0.816588998, 0.869730771, -1.00000703, 1.03143287, -0.880817294, -0.443541557, -0.88356626, -0.427683502, 0.814180672, 0.498419553, 0.527234852, -0.749135256, 0.574769258, -0.906902194, -0.601406276, -0.525273085, -0.944630325, 0.96054107, -1.00352395, 0.812626898, -0.630507827, 0.618096471, 0.480205089, 0.84051162, -0.830881298, -0.672740877, -0.424542129, -0.523852289, -0.899116814, -0.609597862, -0.82307452, 0.848293245, -0.82601577, 0.0944526121, -1.03450108, 0.897500873, 0.694547892, -0.182754546, -0.299453527, 0.243903473, 0.152152941, -0.44265753, 0.611877322, 0.824503064, -0.817273259, -0.118649639, -0.260487705, -0.932881713, -0.788241565, 0.887932539, -0.719384849, 0.915576935, -0.822528064, -1.00801718, -0.817445636, 0.487822175, -0.972868621, -0.789416671, -0.164515123, 0.824993432, 1.0453167, 0.354354501, -0.973499417, 0.919373095, -0.777144134, 0.808430672, -0.871208668, 0.824132025, -0.779264331, -0.716419518, -0.834049523, -0.674458325, 0.826367497, 0.679392517, 0.752317786, -0.93660742, 0.754399717, -0.865167797, -0.846726239, -0.719420552, -0.866624653, 0.84739548, -0.947440982, 0.732539356, -0.787194967, 0.925792158, 0.480165601, 0.732789814, -0.81544441, -0.711800933, -0.612993896, -0.473448843, -0.945545018, -0.856743157, -0.909355342, 0.87543112, -0.803813875, -0.439822078, -0.845210373, 1.0326463, 0.899315178, -0.030580882, -0.719331861, 0.541845739, -0.335878223, -0.20505181, 0.291963905, 0.933172584, -0.760733306, 0.0399821214, -0.742113292, -0.947298765, -0.688120842, 0.863982439, -0.894779205, 0.969984472, -0.753294945, -0.953459024, -0.600905359, 0.253932655, -0.985493004, -0.684118211, 0.0549523607, 0.971671522, 0.765570045, 0.304972291, -0.816728652, 0.799813747, -0.852168143, 0.825752318, -0.958667815, 0.998128295, -0.62545383, -0.324288666, -0.743592262, -0.593390346, 0.821690023, 0.633536041, 0.365281403, -0.601394355, 0.764313996, -0.708047211, -0.887171984, -0.440889984, -0.852618217, 0.687865019, -0.703538239, 0.844477713, -0.754793286, 0.621342301, 0.176239669, 0.931521893, -0.681581616, -0.720593512, -0.381482929, -0.433159798, -1.09078968, -0.667128742, -0.677106202, 0.76749295, -0.898184717, -0.0224697217, -0.907822609, 0.968612134, 0.805301011, -0.207517594, -0.473946512, 0.424457073, -0.00338196172, -0.27339831, 0.214707971, 0.914144874, -0.578552306, 0.00051117962, -0.259740561, -0.718720019, -0.691704929, 0.632985055, -0.812450528, 0.888550282, -0.673833549, -0.966824114, -0.817558944, 0.485992312, -0.936645329, -0.817287445, -0.0907262936, 1.09773946, 0.958067656, 0.38255921, -1.01815522, 0.891373158, -0.959374487, 1.00461912, -1.06265748, 1.12125909, -0.574692547, -0.52841866, -1.04114842, -0.757152975, 0.849882603, 0.833392859, 0.770320594, -0.746300936, 0.76509428, -0.954633296, -0.847266853, -0.670829237, -0.898784697, 0.954986036, -0.898273468, 0.78486079, -0.960015237, 0.815841794, 0.235376358, 1.01999354, -0.998362482, -0.77185297, -0.521572351, -0.275175482, -1.08989811, -0.854759157, -0.966544807, 1.11113548, -0.896435559, -0.170752302, -0.943428874, 1.13568366, 0.952051163, -0.0165873785, -0.468039274, 0.625868797, -0.0242228173, -0.130968809, 0.212027967, 0.923119307, -0.79886204, 0.0252223276, -0.536626697, -0.868688226, -0.897437155, 0.805938303, -0.889656305, 0.894871891, -0.678284705, -1.10808825, -1.06255662, 0.323312193, -1.09388602, -0.832231581, 0.304489404, 1.13721406, 1.10198283, -0.0455806963, -0.928042233, 1.10089457, -0.935113847, 0.925236166, -1.11959553, 0.9685992, -0.838369727, -0.489747822, -0.847552121, -0.525443673, 0.844653249, 0.665431738, 0.605067432, -1.04237914, 0.876656175, -1.11805415, -0.99191612, -0.585600793, -0.956043184, 1.1092782, -1.1131748, 1.09151518, -0.78502512, 0.856901944, 0.629819393, 1.0212456, -1.11613202, -1.02250147, -0.443278164, -0.808533907, -1.09294522, -0.895766199, -0.996087551, 0.993358076, -1.05091071, 0.256390482, -1.17618787, 1.12362802, 0.930378318, -0.471164554, -0.437907845, 0.273751527, 0.284316033, -0.762737274, 0.777721703, 0.889968157, -0.973798394, -0.467696726, -0.276850492, -0.952101588, -0.77869153, 0.863922119, -0.972462952, 0.988538623, -0.858974695, -1.08051968, -0.759149373, 0.52772069, -1.04999506, -0.659683347, 0.0117535694, 1.01151359, 1.11238289, 0.398211002, -1.11481512, 0.898744822, -1.04563546, 0.803569257, -0.842653036, 0.949905336, -0.700763047, -0.78028971, -0.9710778, -0.643522739, 0.93565774, 0.762575507, 0.69761759, -0.83656919, 0.937593997, -0.919821441, -0.990025282, -0.742170453, -1.00597656, 0.83546567, -0.981185615, 0.793578148, -0.886171341, 0.783188045, 0.343910426, 1.02735841, -1.00825381, -0.631802738, -0.560468972, -0.336501867, -1.08655119, -0.801837146, -0.723540962, 0.969678462, -1.028458, -0.000842482084, -1.18999386, 1.08291149, 0.873188436, 0.0551245995, -0.413129926, 0.549876571, 0.100124441, -0.397414893, 0.165964231, 0.99963659, -0.756516516, -0.0725842491, -0.522677124, -1.03168833, -0.882433414, 0.727501988, -0.910909355, 0.886263132, -0.763171375, -0.90306741, -1.02164948, 0.562654018, -0.948485017, -0.694936395, -0.222182974, 1.05249691, 1.10250604, 0.408812195, -1.12261093, 1.09155178, -0.899261534, 1.07021356, -0.906940699, 0.935425043, -0.880028844, -0.650212944, -0.884812236, -0.733829737, 0.896124482, 0.886922061, 0.638059437, -0.813690662, 0.71829778, -1.11724079, -0.990601718, -0.481998235, -1.13339043, 0.878371477, -0.903245389, 0.879073203, -0.69482404, 0.714323699, 0.528923392, 1.16980982, -0.862549186, -0.853634179, -0.47158429, -0.438652545, -0.953979075, -0.669543922, -0.876274824, 0.941246331, -0.968127787, -0.252344429, -0.993215501, 1.04132271, 0.938253045, 0.0401512906, -0.360834748, 0.484307617, -0.159859031, -0.306806833, 0.353603542, 0.997254908, -0.863128126, 0.0232510641, -0.385205686, -1.11616337, -0.777577639, 1.05745685, -0.869235158, 0.883288682, -0.765146017, -1.18934882, -0.965456128, 0.477512658, -1.05817914, -0.697171032, -0.15807268, 1.21281433, 1.10640979, 0.511394799, -0.912529707, 1.09973729, -1.01010239, 0.931992829, -1.12894773, 1.05462682, -0.951445103, -0.711644053, -0.836836815, -0.65973103, 0.755652606, 0.72982651, 0.708740532, -0.923789799, 0.883313835, -1.02150893, -0.859018385, -0.652336597, -1.06056261, 1.08454752, -0.983918369, 0.922526658, -0.852333069, 0.930260658, 0.454445541, 1.01583183, -1.13566756, -0.716477811, -0.786858201, -0.346616268, -1.24160314, -0.935656548, -1.00392163, 1.14838195, -0.886216819, -0.236957729, -1.23617971, 1.04308367, 0.937218547, -0.0294403583, -0.494654268, 0.608031988, -0.0875647962, -0.437503338, 0.224637046, 0.981087863, -0.72783947, 0.139756233, -0.729564548, -0.959230125, -0.725957453, 0.930482149, -0.887616992, 0.988028705, -0.842328966, -0.792090476, -0.670441568, 0.0300701354, -0.881175697, -0.438240319, 0.53491956, 0.810557604, 0.831622422, -0.25232017, -0.856232345, 0.759278893, -0.906379402, 0.80940789, -0.716738105, 0.886740029, -0.753706217, -0.126592472, -0.607044101, -0.357984662, 0.458272696, 0.403457761, 0.0654176548, -0.860346794, 0.298449278, -0.834578693, -0.650191069, -0.15592514, -0.714433789, 0.772959232, -0.734123349, 0.914095521, -0.576044798, 0.620039999, 0.479583979, 0.988299072, -0.882439792, -0.731743634, -0.0604174733, -0.748376846, -0.841263831, -0.461956263, -0.863450348, 0.757214963, -0.793172717, 0.339291811, -1.00214148, 0.885348201, 0.729029059, -0.467648894, -0.0716457739, 0.0363362432, 0.595286369, -0.766381979, 0.625612497, 0.753393829, -0.826981544, -0.567100763, 0.125759333, -0.780913949, -0.629091799, 0.900348663, -0.699746132, 0.881745875, -0.615412295, -0.758808196, -0.555578232, 0.261672497, -0.831508458, -0.558282137, 0.181979179, 0.817520261, 0.934221804, 0.0496329665, -0.88269341, 0.940814793, -0.722628236, 0.719642937, -0.768252671, 0.846578479, -0.454786658, -0.417611867, -0.797312438, -0.517541945, 0.60259974, 0.519569039, 0.287127465, -0.591698706, 0.602032125, -0.742424607, -0.859210968, -0.324492484, -0.766255498, 0.734580934, -0.807843745, 0.644142926, -0.756344855, 0.741601169, 0.37793991, 0.755885839, -0.82911706, -0.506487966, -0.309000999, -0.404808462, -0.887884319, -0.783705652, -0.781799674, 0.761692941, -0.653751612, 0.109660521, -0.899198174, 0.738864303, 0.811961412, -0.0746646971, -0.330690831, 0.236063823, 0.16286999, -0.244135201, 0.254997462, 0.70086664, -0.694007397, -0.270426661, -0.239275441, -0.675338745, -0.666000843, 0.761123359, -0.846066654, 0.656381726, -0.452299029, -0.968655169, -0.712994635, -0.159640029, -0.910780072, -0.60800606, 0.379726827, 1.01936507, 0.953597784, -0.235678941, -0.915932655, 0.986563146, -0.750562668, 0.973965049, -0.85545826, 0.966323674, -0.683604121, -0.310208231, -0.869966686, -0.3125754, 0.759332836, 0.425173312, 0.223157331, -0.915502429, 0.664933741, -0.846602142, -0.715007246, -0.0936192572, -0.976047754, 1.01067317, -0.883593917, 0.713848174, -0.592876136, 0.718195736, 0.447578043, 0.926254392, -0.779554844, -0.836337149, -0.244471237, -0.530014038, -0.966891646, -0.642830431, -0.699550152, 0.847063661, -0.716062546, 0.321497768, -0.936521113, 1.07256269, 0.744114697, -0.37231186, -0.0538084805, -0.113423668, 0.542577207, -0.738218367, 0.696359098, 0.811895609, -0.792344272, -0.477001905, 0.02457208, -0.796299279, -0.674420059, 0.916577041, -0.640601814, 0.873451233, -0.819441378, -0.816638231, -0.80349052, 0.471637815, -0.921268523, -0.542855322, -0.0891594812, 0.978114128, 0.961302876, 0.16974929, -0.84097445, 1.04441917, -0.936181962, 0.849858344, -0.883805513, 0.977398574, -0.654956877, -0.614581048, -0.715344787, -0.697615147, 0.859832227, 0.636470735, 0.37946412, -0.80959487, 0.798462868, -1.01728022, -0.787714779, -0.404177964, -0.886745334, 0.840279698, -0.887163103, 0.843767107, -0.842060864, 0.658450246, 0.36931482, 0.993214369, -0.980704725, -0.828209698, -0.447140545, -0.471337795, -1.01517701, -0.599507689, -0.924285769, 0.939803779, -0.719067812, -0.165062428, -0.897974551, 1.04035592, 0.775715172, 0.0181991719, -0.535969496, 0.274033904, 0.0918607712, -0.378453404, 0.314324677, 0.909226835, -0.685361981, -0.129584819, -0.308290213, -0.85573864, -0.673500717, 0.780632615, -0.736774921, 0.800696313, -0.791894972, -0.846441031, -0.815497339, 0.0217434093, -0.916837394, -0.508723736, 0.115324259, 0.974974334, 0.864486456, -0.161361516, -0.950496614, 0.922108531, -0.954298973, 0.850754857, -0.975950599, 0.966019154, -0.73440975, -0.33703503, -0.852672637, -0.280592561, 0.840091705, 0.472856075, 0.188667953, -0.657141447, 0.643595517, -0.92535007, -0.918782473, -0.383526325, -0.753213942, 0.915782928, -0.693038046, 0.728420436, -0.593485832, 0.748035192, 0.437922567, 0.952039242, -0.761089265, -0.605134785, -0.315682709, -0.582576096, -1.05821884, -0.627691209, -0.809873164, 0.917406559, -0.923862636, -0.0197111238, -1.04808128, 0.824178457, 0.738282979, -0.189726129, -0.147668839, 0.117851004, 0.271021366, -0.537482321, 0.507217526, 0.810153842, -0.784860969, -0.271175295, -0.286517859, -0.989632845, -0.775955915, 0.758684993, -0.780177116, 0.920935333, -0.770521998, -1.09896958, -0.913210809, 0.14743869, -0.997456133, -0.561877191, 0.249567315, 0.920378447, 0.893390417, -0.217661411, -0.857441604, 0.975236416, -0.919962704, 0.880448937, -0.973008215, 0.909922123, -0.728138804, -0.333273709, -0.826762557, -0.46681878, 0.904040873, 0.777379096, 0.401090384, -0.804922104, 0.760257721, -0.940277994, -0.994910657, -0.324435234, -0.977304578, 0.958711088, -0.977880955, 0.77532351, -0.81360656, 0.750584185, 0.636889458, 0.962432623, -0.926967144, -0.784475625, -0.369279504, -0.59172523, -1.10861695, -0.677711189, -0.848594487, 0.9685812, -0.863759458, 0.319024473, -1.18393064, 1.14742708, 0.918598413, -0.395315289, -0.00844334811, -0.0408792906, 0.491947353, -0.503088713, 0.435376495, 1.04138827, -0.783190846, -0.532903433, -0.229609758, -0.887545884, -0.902766347, 0.825376213, -0.89317739, 0.95029825, -0.758211613, -1.04166973, -0.807916641, 0.561932385, -0.883095682, -0.690106511, -0.205714479, 1.11524117, 1.11531162, 0.366474301, -0.867595017, 0.93494755, -1.06055856, 0.952125549, -1.02646875, 1.07473516, -0.746242821, -0.503588974, -0.884567559, -0.765060842, 0.866778195, 0.733334363, 0.655939162, -0.835318685, 0.831832707, -0.933980763, -0.916061342, -0.511183202, -0.913283646, 0.911170483, -0.894062817, 1.0100801, -0.780753791, 0.701069593, 0.482225567, 0.91133213, -1.01987433, -0.658463418, -0.494292498, -0.535505891, -1.15360796, -0.856469214, -0.997964263, 1.10171413, -0.968633354, -0.137197793, -1.04813302, 0.948315203, 0.78426671, -0.0600807406, -0.504433632, 0.565597057, -0.102513008, -0.448391438, 0.415334791, 0.983016074, -0.76524514, 0.0311283544, -0.517006934, -0.91556704, -0.791224957, 0.895029902, -0.915585577, 0.983500361, -0.928438723, -1.03406978, -1.08303034, 0.593069911, -0.966300011, -0.895419002, -0.0831895694, 1.00097859, 1.15092623, 0.475688368, -1.07410848, 1.11494958, -1.0881263, 1.03608155, -1.0770756, 1.2061969, -0.795345008, -0.695340455, -1.0396142, -0.882051826, 0.799437165, 0.888003886, 0.812065959, -0.846854031, 0.949035823, -1.01090109, -1.03668165, -0.794045329, -1.0865401, 1.17227089, -1.02369237, 0.835212111, -0.920741081, 0.805937171, 0.377676934, 1.16462588, -0.96840167, -0.774968624, -0.645982325, -0.425984651, -1.08848512, -0.840759397, -0.8932634, 1.08590651, -0.985020101, -0.306075305, -1.10577548, 0.978632331, 0.863674343, 0.0776144862, -0.514621258, 0.627155244, -0.0781887844, -0.231704667, 0.156509012, 1.15933418, -0.852298796, -0.0475793257, -0.497312486, -1.11962271, -0.930182397, 0.858195603, -0.973948538, 1.11558771, -0.938831508, -0.867746592, -0.863978624, 0.161411345, -1.08415747, -0.638186693, 0.117466122, 1.11144483, 0.985854387, 0.0497543812, -1.00623786, 0.979995668, -0.852036238, 0.765706122, -0.775051355, 1.06992733, -0.720672429, -0.436103582, -0.959627748, -0.528075397, 0.698085606, 0.760062814, 0.342677534, -0.652949691, 0.576641858, -0.906636834, -0.809891999, -0.312737167, -1.00150824, 0.877051532, -0.781708121, 0.893969059, -0.597018301, 0.766473353, 0.360368967, 1.15775716, -0.905454814, -0.675140917, -0.340480745, -0.507193863, -1.19997323, -0.644891024, -0.728058577, 0.818478882, -0.814920723, 0.187791288, -0.98739934, 0.953460574, 0.880523324, -0.340227067, -0.190726727, 0.174094856, 0.366152555, -0.430888921, 0.436932355, 0.807621717, -0.690511644, -0.221229002, -0.144982845, -0.837571263, -0.834334195, 0.893289506, -0.683453381, 0.906138897, -0.858801425, -0.910994172, -0.741055548, -0.0906451866, -0.750089347, -0.179178044, 0.711199224, 0.939223051, 0.838674486, -0.557342589, -0.931792378, 0.780850649, -0.82053566, 0.729475856, -0.798631728, 0.906719446, -0.835863471, 0.0397252738, -0.409141123, -0.0270589311, 0.504007459, 0.246139526, -0.070134148, -0.872599781, 0.160449758, -0.805105925, -0.545978189, 0.0277858321, -0.936650217, 0.911276102, -0.710964739, 0.774356723, -0.411576539, 0.448663175, 0.81014961, 0.866183043, -0.914341092, -0.670375049, 0.0339476466, -0.780256331, -0.785773814, -0.24337855, -0.748005986, 0.68598336, -0.356214583, 0.503674805, -0.713992655, 0.781561613, 0.311122417, -0.593362272, 0.206501067, -0.182407051, 0.555568397, -0.768952072, 0.690493822, 0.678100109, -0.690579355, -0.764402092, 0.184428468, -0.697541177, -0.50068146, 0.755816996, -0.327860236, 0.831468284, -0.749435067, -1.06540573, -0.982817411, 0.18890506, -1.00976098, -0.619255841, 0.147960603, 1.00080621, 1.12704122, -0.0488918573, -0.96573478, 1.07354128, -1.06324792, 0.804897547, -0.922943056, 1.08886957, -0.711678863, -0.513009906, -0.855891943, -0.578175426, 0.682360172, 0.617384493, 0.37783277, -0.777455389, 0.674189985, -0.870981753, -0.919557989, -0.538088143, -0.960185468, 0.975223839, -0.819583952, 0.980190814, -0.780355632, 0.841829956, 0.489903003, 1.05785203, -0.849623501, -0.860916913, -0.395284265, -0.623380244, -1.04620266, -0.674330533, -0.924329937, 0.84630996, -0.89330554, 0.116599709, -1.08148801, 1.1350168, 0.816165447, -0.222211391, -0.396473318, 0.369639605, 0.283509135, -0.622343719, 0.497577757, 0.843381464, -0.945206046, -0.269997001, -0.380826235, -0.973428488, -0.699160397, 0.975462854, -0.862314999, 1.02842128, -0.953981221, -0.750514567, -0.688439429, -0.277252316, -0.977173984, -0.309784561, 0.655972958, 0.884081781, 0.987296999, -0.458941042, -0.711202443, 0.981444001, -0.85346508, 0.937917948, -0.787044883, 0.747037649, -0.743543267, 0.0251842607, -0.522004664, -0.0839740485, 0.420434713, 0.184030026, 0.144405425, -0.84163481, 0.426001579, -0.784844577, -0.455770373, 0.00759232556, -0.77793932, 0.948131204, -0.911694169, 0.714292228, -0.329961568, 0.295224756, 0.520546019, 0.864608109, -0.867312133, -0.674962044, 0.148374364, -0.604444087, -0.847814858, -0.547508061, -0.74897182, 0.77784729, -0.607136428, 0.38284409, -0.923359275, 0.865110755, 0.337771416, -0.488369375, 0.0974853784, -0.189915836, 0.436232537, -0.667221606, 0.790938377, 0.770621121, -0.736455977, -0.646956742, 0.132405788, -0.958602071, -0.521056592, 0.893951356, -0.406006992, 0.738090813, -0.65931946, -0.996614039, -0.805866599, 0.241578802, -0.966110468, -0.596575797, 0.00621271739, 0.868061125, 0.994057, 0.26074782, -1.03123319, 1.00777936, -0.964930236, 0.791451871, -0.832785547, 0.817733824, -0.808596671, -0.518564761, -0.877115846, -0.586268902, 0.865031362, 0.722628057, 0.340871543, -0.788305759, 0.628780484, -0.829450965, -0.6813187, -0.453804076, -0.952066422, 0.73108232, -0.962357938, 0.791199625, -0.598254204, 0.670205057, 0.467287272, 0.807801247, -0.941978037, -0.681576967, -0.524434507, -0.47845608, -1.03611553, -0.650788724, -0.695517719, 0.946980476, -0.757736206, -0.0610983819, -1.07657337, 1.06499672, 0.758542299, -0.215620369, -0.393702865, 0.340857595, -0.0976904333, -0.221364141, 0.181904316, 0.876920342, -0.639999866, -0.111582018, -0.425084323, -0.867833912, -0.692504704, 0.893275619, -0.739153028, 0.954588175, -0.812311947, -1.21184802, -0.844080746, 0.570108473, -0.975573957, -0.723409176, -0.0131961405, 1.08833027, 1.05577898, 0.224035561, -1.1606859, 1.08909333, -0.969332516, 1.10719109, -1.04015195, 1.05004656, -0.678198874, -0.716714859, -0.977309644, -0.834499598, 0.973265588, 0.797283769, 0.75368458, -0.835332811, 0.808740079, -1.10811818, -0.896469891, -0.771928966, -1.07127702, 1.11476052, -1.14046824, 0.955279708, -0.959254205, 0.819234669, 0.426164985, 1.0381788, -0.936059475, -0.604959369, -0.65494442, -0.372639567, -1.19064605, -0.745349944, -0.817401886, 0.939729035, -1.00588417, -0.267551363, -1.20652568, 1.058833, 0.924105704, 0.10949903, -0.527458906, 0.619390011, -0.0652809069, -0.307280123, 0.34440726, 1.02386594, -0.872809112, 0.133331463, -0.517471969, -0.914980531, -1.0185554, 0.974691629, -1.00686669, 0.964569807, -0.664775312, -0.647060215, -0.659819782, -0.203391761, -0.663825512, -0.194261402, 0.414617538, 0.599808335, 0.595124424, -0.42691943, -0.708030641, 0.754834592, -0.746999562, 0.781613886, -0.74068284, 0.731891632, -0.574534357, -0.0437335931, -0.322872341, -0.0655643567, 0.337026298, 0.136019453, -0.0205819495, -0.665302038, 0.154436976, -0.630010962, -0.41903761, -0.00546499994, -0.702008784, 0.675100029, -0.599324048, 0.746405721, -0.413539171, 0.348993242, 0.58388418, 0.860259056, -0.798965096, -0.606727779, -0.0287924837, -0.667034626, -0.757388234, -0.19465521, -0.673445404, 0.608740449, -0.471730232, 0.497264177, -0.683601558, 0.698435307, 0.358315885, -0.476642251, 0.140274376, -0.0743753687, 0.590071857, -0.630947709, 0.735952199, 0.73390013, -0.803921461, -0.623386681, 0.128250197, -0.733342707, -0.278798878, 0.564716756, -0.251306683, 0.808975518, -0.691078246, -1.13780224, -1.03294492, 0.280970395, -1.00044453, -0.67680043, 0.347801715, 1.12598705, 0.893964171, -0.151982576, -1.05082977, 1.00025547, -1.11109722, 0.874447405, -0.907184541, 0.919569552, -0.711464703, -0.544213533, -0.828579128, -0.70937562, 1.01005268, 0.743564725, 0.514153838, -0.894601226, 0.700024903, -0.890127242, -0.925134838, -0.578231335, -0.874077082, 0.911543727, -1.0773921, 0.878839314, -0.738351107, 0.930854023, 0.51254046, 1.08822978, -0.891368091, -0.7510975, -0.324289918, -0.67497611, -1.07733274, -0.912501156, -0.906857312, 1.00731552, -0.84553206, 0.18235831, -1.14469647, 1.01296222, 0.842359126, -0.324698657, -0.224978849, 0.187029555, 0.402082086, -0.676193416, 0.709454894, 0.96477741, -0.926402867, -0.450022608, -0.243575856, -1.05365515, -0.943787277, 0.788061202, -0.930278242, 1.09640551, -0.84099406, -1.00080168, -0.825322568, 0.341880172, -1.05806601, -0.683522403, 0.11472331, 0.91114974, 0.873009443, 0.0018817751, -0.825888991, 1.13497913, -0.823179543, 0.80214864, -0.824991345, 0.970322847, -0.847236931, -0.510233402, -0.971776962, -0.401460707, 0.906775832, 0.5636217, 0.473190904, -0.909424663, 0.744375527, -0.874619305, -0.797892988, -0.517945349, -0.996560276, 1.02788782, -0.977011204, 0.761212647, -0.674539685, 0.667898238, 0.604148448, 1.15148389, -1.00630593, -0.80945313, -0.250946552, -0.538010299, -1.09676039, -0.696952403, -0.951910555, 0.865034759, -0.750389695, 0.110189751, -1.07638931, 1.08666193, 0.752868414, -0.312779814, -0.245955124, 0.183307394, 0.274840951, -0.460807383, 0.430708945, 0.806925237, -0.971363842, -0.201447383, -0.348557115, -1.06920755, -0.88614893, 0.935667753, -0.818521023, 1.07726741, -0.89764595, -0.990761399, -0.863233685, 0.0411759876, -1.13398433, -0.671033382, 0.479406565, 1.15445054, 1.04937005, -0.345098406, -1.08946002, 0.986090958, -1.04164982, 0.824137926, -0.980774462, 0.871760249, -0.773705006, -0.205187514, -1.03152287, -0.373452574, 0.772749126, 0.556335449, 0.314310968, -0.793766618, 0.56686765, -0.807256341, -0.928150117, -0.26205191, -1.07658386, 0.837845802, -0.793071151, 0.908378243, -0.736154079, 0.793367863, 0.600711107, 1.06671357, -0.7806108, -0.855808079, -0.234251305, -0.512653768, -1.12065315, -0.779898942, -0.769633651, 1.06528866, -1.04135513, 0.219725981, -0.978415132, 1.02230132, 0.892620742, -0.469449788, 0.00762188481, 0.106708132, 0.508779049, -0.624940991, 0.577260613, 0.946124792, -0.786776304, -0.407321811, -0.0388800129, -1.07600164, -0.840634227, 0.858025491, -0.801332295, 1.07156992, -0.7726717, -0.549303889, -0.638356388, -0.0439402238, -0.616375089, -0.0884586275, 0.40849176, 0.692937076, 0.640120745, -0.108789235, -0.425855488, 0.58269757, -0.563694477, 0.41718936, -0.425887614, 0.618270516, -0.570393801, 0.0957398936, -0.389890462, 0.0675123781, 0.272495866, 0.00648389198, -0.0685756803, -0.499544531, 0.27439779, -0.661442816, -0.431017607, 0.0812571123, -0.579040408, 0.474607408, -0.621389329, 0.559733272, -0.0980001166, 0.193707794, 0.366442949, 0.648980916, -0.469305992, -0.416295886, -0.0808261111, -0.397787333, -0.635029078, -0.178170636, -0.581621945, 0.676253617, -0.244879514, 0.291622967, -0.633293688, 0.565957785, 0.145189181, -0.344902992, 0.176559404, -0.132458255, 0.352134436, -0.313530326, 0.376009941, 0.63720119, -0.395942181, -0.253469348, 0.121549822, -0.619641125, -0.360361725, 0.503931046, -0.398058265, 0.491612285, -0.517944634, -0.720233023, -0.615961552, 0.671289921, -0.892400086, -0.910685599, -0.368188411, 0.914290309, 0.812086165, 0.602679312, -0.93445909, 0.711147189, -0.71578145, 0.870088577, -0.808034241, 0.86011678, -0.529967725, -0.644363999, -0.771332741, -0.845984817, 0.73887229, 0.863845825, 0.785664797, -0.749895573, 0.876937151, -1.00794685, -0.772558689, -0.715714037, -0.710956216, 0.783910751, -0.749604106, 0.756131172, -0.793994009, 0.914902747, 0.212008476, 0.613590777, -0.691703141, -0.573437393, -0.814350903, -0.436796516, -0.989124715, -0.706609845, -0.856026411, 0.867407441, -0.739376783, -0.37302658, -0.946519196, 0.95127666, 0.71339047, 0.0663700774, -0.639061868, 0.538956821, -0.362957358, -0.216663152, 0.217286706, 0.853304148, -0.620725274, 0.156644702, -0.567792296, -0.80418539, -0.889051557, 0.736372173, -0.808001578, 0.837038636, -0.576460958, -0.920148551, -0.898714304, 0.201782927, -0.839212835, -0.648532569, 0.0799565688, 1.08776164, 1.02611005, 0.116943635, -0.860131919, 1.02636468, -0.972904325, 0.790614426, -0.978492081, 0.794461787, -0.802973449, -0.346741706, -0.904234946, -0.460512817, 0.703312874, 0.489981383, 0.442758858, -0.836377501, 0.591198862, -0.743168175, -0.906577468, -0.437090486, -0.956070662, 0.830190241, -0.75756675, 0.755258501, -0.766777933, 0.720925927, 0.400990158, 0.859190524, -0.78292793, -0.620329857, -0.420223057, -0.527267873, -1.05339038, -0.622338474, -0.682140768, 1.03030086, -0.737843335, 0.131305009, -0.86850059, 1.0566684, 0.655864835, -0.313640445, -0.172575861, 0.35854122, 0.14339067, -0.56331563, 0.562504351, 0.828884125, -0.737003565, -0.190239966, -0.275263935, -0.982070208, -0.766988993, 0.852386594, -0.62799716, 0.904230416, -0.698065102, -1.0385257, -0.733011127, 0.27447924, -0.858885348, -0.550420523, 0.069836013, 1.03368235, 0.824826717, 0.00888017844, -0.965300798, 0.959463894, -0.874589384, 0.931506276, -1.03086782, 0.821991742, -0.812327802, -0.543480933, -0.755613506, -0.488953978, 0.793423414, 0.622666955, 0.398159683, -0.689910948, 0.629190028, -1.00548244, -0.784237742, -0.389830917, -0.935308158, 0.793312967, -0.768476486, 0.723726332, -0.638026297, 0.76798737, 0.401863486, 1.13336432, -0.808560848, -0.617281914, -0.418464154, -0.513358653, -1.14974988, -0.843147278, -0.726142049, 1.00907207, -0.73156178, -0.123481221, -0.883033276, 0.902231693, 0.842271626, -0.263394654, -0.390603602, 0.38680473, 0.197833359, -0.39950639, 0.439472914, 0.861869812, -0.797353685, -0.153385311, -0.237103149, -0.991820335, -0.688924611, 0.917775452, -0.811977088, 0.87590313, -0.810714066, -0.981729031, -0.88219738, 0.648488164, -1.03987753, -0.862566054, -0.177724645, 1.08571625, 1.07452881, 0.368714035, -0.994782269, 1.03743708, -1.00842714, 0.844676793, -1.05588603, 0.969592392, -0.792215943, -0.737406075, -0.991951287, -0.828681827, 0.771260977, 0.82473737, 0.789083481, -0.750544965, 0.894961059, -0.990762949, -0.884568274, -0.689292014, -1.1210916, 0.997003376, -0.920547247, 0.868750453, -0.899999142, 0.981734216, 0.37072596, 1.08225477, -0.956426919, -0.614243567, -0.560629785, -0.238357544, -1.09568942, -0.958396256, -0.901943028, 0.922318578, -1.03397608, -0.218839824, -1.05735075, 0.937167048, 0.94077307, 0.156876802, -0.54023993, 0.579226136, -0.243987396, -0.305969894, 0.207878768, 1.0163815, -0.765354574, 0.0348801799, -0.550502598, -1.08040571, -1.00219464, 0.853471756, -0.874036729, 1.04468739, -0.913006008, -1.0017972, -0.878947139, 0.255303234, -0.946021795, -0.624148905, 0.124308653, 1.05950809, 1.01422679, 0.0944362506, -1.07101858, 1.14251006, -0.861802638, 1.06708288, -0.860284209, 1.04953408, -0.809230566, -0.436149567, -0.93576175, -0.502566218, 0.890743077, 0.60882175, 0.422579557, -0.844233274, 0.623083472, -0.851229906, -0.726708233, -0.365490675, -0.865034223, 0.913283467, -0.844852269, 1.02171373, -0.848013222, 0.634785473, 0.536277652, 1.17107892, -0.999777913, -0.874782264, -0.521103263, -0.704013944, -1.08592796, -0.685212851, -0.979801536, 0.850257337, -0.833382428, 0.0114112915, -0.966780961, 1.11081493, 0.72694838, -0.24590297, -0.42065838, 0.244061083, 0.277858466, -0.562986255, 0.559036016, 0.933329344, -0.902888954, -0.233993232, -0.310846239, -1.01807129, -0.706233919, 1.0126133, -0.769901156, 1.0402534, -0.882325351, -0.995352685, -0.77962029, 0.0672754124, -0.998681247, -0.473735392, 0.515082419, 1.09194529, 1.0777297, -0.407653332, -0.794678152, 0.902068794, -1.00750613, 0.844537437, -0.850816667, 1.00689089, -0.628118038, -0.0654336363, -0.924520612, -0.266657799, 0.865810275, 0.515253484, 0.258601457, -0.667572737, 0.696138799, -0.993053317, -0.838807523, -0.0655307472, -1.02815151, 0.798331976, -0.815726459, 0.724503458, -0.649456739, 0.614294291, 0.460416168, 0.873559475, -0.949510813, -0.657532334, -0.0608879104, -0.570373476, -1.10029089, -0.822736502, -0.922478616, 0.940835595, -0.899077058, 0.368855715, -1.00277901, 0.92730552, 0.798269868, -0.478674918, 0.0883339942, -0.071504049, 0.541180789, -0.65729475, 0.672089219, 0.947205484, -0.791406691, -0.387015492, -0.0482109673, -0.990223885, -0.723315716, 0.822611749, -0.682777584, 0.875303209, -0.740133286, -1.12873936, -1.03113019, 0.646610975, -1.02559292, -0.839020729, -0.185920268, 1.06680262, 1.1079874, 0.2977615, -1.09732425, 0.924898922, -1.14836562, 0.926818967, -1.08597827, 1.16788375, -0.814071119, -0.753048182, -0.916297138, -0.699535728, 0.864776492, 0.913399637, 0.780896723, -1.04600251, 0.896025121, -1.04204464, -1.00725353, -0.756341934, -1.1111846, 1.00979757, -0.964928448, 0.854104459, -0.710465908, 0.706667006, 0.451359332, 1.19445527, -1.04390681, -0.70082742, -0.599669516, -0.564466417, -0.97518903, -0.821191967, -1.07865798, 1.06515336, -1.03696811, -0.360870332, -1.04832506, 0.949002922, 0.843557, 0.114579149, -0.582424879, 0.458579004, -0.0585701056, -0.282757044, 0.370782673, 1.12461412, -0.743403494, 0.0292093642, -0.698496044, -1.15166843, -0.91422677, 0.859345734, -0.7979846, 1.11669254, -0.942408741, -0.971266806, -0.839450717, 0.265400976, -0.957968533, -0.642010689, 0.0681718066, 0.92869854, 0.871223867, 0.00141623942, -0.832739472, 0.859192967, -0.900926709, 0.905400813, -0.97872901, 0.857826412, -0.864768803, -0.527807772, -0.922775745, -0.564288378, 0.640877545, 0.496911645, 0.346623063, -0.827323258, 0.690292656, -0.957691371, -0.682329834, -0.526140094, -0.966633081, 0.814687014, -0.842431664, 0.901609242, -0.778759956, 0.723447382, 0.584694147, 0.902182043, -0.925217867, -0.74964726, -0.40994525, -0.444771945, -1.03940105, -0.77091974, -0.915254891, 1.03188205, -0.716094017, -0.0730709881, -0.875644445, 1.00034475, 0.802461684, -0.18070288, -0.186475143, 0.326547205, 0.0978334993, -0.40762502, 0.456318825, 0.88022536, -0.918429792, -0.180900455, -0.408369809, -0.979026794, -0.794344068, 0.725096703, -0.819285333, 0.974922955, -0.665378451, -0.957049549, -0.90338701, 0.0117121758, -0.958540559, -0.369567811, 0.426849037, 1.08412206, 0.999146521, -0.457600266, -0.836898386, 0.976403356, -0.787701726, 0.761778176, -0.817251086, 0.854241192, -0.688637435, -0.06189996, -0.870071232, -0.207452789, 0.730751336, 0.474085152, 0.0717327297, -0.732244074, 0.522166133, -0.911408961, -0.733314335, -0.0541811772, -0.902774572, 0.854152024, -0.8356722, 0.973957896, -0.513721168, 0.530448258, 0.5178653, 0.883517206, -0.779456973, -0.876037419, -0.0545621067, -0.581693232, -1.03839672, -0.561269879, -0.884293139, 0.90004611, -0.894381225, 0.329745978, -1.09925151, 1.07232964, 0.588010967, -0.44480446, -0.0150289955, -0.135732114, 0.449506044, -0.564474761, 0.573967218, 0.923888683, -0.830143094, -0.48354727, -0.0832665041, -0.932321787, -0.707611501, 0.837150931, -0.589895606, 0.884020984, -0.700715184, -1.07129419, -0.94995594, -0.00976584293, -0.94228363, -0.781064391, 0.341988683, 0.989681959, 1.05134106, -0.235938579, -0.882476687, 1.01740777, -0.860665202, 0.873909056, -1.04988039, 0.969247997, -0.843372107, -0.373168916, -1.05513656, -0.543990791, 0.902973592, 0.727481186, 0.420580238, -0.72556293, 0.67583847, -0.872810423, -0.809691727, -0.267048627, -0.880384624, 0.952611685, -0.878111124, 0.75098896, -0.905347526, 0.846189082, 0.69805342, 1.09651959, -1.05237222, -0.714071691, -0.193896756, -0.722881973, -1.19934773, -0.788069904, -0.789794445, 1.06000125, -0.970254421, 0.197426975, -1.16599083, 1.12352848, 0.764925361, -0.490962476, -0.0293805785, 0.00408987841, 0.547814965, -0.625176251, 0.731678784, 0.830836356, -0.718104124, -0.571434796, -0.249035984, -1.04093373, -0.854917109, 0.926286042, -0.862562239, 0.946636558, -0.944305599, -0.864344001, -0.910897791, 0.68150562, -0.845130801, -0.767355025, -0.114011943, 0.915433884, 0.943817258, 0.422875434, -0.985541284, 0.847730935, -0.897607744, 0.947556019, -0.968665361, 0.977826774, -0.826483965, -0.590630472, -0.813964248, -0.671755373, 0.914518654, 0.863830805, 0.596408129, -0.833931208, 0.661211967, -0.909825325, -0.786110222, -0.685446739, -0.762152195, 0.644028187, -0.927412987, 0.890666306, -0.803931832, 0.778359175, 0.333450198, 0.912733078, -0.847847164, -0.668307245, -0.691494465, -0.485319674, -0.877907872, -0.841263831, -0.794061542, 0.911942244, -0.912737072, -0.374022633, -0.851201892, 0.917727351, 0.73525089, 0.168483675, -0.720677555, 0.479414254, -0.317186952, -0.420087814, 0.184136882, 0.976621091, -0.574174225, 0.0170140956, -0.751726031, -0.84854877, -0.835730612, 0.905328512, -0.911752164, 0.913094819, -0.606425166, -0.720393538, -0.7295748, 0.344403982, -0.86116308, -0.678945899, 0.156386048, 0.953555405, 0.958199739, 0.236053288, -0.923352778, 0.959935367, -0.819540143, 0.747258306, -0.81029886, 0.928490877, -0.510812819, -0.442689329, -0.753787875, -0.489949971, 0.716122806, 0.511437953, 0.265272439, -0.617701232, 0.737136006, -0.79793036, -0.861609399, -0.474431813, -0.82002455, 0.776415646, -0.819094956, 0.772338271, -0.744754732, 0.727091491, 0.209494978, 0.773643255, -0.739520848, -0.582251787, -0.261787802, -0.388570815, -1.09793127, -0.716441214, -0.578344285, 0.795916021, -0.696612298, -0.00033725932, -0.890256584, 0.788283408, 0.572737217, -0.0883816704, -0.197841734, 0.212345377, 0.0361416079, -0.283466429, 0.232493818, 0.797204554, -0.486870259, 0.0134175075, -0.258473247, -0.682537138, -0.577550709, 0.745770693, -0.75896287, 0.884109318, -0.623207211, -0.867220581, -0.710948288, 0.379665762, -0.955271006, -0.58400768, 0.0693375394, 0.876787901, 0.94924444, 0.219433963, -0.864140511, 0.968326449, -0.811451197, 0.909300387, -0.969635069, 0.980972588, -0.748623669, -0.373714656, -0.786709964, -0.603908598, 0.662294984, 0.610149443, 0.582091868, -0.838529885, 0.630883157, -0.872823894, -0.819868982, -0.34627679, -0.784237802, 0.922452807, -0.829904854, 0.831491649, -0.763492286, 0.610323131, 0.182136059, 0.982402325, -0.871043146, -0.66922152, -0.351899326, -0.324097514, -0.966637254, -0.830069661, -0.704668701, 0.968638301, -0.840793788, -0.0588751137, -1.01591802, 0.898328125, 0.775750339, -0.00615634909, -0.366069883, 0.481870472, 0.0964924991, -0.169103563, 0.396754295, 0.778298557, -0.706937671, 0.0434820503, -0.455761284, -0.858888507, -0.740659833, 0.882302999, -0.84394896, 0.888337612, -0.535447717, -1.03198898, -0.895029485, 0.127248153, -0.945930481, -0.769857585, 0.562765777, 1.08108449, 0.973237276, -0.278321922, -1.00203419, 1.0468998, -0.934166908, 0.930195808, -1.12658882, 1.13442659, -0.844970882, -0.347985625, -0.844344795, -0.595144331, 0.787541151, 0.66479224, 0.257733136, -0.914903939, 0.661600709, -0.887846649, -0.962706029, -0.301309258, -0.951397181, 0.879043639, -1.01958907, 0.957660317, -0.894825041, 0.910873353, 0.714688003, 1.01584494, -1.00434387, -0.855702281, -0.27848807, -0.648084283, -1.12428451, -0.887056768, -0.983325183, 0.952878714, -0.942436814, 0.3327052, -1.05330729, 0.984519899, 0.988032281, -0.358916074, -0.282477677, 0.045628868, 0.512000442, -0.529566646, 0.560500503, 1.10886931, -1.00151324, -0.502405167, -0.285424024, -1.0863452, -0.906020164, 0.932744801, -0.925766945, 0.920359969, -0.871665955, -0.817522347, -0.717796504, -0.158151135, -0.863889277, -0.152621597, 0.688364267, 0.856443346, 0.771175086, -0.352219135, -0.674328327, 0.876321375, -0.670305192, 0.843350589, -0.810701311, 0.819873393, -0.714629114, -0.0204545502, -0.378520131, -0.0482513569, 0.242488727, 0.0897907093, 0.0545988567, -0.787264764, 0.0480587967, -0.882032633, -0.442056656, 0.0729326531, -0.657725036, 0.671104193, -0.813675404, 0.853086352, -0.265330464, 0.331832349, 0.595983624, 0.739224374, -0.658296227, -0.706247509, -0.0336610824, -0.703258991, -0.767020404, -0.345975459, -0.670200765, 0.81023109, -0.436149299, 0.552532375, -0.704727888, 0.911493361, 0.26556921, -0.45797956, 0.0300160442, -0.135582045, 0.692435324, -0.649664879, 0.724178016, 0.791167319, -0.790905714, -0.700752556, 0.219975486, -0.697214186, -0.321251899, 0.810950577, -0.340426624, 0.754207373, -0.74222219, -0.819306135, -0.766723752, 0.314272404, -0.935828149, -0.65202117, -0.18344748, 0.929053664, 0.91260159, 0.303058803, -0.800495148, 0.8713696, -0.978657484, 0.808263004, -0.838800609, 0.894504189, -0.769154191, -0.474667847, -0.890345633, -0.482116401, 0.693107367, 0.771432281, 0.442364931, -0.885446906, 0.713657737, -0.78001231, -0.755061567, -0.507024229, -0.982696831, 0.936754942, -0.793481112, 0.706687093, -0.734841406, 0.859075546, 0.340908557, 0.833788395, -0.923908651, -0.848967314, -0.445634305, -0.551591039, -0.933882296, -0.682923257, -0.852004349, 0.970587134, -0.928369403, -0.210079119, -0.934322774, 0.916409254, 0.775862932, 0.0422250032, -0.39993611, 0.403054774, -0.00731305499, -0.3526223, 0.326264381, 0.925620496, -0.781861186, -0.00949419197, -0.387069046, -0.809717894, -0.820062637, 0.859523118, -0.76733762, 0.765727401, -0.784216285, -1.11812997, -0.859784126, 0.561689198, -1.17836523, -0.859569669, -0.0625344366, 1.14610291, 0.939392269, 0.34284386, -1.0861398, 1.05282509, -1.02815473, 0.997420728, -0.861877143, 0.983874798, -0.787852466, -0.627726138, -0.967456102, -0.698395312, 0.801503778, 0.769794881, 0.753206849, -0.813829124, 0.968657494, -1.04559875, -0.871890247, -0.649935424, -1.08626008, 1.00657034, -0.901096225, 0.758995354, -0.975984812, 0.952033877, 0.387914717, 1.19572413, -0.873779893, -0.75214678, -0.536943436, -0.281765401, -1.25894392, -0.852993906, -0.817538559, 0.986916542, -0.889575183, -0.0633313432, -1.10451198, 1.08292651, 0.807317436, -0.0711139217, -0.559311986, 0.487922519, -0.12266469, -0.262568772, 0.382075876, 0.84499675, -0.856390953, -0.00263357954, -0.567296922, -1.0022068, -1.0351007, 0.828041255, -0.811619401, 0.850459337, -0.66757822, -1.01101673, -0.691120863, 0.674151719, -0.852256477, -0.733033955, -0.402994603, 0.972786844, 1.00774634, 0.681202114, -0.96730262, 0.797137618, -0.786753058, 0.859865248, -1.00905955, 1.05705845, -0.680681109, -0.900515974, -0.812533915, -0.917396307, 1.02717853, 0.940837026, 0.798831761, -0.806271732, 0.945535362, -1.00621688, -0.871542335, -0.68930161, -0.867748559, 0.810870469, -0.826174796, 0.756949842, -0.770619273, 0.837704062, 0.379606724, 0.95077455, -0.832608163, -0.740756869, -0.834090948, -0.347329348, -1.02992558, -1.01722944, -0.81105423, 0.99357599, -0.930593729, -0.624682128, -1.06663835, 0.948874414, 0.884503841, 0.314552873, -0.662997782, 0.852961361, -0.307718426, -0.233914047, 0.0506733842, 0.889522016, -0.594542623, 0.10731367, -0.839280009, -0.805817366, -0.990870893, 0.860335827, -0.971334398, 0.695464194, -0.590175569, -0.992984831, -0.916395068, 0.23752214, -0.811707914, -0.605515122, -0.0289754141, 1.01348734, 0.885276437, -0.0195621662, -0.930562556, 0.879725218, -0.791247368, 0.818392634, -0.887332559, 0.830451667, -0.81298095, -0.364100933, -0.95015794, -0.532445252, 0.723904669, 0.489164263, 0.53073287, -0.770344555, 0.516097724, -0.77816397, -0.819258988, -0.527508438, -0.782685339, 0.917488337, -0.987100363, 0.880340993, -0.676350951, 0.785340846, 0.411043912, 0.94011718, -0.836034477, -0.787358463, -0.492183775, -0.377437592, -1.07014406, -0.77786088, -0.858503938, 0.758644164, -0.816026211, 0.0425491221, -0.937254548, 1.03547621, 0.640421748, -0.0199737195, -0.454919845, 0.369799823, 0.184253171, -0.419892371, 0.2992706, 0.81585288, -0.672169447, -0.106847234, -0.33666116, -0.955514789, -0.746241271, 0.78523308, -0.723766387, 0.747978032, -0.6113